(* IEC 61131-3 sources: tf-plc/examples/models/structured_text (part 7) *)

    weights_2 : ARRAY[0..287] OF REAL := [-0.187368, -0.051744, -0.039838, -0.182706, 0.020143, 0.109520, 0.194103, 0.170830, 0.202326, -0.167691, -0.195653, -0.237644, 0.106375, -0.036592, -0.006802, 0.135748, 0.022817, -0.062333, -0.017378, 0.128592, 0.187297, 0.185332, -0.152342, -0.201742, -0.104000, 0.041331, 0.068691, -0.044867, -0.198049, 0.149257, 0.125627, -0.021191, 0.074122, -0.145982, 0.118018, -0.081354, -0.131859, -0.051540, 0.168976, 0.046712, -0.040107, -0.054049, 0.084196, -0.269932, -0.139673, -0.139174, 0.131241, -0.010010, 0.138380, -0.188378, -0.036906, 0.057354, 0.008294, -0.113937, -0.038322, -0.006458, -0.001382, 0.096871, -0.011427, -0.108642, -0.113846, 0.096256, -0.134778, -0.045314, 0.048023, -0.015410, -0.087083, 0.081638, 0.095536, 0.014215, 0.110213, 0.167564, 0.020146, -0.133820, -0.078020, 0.007872, -0.044209, 0.044677, 0.131990, -0.089845, 0.145099, -0.119614, -0.106027, -0.091758, 0.077236, 0.042917, 0.118902, 0.120238, -0.244683, 0.045377, 0.197385, -0.131725, 0.193356, 0.124749, -0.181955, 0.108950, 0.119074, -0.070678, -0.009053, -0.087902, -0.065026, 0.183027, -0.196468, 0.195945, -0.166252, -0.165656, -0.164554, -0.076295, 0.139092, 0.190423, -0.007008, 0.013343, 0.018061, -0.073660, -0.022792, 0.075813, 0.097410, 0.177929, -0.145417, 0.025251, 0.175258, -0.197919, -0.079814, -0.340062, -0.006446, 0.052857, 0.114206, 0.051889, 0.145295, -0.146757, 0.093871, -0.111949, -0.084611, -0.067383, -0.099881, -0.057531, -0.233824, -0.186072, 0.174656, 0.076755, 0.009728, 0.104689, 0.106295, -0.179713, -0.113384, 0.079812, 0.132616, 0.004269, -0.171604, -0.030952, -0.045874, -0.015698, 0.004115, 0.010316, -0.183566, 0.082135, 0.082901, 0.090530, 0.143641, -0.040666, -0.152231, 0.207951, 0.124544, 0.016117, 0.046549, 0.030973, 0.043746, 0.036781, -0.086853, -0.171788, -0.013353, 0.078074, -0.141704, -0.113534, -0.045675, 0.082511, 0.031405, 0.099222, 0.061383, -0.090559, 0.025971, 0.117368, -0.137792, -0.203968, -0.087473, 0.150403, 0.221516, -0.053973, 0.100427, -0.012862, 0.224251, 0.226762, -0.101491, 0.057445, 0.086675, 0.134510, -0.058083, -0.216293, -0.036254, -0.225297, -0.080859, 0.008825, 0.033891, 0.143634, 0.059084, 0.023081, 0.094791, -0.194769, -0.001480, 0.073488, 0.115785, -0.061513, -0.130487, 0.057053, 0.185202, -0.062696, -0.098506, -0.052882, -0.012272, -0.177827, 0.048385, 0.121327, 0.044788, -0.111825, -0.129649, 0.139996, 0.051313, -0.047422, -0.002531, -0.233266, -0.124867, -0.128167, -0.082153, -0.073802, 0.102312, -0.003983, 0.033367, -0.024256, -0.227793, -0.130058, -0.093124, -0.002918, 0.156583, -0.133267, -0.070283, -0.019832, 0.240679, 0.192125, 0.226900, -0.215979, -0.037737, -0.027495, 0.257100, 0.067004, 0.162718, -0.035639, -0.025185, 0.145988, -0.062046, 0.179573, 0.208897, -0.050213, 0.200720, 0.185337, 0.195171, 0.145625, 0.199399, 0.174908, -0.021887, 0.128953, -0.153483, -0.080969, -0.116301, 0.002837, 0.088707, 0.122016, -0.069452, -0.073120, -0.099167, -0.086314, 0.211113, 0.213622, 0.087920, -0.150208, -0.143647, -0.111789, 0.093171, 0.048712];
    bias_2 : ARRAY[0..2] OF REAL := [0.178373, 1.153172, -1.176576];

END_VAR

VAR
    (* Buffer allocation variables *)
    buffer_0 : ARRAY[0..95] OF REAL;
    buffer_1 : ARRAY[0..127] OF REAL;

    (* Temporary computation variables *)
    i : DINT;
    j : DINT;
    sum : REAL;
    max_val : REAL;
    exp_sum : REAL;

END_VAR

(* Layer 0: Fused Linear + RELU *)
FOR j := 0 TO 127 DO
    sum := 0.0;
    FOR i := 0 TO 4 DO
        sum := sum + input_data[i] * weights_0[i * 128 + j];
    END_FOR;
    buffer_1[j] := MAX(sum + bias_0[j], 0.0);
END_FOR;

(* Layer 1: Fused Linear + RELU *)
FOR j := 0 TO 95 DO
    sum := 0.0;
    FOR i := 0 TO 127 DO
        sum := sum + buffer_1[i] * weights_1[i * 96 + j];
    END_FOR;
    buffer_0[j] := MAX(sum + bias_1[j], 0.0);
END_FOR;

(* Layer 2: Fused Linear + SOFTMAX *)
FOR j := 0 TO 2 DO
    sum := 0.0;
    FOR i := 0 TO 95 DO
        sum := sum + buffer_0[i] * weights_2[i * 3 + j];
    END_FOR;
    output_data[j] := sum + bias_2[j];
END_FOR;

max_val := output_data[0];
FOR i := 1 TO 2 DO
    IF output_data[i] > max_val THEN
        max_val := output_data[i];
    END_IF;
END_FOR;

exp_sum := 0.0;
FOR i := 0 TO 2 DO
    output_data[i] := EXP(output_data[i] - max_val);
    exp_sum := exp_sum + output_data[i];
END_FOR;

FOR i := 0 TO 2 DO
    output_data[i] := output_data[i] / exp_sum;
END_FOR;

END_FUNCTION_BLOCK

(* ---- test6_52k.st ---- *)
FUNCTION_BLOCK NeuralNetworkFB

VAR_INPUT
    input_data : ARRAY[0..4] OF REAL;
END_VAR

VAR_OUTPUT
    output_data : ARRAY[0..2] OF REAL;
END_VAR

VAR CONSTANT
    weights_0 : ARRAY[0..1279] OF REAL := [-0.070155, -0.038928, -0.060831, 0.071798, 0.002485, -0.001928, 0.071168, 0.040746, -0.011541, 0.011445, 0.033770, -0.092213, 0.017192, -0.118437, -0.098900, -0.051498, 0.004445, -0.006958, -0.025937, -0.127331, -0.033657, -0.020618, -0.089709, 0.067849, 0.032140, 0.027497, 0.034283, 0.044327, -0.041753, -0.071082, -0.023682, -0.090062, 0.088008, 0.007363, -0.073022, -0.031094, 0.042343, -0.067819, -0.017369, 0.056200, -0.086665, 0.056540, 0.024530, -0.093938, 0.012128, -0.109124, 0.043440, -0.042579, -0.016699, 0.004629, -0.082224, 0.015294, 0.014115, 0.027542, 0.014956, -0.021326, -0.135801, -0.044497, 0.006702, -0.013372, 0.013572, -0.004992, -0.067393, 0.015628, -0.044148, -0.024818, -0.001204, -0.007329, -0.112170, -0.094539, 0.009056, -0.031292, 0.066635, -0.026743, 0.002959, -0.164818, 0.041633, -0.146296, -0.119213, -0.024292, -0.025669, -0.181450, -0.006220, -0.075742, -0.011598, -0.002342, -0.026022, -0.097560, -0.021554, -0.012841, -0.050252, -0.103415, -0.029755, 0.012920, -0.010506, 0.006163, -0.086429, -0.082030, 0.041432, -0.020474, 0.059144, -0.007111, 0.003627, -0.155405, 0.002022, -0.031367, 0.028444, 0.041676, 0.054722, -0.002389, -0.071904, -0.012697, -0.021735, 0.006464, 0.051797, -0.067293, -0.057014, 0.035573, -0.061071, -0.045083, 0.003018, 0.041802, -0.097514, 0.002537, -0.057788, -0.071212, -0.054268, -0.012065, -0.017229, -0.022461, 0.063413, 0.005719, 0.022329, -0.099895, -0.169818, -0.108498, -0.092381, -0.012462, -0.023149, -0.024445, 0.001542, -0.032483, -0.113439, -0.054737, -0.004174, -0.010661, -0.019861, 0.037820, -0.132428, 0.022416, 0.011167, -0.055828, -0.034627, -0.058847, 0.018462, 0.025207, 0.008687, -0.013364, 0.049810, -0.020141, -0.018092, 0.025560, -0.021438, -0.034213, -0.023112, -0.027428, -0.112417, -0.060424, -0.006416, -0.000760, -0.237476, -0.086897, -0.081624, -0.070778, -0.009070, 0.027652, -0.129067, -0.014944, 0.070686, -0.006345, 0.018438, -0.048882, -0.056557, 0.062420, -0.013772, 0.014728, -0.015230, -0.076275, 0.001375, -0.011276, 0.055686, -0.049352, -0.030465, -0.023252, 0.003113, -0.023272, -0.035683, -0.076872, -0.011587, 0.004628, -0.030451, -0.045972, -0.004618, -0.025772, -0.087139, 0.004941, -0.025864, 0.024506, -0.078173, -0.092430, 0.019720, -0.007388, -0.031572, -0.029024, -0.016634, 0.007754, -0.131151, 0.000328, -0.051390, -0.012149, 0.023158, -0.010932, 0.001055, 0.019128, -0.102080, -0.010931, -0.004006, 0.002197, -0.046069, -0.077169, 0.041212, -0.009728, 0.006004, -0.136275, 0.041067, 0.023654, 0.053500, 0.007832, -0.052076, -0.010449, -0.061968, 0.004481, -0.017595, -0.114258, -0.086593, -0.011651, 0.022509, -0.070902, -0.014800, -0.082160, -0.123492, -0.043907, 0.016663, -0.004434, -0.054333, 0.003070, 0.089158, 0.025455, 0.057796, -0.060061, -0.053971, -0.149259, -0.048506, -0.131124, -0.069589, -0.080767, -0.101356, 0.024470, 0.060420, 0.024438, -0.048683, 0.003822, 0.001343, -0.000167, 0.044828, 0.070380, -0.072733, -0.003184, 0.066587, -0.008192, -0.074305, -0.068878, -0.004405, -0.115034, 0.052002, 0.015329, -0.068499, 0.086396, 0.005960, -0.052240, 0.085370, -0.002848, -0.093293, 0.056188, -0.044788, -0.007773, 0.056717, 0.055797, 0.034819, 0.070412, 0.016734, 0.026962, -0.057618, 0.037052, -0.052987, -0.121634, 0.024814, -0.146882, -0.013487, -0.083349, -0.024382, 0.026361, 0.101833, -0.002916, -0.006728, 0.015952, -0.015001, -0.004409, 0.042099, -0.126239, -0.019967, -0.013365, -0.089322, -0.006933, 0.059515, 0.037254, 0.045940, -0.074429, 0.040376, -0.027424, -0.080917, 0.035436, -0.094184, 0.086872, 0.085092, -0.091239, -0.026700, 0.043759, -0.012511, 0.063707, -0.027418, -0.008543, -0.119174, 0.009577, -0.061811, -0.094772, -0.022777, 0.022945, -0.005291, -0.032016, -0.059554, 0.046357, 0.075232, 0.040890, -0.148068, -0.049176, -0.063437, -0.004632, -0.026976, 0.105835, -0.039771, -0.031932, 0.011247, -0.132174, -0.032898, -0.073880, 0.088190, -0.053595, -0.043657, -0.188433, 0.014483, -0.032608, 0.091753, -0.101293, 0.051511, 0.070593, 0.004308, -0.037419, 0.076578, -0.054873, 0.099081, 0.003978, -0.081189, -0.127868, 0.054014, 0.114358, -0.023209, -0.011056, -0.110387, 0.098939, 0.080905, 0.080982, 0.096756, -0.078019, 0.020367, -0.011403, -0.049023, 0.027064, 0.045508, -0.029634, -0.027102, -0.001639, -0.051489, 0.038324, -0.060108, -0.090780, -0.070994, 0.013411, 0.029360, 0.048912, 0.032128, -0.033461, -0.088759, -0.006212, -0.115797, -0.025116, -0.056739, -0.064863, -0.018670, -0.114987, -0.056438, -0.030989, 0.092064, 0.189426, -0.025521, 0.023734, 0.049321, 0.059772, 0.003554, 0.131488, 0.021443, -0.112435, 0.054834, 0.073230, -0.001986, -0.073395, -0.088302, -0.088925, -0.006384, -0.017310, -0.022798, -0.173727, -0.023516, 0.107446, -0.011929, -0.035021, 0.039987, -0.033331, 0.028726, 0.007168, -0.073183, -0.021234, 0.039145, 0.072611, -0.171738, 0.066412, 0.031766, -0.144949, -0.042576, 0.096573, 0.008219, -0.068725, 0.015551, 0.032414, 0.043340, 0.033251, -0.078822, -0.124831, -0.110806, -0.004724, 0.045751, -0.038142, 0.191380, -0.055027, 0.060193, -0.041085, -0.025719, 0.040618, -0.056256, -0.008186, 0.069378, -0.035653, -0.084666, -0.038777, -0.058272, 0.019557, -0.136677, 0.065821, -0.102945, 0.050225, 0.018768, -0.064491, -0.091170, -0.006610, -0.032372, -0.123312, -0.026740, 0.070938, 0.001682, 0.065152, 0.035602, -0.010920, -0.117728, -0.045748, -0.028254, 0.012258, 0.147745, -0.019861, 0.060016, -0.048321, 0.020267, -0.102670, 0.020371, 0.036374, 0.049515, -0.085354, -0.004292, 0.032160, -0.047433, 0.015542, 0.003641, -0.001895, 0.039274, -0.046615, -0.016797, 0.007867, 0.096931, -0.006988, -0.073010, 0.025101, -0.081308, 0.030847, 0.031478, 0.015346, -0.066517, -0.199175, 0.092511, -0.083915, -0.144285, 0.058104, -0.086546, -0.018784, 0.035585, -0.058032, 0.018627, 0.052126, 0.017639, -0.000476, 0.115320, -0.064683, -0.022925, 0.007203, -0.020902, -0.037572, -0.042251, -0.046520, -0.123537, 0.049099, -0.212938, 0.041265, 0.029031, 0.034293, 0.038876, 0.019368, -0.166769, -0.036728, 0.011981, -0.056179, 0.014853, -0.017817, -0.052471, -0.052235, -0.109694, -0.017080, 0.027348, 0.072501, -0.023639, 0.039061, -0.021487, 0.004655, -0.077402, -0.030520, 0.049986, 0.015832, -0.107897, 0.019971, 0.077300, -0.067741, -0.016473, -0.016751, -0.142127, 0.027512, -0.076044, -0.049235, -0.036304, 0.005174, 0.034315, -0.048157, -0.019821, 0.034346, 0.021618, -0.014229, -0.108075, 0.031648, 0.023075, -0.146272, 0.066495, -0.103423, -0.090994, -0.007711, 0.138765, 0.023170, -0.011847, -0.025818, 0.004740, -0.090616, -0.039913, -0.036852, 0.018737, 0.024087, -0.099178, 0.090088, -0.022893, -0.002647, -0.036183, 0.054486, -0.109386, 0.009673, -0.054158, -0.036976, 0.037600, 0.022299, -0.092783, -0.059639, 0.001632, -0.018608, -0.112979, 0.022739, 0.040180, -0.030441, -0.105134, 0.033549, -0.106905, -0.046508, -0.094102, 0.000469, 0.057010, 0.023167, -0.086274, 0.045263, -0.049488, -0.052119, -0.037550, -0.022030, -0.010889, 0.003728, -0.008856, -0.083921, 0.133954, -0.080053, -0.017677, 0.094552, 0.068978, 0.020386, -0.025452, -0.168631, -0.090440, -0.195507, -0.003636, -0.084083, -0.068182, 0.058592, 0.029474, 0.040437, 0.061063, 0.025880, -0.001188, 0.000644, 0.010631, -0.110092, -0.000888, -0.141433, 0.108213, -0.022925, 0.000002, -0.130711, -0.062924, 0.008210, 0.019788, -0.175506, -0.039343, 0.045400, 0.123293, 0.092991, 0.016389, 0.004282, -0.004402, 0.075178, 0.003878, -0.106472, -0.002041, -0.004386, -0.036288, -0.002075, -0.062324, -0.014999, 0.041272, -0.017299, -0.065019, 0.063675, -0.028323, 0.020868, 0.058101, -0.043334, -0.045801, -0.052023, -0.069590, 0.053231, -0.069505, -0.033325, -0.063689, 0.014256, -0.067391, 0.005150, 0.014229, -0.018608, -0.039890, -0.104577, -0.153014, 0.020215, -0.030304, 0.036193, -0.106386, 0.008862, 0.040607, 0.011998, -0.043155, -0.008992, -0.005723, -0.012143, 0.037371, -0.016482, 0.095962, 0.051428, 0.012461, 0.050556, -0.075283, 0.013162, -0.012846, 0.062124, 0.080743, -0.025501, 0.139815, -0.065035, -0.005680, 0.005855, 0.048577, -0.014476, 0.120541, 0.069732, 0.030624, 0.049617, -0.192638, -0.032519, -0.154690, -0.022641, -0.025504, 0.012953, -0.027163, -0.031450, 0.065519, -0.104127, 0.037112, -0.119223, -0.095449, 0.035030, 0.034269, 0.024936, -0.046396, -0.025763, 0.005578, -0.043447, 0.019468, 0.028594, 0.004105, -0.158852, 0.010332, -0.055373, -0.080652, -0.053025, 0.093439, -0.167693, -0.056412, 0.084124, 0.138518, 0.010848, 0.047750, 0.065364, -0.054384, -0.045877, -0.157582, -0.058733, 0.018936, 0.010344, -0.077384, 0.028530, -0.036928, -0.080216, -0.012947, -0.183244, -0.072780, 0.075381, 0.062871, -0.028872, -0.298677, -0.122305, 0.024540, -0.183726, -0.086483, 0.028399, -0.020734, -0.022262, -0.050299, 0.060296, -0.118434, 0.011326, -0.046636, -0.025086, 0.066485, 0.015072, -0.007407, -0.044429, 0.119766, -0.047552, 0.063841, 0.005677, -0.020033, -0.024924, -0.233876, -0.022696, -0.111984, -0.043489, -0.051726, 0.036200, 0.070647, -0.001496, 0.052031, 0.090468, -0.004369, -0.060146, 0.019014, -0.042590, 0.009331, 0.075433, 0.015205, 0.045605, -0.016796, -0.001694, -0.110277, -0.107970, -0.011359, 0.017214, -0.087149, -0.066041, -0.040559, 0.002534, 0.000869, -0.049051, -0.134641, -0.071958, -0.090083, -0.033740, -0.027785, -0.014719, -0.067009, 0.054519, -0.112509, -0.141188, -0.101297, 0.027771, -0.021707, -0.026334, -0.046971, 0.081692, -0.052515, 0.042934, 0.002791, -0.025111, -0.005613, -0.003938, -0.041332, -0.026735, -0.021925, -0.056798, 0.066753, -0.013360, 0.035447, 0.029946, -0.050330, -0.020345, 0.102162, -0.016480, -0.009511, 0.017979, -0.000835, -0.016305, -0.005105, -0.034165, -0.094269, -0.030100, -0.018412, -0.009383, 0.003034, 0.058877, -0.094282, -0.001475, -0.008207, -0.135370, -0.018500, -0.028991, 0.023336, -0.155066, 0.068173, 0.106962, 0.025825, -0.009390, 0.192936, -0.002078, -0.033218, -0.064921, -0.042340, 0.023166, 0.001465, 0.003338, -0.087242, 0.088695, -0.064151, 0.023704, -0.042815, 0.040228, -0.088100, 0.029738, 0.052976, -0.017066, -0.013374, -0.115260, -0.151356, -0.057710, -0.126411, 0.031555, -0.056856, 0.036591, 0.034966, 0.008604, -0.002094, -0.092756, -0.202693, 0.028386, 0.024546, 0.076751, 0.017080, -0.018400, -0.037468, 0.032381, -0.089056, -0.187506, 0.129519, -0.021868, -0.080211, 0.100733, 0.030251, -0.004738, -0.024252, -0.009992, -0.027219, -0.172047, 0.029982, -0.126244, 0.126345, -0.019377, 0.012645, -0.025258, -0.065075, 0.028387, -0.041856, -0.017149, 0.030092, 0.000136, -0.004336, -0.093402, -0.012175, 0.005064, 0.021007, 0.024673, 0.024129, -0.034974, 0.004802, -0.013058, -0.053403, -0.190563, -0.019771, -0.090807, 0.061242, -0.032385, 0.046829, 0.005640, -0.098551, 0.083228, -0.062776, -0.092552, -0.069659, -0.059411, -0.109861, -0.007731, -0.057467, -0.123494, 0.004573, -0.083022, -0.016332, 0.051041, 0.110085, 0.073775, 0.004332, 0.020398, -0.023250, -0.240979, 0.044898, -0.046601, -0.058876, 0.054855, 0.074309, -0.081339, -0.042678, -0.073336, -0.128968, -0.047388, 0.046222, -0.051490, -0.121539, -0.014110, 0.015559, -0.096600, -0.026040, 0.032576, -0.048588, -0.136002, -0.095979, 0.036955, 0.120072, 0.117148, -0.211939, 0.082600, -0.083967, 0.111170, -0.045167, -0.052241, -0.135401, -0.065841, -0.088071, -0.020966, -0.022402, -0.022904, 0.015520, 0.135462, -0.039160, 0.030723, 0.095178, -0.072782, -0.122238, 0.017292, 0.137500, -0.023816, -0.043778, 0.078469, -0.029312, -0.022650, 0.019829, -0.054630, 0.004616, -0.052215, -0.042087, -0.029251, -0.010856, 0.017121, 0.000070, -0.000649, -0.167285, -0.133736, -0.115300, -0.070077, -0.072475, -0.028821, 0.017386, -0.026148, -0.075110, -0.140864, -0.265319, 0.034329, -0.032104, -0.108525, 0.078500, -0.021793, -0.019431, -0.080346, 0.010413, -0.075056, -0.007622, 0.000705, 0.074607, -0.090247, -0.168186, -0.039990, 0.031701, -0.071391, -0.018511, 0.014074, -0.022277, -0.023848, -0.025741, 0.026712, -0.067890, -0.028615, -0.066786, -0.023857, 0.044643, -0.013439, 0.111842, -0.073162, 0.005626, 0.026295, 0.080199, -0.108263, 0.001735, -0.108968, -0.149550, -0.043386, -0.001566, 0.012777, -0.011432, -0.195532, -0.000366, -0.033416, -0.085170, -0.005145, -0.030513, -0.069574, -0.100038, -0.027521, -0.074923, -0.100165, -0.104816, -0.065458, -0.013671, -0.442613, 0.025321, -0.030204, 0.013435, -0.012925, 0.006500, -0.379789, -0.014098, -0.052213, -0.030067, -0.087624, 0.038926, -0.044570, 0.059827, -0.018701, -0.029826, -0.133173, -0.116575, -0.012915, -0.023978, -0.024605, -0.153727, 0.037398, -0.021229, -0.068256, 0.080290, 0.051136, -0.059677, -0.024896, -0.248148, -0.052647, -0.045824, -0.042903, -0.291025, -0.024924, -0.014856, -0.032847, -0.013471, -0.064484, -0.000900, -0.064762, 0.063787, -0.061784, 0.022854, 0.069113, -0.139692, -0.025717, 0.024155, 0.025020, 0.013773, -0.025551, -0.028811, 0.002795, -0.056229, -0.253997, -0.059094, -0.055135, -0.027552, -0.055112, -0.061042, -0.090559, -0.302910, -0.153096, -0.108954, 0.002854, -0.065210, -0.058173, 0.042017, -0.152229, -0.018775, -0.276441, 0.115907, -0.061645, -0.046450, 0.088557, -0.030303, 0.108731, -0.035072, -0.089776, -0.036277, 0.031124, -0.120535, -0.084175, -0.034725, -0.048802, -0.314331, 0.044946, -0.064024, 0.040152, -0.048355, -0.067662, -0.021274, -0.042630, -0.228118, -0.142731, -0.022468, -0.072343, -0.034337, -0.025426, -0.029231, -0.028560, -0.059697, -0.185525, -0.011706, -0.098026, 0.066904, -0.028047, 0.102726, 0.096580, -0.092999, -0.048373, -0.263141, 0.136710, -0.097510, -0.041869, 0.014649, -0.041501, -0.043015, -0.089343, -0.077332, -0.101542, -0.098549, -0.095657, -0.183604, -0.095671, -0.010110, -0.157311];
    bias_0 : ARRAY[0..255] OF REAL := [1.761415, 0.448067, -0.616874, -0.484059, 0.264607, -0.939340, 1.879217, 0.387234, -0.224406, -0.592480, 0.573221, -0.500961, -1.606627, 0.053632, -0.815345, -0.331633, -0.254809, 0.114883, 0.034678, -0.491211, -0.556383, 0.517875, -0.619894, -0.175753, -1.234692, -0.794876, 0.608074, -1.463195, -0.042061, -0.962730, -0.235608, 0.198914, -0.023740, 0.011105, 0.650481, 0.174745, 0.899415, -0.358974, -0.603442, -1.367541, -0.065719, -0.929502, -0.847885, -0.365598, -0.106994, -0.493744, -0.071272, -0.507953, -0.072654, 0.642076, -0.468674, -0.864381, -1.117401, -0.245438, -0.073791, -0.435633, 0.299667, -0.095896, -0.052645, 0.095357, -0.586712, -0.615622, -0.026960, -0.250394, -0.784761, -0.225061, -0.657271, -0.407327, -0.230763, -0.098783, -0.037782, 0.199574, 0.593063, -0.725165, -0.492830, 0.248655, -1.223977, 0.003933, -0.103927, -0.255865, -0.239717, 0.080054, -0.552899, -0.238874, -1.349266, 0.138204, -1.088216, -0.206781, -0.391251, -0.378652, -0.585402, -0.228141, -0.377184, -0.224824, -0.723177, -0.617806, 0.083839, -0.155374, 1.478903, -0.308232, -0.179639, -0.159381, -0.263020, -0.181034, -0.507353, -0.264171, -1.168516, -0.972790, 0.189400, 0.139605, 0.125825, -0.717963, -0.294487, -0.057633, 0.015071, 0.269775, -0.534699, -0.084028, -0.079780, -0.401683, 0.027464, 0.074169, -0.013114, 0.126892, -0.778323, 0.311368, -0.224082, -1.059481, -1.343553, -0.005818, -0.149338, 0.081988, -0.058032, -0.328252, -0.384153, 0.146061, -0.012248, -0.017525, -0.254924, -0.230246, -0.753802, -0.348697, -0.681305, -0.580557, -0.063855, 1.148852, 0.216549, 1.353733, -0.041907, -0.766222, -0.039394, -0.722909, -0.515027, -0.293167, -1.141858, -0.532181, -0.700502, -0.093383, 0.853853, -0.491534, -0.364100, 1.343948, 0.206487, -0.739496, -0.120556, -0.194485, 0.531750, -0.071946, -0.429285, -1.223201, -0.799083, -0.240277, -0.253012, -1.097437, 1.321796, -0.732158, -0.643209, 0.023920, -1.042058, -0.577268, -0.130637, -0.380038, -0.697286, 0.272227, -0.397080, -0.299311, -0.152759, -0.012990, -0.102990, -0.175804, 0.514636, 0.076499, -0.173979, -0.501178, -0.362724, -0.373031, -0.193449, 0.413115, -0.477030, 0.085947, -0.924347, -0.343727, 0.956858, -1.252704, 0.042583, -0.986913, 0.150553, 0.331016, 0.022171, 0.308270, -0.172095, -0.276784, -0.621540, -0.314609, 0.217584, 0.068779, -0.080378, -0.521706, -0.216527, -0.760283, -0.076289, 1.077613, 0.342408, 1.537670, -0.199558, 0.696804, -0.477082, -0.216091, -0.627426, -0.344922, -0.476790, 0.048585, -0.653165, 0.220433, -1.102417, 0.015778, -1.255825, -1.064247, 0.158786, 1.424948, -0.014341, -1.144714, 0.264992, -0.409402, -0.673654, 0.344695, -0.371929, -0.803940, 0.197236, 0.139407, -0.046033, -0.167134, -0.541114, -0.539192, -0.470981, -0.991606];

    weights_1 : ARRAY[0..50175] OF REAL := [0.019087, 0.112252, 0.211727, 0.072814, 0.087899, -0.175614, -0.015506, 0.164059, 0.236532, -0.229048, -0.055866, 0.004746, 0.085537, -0.126006, -0.170778, 0.039044, -0.227048, -0.200908, 0.085609, -0.210631, 0.017052, 0.078471, -0.091614, -0.312604, -0.219523, -0.039882, 0.227878, 0.098304, 0.053254, 0.175391, 0.027453, 0.004954, 0.256044, 0.220982, -0.118379, -0.043911, 0.113699, -0.067441, 0.121477, -0.081606, 0.017963, -0.108318, -0.122663, 0.122943, -0.098493, -0.129229, -0.104070, -0.040965, -0.030263, 0.103501, 0.114757, -0.033213, -0.097106, -0.003870, -0.064622, -0.031450, 0.136162, 0.043457, 0.119389, 0.086272, 0.086328, -0.054092, 0.022835, 0.076201, 0.115069, -0.146640, -0.019403, 0.182401, -0.070480, 0.040452, 0.252047, 0.027936, 0.131226, -0.044332, -0.068760, -0.075233, 0.136624, 0.010865, 0.031996, 0.217943, 0.132278, 0.094806, -0.081434, -0.018107, -0.011303, -0.132485, -0.155610, 0.010216, 0.251893, 0.008599, 0.088021, -0.110349, -0.184611, -0.165733, -0.023405, 0.070966, 0.052070, -0.066027, 0.206689, -0.139396, 0.065651, 0.040476, 0.265397, 0.200300, -0.161854, -0.035440, -0.100544, 0.060114, 0.132822, 0.181317, 0.162731, -0.157100, 0.032291, -0.024872, 0.026177, -0.062704, -0.227261, -0.061749, 0.001810, 0.143090, 0.297814, -0.094348, -0.189725, 0.023125, 0.100221, -0.079787, 0.014617, 0.045027, 0.126831, 0.107187, -0.033158, 0.172206, 0.084450, 0.023537, -0.137875, -0.059479, -0.015502, 0.066624, -0.388477, 0.056747, 0.095752, -0.076781, -0.090368, -0.033154, 0.006288, 0.066518, -0.177086, 0.016229, 0.237689, -0.198316, -0.126118, -0.093328, 0.283691, -0.024487, -0.033743, -0.047251, 0.048239, 0.011724, 0.182427, -0.122201, -0.063529, 0.153458, -0.024413, 0.046109, -0.057552, -0.027173, 0.109429, 0.110716, 0.187617, 0.078747, 0.105684, 0.073501, -0.010930, 0.094036, 0.255130, -0.016355, 0.064772, 0.166211, 0.051418, -0.100114, 0.103828, -0.122074, -0.013134, -0.013142, 0.051070, -0.141888, -0.073589, 0.047752, 0.118184, -0.150595, -0.069933, -0.111839, 0.201886, 0.157238, -0.000566, -0.241842, -0.103816, -0.167649, 0.036014, -0.071474, -0.197229, -0.093806, -0.117186, -0.121392, 0.090752, 0.057172, -0.101006, -0.146829, -0.162285, -0.114287, 0.041882, -0.021359, 0.039685, -0.051023, -0.088828, -0.130283, 0.071467, -0.027591, 0.063893, -0.060089, -0.039073, -0.080926, -0.039526, -0.175741, -0.072726, -0.002156, -0.064652, -0.032380, -0.078773, -0.139573, -0.095449, 0.025900, 0.061990, 0.011282, -0.073379, -0.164573, -0.087662, -0.047434, -0.138482, 0.065975, 0.141275, 0.072849, 0.009651, 0.000184, 0.034366, -0.001639, 0.064527, -0.039849, 0.042872, -0.078356, -0.159165, -0.127313, 0.015479, -0.087568, 0.051244, -0.121865, 0.175445, 0.066785, -0.115017, -0.018106, -0.043598, -0.076265, 0.050338, 0.012569, -0.034868, 0.027134, -0.010178, -0.155097, -0.073559, -0.000278, -0.203096, -0.004941, -0.078585, -0.036923, -0.136309, 0.039640, 0.015160, -0.024950, -0.040108, 0.099179, -0.043566, -0.138085, 0.057145, -0.027623, 0.116453, 0.067655, -0.149188, -0.011659, -0.000152, -0.117239, -0.058557, -0.025922, -0.115761, -0.008718, 0.041052, 0.021877, -0.164530, -0.025719, 0.039448, -0.033210, -0.094054, -0.074904, -0.038552, -0.028109, 0.020906, 0.042368, -0.050518, -0.069741, -0.009646, -0.030400, 0.121980, -0.068921, -0.010179, 0.075115, -0.071092, -0.000068, 0.128066, -0.175240, -0.048073, -0.201908, 0.025278, -0.106169, -0.136777, -0.038482, -0.042894, -0.052749, 0.034706, -0.067714, 0.011700, -0.130630, 0.012471, 0.040072, 0.030638, 0.185444, 0.078900, -0.113858, 0.072917, -0.095026, -0.064184, -0.069011, -0.084066, -0.010202, -0.007493, -0.054461, 0.132179, -0.108565, -0.133447, -0.020019, 0.089484, 0.010921, -0.015147, -0.073809, -0.164842, 0.019242, -0.128817, -0.021889, -0.098907, -0.155679, -0.077994, -0.055610, -0.079722, -0.093138, 0.089238, -0.071704, -0.084965, 0.003876, 0.010080, -0.184207, -0.008479, 0.002302, -0.123802, 0.014025, 0.039673, 0.027165, 0.140232, 0.081911, -0.104612, -0.136547, -0.125663, -0.017690, -0.028861, -0.128213, 0.053530, -0.037016, -0.005354, -0.007881, -0.072455, 0.075998, -0.150186, 0.003538, 0.025154, -0.181750, -0.005627, 0.015931, -0.145865, 0.164566, -0.022345, -0.086018, 0.052187, -0.007339, 0.163025, 0.085218, 0.076081, 0.144517, -0.071499, -0.039545, -0.047413, 0.016911, 0.129909, 0.120274, 0.052777, 0.029113, 0.102280, 0.120183, 0.012646, 0.080433, -0.019135, -0.114755, 0.075379, -0.077169, 0.044199, -0.147909, -0.122363, -0.066505, -0.016582, -0.016903, -0.069173, -0.002722, -0.042748, -0.019419, -0.013751, 0.110063, -0.042846, 0.029374, 0.013619, -0.084677, -0.082738, 0.017447, -0.019679, 0.008661, 0.089650, 0.223866, -0.037423, 0.058718, 0.223306, 0.035864, 0.061035, -0.054710, 0.075441, 0.058958, 0.202108, -0.101563, -0.099383, -0.008222, -0.200740, 0.097243, 0.014732, 0.154570, 0.043766, -0.009304, -0.055844, -0.018659, 0.183471, -0.023827, 0.070002, 0.041760, 0.167490, -0.048266, 0.108233, -0.010787, 0.121722, -0.003856, 0.025528, 0.020465, -0.052595, -0.048578, -0.036409, 0.000491, -0.016168, 0.053307, -0.145291, 0.054400, 0.187202, -0.089671, -0.101879, 0.162248, -0.019973, -0.055917, 0.119184, -0.150383, 0.042248, 0.096906, 0.109155, 0.080165, -0.009909, 0.280200, 0.051996, 0.042644, 0.000768, 0.002605, 0.072514, 0.213357, 0.038522, 0.085074, 0.070995, 0.219419, -0.074172, 0.008887, 0.246615, -0.095728, -0.020076, 0.116962, 0.027811, -0.013989, 0.056890, 0.101884, 0.060451, -0.099294, 0.022870, 0.156072, -0.047571, -0.026024, 0.058590, 0.019635, 0.026216, -0.001581, -0.081485, 0.033548, 0.034559, -0.034313, 0.048365, 0.110622, 0.094056, -0.001664, -0.018744, 0.050562, 0.021697, 0.056702, -0.092299, -0.073527, 0.006214, -0.079798, -0.052168, -0.086453, -0.006532, -0.010577, -0.029513, 0.105852, -0.275099, -0.128755, 0.041453, -0.093995, -0.003681, -0.124704, -0.124020, -0.049122, 0.117641, 0.059697, -0.044566, -0.101940, 0.188092, 0.142056, 0.134078, 0.041127, 0.035474, 0.107212, 0.060624, 0.034643, -0.181532, 0.039691, 0.012068, -0.031569, 0.090305, 0.069827, 0.143646, -0.038929, 0.079717, 0.128726, -0.068412, -0.046522, 0.105732, -0.025602, 0.079163, -0.096699, 0.045994, 0.034854, -0.067040, 0.086313, 0.064069, 0.036678, -0.156208, -0.150338, -0.102526, 0.039301, 0.086361, -0.024633, -0.132891, 0.080287, -0.100965, -0.057234, -0.111725, -0.022540, -0.090631, 0.031524, -0.120615, -0.017978, -0.022298, -0.006987, 0.061163, -0.102908, -0.148379, -0.098665, 0.018615, 0.056827, 0.089001, -0.013134, -0.003036, 0.143445, -0.010353, -0.062452, -0.013643, 0.092925, -0.034422, 0.085092, -0.043912, 0.076237, -0.048921, 0.056351, 0.061761, -0.141086, 0.003610, -0.085852, -0.045372, -0.121835, 0.088956, 0.082596, 0.034770, -0.057173, 0.029236, -0.166666, -0.009784, -0.116007, 0.000360, -0.056035, -0.068974, -0.045856, -0.091816, 0.026982, -0.136249, 0.016789, -0.079818, -0.083522, -0.032031, -0.117626, -0.064185, -0.216489, -0.129358, -0.072896, -0.075290, 0.053919, 0.022993, -0.031171, 0.036235, -0.062525, -0.079568, 0.104918, -0.111249, 0.090243, -0.156623, 0.106249, 0.110953, -0.002011, 0.011957, 0.076677, -0.117035, 0.045182, 0.084106, 0.054265, 0.049279, -0.170700, 0.088931, 0.077295, -0.106536, -0.223289, -0.180796, -0.054039, 0.063236, -0.039010, -0.003974, -0.097592, -0.099271, -0.088824, 0.036501, -0.121148, 0.071922, 0.064697, -0.030513, -0.146272, 0.033028, 0.146114, -0.181025, 0.025671, -0.066351, 0.005915, -0.036995, -0.065130, 0.010359, 0.143837, -0.194034, -0.035653, 0.072018, -0.101430, -0.324173, -0.106044, -0.043522, -0.049253, -0.088946, 0.142913, 0.064938, -0.135467, -0.037628, -0.108382, -0.075162, 0.025261, -0.026427, -0.002965, -0.103873, 0.026990, 0.118669, -0.077579, -0.118062, 0.075373, -0.055841, 0.047908, -0.016173, -0.000047, 0.001842, -0.132699, -0.101972, -0.085123, -0.123046, 0.083153, -0.157092, -0.147615, -0.186562, -0.079440, -0.104795, -0.187915, 0.067444, -0.061773, -0.064322, -0.030680, -0.058348, -0.057221, -0.095582, -0.133214, -0.052529, 0.121469, -0.059717, 0.041280, -0.148639, 0.101247, 0.064651, 0.078919, -0.041949, -0.182256, -0.070102, -0.029421, -0.115502, -0.129157, -0.025260, -0.034863, -0.042848, 0.080907, 0.051103, -0.032286, -0.061058, 0.069918, -0.038627, -0.005238, -0.002159, 0.084238, -0.109072, -0.080085, 0.127401, 0.106197, -0.017038, -0.080919, 0.011097, 0.049521, 0.059727, 0.024202, 0.088085, -0.092945, -0.052078, -0.042216, 0.048724, 0.046643, -0.045592, -0.176796, -0.037914, -0.008196, -0.042904, -0.077948, 0.020485, 0.026218, 0.061671, 0.059945, -0.016648, -0.121312, -0.098689, -0.181613, 0.078740, 0.023735, -0.098268, -0.071533, 0.035284, -0.056109, -0.001989, -0.139051, -0.020433, -0.004766, -0.007580, -0.174961, -0.092434, 0.066625, -0.117502, -0.037798, 0.057671, 0.053905, -0.065360, -0.019672, -0.186390, 0.002110, 0.100599, -0.014125, -0.004204, 0.122479, -0.104440, 0.035850, -0.152272, -0.026409, 0.114577, -0.067488, -0.091784, 0.008339, 0.052320, 0.048703, -0.062640, 0.025489, 0.095889, -0.023739, -0.097751, -0.099172, 0.053132, 0.114207, -0.177148, 0.105202, -0.111281, 0.038844, -0.015349, 0.056444, 0.054711, 0.136033, -0.082014, 0.010470, -0.030293, -0.099113, -0.047619, -0.181317, 0.103047, 0.127858, 0.078801, -0.086867, -0.117279, -0.033613, 0.019201, -0.180484, -0.154765, 0.061346, -0.064952, -0.056183, 0.084271, 0.102972, 0.065615, -0.111835, 0.056108, 0.176568, 0.016379, 0.017522, -0.142013, -0.007219, -0.104620, -0.144636, -0.063979, -0.060847, -0.032692, 0.122917, -0.147106, -0.062755, 0.012541, -0.148126, -0.043110, 0.021487, -0.009996, 0.061543, -0.206080, -0.195564, -0.020537, -0.133944, 0.025850, 0.096806, -0.112063, 0.029370, -0.049795, -0.056473, 0.055213, -0.151802, -0.160091, -0.151661, -0.038781, 0.036104, 0.053520, -0.132503, -0.032326, -0.077364, -0.217113, 0.053834, -0.219743, 0.105419, -0.095950, -0.151808, -0.066669, -0.081858, 0.098166, -0.021824, -0.067333, -0.019496, 0.015563, -0.059110, -0.076128, 0.178659, 0.091090, -0.074106, 0.070255, -0.077358, -0.112879, 0.077412, 0.025083, 0.026152, 0.012809, -0.142545, -0.087881, -0.015273, 0.178429, 0.170337, -0.106502, 0.054853, 0.021515, -0.089748, -0.100349, -0.164853, 0.000667, -0.090071, -0.008077, 0.185323, -0.085372, -0.112397, 0.014247, -0.083588, -0.036136, 0.127643, 0.064369, 0.073729, -0.050948, -0.014044, -0.182222, 0.056814, -0.056092, -0.040727, -0.213120, -0.098599, 0.045975, -0.181463, -0.071185, 0.100344, 0.052472, -0.215122, -0.065159, 0.015217, 0.032520, 0.094486, -0.197438, -0.026454, -0.044753, -0.152395, -0.051332, -0.019524, -0.172293, 0.082108, 0.142434, 0.074673, 0.074597, 0.078569, -0.072255, -0.136009, -0.056322, -0.054084, -0.104861, 0.044404, 0.076383, 0.033862, 0.080257, -0.058024, -0.078371, -0.097096, -0.063691, -0.029839, 0.044378, 0.078426, 0.033354, -0.070337, 0.138203, -0.142656, -0.056512, 0.021528, -0.066354, -0.083081, -0.236461, 0.064244, -0.153117, -0.029091, 0.042190, -0.117686, 0.145115, -0.048079, 0.099946, -0.071859, 0.059696, -0.095557, -0.054787, -0.122110, -0.088782, 0.083703, 0.048141, -0.064529, 0.005618, -0.097177, -0.110536, -0.142819, -0.065839, -0.094944, 0.018961, -0.099151, -0.198094, -0.013984, -0.011091, -0.008252, 0.022140, -0.039377, -0.010458, -0.208391, -0.091304, -0.078158, -0.049752, 0.125188, -0.100087, 0.097491, -0.116807, 0.004508, -0.070719, -0.002883, -0.030286, -0.030703, 0.005226, -0.262217, 0.022196, 0.015927, -0.040104, 0.068360, -0.026407, 0.046189, -0.049886, 0.173153, 0.108369, -0.022076, 0.064689, 0.085553, 0.000238, 0.044140, 0.093514, -0.045166, -0.012393, 0.079811, -0.082676, -0.056477, -0.087986, -0.100695, -0.041185, -0.146482, 0.023451, -0.058040, 0.058801, -0.107925, -0.152068, -0.172320, 0.044384, 0.052113, -0.172874, -0.170240, 0.014697, 0.150143, 0.081321, -0.030740, -0.113979, 0.022836, -0.167214, -0.050602, -0.099422, -0.131082, 0.038192, -0.082917, -0.108151, -0.052472, -0.134135, -0.045075, -0.064432, 0.250552, -0.143789, 0.015460, 0.180920, 0.029685, -0.050402, 0.035008, -0.073346, 0.071804, -0.157414, 0.052726, -0.118639, 0.065929, 0.069186, -0.253910, -0.017151, 0.089519, 0.183066, 0.137547, 0.122671, -0.145832, -0.008087, -0.051812, -0.036468, -0.046325, 0.043646, -0.134134, -0.129915, 0.044372, -0.091126, -0.050619, 0.050467, -0.013290, -0.031310, -0.114490, 0.042256, 0.070883, 0.047820, 0.008023, 0.104225, 0.125312, 0.034384, -0.039841, 0.094834, 0.042942, -0.005580, -0.257027, -0.154987, 0.009421, 0.045741, 0.080904, 0.035393, 0.111025, 0.082148, -0.089763, 0.035221, 0.094880, 0.108935, 0.001577, -0.023088, -0.037592, 0.033744, 0.075051, -0.100634, -0.053072, 0.026299, -0.003795, 0.127786, 0.094785, 0.232596, -0.056839, 0.033139, -0.090313, -0.149171, 0.117668, 0.174688, 0.097817, -0.145184, 0.068671, 0.180850, -0.030937, 0.215770, 0.156902, -0.119691, 0.059523, -0.055236, -0.226490, -0.237438, -0.127971, -0.000791, 0.089595, -0.034488, 0.138498, -0.114008, -0.028960, -0.095210, 0.029992, 0.065373, -0.151819, 0.062377, -0.041755, -0.059274, -0.054100, -0.021659, 0.089076, 0.127801, -0.023952, 0.062740, -0.032144, 0.187913, -0.136559, -0.009302, -0.007558, -0.169485, -0.084244, -0.059545, 0.105821, -0.120696, 0.141241, 0.203729, 0.148026, 0.088018, -0.080925, 0.096096, 0.027410, -0.156046, -0.158756, 0.032207, 0.007221, 0.344494, -0.036998, -0.047743, 0.016457, 0.005089, -0.000682, 0.026303, -0.014775, 0.272801, -0.041455, 0.040938, 0.034764, 0.050673, -0.038220, 0.033246, 0.098095, 0.027850, -0.073006, 0.074952, 0.005706, 0.013382, -0.220796, 0.209334, 0.253340, 0.031337, 0.113429, 0.034453, 0.138160, 0.212788, 0.110564, 0.160061, 0.014191, 0.106261, -0.065506, 0.137208, 0.003077, 0.046537, -0.163562, -0.144258, 0.061503, 0.115026, 0.044925, -0.009267, 0.176470, 0.109477, -0.039916, 0.146964, 0.099196, 0.162142, 0.030322, -0.117109, 0.178354, 0.090466, -0.161766, 0.029943, -0.106840, -0.093958, 0.130050, -0.092636, -0.082686, 0.043057, -0.182247, -0.096600, -0.133091, 0.119896, -0.046350, -0.116248, 0.022831, 0.122150, -0.086858, 0.044733, -0.128481, 0.018598, -0.042498, -0.018465, 0.121027, -0.045440, -0.043158, 0.112994, 0.066515, -0.055506, 0.001144, 0.001762, 0.128164, -0.065124, -0.054133, 0.214650, 0.041804, 0.315379, -0.032408, 0.087979, 0.072041, -0.196844, 0.080406, 0.153377, -0.137726, -0.022882, 0.227910, 0.062962, -0.147406, 0.159909, -0.097056, -0.016344, -0.160364, 0.119470, -0.030065, 0.065594, -0.051290, 0.007540, -0.129645, -0.129634, -0.144952, 0.107958, 0.022748, -0.052174, -0.087933, 0.025262, 0.066282, 0.039028, -0.114060, -0.033210, -0.030558, 0.055064, -0.064431, -0.213004, -0.010090, -0.107847, -0.006497, -0.144362, 0.336409, -0.050992, -0.051211, 0.062435, -0.039551, -0.094448, -0.045941, -0.073822, 0.133791, 0.063238, -0.032661, -0.072728, -0.010004, 0.012471, 0.067459, -0.130388, 0.066889, -0.184211, -0.082500, -0.053863, -0.072569, -0.052074, 0.048992, 0.081268, -0.091059, -0.053469, -0.175719, -0.087657, -0.209073, 0.016879, 0.031966, -0.084577, -0.177720, -0.081343, 0.101700, -0.153151, -0.138370, -0.075105, -0.008808, -0.074839, -0.050318, -0.163576, -0.170850, -0.221416, -0.110951, 0.081662, -0.028462, 0.047567, -0.184248, 0.040988, -0.091325, -0.143539, -0.030374, -0.002269, 0.152714, -0.017201, -0.094564, -0.052210, 0.041706, -0.090776, -0.131064, 0.015830, -0.150425, -0.154221, -0.068794, 0.060521, -0.191235, -0.001042, 0.282362, 0.042888, 0.055028, 0.098971, 0.038474, 0.014420, -0.022587, 0.035149, 0.047814, -0.025055, -0.021019, -0.111718, -0.287602, 0.000253, 0.050583, 0.012616, -0.040234, 0.154187, -0.077570, -0.045584, 0.044512, -0.047277, 0.007406, -0.014795, -0.181500, -0.125628, -0.021537, -0.046749, -0.140914, -0.053525, -0.243101, -0.137482, -0.104698, -0.096924, 0.033680, -0.056733, -0.030535, -0.075371, -0.102772, -0.183080, 0.049507, -0.100398, 0.036516, -0.210650, -0.021577, -0.077714, -0.159015, 0.183548, 0.037474, -0.016995, -0.046999, -0.227799, -0.079963, -0.026326, -0.037037, -0.091802, -0.113556, -0.060374, -0.009194, 0.096339, -0.025744, -0.082264, 0.103064, -0.117133, -0.039137, 0.033967, -0.087033, 0.174108, -0.132678, -0.167555, -0.008391, 0.004518, 0.023418, 0.029971, 0.004577, -0.076275, -0.121223, 0.051243, -0.016593, -0.073084, 0.117548, 0.027623, 0.088855, -0.164806, -0.057957, -0.058351, 0.076715, 0.019879, -0.008117, -0.117966, 0.187369, -0.072366, 0.178441, 0.093355, -0.116011, -0.138751, -0.062116, 0.012776, -0.008796, -0.163777, 0.067828, -0.116379, -0.085175, 0.024777, -0.116945, 0.017072, -0.128596, -0.113390, -0.038784, -0.124178, -0.126629, 0.006454, 0.099044, -0.091827, -0.007732, -0.160089, -0.078124, -0.009004, -0.004980, -0.013874, -0.102244, 0.081286, -0.020725, -0.018777, 0.020967, -0.080072, -0.066568, -0.053473, -0.020241, -0.088039, -0.095797, -0.141911, -0.164115, -0.077702, 0.016036, -0.011268, -0.045965, 0.014893, 0.012777, -0.102961, -0.189625, -0.095094, -0.049763, -0.075690, -0.120070, 0.028730, -0.067642, -0.001965, -0.007239, 0.064283, -0.151160, 0.044597, 0.014399, -0.062381, 0.002024, -0.083654, -0.064107, -0.119602, 0.022915, -0.080297, 0.013349, 0.062126, -0.072363, -0.207237, 0.003734, -0.043662, -0.158454, -0.114404, -0.101448, 0.020741, -0.206459, 0.059534, 0.090559, -0.143550, 0.001672, -0.031304, -0.038508, 0.053129, 0.175834, -0.014710, 0.036988, 0.019318, -0.027118, -0.038198, -0.136480, -0.175305, 0.018628, -0.031914, -0.024771, -0.010782, 0.033243, -0.155769, 0.067826, 0.003758, -0.039986, 0.073341, -0.109548, -0.063142, 0.076973, 0.012936, 0.115559, 0.059937, -0.018252, 0.059264, 0.008156, 0.055209, -0.020416, -0.028660, -0.093089, 0.070549, 0.079156, -0.054899, 0.045430, -0.146777, 0.199928, 0.191229, -0.108392, -0.009619, -0.022477, 0.075113, 0.048136, 0.132529, -0.016129, 0.125690, 0.024077, -0.002285, 0.022616, -0.134391, 0.047702, -0.029570, -0.115425, 0.069332, 0.001313, 0.079069, -0.113597, -0.112819, -0.019466, -0.113795, -0.040433, 0.056663, 0.122918, 0.026737, -0.034013, -0.107641, 0.026462, 0.036141, -0.031089, -0.054573, 0.007394, 0.060948, 0.030305, 0.077312, -0.007448, 0.030940, -0.002564, -0.136700, 0.062775, -0.130955, -0.051405, -0.134777, 0.029866, -0.063722, -0.118298, 0.014863, -0.041507, -0.046326, -0.099231, 0.012791, -0.089044, -0.134637, 0.191558, -0.076247, 0.074888, 0.015094, -0.011294, 0.011376, -0.162267, -0.135580, -0.059208, -0.103904, -0.056071, -0.085404, 0.114298, 0.032905, 0.115623, -0.051892, -0.038895, 0.015444, -0.039494, 0.035762, 0.070795, -0.157048, 0.038876, -0.196186, -0.045179, -0.077474, -0.007454, 0.005102, 0.066898, 0.027204, 0.009113, 0.052094, -0.065906, -0.171679, 0.046485, -0.098911, -0.007187, 0.000240, -0.033393, 0.070073, -0.030711, 0.073362, 0.035598, -0.002507, -0.201307, 0.028633, 0.080203, -0.196043, -0.065957, -0.125021, 0.001547, -0.192467, -0.151143, 0.004591, 0.119832, -0.070920, 0.086491, 0.142954, 0.045717, 0.061341, -0.202144, -0.060203, -0.063361, 0.034158, -0.014267, -0.133672, -0.084147, -0.068462, 0.055255, 0.091635, -0.001075, -0.013580, -0.000664, -0.099291, -0.061880, 0.056597, 0.013572, -0.112947, -0.073521, 0.069699, 0.026268, -0.121181, -0.118742, -0.064180, -0.091876, 0.082797, -0.212855, -0.067485, -0.011989, -0.055563, -0.113979, -0.085965, -0.023988, -0.079515, 0.054800, -0.062980, -0.053606, -0.013759, 0.014781, -0.032490, -0.023336, 0.179701, -0.113594, -0.011894, 0.057133, 0.070240, 0.151126, -0.113374, 0.022945, -0.020242, -0.011959, 0.048784, -0.018162, -0.004894, -0.050443, -0.106047, 0.066109, -0.044677, 0.050467, -0.095524, -0.159400, 0.101974, 0.159742, 0.080277, -0.092075, 0.087559, -0.052313, 0.031599, 0.030421, -0.118346, 0.000175, 0.071803, -0.040223, -0.179201, -0.055939, 0.103731, -0.078320, -0.012671, 0.056494, 0.030093, -0.079507, 0.109278, -0.065657, -0.102386, -0.085533, 0.050784, -0.205683, -0.046242, -0.066881, 0.060181, -0.120047, -0.076139, -0.201692, -0.100922, -0.021243, 0.015871, -0.078541, -0.002240, -0.030480, -0.095572, -0.072460, -0.228379, 0.122723, 0.072628, -0.252539, -0.277393, 0.006553, 0.009668, -0.154670, 0.002855, -0.092451, -0.008875, -0.039893, -0.040272, -0.034766, -0.116732, -0.077112, -0.141940, 0.029427, 0.068693, 0.222056, 0.187592, 0.030192, 0.038319, 0.112310, -0.194210, -0.066446, -0.000920, 0.130781, 0.072736, 0.077486, -0.187105, -0.120419, -0.128611, -0.143621, 0.010328, -0.081794, 0.054265, -0.019573, 0.010238, 0.057413, -0.159222, -0.036712, -0.093249, -0.087319, 0.081351, -0.001184, -0.181214, 0.126413, -0.190884, -0.080189, -0.055854, -0.028841, -0.027709, 0.120972, 0.116504, -0.121195, -0.107296, 0.041077, 0.020492, 0.087747, 0.043422, 0.126991, -0.044143, -0.118220, -0.020730, -0.083720, -0.018610, 0.035537, 0.026469, -0.096193, 0.194933, -0.012480, -0.093044, -0.098956, 0.072297, -0.115272, -0.063073, 0.115923, 0.046369, -0.007494, 0.045403, 0.037994, 0.098409, 0.132605, 0.017922, 0.045034, 0.023139, 0.050274, -0.078886, 0.041988, -0.023474, 0.085313, -0.110226, -0.169473, -0.236922, -0.182666, -0.162326, -0.053805, 0.135236, -0.330935, -0.060417, 0.164037, 0.061803, -0.082402, -0.126387, -0.118802, 0.005750, -0.043583, -0.071514, -0.060441, -0.153771, -0.083721, -0.095956, 0.145971, -0.019170, 0.037685, -0.158148, -0.066579, -0.104269, -0.044769, -0.027317, -0.155952, -0.079424, 0.097705, 0.078596, -0.092878, 0.029170, -0.035781, 0.109035, -0.122391, 0.035075, -0.023706, 0.052735, -0.052661, -0.145526, 0.028236, -0.027213, -0.054233, -0.030098, -0.018636, -0.055844, -0.209197, -0.106560, 0.081238, 0.109522, -0.205381, 0.099706, -0.091235, 0.001473, -0.117953, 0.019389, -0.177502, 0.102457, -0.072657, -0.221911, -0.067212, -0.031332, 0.137509, -0.034266, 0.006808, -0.139460, -0.045928, -0.022443, 0.016579, 0.164751, -0.028440, -0.093767, -0.025979, 0.015073, -0.140818, -0.025925, -0.172505, -0.121721, -0.001821, -0.029625, -0.090522, -0.014405, -0.034766, -0.164906, -0.133973, -0.083389, -0.077585, -0.028641, -0.208091, 0.212780, -0.124050, 0.070248, 0.010817, -0.142993, 0.081598, 0.053776, -0.111811, -0.008867, 0.003158, -0.162539, 0.009218, 0.122464, -0.009644, 0.000799, -0.143111, -0.101835, -0.024264, -0.154475, -0.106086, 0.114155, -0.058152, -0.058630, -0.090407, 0.131540, 0.054424, -0.042507, -0.127363, -0.027258, -0.010863, -0.203317, -0.054742, -0.051424, -0.034125, -0.112695, -0.138449, -0.075680, -0.028747, 0.117785, 0.004196, -0.044447, 0.107136, -0.189101, -0.064540, 0.026183, -0.057381, -0.104361, 0.008995, 0.016744, -0.023086, -0.165401, -0.165560, 0.095167, -0.044776, -0.145051, 0.063015, -0.077605, -0.153339, -0.088327, -0.231164, -0.181101, 0.048101, -0.097803, -0.026143, -0.064404, 0.079467, -0.023290, -0.103390, -0.009408, 0.053774, 0.093235, -0.029657, -0.182546, 0.026099, -0.033375, -0.009190, 0.032830, -0.107149, -0.032436, 0.052238, -0.263541, 0.037051, 0.029552, 0.056791, -0.252337, -0.093024, 0.062986, 0.060941, -0.007081, -0.043596, 0.032539, 0.074691, -0.070949, -0.077239, 0.015646, -0.169756, 0.095029, 0.013989, 0.075577, -0.011142, 0.016903, -0.012740, 0.011193, -0.046114, -0.002273, 0.027345, -0.045302, -0.054550, 0.153139, 0.020801, -0.097795, -0.061557, 0.066842, -0.104187, 0.005899, -0.025695, -0.038670, -0.142454, -0.013696, -0.069709, -0.142114, -0.066628, 0.062358, -0.021167, 0.169802, -0.135716, -0.066359, 0.053064, -0.040778, -0.086801, -0.075866, -0.156887, 0.075032, 0.123029, 0.022092, -0.121280, 0.035238, -0.127091, -0.095882, 0.038687, -0.057998, -0.007676, -0.132060, -0.038721, 0.037607, -0.035195, 0.080879, -0.051269, -0.031614, -0.081667, -0.093973, 0.016498, -0.019444, 0.098232, -0.054880, -0.087299, -0.120085, 0.002443, 0.018968, -0.155720, 0.112201, -0.059064, -0.035621, 0.036116, -0.027004, 0.086542, -0.120361, -0.027599, -0.151020, -0.053445, -0.135930, -0.118498, -0.037287, 0.006014, 0.099481, 0.090013, 0.043544, -0.112433, 0.104463, -0.034088, -0.155445, 0.041483, -0.054522, -0.149758, -0.018893, -0.072810, 0.184066, 0.043246, 0.086769, 0.072659, -0.105562, 0.061482, 0.109777, 0.016986, -0.044340, 0.031875, -0.144521, 0.013169, 0.043181, 0.093284, 0.074468, 0.184385, -0.051247, 0.073586, 0.077568, -0.054899, -0.067590, 0.159844, 0.048175, 0.095335, -0.060264, -0.118752, 0.144120, 0.082507, 0.012317, 0.089650, 0.002438, -0.062258, -0.037796, -0.121273, -0.082937, -0.071170, 0.072036, -0.107927, 0.018476, -0.006050, -0.001458, 0.012120, -0.041194, 0.056650, 0.017839, -0.024416, -0.161634, 0.027470, 0.023890, -0.015523, -0.047890, -0.122740, 0.009995, 0.004588, -0.022069, -0.037033, -0.036915, -0.039307, -0.347291, -0.068661, 0.166712, -0.133946, -0.030192, -0.047225, -0.022415, -0.120439, -0.073758, 0.148790, -0.054552, -0.074957, 0.157835, -0.096706, 0.074303, -0.088984, 0.072778, -0.201510, -0.123792, -0.028434, 0.170391, -0.035797, 0.108130, -0.103771, 0.034279, -0.096463, -0.005054, 0.124541, -0.125290, 0.089416, 0.042414, -0.035823, -0.055076, -0.104552, -0.023449, 0.033631, -0.069096, -0.025499, 0.114698, -0.016353, -0.159610, -0.125573, -0.142339, -0.082444, -0.183814, -0.021964, -0.079264, -0.304383, -0.002767, -0.132536, -0.096325, 0.067301, -0.104082, -0.214176, -0.095786, 0.040320, -0.110418, 0.149169, -0.073481, 0.061703, -0.193209, -0.067774, -0.088267, 0.000754, -0.153742, -0.265316, -0.030388, -0.140454, -0.092963, -0.021300, 0.137379, 0.032352, 0.032325, -0.112175, 0.003457, -0.206673, -0.130931, -0.098123, -0.078656, -0.056412, -0.243341, 0.029190, 0.143076, -0.211348, 0.007599, -0.059515, -0.112692, -0.092114, -0.102004, 0.133464, -0.242659, 0.068407, -0.154321, -0.036645, -0.130005, 0.072732, -0.129623, -0.024830, -0.126686, -0.157732, -0.054263, 0.114031, 0.104240, -0.028981, -0.026594, -0.061592, -0.083907, -0.070554, -0.087867, -0.066700, -0.030122, -0.269097, 0.100608, -0.046372, -0.028717, -0.133911, -0.069868, 0.099228, -0.170559, 0.062093, 0.002236, -0.296094, -0.192442, 0.064883, -0.094957, -0.181423, -0.041546, -0.100217, -0.044501, -0.140602, -0.243408, -0.025761, -0.086285, -0.063519, -0.056726, -0.167487, 0.047246, -0.125957, -0.132760, 0.126514, -0.187582, -0.135405, 0.140214, 0.032933, 0.038661, 0.092960, -0.121865, -0.021323, -0.043739, 0.093263, -0.046070, -0.119628, 0.137099, -0.001587, 0.071807, -0.028075, -0.198663, -0.057680, 0.025364, -0.058248, -0.134835, -0.121286, 0.027014, -0.057707, -0.187913, 0.032960, -0.163665, 0.041245, -0.199973, -0.143757, -0.052779, -0.168909, -0.146372, -0.002339, -0.214776, 0.039984, -0.019443, -0.108600, 0.024349, -0.105047, -0.182450, 0.001472, -0.013896, -0.057009, -0.164951, -0.101318, -0.138836, -0.161650, -0.210835, -0.003415, -0.009011, -0.068053, -0.064274, 0.005296, -0.133336, -0.007012, 0.012130, -0.097760, -0.435152, -0.044470, 0.035301, -0.154601, -0.068135, -0.146037, 0.065529, -0.109874, -0.049675, 0.140885, -0.029697, -0.192225, 0.003500, -0.144885, -0.189061, -0.085242, -0.090926, -0.003198, -0.228940, 0.021831, -0.197883, -0.045680, 0.131188, -0.116335, 0.018045, -0.020853, -0.178866, -0.168448, -0.035180, -0.174030, -0.058121, 0.017344, -0.016081, -0.246462, -0.053458, -0.154282, -0.178749, 0.052529, -0.147745, 0.077385, -0.062275, -0.115843, -0.005264, 0.003910, 0.049700, -0.020530, -0.192279, -0.079080, 0.087107, -0.325585, -0.061374, 0.092730, 0.080280, -0.124476, 0.013983, -0.153576, -0.022479, 0.023825, 0.020818, -0.028854, -0.121934, -0.107864, -0.056019, -0.052255, 0.078968, 0.011126, 0.012962, -0.059262, -0.029813, -0.138145, -0.034773, 0.054480, 0.069958, -0.055701, -0.003352, 0.009370, -0.017522, -0.009066, -0.126615, -0.002882, -0.192078, -0.136099, -0.150764, 0.050751, 0.073025, -0.081593, -0.068313, -0.190202, -0.101080, 0.066659, -0.124887, -0.038662, 0.073330, -0.054553, -0.305221, -0.003392, 0.058004, -0.047934, 0.040097, 0.102967, -0.026782, 0.025573, -0.086253, -0.095216, 0.095567, -0.115651, -0.113359, -0.074895, -0.067474, -0.193817, 0.024670, 0.005042, -0.043217, -0.181589, -0.139558, 0.120287, -0.046967, 0.105773, -0.079070, -0.235334, -0.029267, 0.056830, 0.026388, -0.151306, 0.046752, -0.224455, 0.095211, -0.012172, -0.019097, 0.060606, -0.058891, -0.221758, 0.126744, -0.013248, -0.203035, 0.035841, -0.156769, 0.095524, -0.021415, 0.075800, -0.062436, -0.083513, 0.219822, -0.020604, 0.006724, -0.165978, -0.372533, -0.119710, 0.044033, 0.008928, -0.433636, -0.234675, -0.146079, 0.003303, -0.046552, -0.112135, -0.077509, -0.158093, -0.234958, -0.078717, 0.213535, 0.059069, 0.191849, 0.065640, 0.143610, -0.239684, -0.076163, -0.070503, 0.011417, -0.024035, 0.207786, -0.105763, -0.200766, 0.002038, -0.072414, 0.054924, 0.077387, 0.026869, -0.156442, -0.009138, -0.058285, -0.199708, -0.019956, -0.100663, -0.109681, -0.037448, 0.256107, -0.099835, -0.080525, -0.019100, -0.033991, -0.147076, -0.093837, -0.029817, -0.052364, -0.136723, 0.027086, 0.084430, 0.022162, -0.190539, 0.035415, 0.000806, -0.035769, -0.385158, -0.357358, -0.221977, -0.067018, 0.075678, -0.110639, 0.015855, 0.030232, 0.022461, 0.023747, 0.015568, -0.100060, -0.364533, -0.040461, -0.004988, -0.228169, -0.074997, -0.016723, -0.082738, -0.211165, -0.329567, -0.028588, -0.059708, -0.051029, 0.101628, 0.128107, 0.025882, -0.004721, 0.070833, -0.144995, -0.047396, -0.059485, -0.174326, -0.196945, -0.177992, -0.103623, -0.016748, -0.079357, -0.114142, -0.040439, 0.075442, 0.071951, -0.121837, -0.131791, 0.173629, -0.141120, 0.027474, -0.093048, -0.033247, -0.052539, -0.100527, 0.084374, 0.046823, 0.037147, -0.179601, -0.096900, -0.131676, -0.142185, 0.059563, -0.045363, -0.044397, -0.123087, -0.023015, -0.076475, -0.055046, -0.026545, -0.019593, -0.091789, -0.015027, 0.077177, -0.023897, 0.083421, -0.021897, 0.113625, -0.116027, -0.054452, 0.017473, -0.024014, -0.148910, -0.110849, -0.011972, -0.166899, 0.063058, 0.024954, -0.017574, -0.028549, -0.132254, -0.090857, -0.109773, -0.141056, -0.022536, 0.024924, -0.048091, -0.016754, -0.098519, 0.080100, -0.098552, -0.069122, -0.113134, 0.025553, -0.111853, 0.060200, -0.140128, -0.094525, 0.053798, -0.059619, -0.116877, -0.033758, 0.057168, 0.099797, 0.002290, -0.020689, -0.011083, -0.110233, -0.096956, 0.067461, -0.006061, -0.133520, -0.062682, -0.123421, -0.067516, 0.067293, -0.084571, -0.078932, 0.012629, 0.038806, -0.055639, 0.007363, -0.024023, -0.063624, 0.115203, 0.119328, -0.000051, -0.025234, -0.123329, 0.091965, -0.017763, -0.153317, -0.013709, -0.050928, -0.235270, -0.161229, -0.056051, -0.075273, -0.124565, -0.147145, -0.001261, -0.152334, -0.187168, -0.047326, -0.052173, -0.238113, 0.065726, 0.104003, -0.066369, 0.022359, -0.142507, 0.091698, -0.061968, -0.062454, 0.025669, -0.002330, 0.125744, -0.090312, -0.175322, -0.076810, -0.103594, -0.009597, -0.162850, -0.095368, 0.081653, -0.040522, 0.011559, 0.058787, 0.034153, 0.018117, 0.060779, 0.049629, 0.008666, -0.023060, 0.007225, -0.029763, 0.049383, -0.145896, -0.102978, 0.019372, 0.065187, -0.185356, 0.010111, -0.056371, -0.084967, -0.030131, -0.151355, -0.068010, 0.002111, -0.039701, -0.201487, -0.260601, -0.002647, -0.073961, 0.006952, -0.078208, -0.081915, -0.065358, 0.162113, 0.074604, -0.035159, -0.000763, -0.143871, -0.010183, -0.008682, -0.081857, 0.045224, -0.135508, 0.000319, -0.198289, -0.147073, -0.046908, 0.036359, -0.133954, 0.002975, 0.108507, -0.138581, -0.045861, 0.015162, -0.075112, -0.013375, 0.047677, -0.093441, 0.037267, -0.075997, 0.061607, -0.068909, 0.049660, -0.140163, 0.069048, 0.011648, -0.152991, 0.041181, 0.046013, 0.003656, 0.012783, 0.203628, -0.058242, 0.167972, -0.026348, -0.122479, -0.069336, 0.052834, -0.039294, 0.008059, 0.056264, 0.130947, -0.093885, -0.144072, 0.015358, 0.037974, 0.138899, -0.119804, 0.049484, -0.018998, -0.138845, -0.028653, -0.130479, -0.095948, -0.061333, -0.051929, 0.152148, -0.062989, 0.036603, 0.134599, 0.140234, 0.037752, 0.039781, 0.059013, 0.108256, 0.019346, 0.000797, 0.003160, -0.014864, 0.028225, 0.017749, -0.020234, 0.065106, -0.034647, 0.062206, -0.018270, -0.078950, 0.014991, 0.041244, -0.032646, -0.040795, 0.034070, -0.067503, -0.135368, -0.091426, 0.086328, -0.042814, 0.033086, -0.026986, 0.041271, -0.114991, 0.010664, -0.003690, 0.146406, -0.114275, -0.086341, 0.094540, 0.001637, -0.030737, 0.071344, 0.085621, -0.182983, 0.051418, -0.019718, 0.072537, -0.093087, 0.111494, -0.101459, -0.023699, 0.071369, 0.018671, 0.001229, 0.059204, -0.013593, 0.074542, -0.110264, -0.055075, -0.027838, -0.054335, 0.097348, 0.020577, 0.068916, 0.107039, 0.011772, -0.072780, -0.084506, 0.106147, -0.138462, -0.057223, 0.019620, -0.050388, 0.029875, 0.138136, 0.053163, 0.055840, -0.176175, 0.114934, 0.016680, -0.068455, -0.087203, 0.064099, -0.056567, -0.168697, 0.077517, -0.214364, -0.001430, -0.020959, -0.086716, -0.056709, 0.144707, 0.053366, 0.102451, 0.090011, 0.039274, 0.017870, -0.103485, 0.116097, -0.040037, -0.054777, 0.126079, -0.074423, 0.011791, -0.100010, 0.062148, 0.033072, 0.005502, -0.038822, 0.008529, -0.117446, 0.023762, -0.112772, -0.009901, 0.009360, -0.057126, 0.190816, 0.073941, 0.018355, -0.130529, 0.012463, 0.100470, -0.030437, 0.181699, -0.044676, -0.019230, -0.093345, -0.093089, 0.029931, 0.110651, 0.046043, 0.171809, 0.082464, 0.001066, -0.074358, 0.126926, -0.028155, -0.046436, 0.050406, -0.168920, -0.072015, -0.033478, -0.050125, -0.043479, 0.031158, -0.044136, 0.095465, 0.023192, -0.072044, -0.062716, -0.036005, 0.113594, 0.099973, -0.018794, -0.004461, -0.190591, 0.031607, -0.116120, 0.004099, -0.085797, 0.089681, 0.022658, 0.148813, -0.124902, 0.090635, 0.014614, -0.097756, -0.242078, 0.073628, 0.019843, -0.054724, -0.059661, 0.006279, 0.024353, -0.168932, 0.053927, 0.006301, -0.074176, -0.023818, 0.028727, -0.057886, -0.052302, 0.020428, -0.068597, -0.047236, -0.079005, -0.091185, -0.073569, -0.088530, 0.060150, -0.131975, -0.036506, -0.018834, -0.038552, -0.122502, 0.054835, 0.075879, -0.021335, 0.146962, -0.058336, -0.087290, 0.089687, -0.021143, -0.010161, 0.122782, -0.095042, -0.146120, 0.208879, -0.054203, 0.010463, -0.050359, -0.081405, 0.038086, -0.041686, -0.205757, -0.168329, -0.025926, 0.015814, 0.072949, -0.063454, -0.005879, -0.086528, -0.086613, -0.081872, -0.111511, -0.044107, 0.001502, 0.097951, -0.070983, 0.013071, -0.218000, 0.045928, 0.036345, 0.015297, -0.063999, -0.134623, -0.143680, 0.010347, -0.166799, -0.077430, -0.094337, -0.041325, 0.007421, 0.085554, -0.220417, -0.074392, -0.045473, -0.004537, -0.107514, 0.104693, -0.067416, -0.117774, -0.100649, -0.131449, 0.003238, -0.029459, 0.098295, -0.031098, 0.083079, 0.046918, 0.049274, 0.008466, -0.062693, 0.098637, -0.108772, 0.062500, -0.074120, 0.046568, -0.017530, -0.063932, -0.038669, 0.033951, 0.199346, -0.050113, -0.138489, 0.040220, -0.058408, 0.099074, -0.152265, 0.113193, 0.104128, 0.096634, -0.045871, -0.136480, 0.006801, 0.015815, -0.126718, 0.075590, 0.016429, 0.064568, -0.058904, 0.069883, 0.187780, 0.053879, -0.072304, -0.081966, -0.094970, -0.126066, -0.142198, 0.006573, 0.001783, -0.006990, 0.016942, -0.021147, 0.132214, -0.008446, 0.016273, -0.083971, -0.117231, -0.041870, 0.019675, -0.128394, 0.012964, 0.019175, -0.044400, -0.051952, -0.204019, 0.132498, 0.149170, 0.056909, -0.020648, -0.037201, 0.059877, -0.044375, 0.038615, 0.000627, 0.142140, -0.040076, 0.015490, -0.016664, 0.088257, -0.198647, -0.069621, 0.011015, 0.127128, -0.104116, 0.098732, -0.127153, 0.098776, -0.108447, -0.000428, -0.082623, -0.026132, -0.016761, -0.038015, 0.121798, 0.034316, 0.090678, -0.067154, 0.089492, 0.019632, -0.038679, 0.099009, 0.057944, 0.029281, 0.000409, -0.027494, 0.062662, -0.124168, 0.040687, 0.022160, -0.055331, -0.048190, -0.080587, -0.028514, 0.043123, -0.245596, -0.182641, 0.044531, -0.024949, 0.007206, 0.010216, -0.148411, -0.044334, -0.019283, 0.126113, 0.082067, -0.190736, 0.017685, 0.023508, 0.042169, -0.079757, 0.122315, -0.036046, -0.069359, -0.051944, -0.062178, 0.115055, 0.040306, -0.183491, 0.019392, -0.019991, 0.018811, -0.112608, -0.137771, 0.030295, -0.027283, -0.134316, 0.090266, -0.107783, -0.010321, -0.135497, 0.072288, -0.084060, -0.129109, 0.079897, -0.016866, 0.043828, -0.174852, 0.062438, 0.079805, -0.003929, -0.118412, -0.032092, -0.023406, 0.037815, 0.070854, 0.008882, -0.013117, -0.036381, -0.145240, -0.095026, -0.032649, -0.106797, -0.112104, 0.031933, 0.068449, -0.029149, -0.098384, -0.082480, 0.000643, -0.103027, 0.033714, 0.086354, -0.008428, 0.110576, -0.007864, -0.097262, -0.180885, 0.034460, 0.006498, -0.038993, -0.081411, -0.225106, -0.041844, -0.129164, -0.064087, -0.106992, -0.042072, -0.155786, -0.037159, 0.058244, 0.007018, -0.292664, 0.072258, -0.249745, -0.121693, -0.182519, -0.153451, -0.076374, -0.001731, -0.047619, -0.053593, 0.116778, -0.107736, -0.094979, -0.098637, -0.034375, -0.055126, 0.087810, -0.042993, -0.130296, -0.005233, -0.073222, -0.078988, -0.005794, -0.115612, 0.032973, 0.050318, -0.010285, -0.077051, -0.216627, -0.031803, 0.124005, -0.102523, -0.069515, -0.080839, 0.001438, -0.023432, 0.015457, -0.050717, -0.029156, -0.075381, -0.037715, 0.123255, -0.056802, -0.042032, 0.100244, -0.162414, -0.035163, 0.005517, -0.131325, -0.092598, -0.049279, -0.020315, 0.030483, 0.051690, -0.096460, -0.147453, -0.085629, -0.064820, 0.046792, -0.009387, -0.030789, -0.013869, 0.015571, -0.162979, -0.119113, -0.136663, 0.000783, -0.052611, -0.074448, -0.026619, -0.072115, -0.072530, -0.091429, -0.035569, -0.061765, 0.119485, -0.068363, -0.287902, -0.018046, -0.022451, 0.000028, 0.076027, 0.034049, -0.123502, 0.020447, 0.075165, -0.023378, 0.055744, -0.058038, -0.062636, 0.121339, -0.013051, 0.037661, -0.029063, 0.054065, -0.140765, 0.002105, 0.012374, -0.134888, 0.044262, -0.027604, -0.175688, -0.058845, 0.171828, 0.009248, -0.029104, -0.016661, 0.223975, 0.130438, -0.038260, -0.017648, -0.069363, -0.022101, 0.111524, -0.109093, 0.102940, -0.151455, 0.208134, -0.072306, -0.031215, -0.069374, -0.101493, -0.254544, 0.067483, -0.018431, 0.013245, 0.013553, 0.076736, -0.055793, -0.024447, 0.060326, 0.083566, 0.039073, -0.095280, 0.014408, 0.044301, -0.070744, -0.190903, -0.008299, 0.018804, 0.022930, -0.108671, 0.014493, 0.064324, -0.141594, -0.129037, -0.030659, 0.062191, -0.149435, -0.159981, 0.044609, 0.119048, 0.142492, 0.094042, 0.029357, 0.051722, -0.056652, -0.023510, 0.127183, -0.016280, -0.038552, -0.198949, -0.147464, 0.087198, 0.031614, 0.036145, -0.017352, -0.038559, -0.086792, -0.031823, 0.103093, 0.008135, 0.067778, -0.134567, -0.088446, -0.050763, -0.030137, -0.050223, -0.119532, 0.040044, -0.005919, 0.061318, -0.054375, -0.082281, -0.097600, -0.068808, -0.084127, -0.105033, 0.002077, -0.082140, 0.062786, -0.066852, -0.006593, 0.005070, -0.016905, 0.092082, -0.176027, 0.204910, 0.093863, -0.119235, -0.115423, -0.274976, -0.225057, 0.046238, -0.149975, -0.079404, -0.332325, 0.124737, -0.058707, 0.061638, 0.110805, 0.127129, -0.165928, -0.185743, -0.035228, -0.176918, -0.008101, 0.068449, -0.063268, -0.166279, -0.030102, -0.118573, -0.227808, -0.024509, -0.137099, -0.012383, -0.066046, -0.042926, 0.005177, -0.094976, -0.013117, 0.018711, -0.051383, -0.016900, -0.007156, -0.020425, 0.073003, -0.078669, 0.014017, 0.039352, 0.020145, -0.043552, -0.005199, 0.091879, 0.060729, -0.090801, 0.054089, -0.061018, 0.119698, -0.115594, -0.099541, -0.053763, -0.038999, -0.095404, -0.003955, 0.018399, 0.182729, -0.179721, -0.079970, -0.261002, -0.196496, -0.216771, -0.031651, -0.032150, -0.003531, 0.026535, 0.167153, -0.131749, -0.055433, 0.090566, -0.060284, -0.005399, -0.048728, -0.007436, -0.000272, -0.012569, 0.021800, 0.029359, -0.030026, -0.096823, -0.070797, -0.105219, -0.061489, -0.011105, 0.111241, -0.035469, 0.019216, -0.019821, 0.057768, -0.095234, -0.070371, 0.057568, 0.068834, 0.165882, 0.038837, -0.179494, -0.112829, 0.088466, 0.045454, 0.039259, 0.070924, -0.102202, -0.058179, 0.031527, 0.046909, -0.062567, -0.174287, -0.093190, 0.119169, -0.023643, 0.105330, 0.022387, 0.067000, -0.010873, 0.057861, 0.040474, 0.026070, -0.116047, -0.000810, 0.011510, 0.007864, -0.139058, -0.034463, 0.073313, 0.067841, -0.081335, 0.060430, -0.071300, -0.081929, -0.035771, 0.020305, -0.025826, 0.048588, -0.008804, -0.126809, -0.193321, -0.066686, 0.101628, -0.029525, 0.118877, -0.017622, -0.030064, 0.022763, -0.118488, -0.106003, 0.007339, -0.032362, 0.175508, 0.106023, 0.078912, 0.061872, -0.139555, -0.016383, -0.006526, -0.042544, 0.011826, -0.012201, 0.076302, -0.003576, -0.163289, 0.078688, 0.002217, -0.008301, -0.093748, 0.007359, -0.112806, 0.076594, 0.042535, 0.221136, -0.206835, -0.229130, 0.035516, 0.104121, -0.014032, 0.095444, -0.130961, -0.030264, -0.040374, -0.012330, -0.025552, -0.020989, 0.059928, 0.046894, 0.110158, -0.213501, -0.005954, -0.069962, 0.036661, -0.048987, 0.069931, -0.037897, -0.050485, 0.069588, -0.033645, 0.082831, 0.059432, 0.078829, -0.173516, -0.011831, 0.007269, 0.093592, -0.224196, 0.195422, 0.129130, -0.017316, -0.065978, 0.071086, -0.095350, 0.071101, 0.103121, 0.004518, 0.038557, 0.023136, -0.060841, 0.058827, -0.009534, -0.222815, -0.051922, -0.039274, -0.134631, -0.037860, 0.086253, -0.174725, -0.145306, 0.060124, -0.127489, -0.073043, 0.049601, 0.192907, -0.123709, -0.129380, 0.016020, 0.015858, -0.136824, -0.069150, 0.086734, 0.021087, -0.031258, -0.053344, -0.027790, -0.007340, 0.033700, -0.076475, 0.061390, 0.027040, 0.004191, -0.007257, 0.102520, -0.194497, -0.064849, 0.030611, 0.048210, 0.070614, -0.072884, 0.040259, 0.019559, -0.082818, 0.064373, 0.082822, 0.066337, -0.026658, 0.048960, 0.029637, -0.033332, 0.015372, 0.031995, -0.113763, -0.062519, 0.070400, 0.127192, 0.122241, 0.012558, 0.070762, -0.071880, 0.013834, -0.031658, 0.070073, 0.102732, -0.106265, 0.048822, -0.169062, 0.123907, 0.111989, 0.128458, -0.093820, -0.076286, 0.033886, -0.011811, 0.047638, 0.051459, -0.079107, -0.046385, -0.020387, 0.021618, 0.044388, 0.040465, -0.140248, -0.164357, 0.015417, -0.072033, -0.055933, 0.049196, 0.030368, 0.064201, 0.019329, -0.095539, 0.004250, -0.031017, -0.050449, -0.022888, -0.021269, 0.019517, 0.121720, 0.035497, 0.072216, -0.108030, 0.074772, -0.029942, 0.102610, -0.070233, 0.076666, -0.063612, 0.047368, -0.055417, -0.006878, -0.101862, -0.024956, -0.073378, -0.097012, 0.025693, -0.021930, -0.070376, -0.087773, -0.131919, -0.035085, -0.048346, -0.068094, 0.029060, -0.050153, 0.026375, -0.106136, 0.071767, 0.035678, 0.052745, 0.009462, 0.105244, -0.127938, 0.037765, -0.149585, -0.132042, -0.082670, -0.132427, -0.001540, -0.172115, 0.071959, -0.140200, -0.031160, 0.014245, 0.081011, -0.168253, -0.022828, -0.044315, 0.012108, 0.122460, 0.034895, -0.061572, -0.014355, -0.199724, -0.013875, -0.051021, -0.114935, -0.090823, 0.036393, -0.211950, 0.059983, -0.040143, 0.001740, 0.029647, 0.079594, -0.032817, -0.167964, 0.074551, 0.090106, -0.012153, 0.058021, -0.020662, -0.010300, -0.164301, 0.106935, 0.260431, -0.029741, -0.007944, -0.001828, -0.166766, 0.061915, -0.084093, -0.009174, 0.009618, 0.066373, 0.043103, -0.092679, 0.064870, 0.043049, 0.073493, -0.088806, -0.000102, -0.053090, -0.024611, -0.105786, -0.354259, 0.038793, -0.056625, 0.016190, -0.131007, -0.028511, -0.051598, 0.054320, 0.157242, 0.070199, 0.067184, 0.084486, -0.068777, -0.002112, 0.013564, 0.213083, -0.066406, 0.016064, -0.083865, -0.002959, -0.089523, -0.007364, 0.019501, 0.020058, 0.067514, -0.012181, 0.021012, 0.015207, -0.070544, 0.071557, -0.083219, -0.025638, -0.279106, -0.067233, -0.066479, -0.090283, -0.097288, -0.041080, 0.026277, 0.011736, -0.121760, -0.172139, 0.051294, -0.159049, -0.002481, -0.021770, -0.036156, -0.059248, -0.006296, 0.074399, 0.059307, -0.043883, -0.107494, -0.034386, 0.061804, -0.090981, -0.016392, 0.022166, 0.055119, -0.025145, -0.121037, -0.135580, -0.058106, 0.022025, 0.050271, 0.030859, 0.116210, -0.089142, 0.112157, -0.005407, -0.110430, -0.014726, -0.162739, -0.100278, 0.118483, -0.120908, -0.079123, -0.055674, -0.130761, 0.023478, -0.151181, 0.133052, -0.055106, -0.127126, -0.013812, -0.140643, -0.161795, 0.167317, -0.123816, -0.121085, -0.220647, -0.165418, -0.009087, -0.050460, -0.068853, -0.055026, 0.071934, -0.054732, 0.058304, -0.023844, 0.017639, -0.120493, -0.118126, 0.058040, 0.041169, -0.055727, -0.021230, 0.075947, 0.083886, 0.070128, -0.104871, -0.047722, -0.045510, -0.122013, -0.158473, 0.155251, -0.070215, -0.094254, 0.079598, -0.018151, 0.106714, -0.040596, 0.016450, -0.065476, 0.139143, -0.096886, -0.004576, 0.069536, -0.234696, 0.057974, -0.023785, 0.065491, 0.024792, 0.055723, -0.115271, -0.185299, 0.088142, -0.150510, -0.132312, 0.085020, 0.003106, -0.146295, 0.056258, -0.051820, 0.030736, -0.038717, -0.068603, 0.023153, 0.054021, -0.089970, 0.048851, 0.026736, -0.097624, -0.027582, -0.097729, -0.204503, -0.091907, 0.067270, -0.023791, -0.035106, 0.062176, 0.026610, -0.172351, -0.124447, -0.113672, -0.192875, 0.036261, -0.096645, -0.089714, -0.029796, -0.005171, -0.031457, -0.084642, 0.039710, -0.111771, -0.135783, -0.048955, -0.128304, -0.281269, -0.205512, -0.120098, -0.047603, -0.122811, -0.284401, 0.124258, -0.167586, 0.119977, -0.037083, 0.039982, -0.108833, -0.177149, -0.138470, 0.164335, -0.012523, -0.094132, 0.088551, 0.070285, -0.037885, 0.015147, -0.182813, 0.037156, 0.015818, 0.017367, -0.026103, -0.059657, -0.074451, -0.072117, -0.032202, 0.057886, 0.001654, 0.058711, 0.100391, 0.015541, 0.004152, 0.021422, -0.112271, 0.060068, -0.153015, -0.010529, 0.161568, 0.050634, 0.053643, -0.114443, 0.063591, -0.136020, -0.126297, -0.025016, -0.010572, -0.169593, 0.022024, -0.170734, -0.005525, 0.040260, 0.197998, -0.083081, 0.079327, -0.039900, -0.100057, -0.137291, -0.088154, -0.099276, 0.022371, -0.192036, -0.154942, -0.073324, -0.158078, -0.112393, -0.027118, -0.002877, -0.040991, -0.012942, -0.019356, -0.009375, -0.051952, -0.006641, 0.022929, 0.015091, 0.108199, 0.040318, -0.088270, -0.190541, -0.016933, -0.116838, -0.056290, -0.051902, 0.159244, 0.020761, -0.052232, -0.123964, 0.098832, -0.036826, 0.077738, -0.107882, 0.037663, -0.005430, 0.090681, 0.078899, 0.061013, -0.152627, 0.122984, -0.036893, -0.123482, -0.020064, 0.128325, -0.022540, -0.087252, -0.084057, 0.024780, 0.031234, -0.110676, -0.064162, -0.100468, 0.078091, 0.094900, -0.020669, -0.010057, -0.170540, -0.118959, 0.027017, 0.007574, -0.012434, -0.029411, 0.024195, 0.013798, -0.006570, 0.045159, -0.029393, 0.087169, -0.108666, -0.007843, -0.212875, -0.066675, -0.079006, -0.007737, -0.066800, -0.119319, -0.071637, 0.087302, -0.010658, 0.049033, -0.074197, -0.021607, -0.049924, -0.097063, 0.012777, 0.074501, -0.008716, -0.054696, 0.005727, -0.024067, 0.025372, -0.055069, 0.092109, 0.129738, -0.115144, -0.123790, -0.050720, 0.067710, -0.057972, -0.070279, -0.053308, -0.016014, -0.213560, -0.138886, -0.014101, 0.016838, -0.203820, 0.016753, 0.068865, -0.060205, 0.001634, 0.088078, 0.144537, -0.145244, -0.066068, -0.025455, -0.067123, 0.041828, -0.019499, -0.003338, -0.012798, -0.001443, -0.065340, -0.023787, -0.088199, -0.106870, 0.086379, -0.058711, -0.049113, -0.065910, -0.094060, -0.006762, 0.001172, -0.041658, 0.187839, -0.002685, -0.049181, -0.039465, -0.018347, -0.100779, 0.001526, -0.056302, 0.025021, 0.038479, 0.040542, -0.100450, -0.024246, -0.153138, -0.042795, -0.167190, 0.050730, 0.058303, 0.141334, 0.044526, 0.058873, 0.143144, -0.003947, -0.137729, -0.107334, -0.031527, -0.013312, 0.008832, -0.081272, -0.009417, 0.050453, 0.030817, -0.017685, -0.022402, -0.105225, -0.044858, 0.031899, 0.209029, -0.122391, -0.052477, 0.071320, -0.128502, 0.111084, 0.021287, 0.052869, -0.063602, 0.010122, -0.011385, 0.096793, 0.079424, -0.120927, 0.067186, -0.048985, -0.064627, -0.007341, 0.023025, -0.063792, -0.205782, -0.231632, 0.176161, 0.015777, -0.137782, -0.180000, 0.071903, 0.074973, 0.003187, -0.037289, -0.041300, 0.093357, 0.003070, 0.004946, -0.039536, 0.052924, -0.077118, -0.043539, -0.089842, 0.012481, -0.097825, 0.032228, 0.032803, -0.006559, -0.041052, 0.055771, 0.049250, -0.072071, 0.000555, -0.158054, -0.047668, 0.064026, -0.090133, -0.056910, -0.069543, 0.007716, -0.027090, -0.214130, 0.014789, 0.116021, 0.049864, -0.136626, -0.058964, -0.042253, -0.042876, -0.005233, 0.055879, -0.183548, 0.089182, -0.125520, -0.353067, -0.039579, -0.048661, 0.051359, 0.140446, -0.071182, 0.084293, 0.069767, -0.257759, -0.044037, 0.044264, 0.038131, 0.008525, -0.154235, -0.059081, -0.066722, -0.147072, -0.012935, -0.101006, -0.111193, -0.114904, -0.169241, -0.024248, -0.036257, -0.034095, -0.018850, -0.140328, 0.103927, 0.091620, -0.007594, 0.206907, -0.179893, -0.144197, -0.162345, -0.235265, -0.078595, 0.061855, 0.093645, -0.208349, 0.202928, -0.030785, -0.105420, -0.033730, 0.018039, -0.138314, -0.190440, -0.141635, -0.206586, -0.090117, -0.049468, 0.001742, -0.059584, 0.208721, -0.134961, -0.014449, -0.252731, -0.046835, -0.001556, 0.138565, -0.062602, -0.063364, -0.160925, 0.084114, -0.027819, 0.155323, 0.149241, -0.104495, 0.065426, -0.142228, 0.052523, 0.005036, 0.019921, 0.002065, -0.127720, -0.193936, 0.116309, 0.034046, 0.020931, -0.116367, -0.065739, 0.010041, 0.074589, -0.353351, 0.095083, -0.057956, -0.034941, -0.240649, -0.012093, 0.001841, 0.096869, 0.010607, -0.167603, 0.054229, -0.063451, 0.040409, -0.176723, -0.193609, -0.103997, 0.050583, 0.040682, -0.082689, -0.073978, -0.007730, -0.043997, -0.011804, -0.219556, 0.017417, -0.259160, -0.087331, 0.030993, -0.072511, -0.160959, 0.062435, -0.015777, 0.042320, -0.109450, -0.017929, -0.013224, -0.007667, -0.045710, 0.081555, -0.081590, 0.024863, 0.103802, 0.068328, 0.004972, -0.142102, 0.171601, -0.079264, 0.074034, -0.076115, -0.056089, -0.001458, 0.002992, -0.035799, -0.112966, 0.068335, -0.046580, 0.097477, -0.161258, 0.078815, -0.069136, -0.202961, 0.034632, 0.177494, 0.003361, 0.022094, -0.104555, 0.124067, -0.009735, -0.181372, -0.011347, -0.043229, -0.132056, -0.087328, 0.066275, 0.177827, -0.026487, 0.050161, -0.027391, -0.234901, -0.027400, 0.073541, 0.034326, -0.100667, -0.038750, -0.058635, 0.077274, -0.060283, -0.076280, 0.022281, -0.040350, 0.074530, 0.043840, 0.060370, -0.078876, -0.056489, -0.035180, -0.030065, -0.237865, -0.318128, -0.301313, -0.255828, -0.106176, -0.053712, -0.227579, -0.317563, 0.096685, -0.075482, -0.198823, -0.080253, -0.153323, -0.246145, 0.006940, -0.056832, -0.031839, 0.071877, -0.031331, 0.165473, -0.100327, -0.083314, -0.100532, 0.042583, -0.014250, -0.177487, -0.028345, -0.278858, -0.012439, 0.086701, -0.087000, -0.073942, -0.017157, -0.042504, -0.042694, 0.093031, -0.053962, 0.127976, -0.132878, -0.014213, -0.091103, 0.093184, 0.050163, -0.230994, -0.150712, -0.109024, -0.063372, -0.336799, -0.312854, -0.042271, -0.226193, 0.055687, -0.131053, -0.071251, -0.072520, 0.114967, 0.045656, 0.051232, -0.119355, -0.171894, -0.221023, 0.018411, 0.032920, 0.134339, -0.135054, -0.049884, -0.029561, -0.039570, -0.142715, -0.041482, 0.046223, -0.173790, -0.045243, -0.086247, -0.045548, 0.042026, -0.024140, 0.077375, -0.302607, -0.086558, -0.061781, -0.119913, -0.119284, -0.008287, -0.175886, -0.171918, -0.024500, -0.125627, -0.092559, 0.014638, -0.075982, 0.054568, -0.006950, -0.110091, 0.037974, -0.219119, -0.027641, 0.022667, -0.153284, -0.000749, -0.220263, 0.103250, 0.034734, 0.024665, 0.076157, -0.028593, 0.072082, -0.052632, 0.095849, 0.103157, -0.165127, 0.080316, -0.048514, -0.022748, -0.206790, -0.146238, 0.069649, -0.190162, -0.042363, -0.340200, 0.007838, -0.160703, 0.006019, -0.103791, -0.051032, -0.033010, -0.099389, 0.021179, -0.192430, -0.061862, 0.032382, -0.110685, -0.062021, -0.035522, 0.109707, -0.120194, -0.099254, -0.138626, -0.077244, -0.345918, -0.124968, -0.060890, 0.046749, -0.182168, -0.106649, 0.014851, -0.212767, -0.143423, -0.144982, -0.065700, 0.007375, -0.099657, -0.073219, -0.065716, -0.290818, 0.090189, 0.005988, -0.147241, -0.321131, 0.210350, 0.046649, -0.222738, 0.018152, -0.019001, 0.001682, -0.309273, 0.098494, 0.075877, 0.032993, -0.011009, 0.109583, -0.174735, 0.083916, -0.254488, -0.057528, 0.024951, -0.205341, -0.090027, -0.256734, -0.064818, -0.006019, 0.014347, 0.169761, -0.011176, -0.183641, 0.012745, 0.043913, -0.030311, 0.081231, -0.137382, 0.062949, -0.179174, -0.052289, -0.075042, -0.127989, 0.158258, -0.213642, -0.059370, -0.083067, -0.109815, -0.135388, -0.162379, -0.149021, -0.148926, 0.018193, 0.116225, 0.131065, -0.182030, -0.030722, -0.112650, -0.132146, -0.226270, -0.013420, 0.065049, -0.085130, 0.087276, -0.028201, 0.066678, -0.060049, 0.066215, -0.062750, -0.067686, -0.018457, -0.249217, -0.174732, -0.063654, -0.006502, -0.039753, -0.040925, -0.026650, -0.058890, -0.137708, -0.165330, -0.166913, 0.048548, 0.067538, -0.044563, -0.054172, -0.078971, -0.182682, -0.048775, 0.047979, 0.012105, -0.105830, -0.121161, 0.112348, -0.206445, -0.047934, -0.172699, -0.120474, -0.033503, -0.225469, 0.040884, -0.087056, -0.080658, 0.004721, -0.148746, -0.058141, 0.143784, 0.050056, -0.105954, 0.085693, -0.120785, -0.037798, -0.072123, -0.058360, 0.005898, -0.078844, -0.063817, -0.159657, -0.065893, -0.042136, 0.067940, -0.075101, -0.068093, 0.020318, 0.038773, -0.121779, -0.021761, 0.031203, 0.103322, -0.201332, 0.011897, -0.125572, -0.039899, 0.019069, -0.166649, -0.128293, -0.094189, -0.191566, -0.122018, -0.026998, -0.000909, -0.048215, -0.179536, 0.012462, -0.195282, -0.063502, 0.040172, 0.038928, -0.001782, 0.050483, -0.003399, 0.082924, -0.047069, 0.064684, -0.092930, -0.013999, -0.155452, -0.106217, -0.139255, -0.090622, -0.128016, -0.105196, -0.049479, -0.194068, -0.025392, 0.004534, 0.024651, -0.082864, -0.154700, -0.065623, -0.177129, 0.023307, -0.085556, -0.065003, -0.129646, -0.111127, -0.201984, -0.050015, -0.117825, -0.190668, -0.105333, -0.231333, 0.044077, -0.237960, -0.081157, -0.046089, -0.110983, -0.025395, -0.094720, 0.066964, 0.038372, 0.003291, -0.057970, -0.117265, -0.093706, -0.039399, 0.042631, -0.058309, 0.051876, 0.013534, 0.002871, -0.091221, -0.003213, -0.132414, 0.070791, -0.113376, 0.029239, -0.016615, -0.006595, -0.102526, -0.070712, -0.056679, -0.005617, -0.033267, 0.010031, -0.113016, 0.137521, -0.154730, 0.003475, -0.005504, -0.040435, 0.035114, -0.134986, -0.142605, -0.043632, 0.062881, 0.138186, 0.148977, -0.018421, 0.033164, -0.120793, -0.033611, -0.083884, -0.202340, -0.096178, -0.120465, -0.016010, -0.201323, -0.221043, 0.090821, -0.062656, -0.012505, 0.140315, 0.040534, -0.170789, 0.055697, -0.005037, 0.152574, -0.009388, -0.030754, -0.024707, -0.098266, 0.124520, 0.007352, -0.183326, 0.002242, -0.037593, -0.248234, -0.234266, 0.041432, 0.045260, -0.027262, -0.146485, -0.067432, -0.158447, -0.002866, 0.138439, 0.123212, 0.139566, -0.046841, -0.026258, -0.062751, -0.153209, -0.012915, -0.138870, -0.170053, 0.062011, 0.201011, 0.013705, -0.046314, -0.252945, -0.067020, -0.200699, 0.103472, 0.141969, -0.144532, -0.009951, -0.077417, 0.071902, 0.087401, 0.003713, -0.063515, -0.099458, 0.107891, -0.011111, -0.033340, -0.224779, -0.090469, -0.116634, -0.031903, 0.026906, -0.159280, -0.188582, -0.109893, -0.020799, 0.026646, -0.102106, -0.033525, -0.014341, -0.149950, -0.046837, 0.051059, -0.054983, 0.116017, -0.098745, 0.099157, -0.149697, -0.000369, -0.019704, -0.104088, -0.060612, 0.058308, 0.154298, -0.057151, 0.035382, -0.107946, -0.176635, -0.063819, 0.119062, 0.056988, 0.069292, 0.004755, -0.132571, 0.048062, -0.157931, 0.085473, -0.065378, -0.072987, 0.018363, -0.176662, -0.025007, -0.094934, -0.191868, 0.028081, -0.072941, -0.069393, -0.140983, -0.179762, -0.151091, -0.282862, 0.114129, -0.192220, -0.135408, -0.022252, 0.124224, -0.078155, 0.054697, 0.050932, -0.233139, 0.092454, -0.041110, 0.071595, -0.020727, 0.011350, 0.066303, -0.214162, 0.158539, -0.083198, 0.023187, -0.023669, -0.038224, 0.136018, -0.009429, -0.032847, -0.135606, -0.018868, -0.051015, 0.011957, -0.060587, 0.038051, -0.011923, -0.113846, -0.033875, 0.244218, -0.036167, -0.275983, -0.102944, 0.011877, -0.047084, -0.043470, -0.106849, -0.012651, -0.184507, -0.122470, 0.024159, -0.166503, -0.131644, -0.085184, 0.004409, -0.000878, -0.121915, -0.112303, 0.024609, 0.060290, -0.082798, 0.049786, -0.246568, 0.004352, -0.148725, 0.021286, -0.232052, -0.018071, -0.163646, 0.070554, -0.007011, -0.161741, -0.000683, -0.231500, 0.138742, -0.026339, -0.154162, 0.107181, 0.003394, -0.067754, 0.149846, -0.092296, 0.003603, -0.134236, 0.098595, -0.142246, -0.045995, 0.096693, -0.101018, 0.029978, -0.045512, -0.101356, -0.117173, -0.003216, -0.065060, -0.131147, -0.110735, -0.047827, -0.200189, -0.027589, 0.063349, 0.132574, 0.136775, 0.075750, -0.181700, -0.089665, -0.164006, -0.184219, -0.009370, 0.088857, -0.052762, 0.043799, -0.075966, -0.129669, 0.084338, -0.007650, -0.124359, -0.074182, -0.128766, -0.150456, -0.064212, -0.107116, -0.008709, -0.126514, -0.069019, -0.112430, -0.114633, -0.126730, -0.113512, 0.025661, -0.169623, -0.017119, -0.057899, -0.005661, -0.048900, -0.114584, 0.037027, -0.076457, -0.079287, -0.099734, -0.126212, 0.036002, -0.108459, 0.054582, -0.177255, 0.095167, -0.038280, 0.026968, -0.052959, -0.038532, -0.115334, -0.210202, -0.134265, 0.126788, -0.071944, -0.029726, -0.169808, -0.115966, -0.155919, -0.171447, -0.080516, -0.155142, -0.039512, -0.177812, 0.036762, 0.010263, 0.091706, 0.040420, 0.104264, 0.026940, -0.245864, -0.115407, -0.044642, -0.106949, -0.015493, 0.040031, -0.093103, -0.134806, -0.061764, -0.027225, -0.091250, 0.007098, -0.057456, 0.021300, -0.179846, -0.019114, 0.009270, -0.110567, 0.048575, -0.099010, -0.003344, 0.083025, -0.006456, -0.011886, -0.016583, 0.011467, 0.002636, -0.113170, 0.112991, 0.073400, -0.130569, -0.014177, 0.004643, 0.020862, 0.099399, 0.040879, -0.157895, 0.062050, 0.019117, -0.000425, -0.131230, -0.174731, -0.023369, -0.173640, 0.090590, -0.135031, -0.038181, -0.048123, -0.074457, -0.008519, 0.032649, -0.062126, -0.002087, -0.133384, -0.140551, 0.081924, 0.083734, -0.185832, -0.147438, -0.162754, -0.035581, 0.008188, -0.073188, 0.022239, -0.108829, -0.118786, -0.036144, -0.187280, -0.070367, 0.072721, -0.055795, -0.043381, 0.115585, -0.010152, 0.074035, -0.072858, -0.184007, -0.014374, -0.006369, -0.072652, -0.067585, -0.122697, -0.068328, 0.004126, -0.005717, 0.138271, 0.062095, -0.034098, 0.029267, -0.195223, -0.019633, -0.096798, 0.103674, -0.185196, 0.061397, -0.213207, -0.116905, -0.106247, -0.061949, 0.075754, -0.075825, -0.134546, 0.064293, -0.154000, -0.116425, -0.179501, -0.129644, -0.121097, 0.045113, -0.010748, -0.076206, -0.029711, -0.070059, -0.074360, -0.107677, -0.212284, -0.009636, 0.153082, -0.073643, -0.126213, -0.088668, -0.052478, -0.106809, -0.047123, -0.100750, -0.015008, -0.074365, -0.004169, 0.031174, 0.060896, -0.111481, -0.027885, 0.047293, -0.073483, 0.018885, -0.058645, -0.098454, 0.063430, 0.019321, 0.078739, -0.078548, -0.024898, -0.113623, -0.065624, 0.017729, -0.001427, 0.018534, -0.239710, -0.058684, -0.022833, -0.036651, 0.103555, 0.059009, -0.003478, 0.111956, 0.071430, -0.042661, 0.088415, -0.106775, 0.042357, 0.038417, -0.038890, 0.064800, 0.077590, -0.102851, -0.123961, -0.128363, -0.052264, 0.078162, 0.143426, 0.012485, 0.020982, 0.059972, -0.013609, 0.087362, 0.055179, -0.021269, -0.068835, -0.009070, -0.027865, 0.073036, 0.014250, -0.062541, 0.179711, -0.119455, -0.111965, -0.135092, 0.090705, 0.084936, -0.068984, 0.044766, -0.071048, -0.020513, 0.105601, -0.047047, -0.127774, -0.068160, -0.002632, -0.074276, 0.028333, 0.025773, 0.038226, 0.126947, 0.019851, 0.026171, -0.058855, 0.067985, -0.091429, -0.040910, -0.040918, -0.002734, 0.237528, -0.122513, 0.119352, 0.016308, -0.009054, 0.004646, 0.028383, -0.009004, -0.004986, -0.209295, -0.030813, 0.045471, 0.084432, -0.033264, 0.157485, -0.244621, -0.047432, -0.040875, -0.087464, 0.072070, -0.084548, 0.088671, -0.013828, -0.039330, -0.078418, 0.087568, -0.157741, 0.032354, 0.153782, -0.040007, 0.007079, 0.021593, -0.011677, -0.009944, 0.000616, -0.020386, 0.036395, -0.052643, 0.002615, -0.068611, 0.110874, -0.052375, 0.047151, 0.009505, -0.098234, 0.004062, -0.031044, -0.130578, -0.080585, 0.108634, 0.211836, -0.160036, 0.050490, -0.049799, -0.068982, 0.152096, -0.129201, 0.089162, -0.080535, -0.020980, 0.012785, 0.100578, -0.008088, -0.109889, -0.090028, -0.060347, -0.151361, -0.057072, -0.082086, 0.130174, 0.190820, 0.040677, -0.069706, -0.099310, -0.136301, -0.112940, 0.005231, -0.030931, 0.008851, 0.120883, -0.019179, -0.034036, 0.055993, -0.003319, 0.052478, 0.036688, 0.050758, -0.030257, -0.067326, -0.064982, 0.048491, -0.102794, -0.087367, -0.034301, -0.040039, 0.038896, -0.024724, -0.092245, -0.065347, -0.147426, 0.118013, -0.060222, 0.052951, -0.226288, -0.237047, -0.061178, -0.230657, -0.032082, -0.078217, -0.107607, -0.001522, 0.052151, -0.003073, -0.037628, 0.009810, -0.209219, -0.216506, 0.041800, -0.098418, -0.065091, 0.018265, -0.051001, 0.149972, -0.011067, 0.016410, -0.224507, -0.052983, 0.005925, -0.278784, -0.024275, -0.114292, 0.076839, -0.030100, 0.071480, -0.015511, 0.041225, -0.032440, 0.025451, 0.020257, -0.068521, 0.020632, -0.116585, -0.147196, 0.021319, -0.132461, 0.135136, -0.279936, -0.099179, -0.051155, 0.033701, -0.306621, -0.141106, 0.099972, -0.234686, -0.024711, -0.132101, -0.053029, -0.082780, 0.090621, -0.065364, -0.046228, -0.182134, -0.085472, -0.224502, 0.009544, -0.138506, 0.113056, -0.116512, -0.111174, -0.102671, -0.000312, -0.159848, 0.002543, 0.080654, -0.145143, 0.111835, 0.052046, -0.260529, -0.024181, 0.156036, 0.017216, -0.212793, -0.079634, 0.000314, -0.192572, 0.032106, 0.014458, -0.011897, 0.096570, -0.071616, -0.018941, -0.004634, -0.008209, -0.142824, -0.079830, -0.130547, -0.080873, -0.139269, -0.222421, 0.013443, -0.084103, -0.226175, 0.040040, -0.249905, -0.039435, 0.042496, -0.024337, 0.076529, -0.109987, -0.033235, 0.089273, 0.005339, -0.031642, -0.285567, -0.112764, -0.116521, 0.052380, -0.039599, 0.036167, -0.136547, -0.067657, 0.021359, -0.189110, 0.012975, -0.170424, 0.089639, -0.250668, -0.204663, 0.008947, -0.170911, -0.148201, -0.242466, -0.194375, -0.028420, -0.296033, -0.220690, 0.104261, 0.006708, -0.103990, 0.004449, -0.299824, 0.065232, -0.212815, -0.177501, 0.079562, -0.043524, -0.115562, -0.303115, -0.004339, -0.045696, -0.034874, -0.163167, -0.048578, -0.082554, -0.079933, -0.012845, 0.023816, -0.090273, 0.035741, 0.045743, -0.164459, -0.263946, -0.176890, -0.099645, -0.279956, 0.063192, -0.052036, 0.125513, 0.099416, -0.007535, 0.030265, 0.023289, -0.247125, -0.124591, -0.299876, -0.098520, -0.265750, -0.050896, -0.083600, -0.102819, -0.092958, -0.175001, -0.065079, 0.029904, -0.041108, 0.082096, -0.044955, -0.159301, 0.057211, 0.056031, 0.052836, 0.070892, -0.153919, 0.013841, 0.001777, 0.000606, -0.093088, 0.060846, 0.089582, 0.005010, -0.054190, -0.074912, -0.029806, 0.069457, -0.061827, 0.041562, 0.053823, 0.048874, 0.085202, -0.008177, -0.029291, -0.172957, 0.040184, 0.087182, -0.114856, 0.106522, 0.138453, 0.024833, 0.050895, -0.025308, -0.046946, -0.112008, 0.049229, -0.022544, -0.017056, -0.054639, 0.147016, -0.139312, -0.022634, 0.015071, 0.060604, -0.301776, 0.091533, 0.057683, 0.023693, -0.056226, 0.187903, 0.048753, -0.083164, -0.092987, -0.078251, 0.064422, -0.190629, 0.062076, -0.052302, -0.069556, 0.033059, -0.060851, 0.228138, -0.044445, 0.019021, -0.068587, 0.172532, 0.034094, 0.104441, 0.206123, 0.077166, 0.315495, 0.144576, 0.079441, -0.113239, -0.005448, 0.112641, -0.001555, 0.054804, -0.053929, 0.087100, 0.049489, -0.021477, -0.058918, 0.000143, -0.053988, -0.063802, -0.018350, 0.094156, -0.037203, 0.067540, 0.263895, -0.225524, 0.095939, 0.034292, -0.154265, 0.137819, -0.119476, -0.003095, -0.071214, 0.123800, -0.061237, -0.025781, 0.090561, -0.077738, -0.098151, 0.070266, 0.148180, -0.136632, 0.122344, 0.085899, 0.043281, 0.057419, -0.001230, 0.031488, 0.013429, 0.054926, 0.077757, 0.058796, -0.012630, -0.156000, 0.051647, 0.012689, 0.097659, -0.039534, -0.039320, -0.057098, -0.047859, -0.050465, 0.027420, -0.142272, -0.019090, 0.190193, -0.267886, -0.040023, 0.089000, 0.063264, -0.227978, 0.003133, -0.063791, -0.104393, -0.063922, -0.004581, -0.049739, 0.096768, -0.042555, -0.177506, 0.042341, -0.060417, 0.072109, 0.044944, -0.048122, 0.043807, -0.070190, 0.019914, -0.121995, 0.103866, 0.002795, 0.012369, -0.165886, -0.110502, 0.019797, 0.029332, 0.075793, -0.046033, -0.214286, 0.076646, -0.023658, -0.031422, -0.007743, -0.115799, -0.049526, 0.002732, -0.009482, -0.179054, -0.239059, -0.041616, 0.057661, 0.122279, 0.038445, -0.015027, -0.036295, 0.036404, -0.163587, 0.044521, -0.023259, 0.116695, -0.080991, -0.056708, 0.019669, 0.114631, 0.070372, -0.145250, 0.131769, -0.124991, -0.147875, -0.104377, -0.026882, -0.012139, 0.131385, -0.055657, -0.027237, -0.054583, 0.181610, -0.028852, 0.027004, 0.092996, 0.018451, 0.020626, -0.004800, -0.178736, -0.030948, 0.016116, 0.036279, 0.017265, 0.083754, -0.013935, -0.413245, 0.002049, -0.021967, 0.004100, -0.054738, -0.008824, 0.150547, -0.069833, 0.060684, -0.059523, -0.043138, -0.005046, 0.025590, -0.206904, -0.038874, -0.118424, 0.052409, -0.036360, 0.067520, 0.036175, -0.075486, -0.105673, -0.043315, 0.079365, -0.072885, -0.044304, -0.049019, -0.117884, 0.202290, -0.017531, -0.142211, -0.119516, -0.034071, -0.115559, -0.205617, -0.164347, 0.039050, 0.219275, -0.056106, 0.019855, 0.070524, -0.098473, 0.214637, -0.125352, -0.064590, -0.124605, -0.072919, -0.109593, 0.015672, 0.012934, 0.154695, 0.010199, -0.100290, 0.012294, 0.034686, 0.000914, -0.018744, -0.010204, 0.056258, -0.064827, -0.071388, 0.137941, -0.138939, -0.153039, -0.101525, -0.093202, 0.037150, -0.039741, -0.068534, 0.228263, -0.139131, 0.148880, -0.041225, 0.011089, -0.073455, 0.032564, -0.013035, 0.020794, -0.012186, -0.073676, -0.045944, 0.026938, 0.019576, -0.017539, -0.099100, -0.251001, 0.106873, 0.063030, 0.010082, -0.068810, -0.005070, 0.006611, 0.043471, 0.088478, -0.010074, -0.309880, 0.060114, -0.325942, -0.284395, -0.244246, -0.226015, -0.147776, 0.129598, -0.080098, -0.068881, -0.165190, 0.113538, -0.095689, 0.080384, -0.011301, -0.147173, -0.021866, -0.097806, 0.006477, -0.032457, -0.114424, -0.070816, -0.007928, 0.070626, -0.150725, -0.069766, -0.083430, -0.100562, -0.006620, 0.092270, -0.089088, -0.019240, -0.041119, -0.035952, 0.005314, -0.107924, -0.155270, -0.035930, -0.095558, 0.000519, 0.063002, 0.094141, -0.031756, -0.066855, 0.079373, 0.002617, -0.121688, -0.041882, -0.001301, 0.069679, 0.051575, -0.091434, 0.063585, -0.060677, 0.033963, 0.092952, 0.040896, 0.025723, 0.062367, -0.066843, -0.029888, 0.048257, -0.176524, -0.180826, -0.259579, -0.241548, 0.138721, -0.266718, -0.100950, -0.057154, -0.188945, -0.190449, 0.083462, 0.060090, -0.065373, 0.120924, -0.017394, -0.140515, -0.076177, -0.013031, -0.138269, -0.159254, -0.122982, -0.033596, -0.089379, -0.310128, -0.069055, -0.133560, 0.095270, 0.003196, 0.072595, -0.126204, -0.059154, 0.021256, -0.058287, -0.022640, -0.011537, -0.082270, -0.054105, -0.007676, 0.095299, -0.041807, 0.118270, -0.253711, 0.087193, -0.059264, -0.108399, -0.123590, -0.005547, -0.047855, -0.108316, -0.221977, -0.119323, 0.131010, -0.051542, 0.032114, -0.055739, -0.068716, -0.138649, 0.002839, -0.031513, -0.224230, -0.110836, -0.144376, 0.046193, -0.203395, 0.103428, 0.011748, -0.011735, -0.063248, -0.043122, 0.018604, -0.010570, 0.038960, 0.025297, -0.257196, -0.137335, -0.104559, -0.093162, -0.024476, 0.068027, 0.084284, -0.059774, 0.138552, -0.055876, 0.052538, 0.027068, 0.030896, -0.163971, 0.097678, -0.070661, 0.069303, -0.219138, 0.008191, -0.011582, -0.041124, -0.023351, -0.082302, -0.043655, 0.005960, -0.075897, -0.052605, 0.001408, -0.199729, 0.072058, -0.017318, 0.016427, -0.151145, -0.001472, 0.142264, -0.048777, 0.101990, -0.041138, 0.082658, -0.097336, 0.052946, -0.135756, -0.072700, 0.039878, -0.117289, -0.225615, -0.130753, -0.080712, 0.037287, -0.070572, -0.074469, -0.023543, -0.065783, -0.018177, -0.227092, -0.095051, -0.015707, -0.193063, -0.108783, 0.012936, -0.122908, 0.057342, 0.012714, 0.103698, -0.275800, 0.001813, 0.052442, -0.070676, 0.144010, -0.059181, -0.094266, -0.125235, 0.087360, -0.110083, 0.025357, -0.120082, -0.107047, -0.082422, -0.199879, -0.075280, -0.095451, 0.016574, -0.430656, -0.023910, 0.029310, 0.037135, 0.080677, 0.139308, -0.105955, -0.038941, 0.077471, -0.086711, -0.049622, -0.075540, -0.067497, 0.042646, -0.157886, 0.065480, 0.018957, -0.012346, -0.096677, -0.148701, -0.119283, -0.110039, -0.091678, -0.036272, 0.267150, 0.161700, -0.068283, -0.129597, -0.037997, -0.040621, -0.163531, -0.202857, 0.038415, 0.004041, -0.127266, -0.130256, 0.044529, -0.135039, -0.252686, -0.086361, 0.088269, 0.006058, -0.351844, -0.023699, -0.033725, 0.108113, 0.055382, 0.102414, -0.121660, -0.066178, -0.063924, -0.043102, -0.076272, -0.204561, -0.059988, 0.008608, -0.155681, 0.054499, -0.212230, 0.008318, 0.031357, 0.094706, 0.037514, -0.089915, -0.105109, 0.048553, -0.095235, -0.012629, 0.043971, 0.146252, -0.026723, -0.218903, -0.188803, -0.003134, 0.165470, -0.102761, 0.019301, -0.074284, -0.052182, -0.143883, 0.039945, 0.066022, -0.027883, -0.109704, 0.056820, -0.088451, 0.094519, 0.026121, -0.022222, -0.095235, -0.067143, 0.005722, 0.002492, 0.001559, 0.127276, -0.091291, -0.026150, 0.058415, 0.060466, -0.080306, -0.094774, 0.057244, -0.093002, 0.054175, -0.063672, -0.006247, -0.111771, 0.073924, -0.149225, 0.007993, 0.230540, -0.096407, -0.081608, -0.089691, 0.022328, -0.077599, -0.029877, -0.001232, 0.016035, -0.118801, 0.042010, -0.015797, 0.058093, -0.141764, -0.007488, -0.032952, -0.125286, -0.236151, -0.060023, -0.000622, -0.061421, 0.010168, 0.058249, -0.087213, -0.111364, 0.106728, -0.018600, -0.035531, -0.116702, 0.140167, -0.061769, 0.111921, -0.008269, 0.009932, 0.036478, -0.102906, 0.050895, -0.122497, -0.107010, -0.026406, -0.116585, -0.053251, 0.041053, 0.094679, -0.021909, -0.074826, 0.011758, -0.121206, -0.069241, -0.147942, -0.112058, 0.007187, -0.004502, 0.053438, 0.002035, -0.013085, -0.038182, 0.003369, 0.022272, -0.017221, -0.094104, -0.055067, -0.034853, -0.022019, -0.087427, -0.019453, 0.080296, 0.018579, -0.109028, -0.036942, 0.062725, 0.040806, 0.034439, -0.227817, -0.013252, -0.060824, 0.056471, 0.080571, -0.006350, 0.010245, -0.097759, 0.024435, -0.047851, 0.067234, -0.046803, 0.163759, -0.391462, -0.038932, 0.009626, -0.136950, 0.084936, 0.050089, 0.031731, -0.108119, -0.033166, 0.094296, -0.086680, 0.081069, -0.037968, 0.037624, -0.038006, 0.353144, -0.130406, -0.102309, -0.046086, -0.180522, 0.068060, -0.134004, 0.079770, -0.059921, -0.002682, 0.016200, -0.230064, -0.006365, 0.035671, -0.116726, -0.093313, -0.045209, -0.210396, 0.080679, -0.041469, 0.000953, 0.017819, 0.090033, 0.012055, -0.043019, -0.012821, 0.019102, 0.109330, -0.016058, 0.049063, -0.020861, 0.004419, -0.121496, 0.041127, 0.116340, 0.017037, 0.054861, -0.095722, -0.024278, -0.040030, 0.087291, -0.068626, 0.064245, -0.021232, 0.055709, -0.129635, 0.092954, 0.017129, -0.075201, -0.148911, -0.042940, -0.094641, 0.108574, -0.066127, -0.028810, -0.102399, -0.090231, -0.017655, 0.079484, 0.011201, 0.015540, 0.022494, -0.004773, 0.091144, 0.062537, -0.428748, 0.044852, -0.015092, -0.087267, 0.114469, 0.169045, 0.057102, -0.066398, -0.009621, 0.024939, -0.001454, 0.036395, 0.019006, -0.234321, 0.142400, -0.331585, -0.150466, 0.241073, 0.108930, -0.021447, 0.058396, -0.482788, -0.091035, -0.107536, -0.101664, -0.152037, -0.108371, 0.009085, 0.281593, -0.002084, 0.038859, 0.105054, -0.131732, 0.096901, 0.000391, 0.198297, -0.049248, 0.050973, 0.066640, -0.003508, -0.001302, 0.124295, 0.197946, 0.087457, -0.164022, -0.047376, -0.103433, -0.267538, -0.083386, -0.051565, 0.233261, -0.100204, -0.030512, 0.066832, 0.049244, 0.019032, 0.193260, -0.090655, -0.140362, -0.096783, 0.243392, -0.026520, 0.119233, -0.005179, 0.028697, 0.024563, 0.080306, 0.014968, 0.067599, 0.173052, -0.052262, 0.083409, -0.124701, 0.044567, 0.291395, -0.017722, -0.056514, 0.086671, -0.093821, -0.031019, 0.114987, 0.005162, 0.081580, -0.027616, -0.198549, -0.203164, 0.097296, -0.147139, 0.115885, -0.035681, 0.000469, -0.032310, -0.095778, 0.182911, 0.068391, -0.317023, 0.246631, -0.057790, -0.167751, -0.003747, -0.080907, -0.207857, -0.056642, -0.132882, -0.078114, -0.210339, 0.138950, -0.023764, 0.009760, 0.051332, -0.135663, 0.040227, 0.232177, 0.039467, 0.216335, 0.134154, 0.096650, 0.039413, -0.050756, -0.276895, -0.005592, 0.147525, 0.000143, 0.034048, 0.131670, -0.215526, -0.175415, -0.088560, -0.101385, 0.074786, -0.026813, 0.063419, -0.023831, 0.019993, -0.191051, -0.160473, -0.153954, -0.058446, 0.010033, 0.250177, 0.017043, 0.127271, -0.165826, -0.155869, 0.096138, -0.019851, 0.066812, 0.005574, -0.039117, -0.221569, 0.150096, 0.142523, -0.055788, 0.222872, -0.350393, -0.084237, 0.215530, -0.241407, -0.319469, -0.097555, -0.229763, 0.129265, -0.143222, -0.052377, 0.122224, 0.055148, 0.093053, -0.011391, 0.120728, -0.400474, 0.183664, -0.025779, -0.067148, 0.012948, -0.193259, -0.038374, 0.015175, -0.125006, -0.000041, 0.007739, -0.007303, 0.024060, -0.096750, 0.091304, -0.074519, 0.236791, -0.037402, 0.091167, 0.043035, 0.145834, 0.089429, -0.008756, 0.148863, -0.116460, 0.094209, -0.007873, -0.197845, 0.081624, 0.055729, -0.084881, -0.060415, 0.039872, 0.055261, -0.129359, -0.011897, -0.073712, -0.067248, 0.107567, -0.207694, -0.154339, 0.090828, -0.011646, -0.096151, -0.096878, -0.124147, 0.069117, -0.107470, -0.171480, -0.010510, -0.012728, -0.043061, -0.054314, 0.016108, 0.032545, -0.313261, 0.123909, -0.093523, -0.003303, -0.123799, 0.106550, -0.014859, -0.163313, -0.018512, 0.077892, -0.061060, 0.037134, -0.217362, 0.034427, 0.060850, 0.058817, -0.008752, -0.141350, -0.000556, 0.095569, -0.167081, 0.096559, 0.145674, -0.035669, 0.103803, -0.031012, -0.061175, 0.064222, 0.000865, -0.031753, 0.079531, -0.116977, 0.000496, -0.150999, -0.119892, 0.056187, -0.098254, -0.065829, 0.047606, -0.114490, 0.111535, -0.081114, 0.090718, 0.067603, -0.035286, 0.028478, 0.192873, -0.085653, -0.021023, -0.147715, -0.098158, 0.053874, 0.008672, -0.041263, -0.084760, -0.095584, -0.105270, -0.012682, 0.002068, -0.041103, 0.122153, -0.099839, 0.082916, -0.049016, 0.040548, -0.245296, 0.075127, -0.297715, 0.170777, 0.027686, -0.016806, -0.101644, -0.203755, -0.147320, 0.088120, 0.039443, -0.006866, 0.049442, 0.042585, 0.071830, 0.023308, 0.021130, -0.125034, 0.106879, -0.099024, -0.042310, 0.001047, -0.101916, 0.054259, 0.003841, -0.087030, -0.122064, -0.069948, 0.158193, -0.059470, 0.022294, 0.022473, -0.060818, -0.059952, 0.086759, 0.085727, 0.068051, 0.132968, -0.029760, 0.051655, 0.016397, -0.062367, -0.200357, 0.001294, -0.045131, 0.046592, -0.201232, -0.046121, 0.130199, -0.103015, 0.021650, -0.359971, 0.071979, -0.015335, 0.035486, 0.076642, -0.116027, -0.027801, 0.202821, 0.056537, -0.102226, -0.037000, 0.012584, 0.016879, -0.075182, -0.208140, 0.008511, -0.157799, 0.024613, -0.006218, 0.096047, -0.147258, 0.169007, 0.098633, -0.069358, -0.044213, -0.104673, 0.136840, 0.046401, -0.024259, -0.034505, -0.047192, 0.112113, -0.081351, -0.114710, 0.047780, -0.027445, 0.070165, -0.052432, -0.153688, -0.157400, -0.004623, 0.107485, -0.179106, -0.071405, 0.173559, -0.054587, 0.061498, 0.023673, -0.080052, -0.175788, -0.065897, 0.021448, -0.035865, -0.048381, -0.042757, -0.064784, -0.128405, -0.041365, -0.124137, -0.057286, -0.144628, -0.089853, -0.140542, -0.041059, -0.259039, -0.161653, -0.019118, -0.041375, -0.079743, -0.066026, 0.076689, 0.002165, -0.027631, -0.131822, 0.114350, -0.063772, 0.025738, 0.093149, -0.125397, 0.077307, 0.029262, 0.090769, 0.042265, 0.071741, -0.173886, -0.024086, -0.151982, 0.051664, 0.016177, -0.179608, -0.059366, 0.039677, 0.072239, -0.085272, 0.204670, -0.016208, -0.038905, -0.080776, -0.197591, -0.062611, 0.074910, -0.139481, 0.032362, -0.002150, 0.053697, 0.136421, 0.072979, -0.086532, -0.054828, -0.112088, -0.149604, -0.018966, -0.120115, -0.011177, 0.152373, -0.019728, -0.134224, -0.026858, -0.015776, -0.132020, 0.075652, -0.041383, 0.052949, 0.036571, -0.029895, -0.037042, 0.257425, -0.069155, -0.172190, -0.017338, -0.125099, -0.071720, 0.082069, 0.005878, -0.078337, -0.034573, 0.012823, -0.059406, 0.024743, 0.078684, 0.020644, -0.079392, 0.125603, 0.066693, 0.073477, -0.120026, 0.114695, -0.167785, -0.180297, -0.077668, -0.044978, 0.109999, -0.009595, -0.088992, 0.098004, 0.053936, 0.038034, 0.049447, -0.011029, -0.019755, -0.104290, 0.054483, 0.044779, 0.136844, 0.004614, -0.094669, -0.050751, -0.128855, -0.027082, -0.110179, -0.004412, -0.040491, 0.026778, -0.127453, 0.017492, 0.106550, 0.087260, 0.043570, -0.040508, -0.123998, -0.149300, 0.082800, -0.009258, -0.074452, 0.039313, -0.039820, -0.143552, -0.194717, -0.020422, -0.059472, -0.001922, -0.125253, -0.063311, -0.045461, -0.236528, -0.172445, 0.052553, -0.116265, 0.115972, -0.213337, 0.092230, -0.027490, -0.000182, 0.082562, -0.041257, -0.008972, -0.122839, 0.274415, 0.109278, 0.048399, -0.132140, -0.033941, -0.185868, -0.122004, -0.200874, 0.158324, -0.042495, 0.133882, -0.103728, -0.013877, -0.012684, 0.048308, 0.146684, -0.074297, -0.064098, -0.033528, -0.223986, -0.117125, -0.031415, 0.051833, -0.121259, 0.108601, 0.049620, 0.034460, 0.053613, -0.134198, -0.084861, 0.037319, 0.022362, -0.175359, -0.099740, -0.025546, 0.046172, 0.032650, -0.003429, 0.004825, 0.078618, -0.044242, -0.081354, 0.048675, 0.154771, 0.139684, 0.077857, 0.044689, 0.139226, -0.083394, 0.140889, -0.006850, -0.115875, -0.001764, -0.042841, -0.059069, 0.050093, 0.033704, 0.063383, -0.075940, -0.045793, -0.095938, -0.096622, -0.004037, 0.039769, -0.019860, -0.170245, -0.038382, 0.067936, 0.056963, -0.021990, -0.126511, -0.181764, -0.030561, -0.081386, 0.040101, 0.071358, 0.016876, 0.015981, -0.036226, 0.064199, -0.047012, 0.077724, -0.112252, 0.063974, 0.095152, -0.056482, -0.051551, -0.126540, 0.060914, -0.030415, 0.014991, -0.034487, -0.006545, -0.022412, 0.123924, 0.110464, 0.029478, -0.129586, 0.144443, -0.048478, 0.054766, -0.046752, 0.037760, 0.113994, -0.054598, 0.118662, -0.048556, -0.064770, 0.119864, 0.034002, 0.040106, -0.076394, 0.064934, -0.166691, -0.113654, -0.106979, 0.179735, 0.082032, -0.062233, 0.043271, 0.064004, -0.012171, -0.081993, -0.071759, 0.028651, 0.049354, 0.042135, 0.024370, -0.101661, 0.090055, -0.123460, -0.176882, -0.060202, 0.193661, 0.082213, 0.050434, 0.075429, 0.031679, 0.007674, 0.006209, 0.040638, 0.013304, -0.044054, 0.092766, 0.039404, 0.017965, -0.066457, 0.009775, 0.096898, 0.014578, 0.043078, -0.061313, 0.026144, 0.014209, 0.038553, 0.060709, -0.115241, -0.078499, -0.189108, 0.006277, 0.039076, -0.038230, 0.111487, -0.045661, -0.253270, -0.159281, -0.054387, -0.111773, -0.092274, -0.078992, -0.046930, -0.009864, 0.029940, -0.068203, -0.080995, -0.063545, -0.000177, -0.030146, -0.071874, -0.024588, 0.008756, -0.089195, 0.020603, -0.043050, 0.003308, 0.117677, -0.017131, -0.167368, 0.057341, -0.206633, -0.018500, -0.125875, 0.072440, 0.055050, -0.021160, -0.171466, 0.060741, 0.047147, 0.146068, 0.044785, -0.133120, -0.070677, 0.071426, -0.037817, -0.074171, 0.100956, 0.038334, -0.156232, -0.128066, -0.048403, 0.059180, -0.088396, 0.035431, 0.059809, 0.143804, 0.045680, -0.032423, -0.105142, 0.089472, -0.054756, -0.004429, -0.130174, 0.030888, -0.016487, -0.082202, 0.043408, -0.000698, -0.074150, 0.079063, -0.094060, -0.095340, 0.055669, -0.034617, 0.083389, -0.010516, -0.019169, -0.023193, -0.067218, 0.044397, 0.100727, 0.048729, -0.158545, 0.124266, -0.033724, -0.145200, -0.080494, -0.044302, 0.104630, -0.130038, -0.154880, 0.107940, 0.003191, 0.131200, -0.130978, 0.047669, 0.065334, 0.077375, -0.106480, 0.088012, 0.037535, 0.042488, 0.090607, 0.137824, -0.008669, -0.101677, -0.184534, -0.138476, -0.054582, 0.079867, 0.035970, 0.001917, -0.068120, -0.135967, 0.102798, 0.024775, 0.042193, -0.132265, -0.035761, -0.151369, 0.029782, -0.045628, 0.042019, 0.110204, -0.033531, -0.004614, 0.131817, -0.046070, 0.000385, 0.038949, -0.044634, -0.046085, -0.069308, -0.077016, -0.157528, -0.100282, -0.124366, 0.010469, -0.057137, 0.013507, -0.139499, -0.008197, -0.177102, -0.021311, -0.081361, 0.050594, -0.102543, 0.050923, -0.108387, -0.013324, 0.001300, 0.001279, 0.021783, -0.041397, -0.036915, -0.068590, 0.002459, -0.037978, 0.030943, -0.068744, 0.012101, -0.047375, -0.028442, 0.075993, -0.187879, -0.089378, 0.101595, -0.106171, 0.072103, -0.130742, 0.008578, -0.038851, -0.052058, 0.102527, 0.002941, -0.053597, 0.018529, 0.056583, -0.067537, 0.132166, -0.025882, 0.080517, 0.064038, 0.050145, 0.076148, 0.041465, 0.054728, 0.120442, -0.015132, -0.063461, 0.000197, -0.041931, 0.051238, -0.227326, -0.038384, -0.111589, -0.020015, 0.087732, -0.053595, -0.155597, -0.030490, -0.142064, -0.116703, 0.131133, -0.011561, 0.005489, 0.092907, -0.113460, -0.022442, 0.089790, -0.041265, -0.119890, 0.093668, 0.033458, -0.014817, -0.103150, -0.037031, -0.095662, -0.059424, 0.051945, 0.096441, -0.075278, -0.109345, 0.003531, -0.053480, 0.199159, -0.125129, 0.034727, -0.052539, 0.126900, -0.108887, 0.062140, 0.055142, -0.069992, -0.083367, -0.027290, 0.033349, -0.047463, 0.066577, -0.065565, -0.129255, -0.070388, 0.029641, 0.165064, -0.147484, -0.109609, -0.176327, -0.047287, 0.233845, 0.107735, 0.061204, -0.061482, 0.044542, -0.080909, -0.007254, 0.006470, -0.033812, -0.150050, 0.065363, 0.059720, -0.016550, 0.018407, -0.094693, 0.088850, -0.075472, 0.092270, -0.214399, -0.349119, -0.177875, -0.237755, 0.021986, -0.051285, -0.195538, -0.223448, 0.126320, -0.184303, 0.024546, 0.115601, -0.204682, -0.173590, 0.017084, -0.134358, -0.091495, 0.064555, -0.055793, 0.090095, -0.097523, -0.190886, -0.078572, -0.194769, -0.009541, -0.250876, -0.020967, -0.370949, -0.160997, 0.056440, 0.089165, -0.153007, 0.051737, -0.108668, 0.018730, -0.005430, -0.264685, -0.247486, 0.020381, -0.005046, -0.072410, -0.202923, 0.149560, -0.117934, -0.050618, -0.033601, 0.041118, -0.162456, -0.259964, -0.137796, -0.124810, -0.038378, -0.028650, 0.100601, -0.000323, 0.018635, 0.032044, 0.005985, -0.155438, -0.202218, -0.081175, -0.002397, 0.065370, -0.050640, -0.102691, -0.091998, 0.006711, -0.062667, -0.205063, -0.051216, 0.012970, -0.101359, 0.168295, -0.028440, -0.023571, -0.174264, -0.194553, -0.035303, -0.206787, 0.106729, -0.017883, 0.018088, -0.062559, -0.020252, -0.076702, -0.223246, 0.025267, 0.009155, -0.044875, -0.022596, -0.113842, -0.024619, 0.011273, 0.029876, 0.046657, -0.236425, 0.105234, -0.079894, -0.111110, 0.153420, -0.146143, -0.091187, 0.022492, -0.067567, 0.009346, 0.083891, -0.115654, -0.008510, -0.064810, 0.065514, -0.326266, -0.030651, -0.003527, -0.134215, 0.016874, -0.097387, 0.011332, -0.129982, -0.027326, -0.242507, 0.038544, -0.065785, 0.118840, -0.010276, -0.200083, -0.105642, -0.186978, -0.069463, -0.072862, -0.072958, -0.077455, -0.194077, -0.010206, 0.021857, -0.085078, 0.031880, -0.147325, -0.086478, 0.109013, -0.191527, 0.025970, -0.078010, -0.085603, -0.167570, -0.077861, -0.119435, -0.109889, -0.146821, -0.182258, 0.056908, -0.120645, -0.010153, -0.050628, -0.145768, -0.097812, 0.084200, -0.271823, -0.106954, -0.199802, -0.002869, 0.040377, -0.252813, -0.114376, -0.094717, 0.081723, -0.010119, -0.084258, 0.006563, -0.012868, -0.121665, 0.085701, 0.020440, 0.024905, -0.124158, -0.048420, -0.012248, -0.100398, 0.008222, -0.244239, -0.092114, 0.071340, -0.049353, -0.141145, -0.152273, -0.188029, -0.217547, -0.060223, 0.021635, 0.125767, -0.005546, -0.170207, -0.213838, -0.004280, -0.023733, -0.118602, 0.123620, -0.173784, 0.014813, -0.142633, 0.051898, -0.059044, -0.098280, 0.013531, -0.174650, -0.055657, 0.092495, -0.042626, -0.078719, 0.044875, -0.007605, -0.043100, -0.086732, 0.049609, -0.014925, 0.040290, -0.023229, -0.005411, -0.043770, -0.006721, 0.016083, -0.087251, 0.022676, 0.057785, 0.056474, -0.142925, -0.254302, 0.008490, 0.010880, 0.016469, -0.158888, 0.052813, -0.025294, -0.020891, 0.168973, -0.130871, -0.068044, -0.138257, -0.126572, -0.087591, -0.132399, -0.035596, 0.001123, 0.093956, -0.001976, 0.007599, 0.097369, 0.187154, 0.217177, -0.107044, 0.023385, 0.015443, -0.049306, 0.134378, 0.098033, -0.077941, 0.033518, 0.179742, -0.049879, -0.144649, -0.156646, -0.085051, -0.144673, -0.116438, -0.018280, 0.142060, -0.031180, -0.121672, -0.061326, 0.053946, 0.017202, 0.000225, -0.093835, 0.056120, -0.001719, -0.071326, -0.158532, -0.128717, -0.142458, 0.060298, -0.116890, -0.221100, -0.094133, -0.078987, -0.056930, -0.032493, -0.126196, 0.005333, -0.030141, -0.065553, -0.213953, -0.028467, 0.062379, -0.059273, -0.119248, -0.170932, 0.052533, -0.097945, -0.160574, 0.078791, -0.131505, 0.220568, -0.111222, 0.084937, 0.162765, -0.091586, -0.002178, 0.014124, -0.083940, -0.247372, -0.328510, -0.178806, -0.007460, 0.139914, 0.026030, -0.127236, -0.088720, -0.008045, -0.136318, 0.295165, -0.051141, -0.043954, -0.016702, 0.025800, -0.247979, -0.035388, 0.069338, 0.043921, -0.227293, 0.139283, -0.212946, -0.116182, -0.019968, -0.099572, -0.097621, 0.073169, -0.091537, -0.202207, -0.037710, -0.117191, -0.040970, -0.209013, -0.135316, -0.100025, 0.007262, 0.100535, 0.032030, -0.223818, -0.101891, -0.010894, -0.012561, 0.018039, -0.010113, 0.056236, -0.129501, 0.128219, -0.000976, -0.032505, 0.011035, -0.148862, -0.101120, 0.027355, -0.118809, -0.212871, -0.193850, -0.118938, 0.113809, -0.022841, -0.027402, -0.128962, 0.060370, 0.087865, -0.117466, -0.025503, -0.036726, 0.107224, 0.062965, 0.033539, -0.024567, 0.060654, -0.140398, -0.083720, -0.143479, 0.073556, -0.083323, 0.099104, -0.022402, -0.134861, -0.077045, -0.014021, -0.081538, -0.130357, 0.163631, -0.025978, -0.112235, 0.041836, -0.222431, 0.033324, -0.034433, -0.005476, -0.068053, 0.008753, 0.022241, -0.199432, -0.154473, 0.001395, -0.090821, 0.025841, -0.030150, 0.023481, -0.041840, 0.020952, -0.052650, -0.071931, -0.096689, 0.086854, 0.098036, -0.103514, -0.058979, 0.042190, -0.189950, 0.078408, 0.011228, 0.104774, -0.039605, 0.027176, 0.023668, 0.063830, 0.008654, -0.069560, -0.142516, 0.096959, -0.062095, -0.093737, 0.003341, -0.123725, -0.145982, -0.071856, -0.018916, 0.074633, 0.056809, -0.080350, -0.055707, -0.252271, -0.030153, 0.062091, 0.104247, -0.139357, -0.043126, -0.004199, 0.031975, 0.171925, -0.025330, 0.031431, 0.028461, 0.160238, -0.114811, 0.096076, 0.015363, -0.049762, 0.006046, 0.049991, -0.049690, -0.025874, -0.084546, -0.039526, -0.031447, 0.026012, -0.150950, 0.045561, -0.179861, -0.141825, -0.190913, 0.168930, 0.021148, -0.210207, -0.081464, -0.051435, 0.015618, 0.010068, -0.078482, 0.079999, -0.005103, -0.001583, -0.106754, -0.053040, 0.134666, -0.103973, -0.133197, -0.172819, -0.089912, -0.102125, -0.004049, -0.144938, -0.044799, 0.017609, 0.028087, -0.186880, 0.022129, -0.047641, 0.096061, 0.074608, 0.093799, -0.009796, 0.138890, 0.158604, -0.230045, 0.109919, 0.058715, -0.106906, 0.097979, -0.041540, -0.087849, 0.037612, -0.136964, -0.160305, 0.117065, -0.009550, -0.101019, -0.039538, 0.029232, -0.004359, -0.019188, -0.086537, -0.036029, -0.111042, -0.074288, 0.001880, -0.051332, -0.045676, 0.029895, -0.201280, 0.052392, -0.044205, -0.098054, -0.044305, -0.003635, -0.085970, -0.066238, -0.110275, -0.083808, 0.024810, -0.088122, -0.106489, -0.064459, -0.116226, -0.067340, -0.080634, -0.014090, -0.012480, 0.007719, -0.021866, -0.132769, 0.075265, -0.051277, -0.015249, -0.148978, 0.014954, -0.004848, -0.093557, -0.128523, 0.035598, -0.154549, 0.059168, 0.032158, -0.004963, -0.148362, -0.021251, -0.088713, -0.131030, 0.147592, 0.045032, 0.013228, -0.025086, -0.131792, -0.009908, -0.010853, 0.040607, -0.083759, -0.132125, -0.168778, 0.009768, -0.050261, -0.114085, 0.023028, -0.136889, -0.058954, 0.087401, -0.037836, -0.096303, -0.234171, -0.204516, -0.094771, 0.052591, -0.148327, -0.058006, -0.199830, -0.046292, -0.210680, -0.051253, 0.063777, -0.144981, -0.118098, -0.008743, -0.054151, -0.097203, 0.015885, -0.021338, -0.153848, -0.075778, -0.039126, 0.013967, -0.231632, 0.005151, -0.020251, 0.026812, -0.122740, -0.168010, 0.145150, 0.089490, -0.024984, 0.032448, -0.005715, -0.144827, 0.021090, -0.217637, -0.020910, -0.085483, -0.168754, -0.070271, -0.139269, 0.225343, -0.095481, -0.065741, 0.025330, -0.082543, -0.149963, -0.043008, -0.018774, -0.301091, -0.033695, -0.101770, -0.133392, -0.045676, -0.007970, 0.098803, -0.005709, -0.048782, -0.103976, -0.014214, -0.063620, -0.136189, -0.034490, -0.175192, -0.233079, -0.177615, -0.007253, -0.062822, -0.029856, 0.115531, -0.196426, 0.039692, -0.065515, -0.009751, 0.034923, 0.136139, -0.066956, -0.144927, -0.082048, -0.044002, -0.036737, -0.093503, -0.106894, -0.111050, 0.007599, -0.217490, 0.064781, -0.047759, -0.127391, -0.040671, -0.074441, -0.054767, -0.208065, -0.079214, -0.166916, -0.041664, -0.122026, 0.046899, -0.037273, 0.004644, -0.003699, 0.052568, -0.002906, -0.005951, -0.032636, -0.005986, 0.086892, 0.079617, 0.120825, -0.165474, -0.126605, -0.184790, 0.047207, 0.086339, 0.007256, -0.027942, -0.030436, 0.063300, 0.027635, -0.075450, 0.031114, -0.019140, -0.021321, -0.103346, -0.087294, -0.216489, -0.049224, -0.046734, -0.048599, -0.102252, -0.158751, -0.009598, -0.014824, -0.139822, -0.110484, -0.012594, -0.097070, 0.061686, -0.097509, -0.080113, -0.041393, -0.001189, -0.175889, -0.122972, -0.148223, -0.006309, -0.136843, 0.016994, -0.023399, 0.006604, -0.080547, 0.018724, -0.030717, -0.004633, 0.082414, -0.034810, -0.114533, -0.200852, 0.077348, -0.124813, -0.160216, 0.085978, -0.091679, -0.113977, -0.098598, -0.019291, 0.010486, -0.020708, 0.023483, -0.078105, -0.198628, -0.063552, -0.182152, -0.001497, -0.116789, -0.069976, 0.054799, -0.185914, -0.103471, -0.053294, 0.013392, -0.000283, -0.173953, -0.160021, 0.066364, -0.132256, 0.026621, 0.049999, 0.006015, -0.067647, -0.111593, 0.006528, -0.120489, 0.086464, -0.028477, -0.126583, 0.023727, -0.036052, -0.068816, 0.029023, 0.091770, -0.086417, -0.202998, 0.102035, 0.021192, -0.138966, -0.066661, -0.042755, 0.069576, 0.082676, 0.030048, 0.023544, 0.049181, 0.071094, -0.090772, 0.159520, -0.013024, -0.060194, -0.024197, 0.021748, -0.056526, -0.122751, -0.022633, 0.040948, -0.007057, 0.000660, 0.015864, -0.119033, -0.055183, -0.041637, 0.082067, 0.202985, -0.126217, 0.058517, -0.186618, -0.164244, -0.117197, 0.117264, -0.037941, 0.144326, 0.117817, -0.143155, -0.120373, 0.059379, -0.015998, 0.129441, 0.102603, -0.168307, 0.022757, 0.055692, 0.035244, -0.033921, 0.039584, 0.145143, 0.086604, 0.138755, 0.037306, 0.184470, 0.042106, -0.029435, 0.171252, -0.066781, 0.049509, -0.055383, -0.030688, 0.092210, 0.105111, 0.035383, 0.038922, -0.153657, -0.067618, -0.004333, 0.024085, -0.012770, -0.116875, -0.147133, -0.072813, -0.038606, -0.044393, 0.068440, -0.065242, 0.012901, 0.144540, 0.058488, -0.101759, -0.019200, -0.164944, 0.083646, 0.041071, -0.117177, -0.041042, 0.117127, 0.103637, 0.034374, 0.147890, 0.148181, 0.090025, -0.039972, 0.026569, 0.021120, 0.036281, -0.016481, 0.163098, -0.167052, 0.169746, -0.049437, -0.100761, 0.139744, 0.199236, -0.045132, 0.073574, 0.138724, 0.152708, 0.015515, -0.235317, -0.083777, 0.101449, 0.155208, -0.057176, -0.071294, -0.012780, 0.046534, 0.142596, 0.036461, -0.044901, -0.074952, -0.016466, -0.164205, -0.044506, 0.008057, -0.093140, -0.015293, -0.067676, 0.026181, -0.142597, -0.044704, -0.056948, -0.157955, 0.115896, -0.064407, 0.034523, -0.110229, -0.098640, 0.125366, -0.029666, -0.090292, -0.045377, 0.051192, 0.099469, 0.076341, -0.021487, 0.022678, 0.046532, -0.114265, 0.017596, 0.020906, 0.049867, -0.078729, 0.012482, -0.030830, 0.122245, -0.129228, -0.029695, 0.169707, 0.026927, -0.084974, -0.040726, 0.059866, -0.011297, 0.094366, -0.130847, -0.069302, 0.035898, -0.155049, 0.066666, 0.088505, -0.060840, 0.100026, 0.099498, -0.110579, 0.086674, -0.127839, 0.016847, -0.054148, -0.117150, -0.198573, -0.070323, -0.026335, -0.098061, 0.017791, -0.014273, 0.079347, -0.018737, 0.179263, -0.002305, -0.050560, 0.015780, 0.041119, 0.086307, 0.001544, -0.013693, -0.119414, 0.066853, 0.119617, -0.217106, -0.023742, -0.006741, -0.010344, -0.024386, -0.131517, -0.028753, 0.084555, 0.021678, 0.023710, -0.010395, 0.047469, -0.052382, 0.098786, -0.008376, -0.069907, 0.085366, -0.165001, -0.028077, 0.015751, 0.085235, -0.010250, 0.002429, 0.203278, -0.093468, -0.053033, 0.072789, 0.043867, 0.062264, 0.099703, 0.154054, 0.079033, -0.056707, -0.070698, 0.121270, -0.117285, -0.148616, 0.086448, -0.090539, 0.030692, 0.034122, -0.093544, -0.089995, 0.059018, -0.038828, 0.037126, -0.136537, 0.070475, -0.046117, 0.053130, 0.170559, 0.053956, 0.018535, -0.030878, 0.022160, -0.077642, -0.189230, 0.059160, -0.062924, -0.180665, -0.099824, -0.098950, 0.002466, -0.019390, -0.004555, 0.020420, -0.024363, 0.058931, 0.073766, 0.068702, -0.087764, -0.032242, 0.073636, 0.071197, 0.097383, -0.173730, 0.029280, -0.054453, -0.015248, -0.148534, -0.084479, 0.005111, 0.130577, -0.105668, 0.079299, 0.003235, -0.081081, -0.130359, 0.070253, -0.110694, 0.037081, -0.041315, 0.074619, 0.071535, 0.024587, -0.174044, -0.094007, 0.118237, -0.024835, -0.046728, 0.182307, 0.088483, -0.023628, -0.036965, 0.019472, -0.045045, 0.039440, 0.017264, 0.097226, -0.022984, -0.003118, -0.304042, -0.047657, -0.051791, 0.158829, -0.066265, 0.097961, -0.058862, 0.019016, -0.090564, 0.005688, -0.070917, 0.116594, -0.056278, -0.076547, 0.003080, 0.142880, 0.018680, -0.096846, 0.048738, 0.142879, 0.031667, -0.128994, -0.090995, -0.063082, 0.073211, -0.043917, -0.113743, -0.063416, -0.071807, -0.035187, 0.110351, 0.053724, -0.117475, 0.020538, -0.026410, 0.062344, 0.052451, -0.013615, -0.147677, 0.056842, -0.057224, 0.039454, 0.100180, -0.039484, 0.014294, 0.168338, -0.076061, 0.046241, 0.080953, -0.117992, 0.000434, -0.012340, 0.115420, 0.014703, -0.036446, 0.018519, -0.147867, 0.019952, -0.044170, -0.043352, 0.049652, 0.043997, -0.070146, -0.024542, -0.142537, -0.028954, -0.029349, 0.022060, 0.008983, -0.053424, -0.016003, 0.006247, 0.061104, 0.050734, 0.032107, -0.044257, 0.092995, 0.057502, 0.017627, 0.091503, 0.118991, 0.013152, -0.169037, 0.125871, -0.176133, -0.019289, 0.111911, 0.009510, 0.008829, -0.157112, -0.016608, 0.042768, -0.072247, 0.058393, -0.117136, 0.017748, -0.057995, -0.129622, -0.014803, -0.066282, 0.015524, 0.127418, -0.074217, 0.024822, -0.197154, 0.042987, -0.081507, 0.067740, 0.060346, 0.118172, -0.094873, 0.048237, -0.033816, 0.092007, -0.014019, -0.087272, 0.028185, -0.184813, 0.087166, 0.025336, 0.005554, 0.051941, 0.011025, 0.030366, 0.013038, 0.194331, 0.074825, -0.224661, 0.159764, 0.014123, 0.109104, 0.109942, -0.080625, -0.101255, 0.148388, 0.070335, -0.003718, 0.003288, -0.027729, 0.127294, -0.099893, -0.019717, -0.001185, -0.006413, -0.071276, 0.006979, -0.116613, 0.053450, -0.046211, -0.016818, 0.105791, 0.120337, 0.078001, -0.106814, 0.023293, 0.062645, -0.037335, 0.018961, -0.034720, 0.100587, 0.006601, 0.018247, 0.080920, -0.133658, -0.100272, 0.144770, 0.005372, -0.105028, 0.043350, -0.073430, 0.116246, -0.105507, 0.083417, 0.076652, -0.001708, 0.255886, -0.103664, -0.121963, 0.029488, -0.106733, 0.096946, 0.109316, 0.095282, -0.063873, 0.038397, 0.273502, -0.014831, -0.045789, 0.148320, -0.116517, -0.119054, -0.087235, 0.062254, -0.145052, 0.084778, -0.075057, -0.301261, 0.043413, 0.068367, 0.125284, -0.063389, -0.023944, 0.053126, 0.147260, 0.119572, -0.053608, 0.033723, -0.004656, -0.119163, 0.096190, -0.146080, 0.046461, -0.170626, -0.088610, -0.036965, -0.036090, -0.102746, -0.126298, -0.018096, -0.029234, 0.056686, -0.083532, 0.019483, 0.049426, -0.101021, -0.073348, 0.053829, -0.080902, -0.021208, -0.073556, 0.105784, 0.213869, -0.025465, -0.064158, -0.381028, 0.063233, -0.094779, 0.187027, -0.006644, -0.069662, 0.002580, -0.053224, 0.045534, -0.028284, 0.136176, -0.016081, 0.028095, 0.034772, -0.022276, -0.178128, -0.041598, 0.005843, -0.086407, -0.007446, 0.028685, -0.022599, 0.089290, 0.319908, 0.075521, -0.003703, 0.010279, -0.097664, -0.072643, -0.024213, 0.100523, -0.033696, -0.002511, -0.133648, 0.002638, 0.134987, -0.057933, -0.092656, -0.105945, -0.126956, 0.084314, -0.001516, -0.186977, 0.020002, -0.193135, 0.020655, 0.036038, -0.031342, -0.175460, -0.180554, 0.009570, -0.154066, -0.099684, -0.025210, -0.020764, 0.087913, -0.076385, 0.107840, -0.146812, 0.032364, 0.094126, 0.058828, -0.144958, -0.004610, -0.118794, -0.065217, -0.039490, -0.013315, 0.054885, 0.075500, -0.051281, -0.042950, -0.132541, -0.124352, -0.211332, -0.037289, -0.216332, 0.021722, -0.020196, -0.171414, -0.035075, 0.056188, -0.000126, -0.012344, 0.116943, -0.227331, -0.066375, -0.087067, 0.009563, -0.040385, 0.097734, -0.101710, -0.046529, -0.051028, -0.104818, -0.144603, -0.105879, -0.014701, -0.129602, -0.016104, -0.183929, -0.059448, -0.055404, 0.094317, -0.126847, 0.019051, -0.033867, -0.039139, -0.050566, -0.094930, -0.194191, 0.085933, -0.367069, 0.046000, -0.104139, -0.097389, -0.027324, 0.069076, -0.061382, -0.091633, 0.015271, 0.014288, 0.020243, -0.125450, -0.226755, -0.031114, -0.100411, 0.111216, -0.009450, -0.078539, -0.116103, -0.140027, -0.087181, -0.191718, -0.070862, -0.069203, 0.042169, -0.072331, -0.100808, -0.013237, 0.009791, -0.089520, -0.180334, 0.005710, 0.107547, -0.057965, -0.242825, -0.077640, -0.229659, -0.107370, -0.130146, -0.026662, -0.141512, 0.058331, 0.079186, 0.004357, -0.219632, -0.058070, -0.238432, -0.047663, 0.072005, 0.019580, -0.175580, 0.133436, 0.014942, -0.112805, -0.041108, -0.004388, 0.078067, 0.055282, -0.013928, -0.021361, -0.102965, -0.022910, 0.190479, 0.038260, -0.011673, -0.129639, 0.134730, -0.086246, -0.041449, 0.040545, -0.195004, -0.019456, 0.086908, -0.119246, -0.014457, -0.066465, -0.091412, 0.048372, 0.043623, 0.056843, -0.022895, -0.120414, 0.022003, 0.046297, -0.080718, 0.076534, 0.178156, -0.178485, -0.136854, -0.017726, -0.008594, -0.013896, -0.056431, -0.326249, -0.082323, 0.065994, -0.087436, 0.027198, 0.038487, -0.080040, 0.000551, -0.060412, -0.001544, 0.008370, 0.047446, -0.059820, -0.116183, -0.087526, -0.084095, -0.087297, 0.081780, -0.084317, 0.090931, -0.003402, -0.050849, 0.112515, -0.157019, -0.276175, -0.075481, -0.059869, 0.036397, -0.000340, -0.009834, -0.151082, -0.055476, 0.016659, -0.102365, 0.191112, -0.102762, -0.031264, 0.028062, -0.154118, 0.022473, -0.028108, -0.136331, -0.073106, 0.083459, 0.092774, 0.010394, 0.010209, -0.015374, -0.041251, 0.018496, -0.015994, -0.094139, 0.075551, -0.032961, 0.068024, 0.028211, 0.062287, -0.048844, -0.022653, 0.006049, -0.049675, -0.141361, -0.102663, 0.032909, -0.064709, -0.114736, 0.028978, -0.065624, -0.056909, -0.031948, -0.017085, -0.140236, -0.180262, 0.041230, 0.057634, -0.042320, 0.086991, -0.024393, 0.108087, -0.103073, 0.090662, -0.018796, -0.098772, -0.051831, -0.099601, -0.063665, -0.091446, 0.099636, -0.020757, 0.031888, -0.031037, -0.005659, 0.112928, -0.047007, -0.028184, -0.017555, -0.056931, -0.168266, -0.096296, -0.069911, -0.047682, -0.173247, 0.030497, 0.089311, 0.082698, 0.055852, -0.132705, -0.091753, -0.000630, 0.052152, -0.079904, -0.017650, 0.063140, 0.045963, 0.010155, -0.112527, 0.021262, 0.073684, 0.059862, 0.009121, -0.081018, 0.084145, 0.043122, 0.018955, 0.001018, 0.002494, -0.052652, 0.006007, -0.075843, -0.025851, -0.062350, -0.073561, -0.155721, 0.040309, 0.068766, -0.035629, 0.056447, 0.117070, -0.052542, -0.119053, -0.107729, -0.102704, 0.056566, -0.054978, -0.082882, -0.117422, 0.042796, -0.000199, 0.016556, -0.256099, -0.070111, -0.023579, -0.006253, 0.062201, 0.147156, 0.050702, -0.007044, 0.073158, 0.085700, -0.024150, 0.078223, 0.086409, -0.072242, 0.046618, 0.108160, -0.174050, -0.107874, 0.127690, -0.139733, -0.006462, 0.036263, 0.078073, -0.050308, 0.016359, -0.052203, -0.085708, 0.019010, -0.011554, -0.116066, -0.061254, -0.022967, -0.227917, -0.018254, -0.048215, 0.007526, -0.036657, 0.047089, 0.013774, -0.034044, -0.112435, -0.094616, 0.033609, -0.188234, 0.152140, 0.084898, -0.107788, -0.049830, -0.055038, -0.028252, -0.054747, -0.024485, -0.017384, -0.073533, 0.031411, 0.031480, 0.044878, 0.087346, 0.013158, -0.120802, -0.044465, 0.042307, -0.043693, 0.034963, 0.051188, -0.114605, 0.022636, 0.094169, 0.041304, 0.129952, -0.086016, -0.036860, 0.098597, -0.028515, -0.233841, -0.012574, -0.038106, 0.142052, -0.122946, 0.022597, -0.108827, -0.161925, 0.136554, -0.073705, -0.075164, 0.050270, -0.113360, -0.027091, -0.037795, 0.135926, 0.023007, -0.179968, 0.039523, 0.114981, -0.081676, 0.044021, 0.008575, -0.035012, -0.130764, 0.057064, -0.045369, -0.034859, -0.100056, -0.106044, -0.162867, -0.106885, -0.111643, -0.141240, 0.083862, -0.133622, -0.013784, 0.142567, -0.025397, -0.075783, 0.165546, -0.045950, 0.016735, -0.041263, -0.133181, -0.110367, -0.218113, -0.088805, -0.103892, 0.061520, -0.048347, 0.062326, -0.017489, -0.030911, -0.062898, -0.021963, 0.242810, 0.025943, 0.106521, -0.070253, 0.050554, 0.067029, -0.003385, 0.012045, -0.000830, -0.090342, -0.161640, 0.043597, -0.082577, 0.010252, 0.023988, -0.018043, -0.190813, -0.118497, -0.121469, 0.037608, 0.129419, 0.035159, -0.126327, -0.037070, -0.028592, 0.047085, -0.023773, -0.012030, 0.055689, 0.074148, 0.029489, 0.044009, 0.052038, -0.059163, -0.025433, -0.172589, 0.053325, 0.046766, 0.012789, -0.120103, 0.119155, -0.075167, -0.075945, -0.126783, -0.043503, -0.164872, -0.023662, 0.004837, 0.054638, -0.229084, -0.192464, -0.121554, 0.057940, 0.033658, -0.086682, -0.058215, 0.073858, -0.139716, 0.024769, 0.097304, -0.095555, -0.066120, -0.305383, -0.075664, 0.017603, 0.172361, 0.011219, -0.055651, -0.146251, -0.005335, -0.004105, -0.120963, 0.070451, -0.016917, -0.124862, 0.089318, 0.044002, -0.001771, -0.091858, 0.109983, -0.033500, 0.012604, -0.081997, -0.079272, 0.041373, 0.005885, -0.228869, 0.068199, -0.037632, 0.071898, 0.251602, -0.107793, -0.050886, -0.091756, -0.203825, -0.165251, 0.109858, 0.095500, -0.051785, 0.060635, -0.053082, -0.086777, 0.079521, -0.154866, 0.000997, -0.042849, -0.056831, 0.006285, -0.019673, -0.003617, -0.131736, 0.008258, -0.246536, 0.087187, -0.045319, 0.053514, -0.127200, 0.013877, -0.183917, -0.043583, 0.015669, -0.105153, -0.035255, -0.071183, -0.059093, -0.070308, -0.127914, 0.057378, 0.073274, -0.013615, -0.050868, -0.098035, -0.173268, -0.146615, 0.088664, 0.012823, 0.044644, -0.034901, -0.056601, -0.067925, -0.049439, -0.188231, 0.079631, -0.083042, -0.093555, 0.023727, -0.186291, 0.020614, -0.068362, 0.053272, -0.002033, 0.058610, -0.173109, 0.112715, 0.054360, -0.034868, -0.009817, 0.005929, -0.104932, -0.246230, -0.224867, -0.075170, -0.048756, 0.122310, 0.006069, -0.229542, 0.053796, -0.133409, 0.061239, 0.032309, 0.147751, -0.005645, 0.072127, -0.015657, 0.133921, -0.024546, -0.059587, 0.027752, -0.079260, -0.170856, -0.117589, -0.033127, -0.014851, -0.163960, -0.019863, -0.017465, 0.106070, 0.031654, -0.094260, -0.157940, 0.026296, -0.145314, -0.208231, -0.099917, -0.009463, -0.099642, -0.050368, 0.124722, -0.056147, 0.021536, -0.010428, -0.064955, 0.089510, -0.114330, -0.047571, -0.042184, -0.053861, -0.051968, -0.142291, -0.069270, -0.041878, -0.180094, 0.068377, 0.015211, -0.159702, 0.048156, 0.153419, 0.040829, 0.076509, -0.013538, -0.029691, 0.006143, -0.123903, -0.353122, 0.031193, -0.147568, 0.145407, -0.140318, 0.042785, -0.175349, -0.021035, -0.018479, -0.032797, 0.003186, -0.049331, 0.062884, -0.009876, -0.017983, 0.161882, 0.048737, -0.175836, -0.109206, -0.175934, -0.023401, 0.036002, 0.078386, -0.078901, -0.126181, 0.150031, 0.066221, -0.087101, -0.089790, -0.059253, -0.033897, -0.036377, 0.066118, 0.118529, -0.151079, 0.186617, -0.077682, -0.047121, 0.067008, -0.280852, -0.036436, -0.071966, -0.140291, -0.075102, 0.045806, -0.161650, -0.052586, 0.112875, -0.150060, -0.096994, -0.070530, -0.057995, -0.140867, -0.103700, -0.009514, -0.068845, -0.078290, -0.143776, -0.169109, -0.058759, -0.135924, 0.160528, -0.057830, -0.044408, 0.006477, -0.021510, -0.113184, -0.079740, -0.111221, -0.013740, 0.030159, -0.019819, 0.043001, -0.023639, -0.006348, -0.025693, 0.123897, -0.167645, 0.213983, 0.008189, -0.024895, -0.076585, -0.038526, -0.009165, 0.142749, -0.253920, 0.098266, -0.023862, -0.059127, -0.200217, -0.012129, -0.008253, 0.050106, 0.128204, 0.064484, 0.019574, 0.108876, 0.091993, -0.228872, 0.035731, -0.003206, 0.016731, -0.174505, -0.032594, 0.001252, 0.128174, 0.026790, 0.018068, -0.026198, 0.013321, -0.120149, -0.026221, 0.093478, -0.054973, 0.074660, 0.043212, -0.026289, -0.168483, -0.087013, 0.098342, -0.152687, -0.170789, 0.155834, -0.194697, -0.008745, 0.031344, -0.055731, -0.049699, 0.053822, 0.031670, -0.093430, 0.035759, 0.049842, -0.034841, -0.022870, -0.117492, -0.236812, 0.031399, -0.061935, -0.140886, -0.080660, 0.032678, -0.024031, -0.018796, 0.027493, -0.055735, -0.070906, 0.005528, 0.040037, -0.022803, -0.019349, 0.074163, -0.165675, -0.098578, -0.118681, -0.006050, 0.070484, -0.014614, 0.031527, -0.056811, 0.024859, 0.030932, 0.165601, -0.115130, -0.049246, -0.076288, -0.045846, 0.034802, -0.006072, 0.132238, 0.033077, 0.080409, 0.085701, -0.048732, -0.021165, -0.071395, -0.213272, 0.001368, 0.026006, 0.056703, 0.030494, 0.065061, -0.067255, 0.037546, 0.030709, 0.097234, -0.051068, 0.115002, 0.088447, 0.017987, -0.036787, -0.077183, -0.090074, -0.040965, 0.121228, 0.029440, -0.064205, -0.060446, 0.140337, -0.080121, 0.076058, -0.035049, -0.100415, -0.067477, 0.098861, 0.059098, 0.110137, 0.079657, -0.084156, -0.133281, 0.014878, 0.091782, 0.005532, -0.187822, 0.101822, 0.011838, 0.017463, 0.112538, -0.017211, -0.065418, 0.235493, 0.054089, 0.147176, -0.087423, -0.059838, 0.037099, 0.023708, 0.045870, -0.006962, -0.032980, -0.067077, 0.067784, -0.029464, -0.036382, 0.008963, -0.204239, -0.156968, 0.057770, 0.019753, -0.037834, 0.025573, -0.073082, 0.080685, -0.051962, 0.051800, -0.017096, -0.062929, 0.015842, -0.037474, -0.077980, -0.016682, -0.025164, -0.029561, -0.128855, -0.060379, -0.114090, 0.032669, -0.101440, 0.009349, -0.186647, -0.134202, 0.007123, -0.080913, -0.161299, 0.066349, -0.114912, 0.087805, -0.105849, -0.063411, 0.072154, -0.049064, -0.016927, 0.033458, 0.001917, -0.002014, 0.204346, 0.142631, 0.048653, 0.070003, -0.028448, -0.077633, -0.057995, -0.000431, 0.034120, -0.072120, 0.004294, -0.065416, -0.138701, 0.052053, 0.054738, 0.004186, 0.075987, 0.025781, 0.100008, 0.006173, -0.002671, 0.132038, -0.067688, 0.009316, 0.071962, -0.092067, 0.039820, 0.054608, -0.066626, 0.062243, -0.032009, -0.111331, -0.063792, 0.010918, 0.007507, -0.164606, -0.065931, -0.081069, -0.040328, -0.016404, -0.058618, 0.003151, -0.043152, 0.176332, 0.025580, -0.028547, -0.176311, -0.057942, 0.003372, 0.119560, 0.013266, -0.009865, -0.026428, 0.041093, -0.086451, 0.248209, -0.062104, -0.166841, 0.033292, 0.076545, -0.084711, -0.048468, 0.135539, -0.038221, -0.114337, -0.059129, 0.028118, 0.012321, -0.174759, 0.057674, 0.019802, 0.012922, -0.014849, -0.016069, 0.112891, -0.079790, -0.003197, 0.037654, 0.035599, -0.116782, -0.252279, -0.063665, -0.043144, 0.053982, -0.112467, 0.014827, 0.084605, 0.095304, 0.007492, 0.072378, 0.080161, -0.038290, -0.044538, 0.040011, -0.010893, 0.172533, 0.018024, 0.058256, -0.136609, -0.065971, 0.045392, 0.000254, 0.093012, 0.095824, 0.101547, 0.011248, 0.075520, -0.156232, -0.002681, 0.025294, 0.095404, -0.022035, -0.037930, -0.058540, -0.145160, -0.149642, -0.153581, 0.016153, -0.071728, 0.049940, -0.145765, 0.087358, 0.013887, -0.084610, -0.033622, 0.057979, -0.051256, -0.013590, 0.004323, 0.002204, 0.096511, 0.069835, -0.120925, 0.031582, -0.114119, 0.250629, 0.094299, 0.117886, 0.095517, -0.014982, -0.067955, 0.128354, -0.091506, -0.027878, 0.058715, 0.067631, -0.078936, 0.029895, -0.150339, -0.062390, 0.044752, -0.010997, 0.019415, 0.014300, 0.005096, -0.061742, -0.076706, -0.021229, -0.007999, 0.073269, -0.191618, 0.040091, 0.060849, -0.014392, -0.002520, 0.004526, 0.042337, 0.013382, -0.124605, 0.075761, 0.049341, 0.054852, 0.086052, 0.077612, -0.021126, 0.061452, -0.215456, 0.021030, 0.068245, -0.166381, -0.016099, 0.092261, -0.031255, -0.077567, -0.116549, 0.003587, -0.005023, 0.000405, -0.030602, 0.082284, 0.000382, 0.054953, 0.073340, -0.093532, 0.022639, -0.029975, -0.053221, 0.109408, -0.058406, -0.025490, -0.005300, -0.083054, 0.043711, 0.117144, 0.104686, 0.049200, -0.035299, 0.032636, -0.141892, 0.119466, -0.101731, 0.012251, 0.064773, 0.017995, 0.008142, 0.087301, -0.006923, 0.023042, -0.049533, 0.007703, -0.050253, -0.127481, 0.062545, 0.002228, -0.052134, -0.068017, -0.015901, 0.006291, 0.004868, 0.018001, -0.057128, 0.021766, 0.048399, 0.011980, 0.119909, -0.029855, -0.098146, 0.130535, 0.117855, 0.109109, 0.063490, -0.005151, -0.088425, 0.021349, -0.021715, 0.018073, -0.127977, -0.059910, -0.050422, 0.114490, -0.003207, -0.136542, 0.059025, 0.067964, -0.138546, 0.001892, 0.039257, 0.118726, 0.050033, -0.051535, 0.014530, -0.038214, -0.144600, -0.009352, -0.023279, -0.121206, -0.035867, -0.127557, -0.180835, 0.164152, 0.032351, 0.057177, 0.055231, 0.019786, -0.069579, -0.213699, 0.035767, -0.043928, -0.121789, 0.016473, -0.062504, 0.010528, -0.108932, -0.022767, 0.140302, -0.079811, -0.071962, -0.209977, -0.108367, 0.095807, -0.111089, -0.005972, -0.098901, 0.001168, -0.030703, -0.099747, 0.043024, 0.013817, 0.004147, -0.058279, -0.191894, -0.069057, -0.099445, -0.135400, 0.015166, 0.061659, 0.024829, 0.023265, 0.027158, -0.034233, -0.019249, 0.054152, -0.139799, -0.139263, -0.008389, 0.116566, -0.153132, -0.079141, -0.118352, 0.079200, -0.056278, -0.026452, -0.053211, -0.134522, -0.052625, 0.097024, -0.178102, 0.068767, -0.013983, -0.024566, -0.185938, -0.115049, 0.101773, 0.173322, 0.052996, 0.276921, -0.005077, 0.131549, 0.165202, 0.124667, 0.049748, 0.049771, -0.107103, 0.015139, 0.096201, -0.063182, -0.148635, -0.104358, -0.042369, 0.020327, 0.057761, -0.054728, -0.075224, -0.019680, 0.072565, 0.077025, -0.135953, 0.059662, 0.044110, -0.106754, -0.171349, 0.198336, -0.129622, -0.069572, -0.017677, 0.021989, -0.024541, -0.053189, 0.044967, -0.102041, 0.070593, -0.095802, -0.048216, 0.059130, -0.077050, -0.029985, -0.117988, -0.025894, 0.162537, 0.001679, -0.125865, -0.067199, -0.022875, 0.000398, -0.078279, -0.081510, -0.113201, -0.105033, -0.026187, 0.088747, -0.009140, -0.056726, -0.078485, -0.143280, 0.060964, -0.032844, 0.070814, -0.130627, -0.111308, -0.158879, 0.096151, -0.060557, 0.051451, -0.131444, -0.164386, -0.162636, -0.025842, 0.014788, -0.063375, -0.128550, 0.177143, -0.015911, -0.078745, 0.111220, -0.062524, -0.092734, 0.078611, -0.098103, 0.060231, 0.005971, -0.030148, -0.087836, -0.037196, -0.087765, 0.089605, -0.074122, -0.098283, 0.086429, 0.006048, -0.107308, -0.127141, 0.107449, 0.022448, 0.072796, -0.060733, -0.100252, -0.083407, -0.099515, 0.009762, -0.068191, -0.059841, 0.013648, -0.202719, -0.144398, 0.033505, 0.061672, -0.001443, -0.182640, 0.049812, -0.083249, 0.064124, 0.053720, -0.033791, 0.056776, -0.089521, -0.076365, -0.007643, 0.003800, -0.059844, 0.054176, 0.086809, 0.075863, -0.059941, -0.136158, -0.023925, -0.090318, 0.000217, -0.007239, -0.018444, -0.074410, -0.055030, 0.088063, -0.182837, -0.138123, -0.085601, -0.091443, -0.006739, 0.022858, -0.055435, 0.024634, 0.133234, -0.013144, 0.113602, -0.105965, 0.048865, -0.197711, -0.136751, 0.065697, -0.021738, -0.020856, -0.098692, 0.027762, -0.176309, -0.105591, 0.034446, -0.073073, -0.042501, 0.069289, 0.046891, -0.097975, -0.146949, -0.146675, 0.018055, -0.045944, 0.053389, 0.143237, 0.140190, 0.041611, -0.076793, -0.099553, -0.128396, -0.072306, -0.124234, -0.130288, -0.106267, -0.074224, -0.086666, -0.091989, 0.103535, -0.016252, -0.134184, -0.027887, -0.140756, -0.100259, -0.015901, -0.028394, -0.149708, -0.122279, 0.012344, 0.082801, -0.148535, 0.104546, 0.009124, 0.002504, 0.019203, -0.067298, -0.024391, 0.108015, -0.025879, 0.006084, 0.160548, -0.137075, 0.003340, 0.213151, -0.092671, 0.018159, -0.014164, 0.028064, -0.078276, -0.180295, 0.007342, -0.090920, 0.034161, 0.166572, 0.063671, -0.179594, -0.052427, -0.049676, 0.010783, -0.015752, -0.073376, 0.022851, -0.267236, 0.141386, -0.162151, -0.003006, -0.030870, -0.037759, -0.167205, 0.029051, 0.070623, 0.035191, 0.009115, 0.021677, -0.089117, 0.077844, -0.179437, 0.061892, -0.031638, -0.099240, -0.005649, -0.104061, 0.013049, -0.025086, -0.065634, -0.010691, 0.060415, -0.066028, -0.044047, -0.171913, -0.151293, 0.077762, -0.105070, 0.028585, 0.053779, -0.053717, 0.027245, 0.049920, -0.046015, 0.059541, -0.112515, -0.091451, -0.190892, -0.028940, -0.214434, 0.019865, -0.014777, -0.021537, -0.108209, -0.135514, 0.066939, -0.121798, 0.006864, 0.002213, 0.025791, 0.029141, -0.039185, -0.113929, -0.049977, -0.118579, 0.014141, 0.001444, -0.126466, -0.031304, 0.070617, -0.106682, -0.074144, -0.010001, 0.120183, -0.088579, 0.091692, -0.059496, -0.123072, 0.136135, -0.075894, 0.038026, -0.079725, 0.019509, 0.039074, -0.014544, -0.162935, 0.006108, 0.069590, -0.165580, -0.162726, -0.102671, 0.124794, 0.177552, -0.061786, 0.092424, -0.087871, 0.003020, -0.114115, 0.006950, 0.075406, 0.053756, -0.172153, 0.089267, 0.028655, 0.152431, 0.106032, 0.019915, -0.063168, 0.032387, 0.020009, -0.129434, 0.047699, 0.164224, -0.096366, -0.059017, -0.034837, 0.111875, -0.077690, -0.184036, -0.029098, -0.098524, -0.102672, 0.011326, 0.047258, 0.095350, 0.000405, 0.009580, 0.064386, -0.020766, -0.004319, -0.076974, -0.036920, 0.034011, -0.065528, -0.017410, -0.016508, -0.002091, 0.029483, -0.138785, -0.020239, -0.051472, 0.005860, 0.093470, -0.111514, 0.037871, 0.044907, 0.031009, 0.039143, -0.069019, -0.016582, 0.008915, -0.167552, -0.027772, 0.026449, 0.011598, 0.070179, 0.040630, 0.003834, 0.004875, -0.013500, -0.097471, -0.084086, -0.083261, -0.010578, -0.108506, 0.027612, -0.108314, 0.011878, 0.151437, -0.073757, 0.063326, 0.063680, 0.050593, 0.006069, 0.133256, 0.144176, -0.011904, 0.100271, 0.065117, -0.051765, -0.123202, -0.011145, -0.065397, -0.233520, -0.116338, -0.072892, -0.010288, -0.117758, -0.263255, -0.129320, -0.080238, 0.156201, 0.088115, 0.059220, 0.093655, -0.164460, -0.049598, -0.095991, -0.086657, -0.038450, -0.115876, -0.063028, -0.089367, -0.034471, 0.041378, 0.103871, 0.043801, 0.088701, -0.117042, -0.099865, 0.003084, -0.127849, -0.039886, 0.130072, -0.042420, 0.099195, 0.045954, -0.004092, -0.054251, -0.044969, -0.062797, -0.061660, -0.090294, 0.078700, 0.017290, -0.026370, -0.041976, -0.018638, 0.092204, 0.095606, -0.056530, -0.063051, -0.076196, 0.106822, -0.089183, -0.082122, 0.080038, 0.035343, 0.071318, -0.020126, -0.030967, -0.074179, 0.079528, 0.004116, -0.036716, 0.002349, 0.046550, 0.013934, -0.168303, 0.058565, -0.039214, -0.102998, 0.119397, 0.156250, -0.008968, 0.033022, 0.072586, 0.039182, 0.178555, 0.030400, 0.028062, 0.012452, 0.063616, 0.011140, -0.067570, 0.064047, 0.023183, -0.079947, 0.020568, 0.145432, -0.042589, -0.088513, 0.036398, 0.030347, -0.119827, -0.090826, 0.107782, -0.073441, -0.101210, 0.017490, -0.187816, -0.133791, 0.133743, 0.124610, 0.089537, -0.001632, -0.061080, -0.040848, 0.069088, 0.144801, -0.187087, 0.132161, 0.052537, 0.050073, -0.095321, 0.105963, -0.113581, -0.099277, -0.017741, 0.067251, 0.009021, -0.110608, 0.074434, 0.017481, -0.072057, 0.069138, -0.139169, -0.029193, -0.040788, -0.080506, -0.035487, 0.026556, -0.070083, 0.043547, -0.058873, -0.100772, -0.003194, 0.055339, -0.008688, -0.035706, 0.002001, 0.058450, 0.144096, -0.014168, -0.071943, 0.043440, 0.124256, 0.055023, -0.002750, -0.074196, 0.110832, 0.078298, -0.026749, -0.135911, -0.124625, -0.082140, -0.077322, -0.130755, -0.178140, -0.034902, -0.091923, 0.080372, 0.056911, -0.016695, -0.113012, 0.066029, -0.086475, -0.091969, 0.175351, 0.108957, 0.052052, -0.114937, -0.056842, -0.069490, 0.077391, -0.041332, -0.083332, 0.156843, -0.088905, -0.055907, -0.081896, 0.021310, 0.013324, -0.021883, -0.102334, 0.098233, 0.078277, 0.116115, -0.161238, -0.065386, -0.114773, -0.010476, 0.037619, 0.011903, 0.120994, -0.102421, -0.058744, -0.114603, 0.029886, 0.002742, 0.010915, -0.010118, 0.096707, -0.084630, 0.033244, 0.025245, 0.037932, -0.135450, 0.055104, -0.048576, 0.022220, 0.004110, 0.019060, -0.072560, -0.086262, -0.018641, 0.047792, -0.029146, -0.104912, -0.010956, 0.003854, -0.054019, 0.101513, -0.062776, 0.095478, 0.017286, -0.032747, 0.040655, -0.107236, 0.099701, -0.031741, 0.042656, -0.019910, -0.139714, -0.083407, -0.205610, -0.064838, -0.088966, -0.002475, 0.036755, 0.115221, -0.080641, -0.032659, 0.097438, -0.150376, -0.111857, -0.036984, 0.200731, -0.049128, 0.037679, -0.244369, 0.249312, -0.088724, 0.019072, -0.033821, -0.033679, -0.120427, -0.168260, -0.152952, -0.082231, -0.013921, 0.064537, -0.100772, -0.070762, 0.132940, 0.025851, -0.034372, 0.073477, 0.131358, 0.037405, -0.019334, 0.019583, -0.032638, -0.141897, 0.032864, -0.034396, 0.046419, -0.179922, -0.031577, 0.032264, -0.052588, 0.074201, -0.104608, 0.129805, 0.048165, -0.145889, 0.010923, 0.038807, -0.167107, 0.088594, 0.071233, 0.022715, -0.009977, 0.032354, -0.153355, 0.215031, 0.072684, -0.100893, -0.041009, -0.075564, -0.054332, 0.032531, -0.094763, 0.137496, 0.086833, 0.001649, -0.255322, -0.110593, 0.088414, -0.035349, 0.055580, -0.116333, 0.007994, 0.093696, 0.018478, -0.038420, -0.067808, -0.075585, 0.026028, -0.051669, 0.109467, -0.178950, 0.095638, -0.125675, 0.118970, 0.117680, 0.057013, 0.044610, 0.052066, -0.039249, -0.017673, -0.110420, -0.153433, -0.118427, -0.067390, -0.058137, 0.113123, -0.017957, 0.025160, -0.052458, 0.110550, 0.069565, -0.100847, -0.045675, 0.039920, -0.016841, -0.146486, 0.045277, -0.070795, -0.124312, -0.105563, -0.000388, -0.070452, -0.149859, 0.072526, 0.063527, -0.039524, 0.205809, -0.142528, 0.020870, 0.039052, -0.081472, 0.133929, 0.009704, -0.192122, -0.088153, -0.171554, -0.145384, 0.091197, 0.010014, -0.252314, 0.123595, 0.049866, -0.004045, -0.022608, -0.047581, 0.006379, -0.111861, 0.061456, -0.022511, 0.141158, 0.090272, -0.078931, -0.115785, 0.023610, -0.226771, -0.011266, 0.017915, -0.257406, 0.066873, -0.233122, 0.162009, -0.106780, 0.095696, 0.020969, -0.115322, -0.077852, -0.113105, 0.062498, 0.022420, 0.081641, -0.033092, -0.097032, 0.078533, -0.272336, 0.042639, 0.026189, -0.075359, -0.082953, 0.223244, -0.141986, -0.043632, -0.105225, 0.044779, -0.047352, 0.027948, 0.057636, -0.156457, 0.019646, -0.072059, 0.024275, -0.166494, -0.106689, -0.055403, 0.131450, -0.067107, 0.027383, 0.044595, -0.097701, -0.064108, -0.017052, 0.102321, -0.062845, -0.069732, -0.126782, 0.167127, -0.035825, -0.031903, -0.062586, -0.105736, -0.005309, 0.057495, -0.058550, -0.182121, 0.081607, -0.088159, 0.063443, -0.123381, 0.032293, -0.190995, 0.043385, 0.016147, 0.089450, 0.082112, -0.167787, -0.061621, 0.052680, 0.067742, 0.021218, -0.018484, -0.128717, -0.025581, 0.019114, -0.005618, -0.005687, 0.119374, 0.045428, 0.109199, 0.004786, -0.023340, 0.189729, 0.002662, -0.067457, -0.057660, -0.123217, -0.135085, -0.130367, 0.150391, -0.090935, 0.011361, -0.061593, 0.057744, 0.009307, 0.110663, 0.102082, -0.147567, 0.008066, 0.038584, -0.223765, 0.021189, 0.024957, 0.121172, -0.074707, -0.125421, -0.049682, 0.119886, -0.104690, 0.110235, -0.036904, -0.008463, -0.120817, -0.029453, -0.022796, -0.046087, -0.049844, -0.068031, -0.099763, -0.082477, -0.083889, 0.096684, 0.032236, 0.000173, -0.107304, -0.052242, 0.005163, 0.044463, 0.058579, -0.113025, -0.014318, -0.046181, -0.111803, 0.065300, -0.173579, 0.031159, -0.058183, 0.004448, -0.061769, -0.056523, 0.032539, -0.000833, -0.091855, 0.005328, 0.168343, 0.081518, -0.092745, -0.068590, 0.095623, -0.013579, -0.070150, 0.041259, -0.137630, 0.142439, -0.071447, 0.041106, -0.187764, -0.106597, -0.151517, -0.104379, -0.119442, -0.063553, 0.050259, 0.076666, 0.023008, -0.129864, 0.070793, 0.030543, -0.142995, 0.136369, -0.022709, -0.023904, -0.075720, -0.057190, -0.030240, 0.110762, -0.173628, -0.020137, -0.122421, -0.011872, -0.105578, 0.036741, -0.015677, 0.079807, 0.004213, -0.103816, -0.003347, 0.015432, -0.140343, 0.000313, 0.041789, -0.019587, 0.053668, 0.036036, 0.055283, 0.162987, 0.126810, 0.020708, 0.104890, -0.029222, -0.027070, -0.155727, 0.098905, -0.178437, -0.016479, -0.179767, 0.026909, -0.006697, -0.039101, -0.195305, 0.031821, -0.031385, 0.007960, -0.038008, -0.116526, -0.064848, -0.033827, 0.010934, 0.112762, -0.041082, -0.099393, 0.020702, 0.070839, -0.130618, -0.077543, -0.092264, 0.024305, 0.078055, -0.026116, -0.319611, -0.043447, 0.057132, -0.018438, 0.013670, -0.108971, 0.045521, -0.106579, 0.003851, 0.023077, 0.045209, -0.144587, 0.028511, -0.024399, 0.069510, -0.095599, -0.089656, -0.016466, 0.045517, -0.212998, 0.070608, 0.056141, -0.090286, -0.054132, -0.127218, -0.080899, 0.156112, 0.126947, -0.111526, 0.042017, 0.048016, -0.123050, -0.119971, 0.139588, -0.044479, -0.089293, -0.083710, 0.072706, -0.014947, 0.067960, -0.074196, -0.169187, 0.024284, -0.038276, -0.111662, 0.054071, -0.007674, -0.100655, 0.080137, 0.155313, 0.062300, -0.146968, -0.107370, -0.060392, -0.078736, -0.089332, 0.018335, -0.017227, -0.031229, 0.050022, 0.009749, -0.134290, -0.028178, -0.122374, -0.132132, -0.093704, -0.066764, -0.123792, -0.088862, -0.045613, -0.005067, -0.135762, -0.032379, -0.015399, -0.013180, 0.071819, -0.091811, 0.149170, 0.121337, 0.072309, -0.016779, 0.081041, 0.001551, 0.065818, 0.141771, 0.014132, -0.070345, -0.144173, 0.059088, 0.081668, 0.000222, -0.174888, -0.020680, -0.064189, 0.012913, -0.019586, -0.055034, 0.048848, -0.025120, -0.084461, -0.024080, -0.042400, 0.015810, -0.070292, -0.023865, -0.047495, -0.021893, -0.079151, -0.163985, 0.056327, -0.180487, -0.119865, -0.009391, 0.053912, -0.202381, -0.068965, -0.013284, -0.057958, -0.062920, -0.055044, -0.136395, 0.016048, 0.024469, -0.041205, -0.097683, -0.051884, -0.112903, 0.042250, -0.178784, 0.046920, -0.077854, 0.014314, -0.061381, -0.009955, -0.079560, 0.011765, -0.061536, 0.069027, -0.003603, -0.117969, 0.082827, -0.084717, -0.128681, 0.006991, -0.014820, -0.052593, -0.039872, -0.011079, -0.107412, 0.032533, -0.029613, -0.069842, -0.009202, -0.068834, -0.119997, 0.010852, 0.151022, -0.150633, 0.081234, -0.004150, -0.124901, -0.177795, -0.137991, 0.121514, -0.039556, -0.133238, -0.265938, 0.011924, -0.121484, -0.068070, -0.105859, 0.117016, -0.176013, -0.063238, 0.008318, 0.054851, -0.319088, -0.150540, 0.055535, -0.056724, -0.113417, 0.042275, -0.039503, 0.035291, 0.009051, -0.126682, -0.116374, -0.091274, -0.137280, 0.053867, -0.037876, 0.010112, -0.008681, -0.019385, -0.078334, 0.012022, 0.034034, -0.016876, 0.028024, -0.188394, 0.055451, -0.138682, 0.123592, -0.051746, -0.028986, -0.090465, -0.123360, 0.053939, -0.213269, -0.008455, -0.101097, 0.010272, 0.082468, 0.062646, -0.132475, -0.015266, -0.126872, -0.027742, 0.047301, -0.108053, -0.037131, -0.039888, 0.094057, -0.192836, -0.034694, -0.132764, 0.092752, -0.030817, 0.061407, -0.029966, -0.132207, 0.058899, -0.023508, 0.050375, -0.025942, -0.059796, -0.142306, 0.007094, -0.072795, -0.116458, 0.061279, -0.092803, 0.030340, 0.051941, -0.127177, -0.084702, -0.120618, -0.145221, 0.123566, -0.101117, 0.108863, 0.094850, -0.052774, -0.164404, -0.117233, -0.171548, -0.133281, 0.122970, 0.037372, -0.073976, 0.004655, -0.006506, 0.065590, -0.051171, -0.030132, 0.019964, 0.040968, 0.040799, 0.025088, -0.008009, 0.058267, 0.197864, -0.217122, 0.027370, 0.018346, 0.011890, 0.101624, 0.019860, -0.122945, -0.054878, 0.199421, 0.049386, -0.061107, -0.028567, 0.048603, -0.103112, -0.100327, -0.024560, -0.023639, -0.246423, 0.045630, -0.035495, -0.039201, 0.017587, 0.118315, 0.030165, 0.046554, -0.219168, -0.109447, -0.241147, -0.008819, -0.019019, -0.156078, -0.044191, 0.090972, -0.031428, 0.063539, 0.064059, -0.058227, 0.265565, 0.040689, -0.036580, -0.111835, -0.090304, 0.047114, 0.001143, 0.001769, 0.022658, 0.031365, -0.039906, -0.029568, -0.037080, 0.088753, -0.132843, 0.009510, 0.085387, 0.055867, -0.190581, -0.019242, -0.090193, 0.118820, 0.148269, -0.055975, -0.043012, -0.032311, -0.158217, 0.049658, 0.017344, -0.150169, 0.091127, 0.022166, -0.088728, -0.145596, -0.054122, 0.051215, -0.074363, -0.083826, -0.163946, -0.007142, -0.099919, -0.116580, -0.163169, 0.105273, -0.204947, 0.130460, -0.039979, 0.050460, -0.063712, 0.009308, -0.063543, -0.160996, 0.008848, -0.024465, -0.113122, 0.055610, -0.158658, 0.070925, 0.289531, -0.087784, -0.016100, -0.108610, -0.006233, 0.042598, 0.009191, 0.108710, -0.008725, 0.005459, 0.049419, 0.061070, -0.208630, 0.022826, -0.287140, -0.129666, 0.035811, 0.048743, -0.006997, 0.014588, 0.042310, 0.095712, -0.005673, 0.040387, -0.249745, 0.093631, -0.059398, -0.081665, 0.001288, -0.000780, 0.006156, -0.088044, 0.061199, 0.109891, -0.103270, -0.028618, -0.005685, 0.153504, -0.118974, -0.096677, -0.023130, -0.097554, 0.022345, -0.088674, 0.176985, 0.125978, -0.265733, 0.041104, -0.045222, 0.206667, -0.032983, -0.076561, -0.108777, 0.141796, -0.095317, -0.110539, -0.074529, -0.023034, -0.032948, 0.107128, 0.025753, -0.207666, 0.004432, 0.130989, -0.063144, 0.016618, 0.110759, 0.045596, 0.039150, -0.014618, -0.077881, 0.070665, 0.004207, 0.051469, 0.002884, -0.100441, -0.000088, -0.139682, -0.052668, -0.057368, -0.014944, -0.089759, 0.026773, -0.056171, -0.008287, 0.064725, 0.036485, -0.006702, -0.036267, 0.023898, -0.144961, -0.042268, -0.057178, 0.099478, -0.074139, 0.056709, 0.147983, 0.026204, -0.007750, -0.100426, 0.049950, -0.067916, -0.037823, -0.004289, -0.042476, -0.023900, -0.179094, -0.072012, -0.110743, -0.000756, 0.046749, 0.001618, -0.080831, -0.068553, 0.092001, 0.084706, -0.037441, 0.041781, -0.085560, 0.076832, -0.081460, -0.067917, -0.137638, -0.001120, -0.066712, 0.010076, -0.146626, 0.047666, -0.017881, 0.093422, -0.110473, -0.082845, 0.037945, -0.111446, 0.064162, -0.046592, -0.004358, -0.030300, 0.065886, -0.063683, 0.030202, 0.028271, 0.049200, -0.020017, 0.069631, -0.050258, 0.006300, -0.110245, -0.013887, -0.118653, -0.093656, -0.068289, -0.125733, 0.052534, 0.075075, 0.048373, 0.003397, -0.077926, 0.127948, 0.025344, -0.056226, 0.079405, -0.081135, 0.050076, 0.102633, -0.024290, -0.070104, 0.026106, 0.148397, -0.140319, -0.012523, -0.196315, 0.130236, -0.066226, -0.119930, 0.014568, 0.005455, 0.072263, -0.133198, -0.034132, -0.001908, 0.023534, 0.095981, -0.004799, 0.003506, 0.061427, 0.116113, 0.212175, 0.091466, -0.036203, 0.063250, -0.049133, -0.086836, 0.013985, -0.069891, 0.047338, -0.044120, -0.015496, -0.069202, 0.075003, -0.019173, -0.239135, -0.026026, -0.075501, -0.105459, -0.117095, 0.034156, -0.155261, 0.069690, -0.079490, 0.149018, -0.088810, -0.115692, -0.103067, 0.011903, 0.027513, -0.028234, -0.082526, -0.122664, -0.074731, 0.086495, -0.212197, -0.082558, -0.111297, -0.092932, 0.068878, -0.096141, 0.137638, -0.050192, -0.053021, 0.003830, 0.088637, -0.066690, -0.045786, 0.023034, -0.074406, -0.047010, 0.084054, -0.049755, -0.009146, -0.079542, -0.038100, -0.024057, -0.144806, -0.123414, 0.072089, 0.021832, 0.130648, 0.049912, -0.097114, -0.023306, -0.112885, -0.073522, -0.000337, -0.002180, -0.121885, -0.075804, 0.138907, -0.037699, 0.100722, 0.121603, 0.119196, 0.140969, -0.047207, -0.022625, 0.039147, -0.068928, 0.035597, -0.037826, 0.009639, -0.081580, -0.065033, 0.102838, 0.002353, 0.125513, -0.068058, 0.008167, 0.059143, -0.185954, -0.140429, -0.039520, -0.058812, 0.073344, 0.031944, -0.023056, -0.043570, -0.006348, 0.060347, 0.013847, -0.079951, -0.078248, 0.026536, -0.131832, 0.031295, 0.043907, 0.186870, -0.070787, -0.079799, -0.173385, 0.026502, -0.050949, 0.074125, -0.049186, 0.204260, -0.051565, -0.143952, -0.052918, 0.078572, 0.067268, -0.195333, -0.060673, 0.043771, 0.138226, -0.112341, -0.002389, 0.084836, -0.006384, 0.086212, 0.021731, 0.034017, 0.025197, -0.137225, -0.020678, -0.050217, 0.072907, -0.077849, -0.070681, -0.103132, 0.024816, 0.029600, -0.090109, -0.073017, -0.046757, -0.040423, 0.131861, -0.018746, -0.029654, -0.151850, 0.041985, -0.044289, 0.014706, 0.098207, -0.036492, 0.058522, -0.119023, -0.012702, -0.080019, -0.081847, -0.030915, 0.184260, -0.006190, -0.037579, 0.008337, 0.038173, -0.081274, -0.057346, -0.048092, 0.046972, -0.126911, -0.140979, 0.023641, -0.056539, -0.019317, 0.060584, 0.057391, 0.046372, 0.119824, 0.004635, -0.099276, 0.065243, 0.088890, -0.134364, -0.031032, -0.085402, 0.065100, -0.015915, 0.017244, 0.097986, 0.031873, 0.067153, -0.069140, 0.095763, 0.117611, 0.033261, -0.014280, 0.201685, 0.129493, -0.008498, -0.100629, 0.013834, 0.022671, -0.159155, -0.096295, -0.013456, 0.074912, -0.080146, -0.017790, 0.023552, 0.121003, -0.131714, 0.024075, -0.070230, 0.101975, -0.028594, 0.022039, -0.025031, 0.175170, -0.101650, 0.050307, -0.022270, 0.048799, -0.141531, 0.134389, -0.059346, -0.123160, -0.117868, -0.015703, 0.164039, -0.093275, 0.104867, 0.082938, -0.005743, -0.113308, 0.088400, -0.014370, 0.118553, -0.032119, 0.123753, -0.099368, 0.053641, 0.048019, 0.053823, -0.110684, -0.089871, 0.013991, -0.077578, 0.016918, -0.160641, 0.071110, 0.183884, 0.013650, 0.181181, -0.068486, -0.003686, 0.117471, 0.091117, -0.063793, -0.016996, -0.006267, 0.049699, -0.108153, -0.020417, -0.119411, 0.001593, 0.032612, -0.067360, 0.041969, -0.073078, -0.096689, -0.099396, -0.007337, 0.054754, 0.059520, -0.039050, -0.158701, -0.028301, 0.096485, 0.011547, 0.070117, 0.089033, -0.029638, 0.142382, 0.010569, 0.070191, 0.155189, -0.135327, -0.018185, -0.079641, 0.064296, 0.013108, -0.106697, -0.126362, -0.052873, -0.074320, 0.134129, 0.064948, -0.050449, 0.062760, -0.133347, -0.049682, 0.080780, 0.022304, 0.005054, -0.123499, 0.210905, -0.110427, -0.068541, -0.169460, -0.045076, -0.178270, -0.097912, 0.028378, -0.029404, 0.000813, -0.192335, -0.034953, -0.026014, 0.077939, -0.100451, 0.174856, -0.147401, -0.071003, -0.075948, -0.042117, 0.048287, -0.011969, -0.011023, 0.135941, 0.095647, 0.075413, -0.147577, 0.037868, 0.041693, -0.020464, 0.020361, -0.080870, -0.077560, -0.171915, 0.046623, 0.129781, -0.131711, -0.037536, -0.058485, 0.124164, 0.012518, -0.141082, 0.060374, -0.008513, -0.008720, -0.000675, 0.104861, 0.049048, 0.061642, -0.025407, -0.006148, -0.056567, -0.103724, -0.179839, -0.073242, -0.088265, 0.083841, -0.053084, 0.032628, -0.024596, -0.081899, 0.037132, 0.059074, -0.143452, -0.131956, -0.254585, -0.024783, -0.157500, -0.079619, 0.068568, -0.037012, -0.200841, -0.094134, 0.090209, -0.286411, -0.273429, -0.077239, 0.087489, -0.043448, -0.098900, -0.039552, -0.051895, -0.131918, 0.088290, -0.047997, -0.023557, -0.163662, -0.116258, 0.064838, 0.093891, 0.014904, -0.018867, -0.172079, -0.002953, 0.010954, -0.002794, -0.092602, -0.069013, -0.019282, -0.066516, 0.071706, -0.016927, 0.148502, -0.007161, 0.082247, 0.071821, 0.014291, 0.186900, 0.167817, -0.107659, -0.010856, -0.002988, 0.106383, -0.124647, 0.071860, -0.149682, -0.002490, -0.069928, -0.057323, 0.128782, -0.043889, -0.039711, 0.131359, -0.005369, -0.170873, -0.145924, -0.047822, -0.028993, -0.038302, 0.074167, 0.011167, 0.131153, -0.040917, -0.009803, -0.121045, 0.088992, 0.042072, -0.019775, -0.110818, -0.060206, -0.061538, -0.128559, 0.019565, -0.000150, 0.029852, 0.036151, -0.158231, -0.147201, -0.141388, -0.174529, -0.023372, 0.037747, -0.178336, 0.090450, 0.016820, 0.029661, 0.099155, 0.024946, 0.182540, -0.111873, -0.002652, 0.056514, 0.024216, 0.064501, 0.046612, -0.066156, 0.082944, -0.057203, -0.071593, 0.106939, 0.049906, -0.086589, 0.051523, -0.116651, 0.033245, -0.130907, 0.014014, 0.042548, 0.010418, -0.044963, 0.168636, -0.057893, -0.309024, -0.124572, -0.034757, -0.119483, -0.058967, 0.078096, -0.097026, -0.230863, -0.043768, -0.032686, 0.131498, -0.072125, -0.164778, -0.124109, -0.088285, -0.010503, -0.001398, 0.063682, -0.143395, -0.155429, 0.082853, -0.205063, -0.053938, -0.105975, 0.041091, -0.116360, 0.034777, 0.038050, 0.047948, -0.086172, -0.099639, -0.149289, -0.085304, -0.154557, -0.074231, -0.039891, -0.048104, 0.134820, -0.058958, -0.121195, -0.094806, -0.024033, 0.102207, -0.068049, -0.071385, -0.141066, -0.006113, 0.049865, 0.080745, 0.079258, -0.091284, 0.027119, -0.052096, 0.021640, -0.016085, -0.083321, -0.067459, -0.001165, -0.103750, -0.141927, -0.019292, 0.115588, 0.101403, 0.089368, -0.118942, -0.177770, 0.055272, -0.053997, -0.090448, 0.168764, 0.024968, 0.012351, 0.145804, 0.049664, -0.173331, -0.061380, -0.067240, -0.204206, 0.022689, 0.096952, -0.155183, -0.131862, -0.058738, 0.100340, 0.007350, -0.029143, -0.089373, -0.108398, -0.010219, 0.114033, 0.004062, 0.022615, -0.247742, 0.169187, -0.183502, -0.308132, -0.158414, -0.164285, -0.266544, -0.056286, -0.135477, -0.188695, 0.189810, -0.085147, -0.080511, -0.009016, -0.131912, 0.083162, 0.003723, -0.032230, -0.172643, 0.051144, -0.100920, -0.045979, 0.174359, -0.114859, -0.232716, -0.184882, 0.201520, 0.006254, 0.075164, 0.072967, -0.091255, -0.021814, 0.035959, -0.099314, -0.081107, -0.087921, 0.210618, 0.171652, -0.034510, -0.052451, -0.226987, -0.179563, 0.058824, -0.000284, -0.124525, 0.104071, -0.041868, -0.109456, -0.085792, -0.159886, -0.011803, -0.040487, 0.080665, -0.114301, 0.014244, -0.031036, -0.133985, -0.159286, -0.036111, -0.104772, -0.061291, 0.091626, -0.136008, -0.310572, -0.135250, -0.131231, -0.064772, -0.146589, -0.098854, -0.054291, -0.009274, -0.152290, 0.019807, -0.077080, -0.016605, -0.074567, -0.123505, -0.107446, -0.055716, -0.064364, -0.025709, -0.173395, -0.017298, 0.046922, 0.016869, 0.090106, -0.021745, 0.044139, 0.064979, 0.004368, 0.063977, 0.024753, -0.179060, 0.006250, -0.003597, 0.097358, -0.103543, -0.115145, 0.048455, 0.017660, -0.150214, -0.199876, 0.105956, -0.143896, 0.164959, -0.081769, -0.130550, -0.033411, -0.075401, -0.083636, 0.023904, -0.064415, -0.061457, 0.031747, -0.042950, -0.035863, -0.124639, 0.070450, 0.105752, -0.115221, -0.080083, 0.094326, 0.019244, -0.060915, -0.052440, -0.020201, -0.169664, -0.065440, 0.067407, -0.020561, -0.078617, 0.189411, -0.071829, 0.011068, -0.135542, -0.075788, -0.034750, 0.088439, 0.071458, -0.114173, 0.044123, -0.152317, -0.106766, -0.082335, -0.046169, 0.035586, -0.018735, 0.018497, 0.052016, 0.036186, 0.038248, 0.038954, -0.099696, 0.034589, 0.022162, -0.081159, 0.042907, 0.059233, 0.218299, -0.078373, -0.127584, 0.053013, -0.038744, -0.023968, -0.139958, -0.014361, -0.013901, 0.020718, -0.087895, 0.032014, 0.057295, -0.109014, 0.043334, -0.044511, -0.164600, 0.066105, 0.035714, 0.181224, -0.013391, 0.042073, -0.022554, -0.216032, -0.010137, 0.082759, 0.073752, -0.030774, -0.159402, -0.094531, -0.202544, 0.075383, -0.043392, 0.116174, -0.049710, -0.133177, 0.101723, -0.046693, -0.084987, 0.004854, -0.001749, 0.032836, 0.078622, 0.070970, 0.061395, -0.053867, 0.049998, -0.026357, -0.071005, 0.035014, 0.062845, -0.177548, -0.110835, 0.151710, 0.156921, -0.059244, -0.061717, -0.021035, -0.009422, 0.056087, -0.109959, -0.107224, 0.087484, -0.084872, 0.060892, -0.053537, 0.066478, -0.160982, -0.040918, 0.109693, -0.024174, -0.045169, -0.018981, -0.018261, -0.099940, -0.017234, -0.072194, 0.089905, 0.079699, -0.179323, -0.082941, 0.052770, -0.067798, -0.087390, -0.046137, -0.087998, 0.006718, 0.017122, 0.004019, -0.031008, 0.177938, -0.005663, -0.065119, -0.046674, -0.090693, -0.007379, -0.046700, -0.062839, -0.098728, -0.141635, 0.091530, -0.079104, 0.158699, -0.023878, 0.038523, 0.120187, 0.034197, -0.048666, -0.065291, -0.066037, 0.011198, -0.075972, 0.041551, -0.140488, -0.117688, 0.091185, -0.080890, -0.002220, 0.025841, 0.016287, -0.147594, -0.064506, -0.008641, 0.023581, -0.096798, 0.062919, -0.179257, -0.037550, -0.199473, -0.075922, -0.043124, -0.036486, 0.016031, -0.044078, 0.063245, 0.005192, -0.076360, -0.001038, -0.063924, -0.041309, 0.031655, 0.138983, 0.167282, -0.077055, -0.072577, 0.028729, 0.006019, -0.081206, -0.053918, 0.050163, 0.044136, 0.042295, -0.068000, -0.159764, 0.117371, -0.096574, 0.010563, -0.100315, 0.041871, -0.147818, 0.053674, -0.024026, 0.061230, -0.106162, -0.123938, 0.000400, 0.063486, -0.111592, 0.084607, 0.070192, -0.096462, -0.045426, -0.155077, 0.081567, -0.109509, -0.058975, 0.068798, -0.078239, -0.125721, -0.145479, -0.119095, -0.028073, 0.098282, -0.155986, -0.051509, -0.001554, 0.014250, -0.017716, -0.045553, -0.037882, -0.082993, -0.067491, -0.227437, 0.007573, 0.125899, 0.015535, -0.117273, -0.005296, -0.130783, -0.102131, 0.002598, -0.117912, -0.179784, -0.034990, 0.037375, -0.003457, -0.037261, 0.001791, 0.063201, -0.055223, -0.207887, -0.096360, -0.140250, 0.020367, 0.029245, -0.029970, -0.007991, -0.086212, -0.130629, -0.053171, -0.081327, -0.037310, -0.081707, -0.014015, 0.011476, 0.053945, 0.015119, 0.006924, -0.026748, -0.026001, 0.088071, -0.108830, -0.062385, -0.038127, 0.030167, 0.009795, 0.035196, -0.091004, 0.070469, -0.045263, -0.033707, 0.109188, -0.139747, 0.041768, -0.050309, -0.004094, -0.072738, -0.107733, -0.079963, 0.073909, 0.014545, 0.057171, -0.095321, -0.025378, 0.172856, -0.357176, -0.175981, 0.019981, -0.123289, -0.048143, -0.111007, -0.103803, -0.187832, 0.144336, 0.046719, -0.111635, -0.094448, -0.112618, -0.136532, 0.081794, 0.067138, -0.038896, 0.030332, -0.244143, 0.034912, -0.272812, -0.119743, -0.026279, 0.016985, 0.074681, 0.043394, -0.248657, -0.127179, -0.028224, -0.133274, -0.035398, 0.107135, -0.045204, -0.072436, -0.073072, 0.144140, -0.154109, -0.011226, -0.181613, -0.036841, 0.114447, -0.023506, 0.178908, -0.111000, -0.083440, -0.000344, 0.110140, -0.042072, 0.006894, -0.015615, 0.023543, -0.061773, -0.057837, -0.056921, 0.142575, -0.012320, -0.091801, -0.125325, 0.118552, -0.182365, -0.230805, 0.081077, -0.058391, -0.044054, 0.106606, -0.020311, 0.194673, 0.029758, 0.005443, -0.025449, -0.018370, 0.127148, 0.024376, -0.138707, -0.092678, 0.088502, 0.022457, -0.028558, -0.066970, -0.125999, 0.053323, -0.006283, 0.095246, 0.038603, -0.069583, 0.129398, -0.024059, -0.093443, 0.087249, -0.087165, -0.036556, -0.154683, 0.075927, 0.010197, 0.077885, 0.006816, 0.048219, -0.038183, -0.168387, 0.041427, -0.103426, -0.008712, -0.007329, -0.005463, 0.107093, -0.007103, -0.091703, -0.074642, -0.063147, -0.080201, -0.091817, 0.119461, -0.103350, 0.090934, -0.031393, 0.020690, -0.002636, 0.066288, -0.080477, 0.015577, -0.131176, 0.027206, -0.139583, 0.075939, 0.155993, -0.098572, -0.058825, 0.080711, 0.101954, 0.026476, -0.035724, 0.028400, 0.025196, -0.100343, -0.024790, -0.028119, -0.025263, 0.218690, 0.037524, -0.014539, -0.016316, -0.138716, 0.068898, 0.046415, 0.120024, 0.030067, -0.115819, 0.035953, 0.017114, -0.260552, -0.013727, -0.041275, 0.110036, 0.036220, 0.047773, -0.024850, 0.203019, -0.090583, 0.058193, -0.003884, 0.009515, 0.024219, 0.087722, -0.043945, -0.048927, -0.062343, 0.067466, 0.045941, -0.047886, -0.099357, 0.140116, 0.008315, 0.092327, 0.005796, 0.042696, 0.006813, -0.157580, 0.082506, 0.079066, 0.026358, 0.170491, 0.034774, 0.309763, -0.089545, 0.078149, -0.059208, -0.089624, -0.079200, -0.062669, -0.068732, 0.113953, -0.153646, -0.049365, -0.086183, 0.014803, -0.031617, -0.276162, 0.004709, 0.063716, 0.087172, -0.085288, -0.116403, 0.032284, 0.102077, -0.045606, 0.110988, 0.191683, -0.069036, -0.126728, -0.097068, 0.013032, -0.122050, 0.031847, 0.016111, -0.077666, 0.142026, -0.042203, 0.041702, 0.102575, -0.075914, 0.043869, 0.127272, 0.180861, 0.089377, -0.082308, -0.088805, -0.098911, 0.014522, -0.039510, -0.021699, 0.009183, -0.044061, 0.164444, -0.144224, 0.051224, -0.126179, 0.007907, 0.020060, 0.010195, 0.017738, -0.123518, -0.161929, 0.024462, -0.136711, 0.040650, -0.090715, -0.057321, 0.023655, -0.064388, 0.002333, 0.189350, 0.096084, -0.117327, -0.040680, -0.000380, 0.051453, -0.122050, 0.066692, 0.102878, -0.000282, -0.035689, -0.038609, 0.032819, -0.055119, -0.077957, -0.041580, 0.008804, 0.082709, 0.115855, -0.007322, 0.124409, -0.036626, 0.091791, 0.077641, -0.020331, -0.059326, 0.323560, -0.127440, 0.121264, 0.092116, -0.019106, -0.027575, 0.013279, -0.027665, 0.101155, -0.066060, -0.026076, -0.034940, -0.117651, -0.107220, -0.062832, 0.014014, -0.016903, 0.024933, 0.105646, 0.016177, -0.078408, 0.085231, 0.020674, -0.063290, -0.232416, -0.032389, -0.002516, -0.119637, -0.188774, -0.100241, 0.094044, 0.046349, -0.095352, 0.191381, 0.044782, -0.067372, 0.196835, 0.071395, -0.091749, 0.020104, -0.072873, -0.121414, 0.129531, 0.038624, -0.111784, 0.149050, 0.079947, -0.160348, -0.039183, 0.088891, 0.018703, 0.093371, 0.122789, -0.022360, -0.145400, 0.044720, 0.028135, -0.137110, 0.011212, 0.011919, 0.114673, -0.010383, -0.004032, -0.085528, 0.058187, -0.006600, -0.055640, 0.058126, -0.048009, 0.115441, 0.123526, -0.082301, -0.017909, 0.022394, -0.075382, -0.114615, -0.022811, -0.106910, -0.056158, 0.176262, -0.008423, -0.082961, -0.158921, 0.013675, -0.181225, 0.070484, -0.187474, -0.042635, 0.079374, 0.014120, 0.144204, -0.088668, 0.071560, -0.123290, 0.018902, 0.076623, 0.062018, 0.222840, 0.100903, -0.080990, -0.176777, 0.008644, -0.051300, 0.060589, 0.117769, 0.190801, -0.018287, 0.003568, -0.001525, 0.050220, 0.154228, -0.015234, -0.112422, 0.089921, -0.028921, -0.045779, -0.064905, 0.062984, -0.060759, -0.012231, -0.066016, 0.054217, -0.087021, 0.125804, -0.018614, -0.045735, -0.005982, -0.035009, -0.000716, 0.102242, -0.009767, 0.092864, -0.170815, 0.080770, -0.052609, -0.235050, -0.196485, 0.075399, 0.029695, -0.160762, 0.001117, -0.112996, 0.002315, 0.045865, 0.012134, 0.022349, 0.059729, 0.075417, 0.104514, -0.051013, 0.137940, -0.060266, -0.078633, 0.093913, -0.068935, -0.137966, 0.124349, 0.082477, -0.126461, 0.090575, 0.018632, -0.163887, 0.123277, 0.211229, 0.024822, 0.016630, 0.000918, -0.109438, 0.101868, 0.082858, 0.003562, -0.066384, -0.012807, -0.004292, -0.056848, -0.000222, -0.056179, -0.001758, 0.053283, -0.047175, 0.164752, 0.000997, -0.086290, -0.103196, 0.201135, -0.087160, -0.125284, -0.089701, 0.016414, 0.111908, 0.061438, 0.020211, -0.020750, -0.086879, 0.089234, 0.022832, -0.138379, -0.045833, 0.040893, -0.144509, -0.080925, -0.011411, -0.124583, -0.039173, -0.184302, -0.022296, 0.064990, -0.125734, -0.115565, -0.050936, 0.110658, -0.106247, -0.028823, -0.107931, 0.123934, 0.160904, 0.001104, -0.111379, -0.101642, -0.060340, 0.000560, -0.123326, -0.103958, -0.048370, 0.113178, -0.009385, -0.032542, 0.061356, -0.226527, 0.183049, -0.051576, 0.007074, 0.020996, -0.029956, 0.087978, -0.033889, 0.069824, -0.074142, -0.033008, 0.030035, 0.041298, 0.110235, -0.013265, -0.075770, 0.121023, 0.043532, 0.121320, 0.111573, 0.099570, 0.027683, -0.170866, -0.103084, 0.009494, -0.184655, 0.116323, -0.112740, 0.034669, -0.005142, -0.013207, -0.110010, -0.106708, 0.067000, 0.131227, 0.122356, -0.057793, 0.045124, 0.009096, 0.171616, -0.218069, 0.015552, 0.036884, 0.030539, -0.148281, 0.028426, -0.139040, 0.011773, 0.065358, -0.046925, 0.061677, -0.162704, 0.113025, 0.209498, -0.205784, 0.051843, -0.151169, -0.099341, 0.016522, -0.012910, 0.161770, 0.089924, -0.055962, -0.187244, 0.017719, 0.077225, 0.113443, -0.019793, -0.039471, 0.067440, 0.049999, 0.065232, -0.010693, 0.123569, -0.064139, 0.067362, 0.210042, -0.001623, 0.009151, -0.039895, 0.037838, 0.006616, 0.111341, -0.090087, 0.018426, 0.041388, -0.006807, -0.004753, -0.082602, -0.123184, 0.068558, -0.090778, 0.032170, -0.031681, 0.006096, 0.089758, -0.063980, -0.042450, -0.095492, 0.001666, 0.058184, 0.010080, -0.042796, -0.303294, -0.118538, 0.028633, -0.072922, -0.011903, 0.061174, -0.166933, -0.089984, -0.068056, 0.117004, 0.020598, -0.070455, 0.035025, 0.090618, -0.054127, 0.068089, 0.055644, -0.030162, -0.051667, -0.012264, -0.131969, 0.023615, 0.096261, 0.013959, -0.030424, -0.034181, 0.087614, 0.137821, -0.108047, -0.106818, 0.019304, -0.111396, 0.107478, 0.054541, -0.153921, 0.063225, -0.062444, -0.046817, 0.045400, 0.104512, 0.110243, -0.085787, -0.152936, 0.086180, 0.029016, 0.145205, 0.058811, 0.000691, -0.061966, -0.114173, 0.121291, 0.200687, 0.006909, -0.065793, 0.214574, -0.040366, -0.053571, 0.126848, -0.074250, -0.091723, -0.151027, -0.198496, -0.026685, -0.012008, -0.042739, -0.094497, 0.151782, 0.132502, -0.114303, -0.088279, 0.009073, 0.077949, -0.164075, -0.054721, 0.103719, 0.026009, -0.065078, -0.035922, -0.065365, 0.014611, 0.014216, -0.131645, 0.084891, -0.204964, 0.027011, -0.167069, -0.043863, -0.083072, -0.029014, 0.076728, 0.069180, 0.048855, 0.144067, -0.140662, -0.219493, -0.315313, -0.095045, -0.129247, 0.149055, 0.026327, -0.007564, -0.057315, 0.006108, 0.089624, -0.014232, -0.005397, -0.081347, 0.050245, -0.032150, -0.111387, -0.141349, 0.006915, 0.076999, -0.060059, 0.145200, -0.082196, -0.226437, 0.041883, 0.045317, -0.090782, -0.016556, 0.051287, 0.037361, 0.057331, -0.085139, 0.014322, 0.176369, 0.065758, 0.079379, 0.044255, 0.133420, 0.140504, -0.080284, -0.234938, -0.082424, 0.059711, -0.100801, -0.041125, 0.027355, 0.064588, -0.050632, 0.001280, 0.011044, 0.124484, -0.107595, 0.021952, 0.095942, 0.136534, 0.084252, -0.048643, -0.010310, -0.129241, 0.158870, 0.111010, 0.039259, -0.024912, 0.020902, 0.250763, 0.025447, 0.075809, 0.097576, -0.240308, -0.147681, 0.060312, 0.007368, -0.029402, 0.081576, -0.013667, -0.100552, 0.118213, 0.101974, 0.080528, -0.125057, -0.080648, 0.078270, 0.135748, -0.182905, 0.133466, 0.006646, -0.013119, 0.079543, 0.057211, 0.044228, 0.026523, -0.111011, 0.129118, -0.042804, 0.077692, 0.101381, -0.038876, -0.096832, -0.081224, -0.150828, 0.031621, 0.062783, -0.035207, -0.177913, -0.030542, 0.037812, -0.087570, 0.084436, 0.147625, -0.023855, -0.165518, -0.018027, -0.035425, -0.094745, -0.002921, -0.053945, 0.113779, -0.139220, 0.084383, -0.208019, 0.032335, 0.002005, -0.079142, -0.063103, -0.161241, -0.003593, -0.018557, -0.130288, -0.034748, -0.035129, -0.095381, -0.126881, -0.131888, 0.182379, -0.119569, 0.096713, -0.045289, 0.016826, 0.016836, -0.068506, -0.161875, -0.012195, -0.048651, -0.111086, 0.073611, -0.182571, -0.089407, 0.007126, -0.043112, -0.030441, -0.029143, -0.029153, 0.015871, 0.164175, 0.020930, -0.009362, 0.007836, 0.005621, 0.081839, 0.048213, -0.104880, -0.050029, -0.043068, -0.025476, -0.003050, 0.065640, -0.159300, -0.062435, 0.044716, -0.134378, -0.028276, 0.039114, -0.203654, -0.023298, 0.029064, 0.016876, -0.018051, -0.182941, 0.041382, -0.069137, 0.015442, 0.103035, 0.071962, -0.188009, 0.053828, 0.029102, -0.084726, 0.034979, -0.059858, 0.060045, -0.128648, 0.095838, -0.082166, -0.048656, 0.017629, -0.023032, -0.076154, -0.024883, 0.006203, 0.005178, -0.195829, 0.026233, 0.005153, -0.023113, 0.211180, -0.066783, -0.125651, -0.164240, -0.017767, -0.042364, 0.045382, -0.141899, -0.038479, -0.052341, -0.152083, 0.042215, -0.056505, -0.257887, 0.090060, -0.192554, 0.037245, -0.041820, 0.035012, 0.012130, 0.005073, 0.019344, -0.279248, -0.030301, -0.064028, -0.086505, -0.019835, -0.044353, -0.197645, -0.014713, -0.023174, -0.096084, 0.073707, 0.041478, 0.085772, -0.127784, -0.044026, 0.037630, -0.078844, -0.169069, -0.117906, 0.023153, 0.005944, -0.046030, -0.089251, -0.058312, -0.075363, -0.099344, -0.057399, -0.051115, -0.108404, -0.046521, 0.093463, -0.120489, -0.143000, -0.000267, -0.163673, -0.240637, -0.077972, 0.019007, -0.260116, 0.079041, 0.088254, -0.054506, -0.103494, -0.135238, -0.077800, -0.005250, -0.126676, -0.068769, -0.028756, 0.039602, -0.308959, -0.151636, -0.169359, -0.001637, -0.487497, 0.030400, 0.062971, -0.046121, 0.133442, -0.064024, 0.024673, 0.024815, 0.130226, -0.072183, -0.101276, 0.027488, 0.021635, 0.079487, -0.217187, 0.074702, 0.019141, -0.011343, -0.134009, -0.053123, 0.069660, 0.075233, -0.027180, -0.065754, -0.101036, -0.107677, -0.045596, -0.064476, -0.336248, 0.024901, 0.039350, -0.094050, -0.036781, -0.082126, 0.017655, -0.078614, 0.128242, 0.127736, -0.092031, -0.150956, -0.049799, -0.082485, -0.141244, -0.088754, -0.081184, -0.142922, -0.099401, -0.163044, -0.062089, -0.027656, 0.078150, -0.089297, -0.050178, -0.074635, -0.003084, 0.076410, -0.243720, 0.007771, -0.023352, 0.050574, 0.002885, -0.052320, -0.050091, -0.012712, -0.055721, -0.042558, -0.039952, -0.100553, 0.074929, 0.097035, 0.010956, 0.079516, -0.093751, 0.081081, -0.039998, -0.026042, 0.079244, -0.055945, -0.100060, 0.023160, -0.092379, -0.005294, 0.039101, -0.106008, -0.086293, -0.242168, -0.018669, 0.038574, 0.032505, -0.126690, -0.094387, 0.034300, 0.004193, -0.017159, -0.120254, -0.113458, -0.102097, 0.081951, 0.136937, -0.064308, 0.002330, 0.016353, -0.014900, 0.029018, 0.090221, -0.076198, -0.128383, 0.000982, 0.091236, -0.000148, -0.031967, -0.032721, -0.183407, -0.056565, 0.052303, -0.031605, -0.125046, -0.011006, -0.025648, -0.044112, -0.029899, 0.002989, -0.063107, 0.013810, -0.007273, 0.061670, -0.016886, 0.035317, -0.174748, -0.079989, 0.058199, -0.038522, -0.215839, 0.109675, -0.135975, -0.023130, -0.120692, 0.019169, 0.010695, 0.069548, -0.158105, -0.166730, 0.117633, -0.007436, 0.017465, -0.046398, -0.102279, -0.026032, -0.082995, -0.075174, -0.080788, -0.070499, -0.056753, 0.077399, -0.108739, -0.046231, -0.071926, -0.121704, 0.072146, -0.145813, 0.048030, 0.088703, 0.018115, -0.147766, -0.161801, -0.164951, -0.104652, 0.064708, -0.168957, -0.007862, 0.020270, -0.094294, -0.031751, 0.031626, -0.054499, 0.009148, 0.093348, -0.043682, -0.195768, -0.000648, -0.009219, -0.169233, -0.041102, -0.080846, -0.140144, -0.014707, -0.088930, -0.071610, 0.147743, 0.025774, -0.091062, 0.002799, 0.005369, -0.171770, -0.123444, -0.176960, 0.088401, -0.047115, -0.094210, -0.150602, -0.063748, -0.051055, -0.014534, 0.045157, 0.144435, -0.128236, 0.082982, -0.126417, -0.013623, -0.043854, -0.050465, 0.019470, -0.068566, 0.023245, -0.118397, -0.220180, -0.111128, -0.112833, -0.115314, -0.038779, 0.082352, 0.034994, -0.234940, 0.073097, -0.154521, 0.057690, -0.155433, -0.048403, -0.073139, 0.000171, -0.100069, 0.034560, -0.090277, 0.007480, -0.139258, -0.002163, -0.094367, -0.079620, 0.133494, -0.109177, -0.004047, 0.119496, -0.110113, -0.034933, -0.057675, -0.137793, -0.102979, -0.059684, -0.040742, -0.187174, -0.029054, 0.051475, 0.010664, -0.007966, 0.090412, -0.158862, -0.154982, -0.172921, 0.016640, -0.040697, 0.039850, -0.158309, 0.152518, 0.112021, -0.168384, -0.050420, -0.067774, -0.150069, 0.062537, -0.013488, 0.054311, 0.036449, -0.072385, -0.093626, -0.087783, -0.038044, -0.039856, 0.027907, -0.130311, 0.033926, 0.144025, -0.305648, -0.278876, 0.122221, 0.057812, -0.071425, -0.261186, -0.054685, -0.100456, -0.172137, -0.191036, -0.070172, -0.016576, -0.076825, -0.098216, -0.094922, 0.142153, -0.084559, 0.069768, -0.117660, -0.159791, -0.021623, -0.034006, -0.085896, -0.007119, 0.135768, 0.057278, -0.000914, -0.111993, -0.222658, -0.076019, 0.072155, 0.047460, -0.169691, -0.071772, 0.004112, 0.059826, 0.061738, 0.109072, -0.080407, 0.004209, -0.038069, -0.146115, -0.147275, 0.031881, -0.091320, 0.159537, -0.015666, -0.011673, -0.016089, -0.171758, -0.134062, 0.033748, -0.023272, 0.049681, 0.000108, -0.043827, -0.099283, -0.069869, 0.065807, -0.116147, -0.114700, 0.048021, -0.030477, -0.104627, -0.257900, -0.150163, 0.058206, 0.255237, 0.155329, 0.051146, -0.088804, -0.058971, -0.142647, -0.091106, -0.120802, 0.072117, -0.114869, 0.007108, -0.083243, 0.114050, 0.135860, -0.110131, 0.036561, -0.079140, 0.025921, 0.137167, -0.041169, 0.000771, -0.060994, -0.191125, 0.119128, -0.083160, 0.108090, -0.057821, -0.245877, 0.002509, -0.115137, 0.041161, -0.033730, 0.100739, 0.122225, 0.029930, -0.026227, -0.079364, -0.094628, 0.033069, -0.025509, -0.158890, -0.156364, -0.062096, 0.026385, -0.036410, -0.161739, -0.082481, -0.169919, 0.091816, -0.057677, 0.029939, 0.081368, 0.002616, 0.068092, -0.052572, -0.064738, -0.112983, -0.009426, -0.050856, 0.139589, 0.051782, 0.063048, 0.085820, -0.029943, 0.101476, -0.032045, 0.053984, 0.197348, 0.239349, -0.055386, 0.002940, -0.124035, -0.027564, -0.101614, -0.074520, -0.016393, -0.155695, -0.121885, -0.068266, 0.015463, 0.045026, 0.106196, -0.141566, -0.001388, -0.018729, -0.055595, -0.070923, -0.047641, -0.239714, 0.239208, 0.062660, -0.066641, -0.207199, -0.076718, -0.265493, -0.038027, 0.010601, -0.108380, 0.136665, 0.021135, -0.178722, 0.224150, -0.068012, -0.027623, -0.008935, -0.070803, -0.048991, -0.074546, -0.156380, -0.066519, -0.082300, 0.044561, 0.087007, 0.157449, -0.048698, -0.217021, -0.016243, 0.044466, -0.061711, -0.023584, -0.026482, 0.009349, -0.009980, -0.012853, 0.150369, -0.138211, -0.112839, 0.163934, 0.003320, -0.024404, -0.139909, -0.037415, -0.116248, 0.010126, 0.031576, 0.117399, -0.056380, 0.158353, -0.106196, 0.151490, -0.025320, -0.074568, -0.062269, 0.041034, 0.058914, 0.053256, -0.016671, -0.062167, 0.008511, 0.075931, -0.082685, -0.069736, 0.051131, -0.180733, -0.007652, -0.046045, -0.103759, -0.025397, 0.010131, -0.102340, 0.008972, 0.012948, 0.077738, -0.126575, -0.000996, -0.090176, -0.063450, 0.017244, -0.000997, 0.019657, 0.010015, -0.094581, 0.018820, -0.054627, -0.055552, -0.082878, -0.026258, -0.045633, 0.006511, -0.029255, -0.019331, -0.104048, 0.046328, -0.172793, 0.029631, 0.012027, -0.009913, 0.038542, 0.054126, -0.108417, 0.048737, -0.090855, 0.016476, 0.033121, 0.028162, -0.084012, -0.056915, -0.180447, 0.126347, -0.095744, 0.006007, -0.006856, -0.002880, 0.047899, -0.009251, 0.023142, 0.047274, -0.078170, -0.005424, 0.024086, -0.034878, 0.037492, -0.018241, -0.089003, -0.019465, 0.100686, -0.056628, -0.159634, 0.109580, -0.061640, -0.010156, 0.046175, -0.011571, 0.092869, 0.045422, 0.028524, 0.125218, 0.079603, -0.011606, 0.035303, -0.044672, -0.033770, 0.009879, 0.021275, -0.156359, -0.015981, 0.090250, -0.011820, 0.081658, -0.073627, -0.128115, -0.085366, 0.045775, 0.035075, -0.134144, -0.081137, -0.109089, 0.006441, -0.119817, 0.050244, -0.141799, 0.096967, -0.020395, -0.048100, 0.181003, -0.134623, 0.027337, 0.028929, 0.088732, -0.137056, -0.040084, -0.115209, -0.022431, -0.058035, -0.154763, 0.044022, 0.083362, 0.071474, 0.115832, 0.045587, -0.020550, 0.139317, -0.115715, -0.063439, -0.042596, -0.136558, 0.112930, -0.017084, -0.092073, -0.006800, 0.098358, -0.017931, 0.091014, 0.004409, 0.159458, -0.116385, 0.139750, -0.011399, 0.007657, 0.027491, 0.052502, -0.061179, -0.059304, -0.022624, -0.001960, -0.066615, 0.007496, 0.103956, 0.092674, -0.081031, 0.007707, 0.054774, 0.074479, 0.035191, -0.045323, 0.010824, 0.045403, -0.010966, 0.048137, 0.035432, 0.057088, -0.055390, 0.028289, 0.076932, -0.166971, 0.001552, -0.036624, 0.031977, -0.011835, -0.031084, 0.045131, -0.008995, 0.063358, 0.109222, -0.162888, -0.030121, -0.049310, -0.119691, 0.071709, 0.129508, 0.045527, -0.064341, 0.011660, 0.117412, 0.011102, 0.035715, -0.135933, -0.086265, -0.065980, -0.063551, -0.117420, -0.179986, 0.110206, -0.126410, -0.068528, 0.020789, 0.029749, -0.013837, 0.055492, 0.090846, -0.004521, -0.074961, -0.018985, 0.003356, 0.024347, -0.021865, -0.130275, 0.015662, -0.035687, -0.140468, -0.070399, -0.031895, 0.002007, -0.064431, 0.026745, 0.000377, 0.095061, 0.172417, -0.008487, -0.037975, 0.077662, -0.058646, 0.034540, -0.130048, -0.099697, -0.000451, -0.059104, -0.089409, 0.067595, -0.135208, -0.032450, 0.016034, 0.136228, 0.034588, -0.059121, -0.047132, -0.025282, -0.088552, 0.063232, 0.044240, 0.026976, 0.034748, -0.119132, -0.096194, -0.150992, -0.017542, -0.125540, 0.053755, -0.076088, 0.060464, -0.100372, -0.119278, -0.054451, -0.221072, 0.042404, 0.033865, 0.112092, 0.019241, 0.018585, -0.076705, 0.097773, 0.163267, 0.111988, -0.048274, -0.077819, 0.112439, 0.024774, 0.063494, -0.028155, -0.010944, 0.042872, 0.090565, 0.082363, 0.030676, 0.157270, -0.005872, 0.012095, -0.081497, 0.050578, -0.017874, 0.088733, -0.032323, 0.083409, -0.042252, 0.060798, 0.009940, -0.251880, 0.063182, -0.164492, 0.004256, 0.011699, -0.037491, 0.036372, 0.093843, -0.087296, -0.105318, 0.095442, 0.055748, 0.037783, -0.055858, -0.043060, 0.172289, -0.110312, -0.055369, -0.142614, -0.019995, 0.020991, 0.046109, 0.056649, -0.200987, -0.083776, -0.070854, -0.083067, 0.060203, -0.027742, -0.045846, 0.111465, 0.188390, 0.026930, -0.069393, 0.145816, 0.040620, -0.109045, -0.028680, -0.027303, -0.015006, 0.031287, 0.019745, 0.036146, 0.023915, 0.084229, 0.067373, 0.053604, 0.118510, -0.014261, -0.124910, -0.105372, -0.011164, 0.032891, -0.001700, 0.094137, -0.017909, -0.072197, 0.179959, -0.137023, -0.011381, 0.066719, 0.158299, -0.095013, -0.046147, 0.056521, 0.042264, 0.053665, -0.090748, 0.066021, 0.042920, -0.133441, -0.053457, 0.118874, 0.092501, 0.056136, 0.069697, 0.005763, 0.097342, 0.093161, 0.096128, -0.130737, -0.083529, -0.096484, -0.103742, -0.136896, 0.099534, 0.071537, -0.068584, -0.153971, -0.012881, -0.008713, -0.012220, 0.016575, -0.003102, -0.005143, -0.035460, 0.040832, -0.160089, 0.307463, 0.020397, -0.023416, -0.108971, -0.277689, 0.035924, -0.168752, -0.282633, 0.020468, -0.133384, 0.198190, 0.100644, -0.083823, 0.038001, -0.152785, 0.113105, 0.052075, 0.111278, -0.017641, 0.233588, 0.007135, 0.033648, -0.169085, -0.039322, -0.060834, 0.132972, -0.082724, -0.090602, 0.008478, -0.014768, -0.182214, -0.072840, 0.030284, 0.170262, 0.002479, 0.094199, -0.129648, -0.196034, -0.089743, 0.195658, -0.050180, -0.230216, 0.110695, -0.060859, 0.139957, -0.121455, -0.116562, -0.146889, -0.010570, 0.050300, -0.050577, -0.059620, 0.098131, -0.137836, -0.164386, -0.041408, 0.092876, -0.043351, 0.153389, -0.097176, -0.123896, 0.114372, 0.081428, -0.049703, 0.175488, 0.028359, -0.147893, -0.112860, -0.074831, -0.078798, -0.055760, -0.025268, -0.018889, -0.026304, 0.069107, 0.035208, -0.036046, -0.207759, 0.193942, -0.004204, -0.053837, 0.025900, -0.371767, -0.097312, 0.031078, 0.028670, 0.010728, 0.039374, -0.034194, -0.035870, 0.179436, -0.015043, -0.212089, -0.129427, -0.308552, 0.006712, -0.038968, 0.060219, 0.112703, 0.007373, 0.011357, -0.055519, -0.151708, -0.119542, 0.012559, -0.048777, 0.008291, 0.041474, -0.027022, -0.101673, -0.037004, 0.063628, 0.027479, -0.066297, -0.022611, 0.046507, 0.030160, 0.180064, -0.322292, -0.091838, -0.112675, -0.019362, 0.001195, 0.004539, -0.112638, -0.077903, -0.023614, -0.010806, 0.065590, 0.072952, -0.057277, -0.102507, 0.116151, -0.154472, -0.021552, 0.019796, 0.024687, 0.118586, -0.128829, 0.023802, -0.528765, -0.056560, -0.195169, 0.042301, -0.249384, 0.068405, -0.059520, 0.044273, -0.271580, 0.068062, 0.009979, -0.067876, -0.052320, -0.044412, -0.073393, 0.191855, 0.005509, -0.034342, -0.075552, -0.156541, 0.010502, -0.077892, -0.005620, -0.079229, -0.319871, 0.066958, -0.203147, 0.171216, -0.200940, -0.006504, -0.130760, -0.368090, -0.010430, -0.118878, -0.133881, 0.029188, 0.114151, -0.368001, 0.020258, 0.078614, -0.070301, -0.087747, -0.161443, -0.197219, -0.066592, -0.068844, -0.170809, 0.119841, -0.075351, -0.097806, -0.108387, -0.076627, -0.035600, 0.151364, -0.082774, -0.066000, -0.120995, -0.164203, -0.053792, 0.060274, -0.079060, -0.060286, -0.061511, -0.100237, -0.105739, -0.015906, 0.040535, -0.010384, 0.006486, -0.067986, -0.116884, -0.023942, 0.058058, -0.245378, -0.000253, 0.007754, 0.004051, -0.200858, -0.310581, 0.061930, -0.178233, -0.090671, -0.038474, -0.006355, 0.030476, 0.178537, -0.060244, -0.128843, -0.075104, -0.165197, -0.095786, 0.067853, -0.043876, -0.008125, 0.051160, -0.046712, -0.088557, -0.058489, -0.068221, -0.071611, -0.044476, -0.170194, 0.025402, 0.001642, -0.042850, -0.013632, -0.017275, -0.036231, -0.216151, -0.000422, -0.113024, -0.067446, -0.033640, 0.080441, -0.057246, -0.165256, 0.022464, 0.097545, -0.058914, -0.100476, -0.081696, 0.011489, -0.038522, -0.078397, -0.114505, -0.181027, 0.041087, -0.000496, -0.268919, -0.065545, -0.274440, -0.107762, -0.051025, 0.002191, 0.075199, 0.110132, -0.074540, 0.088741, -0.086127, -0.033153, 0.028605, -0.008037, 0.033031, 0.049192, -0.101470, -0.136583, -0.206854, -0.181798, 0.006568, -0.258157, -0.030957, 0.006671, 0.034127, 0.039343, -0.081687, 0.116287, -0.195556, 0.043986, -0.217705, -0.078405, -0.152222, -0.237463, -0.175828, 0.041795, -0.048437, -0.171395, -0.039346, -0.085348, 0.009353, -0.212410, -0.109350, -0.057938, -0.113495, -0.042734, -0.131125, 0.040959, -0.143058, -0.171990, -0.038400, 0.042455, -0.021875, 0.006071, 0.024088, -0.120658, -0.170335, -0.119022, -0.199620, -0.089280, 0.001702, 0.072163, 0.084214, -0.274301, -0.031417, -0.101694, -0.147700, -0.146983, 0.059620, -0.098990, 0.046360, -0.051268, 0.011907, -0.326126, -0.086965, -0.048541, -0.078468, -0.035505, 0.006236, -0.041448, -0.293279, -0.029129, 0.014596, 0.060871, -0.060039, 0.124411, -0.006676, -0.025302, -0.097741, 0.057392, -0.088959, -0.082568, -0.018777, -0.134726, -0.054937, -0.141388, -0.212196, -0.001030, -0.027800, 0.082991, -0.031669, -0.004372, 0.170266, -0.022411, 0.036907, -0.041662, -0.102473, 0.003605, -0.076284, 0.063524, -0.086817, 0.032802, 0.047621, -0.210525, -0.049201, -0.063718, -0.128533, -0.138321, 0.048572, 0.201510, 0.094769, -0.291992, 0.128337, -0.113310, 0.147517, 0.160398, -0.051065, -0.052084, -0.031363, -0.126257, 0.060359, 0.102055, 0.076961, 0.059705, 0.101775, 0.025887, -0.057929, 0.048544, -0.059357, 0.037749, -0.072379, -0.078706, 0.054695, 0.071995, -0.043339, -0.106895, -0.008926, 0.137627, 0.036395, 0.165492, -0.194587, 0.096473, -0.048646, -0.199876, -0.034250, 0.023906, 0.020264, 0.159783, 0.081500, -0.073903, -0.182742, -0.126642, -0.060582, -0.236132, -0.013397, -0.073764, -0.002617, 0.027301, -0.033506, -0.143472, 0.061572, 0.054707, -0.095656, -0.069344, -0.030714, 0.035716, 0.040579, 0.001267, -0.109901, -0.072523, 0.208149, -0.017536, 0.014136, -0.219299, -0.158779, 0.095729, 0.063366, 0.025587, 0.108768, 0.000757, -0.076636, 0.223175, -0.063240, 0.030207, -0.078421, -0.136474, 0.041888, 0.192825, 0.144390, 0.103944, -0.042203, -0.222443, 0.262696, 0.124754, -0.015907, 0.365553, -0.231536, 0.260485, 0.101092, -0.079657, 0.140515, 0.035824, 0.038867, -0.071086, 0.180249, -0.035909, -0.047954, -0.034799, -0.137327, 0.067856, 0.181976, 0.043365, 0.040262, -0.003775, -0.020471, -0.029652, -0.082841, -0.113689, -0.097262, -0.106070, 0.082860, 0.030253, 0.031376, -0.098148, 0.089366, -0.142643, -0.128563, -0.109276, 0.090629, 0.018449, -0.007374, -0.368284, -0.211911, -0.005975, -0.090456, 0.061098, 0.039377, 0.135873, -0.082363, -0.058697, -0.145966, -0.064763, 0.037727, 0.155858, -0.027704, -0.155850, 0.026980, -0.078058, -0.038918, -0.058350, -0.009093, 0.110381, -0.045063, 0.069269, -0.165425, 0.154204, -0.055350, 0.130687, 0.049426, -0.022432, -0.066480, -0.011072, 0.118946, -0.064072, -0.168473, 0.050074, -0.066652, -0.018681, 0.092186, -0.111227, 0.046570, 0.151367, -0.053032, -0.234081, -0.070440, -0.139607, -0.000417, -0.070927, -0.107108, -0.135102, -0.000505, 0.088675, -0.006865, -0.028102, -0.000199, 0.030573, -0.078332, 0.091662, 0.124858, -0.069430, 0.133203, -0.053896, 0.086447, -0.034824, 0.166367, 0.015704, 0.075996, -0.018268, -0.085917, -0.064583, -0.196273, -0.125712, 0.058592, -0.193440, -0.063253, 0.088275, -0.018739, 0.026075, 0.035964, -0.189806, 0.162809, 0.076796, 0.003422, 0.006565, 0.058542, -0.087384, -0.025940, -0.062405, 0.065928, -0.013199, 0.007280, -0.068904, -0.071317, -0.075671, -0.009538, -0.005839, -0.116345, -0.018000, 0.055596, -0.125714, -0.178347, -0.116251, -0.166843, -0.113068, -0.022950, -0.007958, 0.092812, -0.014910, -0.062165, -0.067439, -0.189931, -0.088393, -0.174443, 0.101382, 0.219828, 0.159775, 0.022230, 0.167976, -0.184782, 0.080681, 0.075894, 0.051332, 0.044857, -0.016451, 0.102872, -0.129677, 0.117374, 0.046232, -0.013733, 0.027209, 0.028393, -0.049094, 0.116998, 0.123416, -0.142752, -0.032790, 0.072149, -0.049734, 0.194955, -0.066874, -0.089755, 0.000431, 0.043680, -0.022933, -0.137649, -0.133008, 0.035702, -0.112459, -0.215144, -0.060830, -0.071465, 0.077486, -0.083728, 0.049104, 0.114668, 0.113037, -0.022607, 0.128139, -0.022262, 0.178903, -0.015749, 0.025887, -0.148035, 0.051418, 0.032117, -0.040875, 0.045884, 0.024038, 0.054504, -0.020718, 0.054978, -0.086993, -0.061364, 0.037002, 0.121759, -0.165966, 0.106900, -0.095924, 0.100117, -0.023694, -0.336584, -0.079893, 0.007482, 0.000948, -0.086585, 0.067844, -0.091541, 0.075152, 0.030825, 0.032736, 0.040487, 0.089523, 0.185976, 0.128702, -0.129056, -0.117647, 0.124900, 0.114344, -0.183619, 0.014275, -0.056272, -0.161142, -0.028327, 0.076695, -0.015015, 0.015684, -0.073595, -0.120191, -0.139483, 0.067938, -0.143839, -0.067700, -0.058627, 0.035017, -0.120056, -0.056611, -0.143474, -0.139919, -0.129282, 0.070750, 0.064641, 0.044440, -0.055120, -0.109692, 0.046853, 0.034897, 0.064838, 0.164852, -0.130617, -0.166449, -0.076645, -0.006160, 0.116861, 0.094355, 0.171337, -0.057472, -0.107632, -0.039988, 0.144537, 0.120877, -0.096528, -0.033428, -0.042885, -0.126656, -0.039495, -0.115820, 0.082919, -0.042180, -0.057450, -0.027469, 0.080236, -0.014780, -0.176412, -0.107095, 0.060287, 0.024326, 0.081527, -0.133074, 0.040501, 0.149740, 0.003260, 0.064305, -0.066201, 0.135863, -0.110508, 0.064224, -0.018478, -0.097851, -0.064903, -0.058445, 0.089384, -0.028956, -0.061775, 0.014616, -0.048824, -0.059620, -0.086199, 0.113536, -0.150780, -0.071185, -0.000607, 0.019294, -0.071356, -0.047454, -0.119500, -0.073540, 0.054943, -0.132369, -0.017115, 0.011438, -0.152603, -0.042400, -0.079245, 0.064180, -0.143842, 0.095470, -0.086749, -0.037729, -0.075675, -0.032210, -0.009267, -0.104218, 0.320924, -0.088893, -0.051534, 0.107530, -0.073505, 0.016447, -0.082996, 0.007302, -0.008158, 0.067813, 0.092828, -0.025175, 0.022487, 0.164771, 0.058614, -0.083011, -0.012903, -0.066108, -0.209505, -0.098660, 0.051666, -0.083428, -0.051739, -0.117397, -0.000056, -0.063386, -0.012033, -0.066626, -0.160435, 0.034906, -0.145679, 0.047362, 0.066292, 0.069332, 0.115532, -0.036764, 0.006236, -0.046650, 0.126974, 0.076756, 0.046814, 0.008800, -0.109934, -0.102685, -0.113948, -0.032470, -0.023226, 0.085949, 0.092421, -0.015744, -0.156410, 0.014473, -0.071952, 0.042415, -0.003722, 0.084175, 0.097660, -0.087803, -0.008410, 0.042073, 0.036199, 0.186011, -0.089011, -0.080704, -0.088910, -0.082585, 0.028971, 0.126664, -0.123477, -0.027863, 0.040612, 0.007409, 0.104474, 0.041520, -0.129605, 0.223421, -0.049891, -0.055381, 0.016186, 0.161468, -0.036252, -0.037176, -0.069897, -0.076128, -0.044350, -0.000245, -0.126827, 0.086317, -0.124838, -0.022698, -0.070213, 0.077768, 0.012275, 0.031332, -0.100231, -0.222669, -0.005904, -0.075661, 0.154336, -0.074540, -0.126616, -0.091444, 0.135117, -0.034197, -0.144844, 0.008807, 0.125667, -0.064608, -0.000964, -0.124643, 0.038319, -0.164437, -0.002721, -0.024967, 0.023320, -0.013231, -0.067340, 0.059161, 0.116125, 0.279915, 0.052820, 0.083363, 0.047709, -0.024974, -0.122166, 0.008307, 0.018329, 0.065969, -0.012040, -0.067998, -0.105463, 0.115613, -0.092663, 0.087921, -0.000891, 0.065248, -0.025333, 0.034332, -0.039855, 0.055734, -0.049337, -0.003783, -0.054005, -0.106749, -0.097568, -0.100315, 0.116387, -0.048267, -0.041810, -0.073130, 0.128502, 0.115899, 0.199680, 0.065991, 0.142224, 0.090686, 0.018895, 0.172825, -0.061233, -0.096433, 0.038688, -0.218101, 0.013180, 0.055648, 0.003417, 0.064400, -0.113315, -0.018900, -0.004269, 0.043582, -0.019807, 0.196399, 0.119204, 0.064619, 0.159048, 0.064958, -0.170559, 0.042283, -0.054435, 0.032379, 0.250167, -0.013789, -0.163083, -0.026576, -0.064139, 0.189430, 0.210244, -0.100577, 0.027830, -0.008100, -0.029073, -0.036478, 0.056039, -0.105392, 0.042745, -0.201113, -0.106627, 0.013472, -0.033761, -0.016741, -0.112588, -0.114113, -0.231826, 0.032898, 0.079047, 0.045482, -0.045386, -0.071009, -0.138409, -0.241049, 0.075442, -0.093576, -0.065396, -0.049194, -0.212993, -0.126846, 0.002913, 0.066706, -0.017569, -0.082167, -0.089653, 0.137427, 0.067217, 0.181396, -0.121815, -0.119787, -0.045991, -0.155547, -0.245716, -0.071119, 0.078826, 0.008661, -0.032027, 0.066143, -0.161863, -0.016999, -0.106182, 0.085898, -0.124126, -0.045065, 0.040804, -0.115499, -0.126095, -0.035421, -0.035062, -0.045318, 0.026523, -0.043984, 0.103963, 0.031667, 0.110852, 0.093245, 0.212724, 0.042155, 0.025032, 0.048845, 0.011084, -0.050865, -0.034240, -0.125505, -0.078821, 0.104235, -0.073305, 0.186337, -0.137245, 0.016577, -0.177905, -0.051540, -0.296186, 0.076247, 0.100367, 0.106215, 0.080465, -0.125691, 0.022984, -0.064328, 0.105904, -0.092480, -0.019046, -0.129299, 0.024605, 0.027402, 0.122172, 0.113609, 0.100319, -0.102733, -0.134529, -0.144077, -0.079293, 0.019035, -0.117612, 0.072842, -0.025710, 0.040649, 0.065982, -0.028206, -0.108644, -0.071989, 0.047922, 0.116442, 0.083601, -0.128099, -0.022526, 0.049384, 0.028470, -0.011948, -0.207043, -0.099292, 0.015090, 0.007786, 0.171823, 0.051995, 0.068854, -0.079143, -0.020266, 0.046016, -0.052680, 0.087447, 0.083039, 0.000027, 0.070786, -0.315182, 0.048407, -0.011329, -0.057845, 0.060909, 0.225151, -0.044462, 0.018324, -0.023694, -0.095112, -0.068342, -0.063069, -0.112960, -0.154926, 0.093112, 0.003885, -0.069050, 0.051977, -0.013295, -0.174460, -0.059060, 0.028969, 0.048624, 0.122202, 0.053740, -0.063442, -0.030741, -0.361136, 0.178486, -0.036004, -0.339672, -0.169732, -0.102179, 0.270307, -0.080804, -0.087639, 0.011147, -0.065261, -0.051427, 0.054001, -0.094697, -0.092222, -0.280283, 0.083252, -0.220621, 0.036896, 0.071002, -0.045281, -0.178552, -0.203823, 0.090639, 0.004757, 0.028989, -0.038759, -0.011798, 0.161178, -0.097314, -0.002167, -0.094795, -0.071009, -0.047110, -0.057002, -0.032261, 0.066076, 0.087537, -0.081959, 0.053049, 0.059220, 0.044483, -0.035741, 0.144774, 0.061637, -0.206811, -0.054893, -0.092820, -0.071536, -0.066922, -0.069521, -0.046925, 0.156458, -0.020098, -0.121932, -0.192638, 0.102676, -0.014818, 0.088685, -0.140784, -0.074543, -0.116281, -0.098058, -0.202357, 0.040523, -0.034219, 0.121212, -0.131530, -0.120047, 0.030389, -0.112277, 0.022772, -0.048996, -0.256811, -0.002802, 0.086857, 0.066414, -0.180253, -0.017675, -0.284616, 0.041162, -0.010707, 0.111667, -0.116346, 0.014701, -0.327735, 0.068724, -0.126564, -0.227005, -0.045223, -0.049902, 0.111259, 0.033342, 0.047022, 0.052884, -0.340481, 0.368088, -0.165115, -0.197323, -0.124023, -0.068378, -0.238443, 0.002227, -0.133849, -0.135646, -0.143093, 0.100112, 0.059449, -0.077897, -0.001072, -0.094999, -0.167501, -0.040998, -0.017341, 0.281206, 0.057099, 0.217038, 0.015425, 0.024542, -0.050718, -0.094203, 0.103381, 0.038484, -0.242024, 0.251324, -0.030859, -0.062215, 0.085182, -0.102509, -0.085683, 0.089534, -0.209980, -0.178250, -0.037584, 0.033385, -0.193466, -0.282743, -0.046690, -0.028280, -0.027464, 0.057314, 0.031520, -0.170652, 0.099192, 0.011038, -0.032152, 0.158005, -0.050825, -0.115137, -0.114336, -0.068624, -0.093966, 0.031900, -0.024054, 0.098169, -0.059631, 0.065816, -0.351718, -0.384688, -0.159168, -0.288895, 0.233973, -0.148545, -0.028034, 0.001684, -0.043015, -0.050082, 0.054740, 0.079895, -0.140123, 0.038322, -0.097631, -0.204046, -0.084985, -0.045660, -0.012765, -0.040171, -0.131433, -0.007506, -0.011067, -0.153732, 0.093226, -0.163989, -0.043763, -0.107820, 0.012576, -0.122260, 0.120028, -0.098802, 0.175834, -0.109518, 0.161750, -0.119233, 0.096761, -0.035737, 0.029333, -0.005993, -0.056085, 0.106855, -0.069718, -0.006663, 0.049973, 0.126339, 0.074147, 0.058531, 0.018339, -0.048632, -0.112337, -0.001410, 0.046342, 0.138121, -0.011390, -0.143779, -0.042757, -0.062626, -0.062553, 0.026099, 0.132057, -0.040008, -0.014840, 0.007015, 0.000093, 0.070233, -0.063470, 0.003634, -0.189420, -0.128313, -0.130246, -0.000441, 0.021424, 0.065122, -0.030535, 0.065647, -0.061027, 0.087881, -0.136154, -0.054728, -0.144556, 0.018630, 0.030484, -0.052261, 0.113272, -0.116564, -0.174536, 0.072725, 0.030650, 0.021080, -0.137506, -0.050612, -0.020428, 0.038438, 0.042995, -0.001327, 0.145723, 0.104995, -0.056887, -0.099358, -0.047546, 0.146644, -0.067370, 0.034138, -0.079475, 0.005502, 0.025765, -0.063036, -0.018628, 0.100001, 0.047332, -0.138308, -0.043247, 0.007983, 0.021408, 0.068238, 0.066436, 0.100959, -0.044965, 0.012126, 0.071389, -0.010680, 0.042006, 0.031463, -0.017144, -0.040904, -0.071610, 0.058630, -0.032955, -0.062732, 0.069315, 0.012460, -0.063941, 0.051844, 0.005627, 0.076232, 0.012775, -0.027814, 0.021609, -0.013577, 0.044895, 0.009881, 0.120327, -0.030484, -0.148966, -0.092186, -0.110996, 0.066970, -0.011837, -0.057818, 0.016802, -0.058288, 0.078379, -0.079894, -0.037784, -0.130764, -0.065733, 0.040432, 0.132959, -0.004977, -0.012492, 0.020928, 0.003784, -0.088909, 0.068814, 0.029971, 0.031611, 0.038344, -0.013008, -0.117760, 0.006041, 0.029923, -0.071571, -0.108762, 0.002438, -0.033683, 0.081630, -0.097764, -0.090767, -0.037246, -0.009887, 0.076186, 0.078398, -0.042506, -0.012910, -0.025561, 0.059783, -0.123285, 0.031707, 0.087698, 0.056091, -0.012902, -0.074122, -0.043413, -0.085910, -0.129046, -0.040367, 0.089386, -0.063205, -0.060609, 0.024605, 0.128820, -0.012152, 0.082219, 0.013183, 0.047644, 0.023604, 0.002073, -0.043316, -0.080378, 0.017161, 0.054294, 0.086921, 0.023395, -0.080999, 0.046552, 0.146831, -0.042326, 0.053970, -0.034743, -0.053440, 0.004967, 0.051390, -0.070346, -0.110926, -0.138882, -0.021597, -0.094029, 0.079391, -0.060203, 0.080002, 0.113989, -0.116836, 0.079855, 0.024356, 0.101703, -0.027800, -0.149133, -0.092881, -0.040804, 0.128732, -0.015060, -0.177092, 0.101395, -0.286897, 0.028872, -0.074029, -0.205722, -0.089968, 0.061380, -0.024066, -0.006812, -0.052673, 0.003066, 0.035160, 0.020565, 0.105719, -0.127204, -0.025101, 0.084794, 0.047702, -0.003641, -0.130909, 0.120980, 0.070639, -0.122633, -0.079569, 0.000352, -0.024636, -0.038007, -0.131251, -0.058447, -0.055328, -0.148788, -0.123086, 0.042158, 0.029993, -0.121521, -0.029143, -0.114386, -0.126273, -0.086333, 0.013196, -0.008037, 0.006405, 0.137056, 0.121034, 0.116405, -0.026293, -0.090119, -0.065223, 0.025044, -0.228797, -0.066962, -0.019798, -0.075618, -0.056786, -0.086517, 0.022684, -0.173819, -0.066175, -0.010761, 0.099537, 0.025852, -0.111482, 0.113874, 0.038300, 0.060297, 0.036274, 0.045349, -0.122489, -0.131460, 0.183640, -0.023977, 0.050190, -0.039938, 0.006953, 0.045183, -0.065856, 0.015684, 0.050115, -0.116690, -0.011207, 0.035594, 0.094016, -0.139569, 0.033834, 0.128953, 0.099280, 0.098581, 0.046639, 0.054146, -0.058905, 0.092906, 0.046509, -0.224702, 0.093248, 0.050235, -0.010220, 0.074364, 0.132874, 0.050564, -0.115791, -0.065832, 0.066869, -0.103556, -0.052147, -0.067143, -0.001604, -0.027839, -0.014756, 0.069925, -0.088333, -0.112830, 0.050093, 0.071044, -0.139848, 0.099580, -0.108372, 0.003698, 0.190302, 0.162524, -0.137041, -0.124691, 0.065886, 0.061069, 0.002685, -0.217956, -0.036640, -0.046029, -0.327825, -0.023569, -0.113346, -0.003659, 0.030995, -0.202784, -0.174494, -0.082433, 0.082772, 0.034516, -0.012607, 0.199323, 0.158663, -0.069788, 0.113870, -0.005797, -0.137303, -0.067433, -0.006648, -0.189994, 0.175670, 0.193236, 0.041285, -0.075724, 0.082742, 0.086096, -0.011698, -0.011979, 0.013573, 0.098424, 0.051249, 0.049755, -0.032411, -0.078271, -0.037287, 0.105532, 0.002624, 0.191292, -0.134677, 0.099643, 0.060532, -0.070464, 0.215996, 0.066156, -0.046027, -0.007805, -0.027779, -0.055128, -0.028633, 0.035950, 0.004933, 0.065899, 0.020462, -0.320631, -0.281836, -0.273960, -0.323316, -0.417855, 0.092839, -0.030649, -0.380760, -0.062099, -0.136621, -0.010011, -0.036197, -0.142359, -0.167171, 0.003355, -0.096666, 0.106582, 0.040090, -0.101636, 0.017084, -0.157042, -0.157552, -0.030074, 0.055561, -0.047112, -0.088888, -0.086941, -0.175848, 0.037857, -0.184962, 0.056730, -0.055691, -0.013950, -0.045562, -0.100605, 0.158319, 0.195275, -0.033661, -0.051825, -0.115900, 0.002260, -0.070431, 0.251626, -0.238041, 0.140575, -0.071205, -0.047368, -0.120220, -0.205366, -0.079129, -0.354571, 0.001661, 0.071426, -0.135514, 0.047972, -0.087575, -0.044821, -0.096199, -0.200207, -0.190467, -0.252624, 0.049106, 0.073404, -0.035235, -0.164789, -0.103069, 0.025979, -0.096175, -0.105324, -0.083405, -0.134133, -0.321873, 0.046789, -0.058813, -0.072129, -0.064387, -0.035135, -0.026167, -0.321781, -0.121761, -0.147044, -0.376803, -0.212131, 0.080955, -0.061756, -0.154342, -0.164446, -0.043938, -0.145949, -0.028498, -0.249823, 0.010698, -0.091574, 0.007385, 0.044565, -0.277106, 0.079391, -0.062550, -0.247786, 0.079277, -0.198747, -0.049940, -0.032398, 0.009787, 0.036465, -0.013508, 0.043144, -0.068525, -0.022465, 0.016634, -0.329112, -0.013769, -0.060301, 0.029990, -0.207255, -0.104420, -0.110378, -0.065189, 0.042188, -0.115952, -0.048335, -0.089090, 0.125813, -0.009546, -0.219733, -0.019574, -0.322814, -0.165793, -0.164985, -0.155910, -0.062158, -0.310582, -0.135369, 0.003705, -0.158794, -0.049494, -0.052545, -0.125965, -0.061428, -0.414918, -0.149543, -0.078155, -0.153025, 0.046215, -0.220992, -0.016386, -0.008890, -0.097929, -0.034545, -0.138515, -0.011945, -0.188789, 0.069118, -0.028001, -0.293557, 0.091387, -0.093256, -0.005673, -0.223653, -0.117339, -0.167852, -0.245122, -0.091290, -0.104819, -0.019394, 0.045247, -0.033260, 0.201083, -0.064026, -0.154743, -0.082042, -0.295479, -0.095284, -0.444657, -0.087330, -0.097887, -0.198394, 0.017064, -0.223860, -0.064489, 0.022250, -0.097288, 0.125187, -0.022067, -0.232618, 0.094854, -0.097888, -0.075581, 0.073562, -0.112346, -0.136780, 0.033985, -0.125276, -0.321069, 0.032384, 0.099893, 0.024167, 0.054283, 0.034128, -0.092456, -0.019133, 0.088654, -0.083230, -0.118362, -0.015762, 0.037959, -0.079354, 0.039312, -0.150997, -0.094924, 0.015776, -0.126137, -0.081712, 0.055804, -0.078698, 0.007256, -0.091899, -0.135883, -0.031552, -0.008581, -0.038109, -0.080549, 0.033400, -0.010590, 0.061655, -0.042998, 0.093812, 0.070115, -0.092453, -0.046645, -0.046337, 0.053829, -0.035560, -0.095752, -0.041504, -0.140637, -0.108931, -0.044518, -0.163751, -0.015510, 0.018417, -0.133559, 0.060327, 0.055841, -0.084184, -0.040802, -0.005292, 0.003381, 0.018329, 0.116703, -0.059311, -0.049561, -0.053835, -0.035965, 0.058987, 0.049497, 0.044153, -0.037292, -0.141432, -0.161087, -0.121527, 0.117311, -0.030272, -0.001184, -0.055795, -0.002486, -0.068789, 0.034904, -0.010284, 0.036350, 0.078311, -0.059228, -0.015435, -0.077254, -0.064175, -0.123681, 0.041613, 0.089121, -0.002873, -0.114284, 0.029440, -0.017309, -0.044754, -0.026124, 0.039786, -0.081021, -0.095334, 0.118441, -0.081264, -0.115500, 0.046917, -0.077877, 0.029928, -0.102471, 0.014797, -0.090446, 0.017926, 0.048931, 0.067393, -0.095960, -0.174307, -0.039299, -0.041900, 0.127161, -0.041253, 0.118785, -0.061346, -0.123313, -0.037561, -0.004211, -0.117890, 0.015136, 0.105246, -0.121119, -0.123018, -0.028441, -0.014214, 0.055299, 0.051977, 0.000731, 0.096077, -0.052905, -0.094523, 0.138934, 0.111123, 0.026282, -0.009975, 0.094072, 0.014219, -0.006404, -0.025369, -0.121986, 0.047188, -0.002728, 0.040961, 0.057789, -0.106470, -0.122462, 0.052882, 0.155134, 0.055254, -0.117730, -0.008940, -0.208140, -0.031824, -0.093844, -0.027801, -0.079768, 0.032856, 0.043761, 0.000708, -0.063234, -0.032128, 0.015770, -0.115096, -0.082891, 0.048678, -0.056779, -0.073184, -0.039189, 0.027632, -0.074326, 0.108843, -0.063087, -0.015077, -0.040940, 0.005305, 0.035519, 0.065066, 0.087835, -0.064585, 0.034441, -0.066236, -0.111902, 0.088476, -0.005130, -0.015603, 0.066666, 0.085037, 0.007765, 0.117824, -0.084906, -0.142216, -0.093463, 0.004740, 0.075673, -0.077250, 0.120591, -0.332697, -0.041148, -0.033691, -0.129794, -0.101185, 0.010905, -0.006170, -0.185505, -0.064564, 0.037324, -0.101491, 0.000366, -0.152152, 0.056040, 0.017028, -0.026707, -0.328550, -0.087478, -0.071055, -0.028419, 0.065051, -0.094925, -0.150722, -0.007161, -0.091055, -0.060933, -0.103757, 0.000752, 0.017284, 0.036489, -0.020032, 0.054709, 0.005742, -0.001819, -0.073051, 0.071649, -0.099291, -0.013985, -0.035283, -0.103378, 0.077881, -0.182806, 0.012076, 0.061502, 0.019338, -0.017459, 0.003289, -0.249176, 0.048872, 0.071768, -0.058683, -0.044261, -0.098442, -0.067731, -0.135689, 0.110124, 0.015198, -0.132140, 0.014221, -0.052108, 0.003471, -0.090089, -0.080421, -0.028540, 0.046194, -0.017742, 0.060060, -0.030137, -0.179193, -0.080912, -0.105910, -0.066747, -0.056803, -0.031311, -0.198117, -0.186682, 0.062273, -0.091352, -0.168795, 0.036792, -0.128357, -0.030541, 0.003755, -0.005971, -0.008363, -0.143691, -0.003922, 0.027619, 0.066269, -0.120075, 0.015092, 0.091244, -0.244811, -0.052686, 0.052174, -0.108148, 0.018901, -0.042860, 0.003212, 0.025170, 0.070424, 0.008142, 0.256699, -0.027637, -0.042487, -0.027892, -0.126491, -0.067974, 0.171102, -0.105774, -0.128959, -0.079572, -0.098444, -0.023540, -0.040118, -0.113935, -0.084683, -0.114781, -0.085792, 0.034368, -0.200892, -0.169142, 0.011520, -0.015275, -0.100881, 0.008438, -0.058977, 0.026906, -0.267861, 0.078009, 0.026461, -0.107124, -0.178896, -0.157631, 0.047328, -0.025748, -0.040126, 0.012371, 0.050066, 0.097968, -0.013780, -0.033341, -0.095901, -0.053693, 0.198500, -0.071247, 0.022768, -0.042791, -0.032637, 0.006505, -0.087021, -0.000076, -0.032508, 0.035979, -0.033953, 0.031686, -0.198845, 0.058936, -0.061763, -0.101328, -0.131337, 0.044351, 0.146480, 0.009326, -0.067068, -0.102900, 0.095212, -0.072848, -0.090250, -0.036714, 0.029892, -0.116298, -0.027662, -0.062231, 0.038844, -0.038784, -0.146376, -0.166188, 0.313560, -0.014587, -0.028223, -0.060164, -0.031235, -0.019822, -0.111088, -0.068100, -0.170124, -0.033628, -0.165687, -0.055185, 0.073528, -0.085137, -0.069467, -0.049083, -0.100256, 0.002354, 0.108595, -0.051864, 0.104063, 0.050921, -0.061192, -0.096299, 0.109858, 0.055076, 0.028130, -0.045724, -0.080546, -0.038850, 0.125929, -0.037071, -0.013955, -0.031692, -0.107318, 0.085611, -0.057431, -0.119878, -0.070149, 0.037998, -0.098855, -0.054922, 0.049407, 0.069929, -0.067527, 0.013999, 0.060339, -0.057807, -0.167466, -0.020730, -0.100983, -0.151332, -0.053338, 0.057532, -0.032879, -0.078396, -0.058914, -0.097518, 0.037446, -0.036823, -0.091370, 0.159987, -0.041251, -0.117258, -0.175549, 0.100423, -0.027831, 0.157677, -0.115334, 0.032967, -0.016487, 0.063812, 0.132784, 0.006840, -0.060574, 0.126458, -0.035177, -0.051341, -0.027286, -0.149214, -0.054435, 0.017076, 0.044087, 0.112145, -0.204964, 0.133145, 0.047321, 0.095190, -0.027215, -0.013910, 0.049583, 0.119319, -0.138798, 0.010634, 0.104724, 0.070723, -0.040704, -0.052029, -0.075257, 0.024035, -0.141484, 0.067893, 0.073598, -0.249688, 0.162998, 0.114631, 0.121823, -0.230230, -0.098277, -0.003301, 0.075494, 0.065268, 0.096625, -0.101807, 0.001191, 0.114923, 0.081898, 0.123994, 0.092250, 0.001312, -0.024086, 0.149521, 0.122739, 0.036923, 0.008668, -0.037993, 0.119124, -0.022211, 0.147741, 0.022628, -0.077001, 0.058671, -0.039667, 0.040180, -0.059933, 0.113862, -0.109439, -0.020264, -0.019407, 0.085476, -0.016839, -0.166066, -0.134895, -0.065935, 0.055401, 0.161524, 0.090011, 0.047616, -0.057956, 0.268957, 0.003896, 0.076125, -0.014026, 0.178900, -0.024760, -0.142704, -0.030860, -0.154514, -0.020011, -0.005124, -0.171485, -0.110742, 0.007665, -0.024232, 0.033851, 0.095018, -0.043649, 0.005022, 0.049750, 0.061858, -0.052117, 0.146874, 0.051195, 0.049508, 0.034214, -0.037279, 0.120692, -0.156351, -0.077434, 0.007859, 0.082764, 0.001432, -0.109189, -0.039274, -0.093652, -0.144355, -0.077210, 0.110319, -0.110534, 0.026715, 0.004551, 0.067639, 0.097769, 0.209425, 0.057577, 0.121009, 0.001004, 0.008010, -0.069654, 0.012200, -0.163975, -0.018584, 0.051852, 0.058262, -0.195871, -0.008093, -0.069087, -0.113725, -0.035638, 0.005737, -0.024957, -0.046218, -0.026900, -0.044425, -0.135961, 0.061226, 0.134940, 0.004697, -0.010512, 0.062074, 0.003400, -0.057330, 0.201516, -0.073157, -0.007947, -0.198857, -0.051318, -0.258609, 0.077456, -0.050570, -0.177912, 0.074926, 0.084481, 0.069762, -0.028691, 0.006759, -0.083524, -0.049425, -0.047759, 0.005801, -0.071233, 0.160923, -0.034509, -0.005583, -0.067399, 0.073877, -0.162912, -0.068442, 0.186825, 0.048431, -0.260859, 0.005083, 0.080071, 0.090315, -0.073162, 0.134181, 0.001289, -0.076654, 0.029558, 0.008495, 0.071675, -0.065701, -0.082156, -0.044954, 0.034952, -0.057017, 0.024779, -0.099009, 0.003829, -0.025087, 0.012239, -0.116820, 0.074734, -0.024627, -0.140065, 0.034288, 0.084276, 0.099425, 0.160483, 0.079851, 0.117225, 0.030030, -0.175479, -0.090567, -0.047473, -0.049218, -0.133766, -0.113354, -0.173324, 0.013594, 0.006190, 0.011925, 0.070885, 0.042836, -0.063331, 0.063460, 0.157142, -0.110262, -0.139218, -0.000370, -0.096600, 0.053864, -0.079215, -0.059331, 0.055188, 0.065775, -0.035835, -0.079258, 0.028979, -0.206867, 0.030253, 0.132931, -0.043722, 0.222228, -0.118610, -0.001973, 0.000565, 0.105224, 0.095284, -0.026608, -0.247171, -0.026762, 0.077891, 0.017440, 0.018515, 0.028772, 0.060826, 0.031960, 0.060915, -0.115517, -0.055242, -0.003539, -0.011686, -0.009660, -0.119105, 0.097084, -0.047040, -0.037964, -0.182104, -0.056219, -0.045938, -0.144456, -0.212142, -0.169760, 0.011684, 0.100647, -0.036757, 0.099388, 0.006961, 0.047116, -0.038425, -0.136439, 0.164479, -0.050046, 0.090201, 0.078795, 0.022470, 0.089379, -0.069072, 0.052122, -0.057131, -0.233778, -0.037374, 0.014706, 0.087299, -0.095431, 0.115591, -0.131035, 0.097803, -0.024574, -0.314615, 0.044222, 0.188964, 0.027303, 0.059504, 0.009073, 0.121399, 0.016886, -0.054758, -0.169657, -0.139456, 0.028155, 0.018538, 0.052148, 0.146474, -0.255966, 0.077720, -0.060795, 0.022088, 0.049411, 0.080412, 0.192936, -0.078614, 0.003615, -0.126701, -0.053882, -0.058713, 0.064483, -0.011054, -0.000738, 0.030828, -0.086642, 0.077441, 0.027402, -0.051702, -0.190825, 0.078878, -0.055278, 0.011310, 0.005660, 0.071821, 0.067429, 0.029839, -0.123993, -0.114707, -0.049661, -0.167617, 0.056342, -0.116663, 0.046143, 0.029724, -0.081427, 0.041639, 0.051811, -0.020210, 0.129666, -0.050771, 0.188207, 0.032444, -0.137360, -0.057769, -0.020588, 0.030857, -0.057394, 0.000165, -0.000621, 0.007913, 0.095192, 0.022772, -0.149600, -0.085870, 0.033742, 0.015381, -0.007207, -0.072266, -0.013185, -0.263171, -0.197043, 0.082751, 0.067706, -0.235078, 0.061937, 0.034586, -0.033142, -0.031018, 0.054441, 0.014488, 0.043356, 0.165276, 0.020465, 0.026978, -0.007448, -0.130390, -0.040962, 0.093885, -0.029519, 0.151588, 0.058191, -0.035450, -0.045470, -0.052258, -0.008227, -0.096110, 0.128421, 0.041831, -0.004093, 0.000744, 0.000220, -0.174368, 0.002190, -0.045175, -0.058838, -0.002403, -0.167034, -0.013614, -0.118622, -0.020385, -0.097728, 0.014369, -0.001716, -0.071835, -0.005660, 0.079677, -0.017964, -0.129655, -0.139002, -0.109957, 0.101661, -0.058004, -0.009959, -0.023073, 0.067251, -0.120252, -0.134495, 0.101426, -0.129498, 0.018512, 0.017842, 0.036049, -0.053081, 0.060214, -0.044770, 0.063738, 0.009737, 0.059572, -0.062405, -0.174845, -0.048404, -0.015829, -0.046462, 0.156257, -0.081339, 0.017098, -0.004372, 0.014883, -0.118947, -0.098997, 0.074073, -0.039814, -0.004702, 0.039182, -0.037912, 0.081815, 0.031044, -0.099265, 0.077115, -0.083712, -0.042703, -0.250900, -0.166667, 0.071617, 0.075986, -0.159852, -0.142337, -0.131475, 0.160736, -0.149554, -0.064750, 0.087684, 0.024418, -0.040513, 0.090897, -0.127098, -0.010633, -0.066225, -0.043778, 0.040936, 0.057844, -0.267469, 0.000931, 0.054244, -0.077933, 0.124728, 0.069738, -0.045607, -0.020835, -0.356803, 0.007945, -0.148171, -0.033532, 0.065665, -0.064175, 0.179317, -0.085005, 0.027863, -0.261506, 0.076569, 0.042682, 0.100302, -0.069790, -0.100066, 0.048303, -0.106157, -0.091787, 0.116303, 0.004552, -0.041670, 0.063340, 0.082825, -0.068005, -0.105224, -0.022005, 0.022982, 0.010475, 0.019081, -0.004345, -0.215589, 0.126259, -0.038649, 0.099271, 0.101168, 0.009555, -0.175877, -0.038100, 0.162414, -0.059705, -0.122116, 0.078227, -0.010089, -0.024037, 0.030286, 0.223085, 0.052676, -0.067553, 0.028301, -0.084342, -0.026597, 0.015056, -0.036686, -0.001457, 0.037651, -0.015583, 0.052154, -0.063114, -0.053204, -0.155237, -0.093895, -0.046258, -0.073418, 0.003406, 0.064511, 0.019325, -0.184678, -0.017165, -0.031616, -0.123489, -0.069799, 0.361381, 0.092272, -0.004060, 0.008062, 0.043219, -0.141910, -0.050251, 0.002551, 0.060260, -0.046441, -0.132724, -0.013720, -0.067291, -0.014790, -0.165338, 0.040678, -0.068499, -0.034852, -0.188337, 0.046784, 0.045634, 0.022247, 0.015906, 0.016942, 0.024885, 0.015514, 0.020077, 0.026067, -0.092715, -0.119386, -0.031013, -0.004238, 0.049967, -0.097354, -0.008325, -0.072182, -0.045106, -0.194680, -0.015742, 0.017410, 0.000134, -0.038757, -0.050300, -0.104252, -0.045844, -0.077165, 0.007889, -0.011204, -0.040528, 0.097182, -0.003449, -0.049089, -0.072533, -0.078685, -0.115992, -0.007082, -0.050899, -0.096230, 0.043973, -0.074465, -0.022626, -0.032246, -0.013314, -0.052089, -0.125287, -0.138799, 0.036846, -0.121875, 0.103521, 0.024576, -0.057750, -0.026243, -0.082276, 0.046250, 0.013340, 0.001795, -0.009054, 0.106019, -0.103261, 0.103401, -0.160286, -0.060691, -0.094014, 0.112333, 0.128201, -0.096710, -0.038025, 0.035923, 0.045668, -0.016678, -0.031534, -0.034349, -0.123206, -0.056150, -0.019148, -0.093186, -0.016536, -0.349115, -0.069248, -0.133397, -0.107857, -0.069917, 0.003013, -0.074416, -0.069234, 0.122266, 0.082947, -0.042563, -0.103198, 0.011277, -0.137110, 0.074876, 0.009112, 0.089675, 0.058513, -0.051016, -0.029926, 0.125699, -0.132190, -0.066214, -0.040979, 0.148902, -0.006171, 0.048697, -0.067727, -0.072220, 0.014549, -0.071796, -0.066780, 0.054162, -0.129418, -0.013728, -0.003547, 0.099971, 0.022282, -0.127128, -0.108193, -0.041520, 0.085874, 0.192319, -0.067525, 0.127843, -0.148406, -0.237751, -0.065256, -0.111757, 0.042962, -0.053458, 0.027547, -0.050078, -0.128561, 0.256082, 0.040443, 0.026108, 0.084282, 0.007726, 0.011843, 0.019832, -0.046665, -0.086357, -0.048966, -0.089083, 0.014328, -0.087195, 0.013074, -0.013402, -0.020059, 0.050874, -0.223518, 0.079337, -0.101486, 0.104044, -0.077222, 0.076144, -0.071063, -0.174972, -0.103591, -0.063536, 0.056479, -0.008231, -0.089534, -0.058432, -0.071028, -0.104539, 0.025890, -0.090563, -0.074682, -0.031716, -0.069125, -0.006225, -0.025241, -0.091135, -0.140160, 0.118179, -0.000858, -0.008358, 0.084175, 0.043443, -0.031612, -0.030553, -0.051145, -0.037136, -0.019582, 0.025805, -0.063706, -0.059474, 0.045085, 0.031876, -0.118870, 0.008425, -0.085046, 0.022466, 0.002574, 0.026983, -0.113695, -0.102028, -0.079537, 0.015512, 0.031698, -0.003478, 0.063516, 0.067535, 0.039897, -0.100763, -0.012151, 0.077709, -0.105966, -0.029072, 0.145351, 0.033875, -0.152267, 0.042528, -0.056599, -0.093187, -0.122141, -0.066502, 0.017661, 0.006524, 0.005956, -0.268206, -0.100266, -0.045581, -0.089011, 0.091104, 0.020957, -0.018513, -0.105020, 0.098319, -0.190358, -0.033712, 0.087400, -0.077930, -0.082555, -0.135251, -0.024772, 0.006085, -0.133967, 0.043046, -0.051226, -0.068687, -0.192576, -0.037178, 0.036400, 0.035664, -0.148301, 0.019482, -0.077409, -0.044221, 0.039328, 0.079281, -0.066808, 0.012500, 0.097220, 0.062767, -0.133576, 0.101343, 0.133730, -0.071188, 0.126486, -0.019371, 0.039823, -0.086438, 0.056880, 0.127526, 0.013699, -0.055537, 0.044520, -0.160393, -0.121234, -0.052648, -0.018657, -0.013512, -0.018087, -0.103853, -0.015687, 0.110502, -0.018452, -0.024131, -0.000849, -0.099036, 0.042808, -0.120268, -0.046553, 0.009323, 0.045664, -0.003770, 0.005568, 0.095911, -0.019236, -0.131976, 0.063919, 0.076454, -0.030544, -0.043730, 0.009750, -0.134336, -0.145342, 0.029552, -0.142949, 0.132252, -0.010223, -0.049474, 0.052000, -0.113810, -0.011091, -0.042991, 0.041066, 0.178327, -0.136655, -0.051790, 0.028465, -0.021827, 0.022607, 0.120952, -0.073410, -0.106257, 0.023091, 0.045165, -0.103191, -0.110413, -0.004590, 0.021639, 0.132746, -0.080934, -0.132735, -0.031588, -0.018021, 0.018236, -0.052814, -0.008881, 0.001844, -0.082097, -0.197083, -0.144542, -0.060567, 0.000027, -0.117389, 0.022598, 0.016634, 0.039845, -0.015449, 0.083081, 0.014805, -0.140595, -0.093013, -0.032607, 0.045805, 0.006147, -0.081341, 0.147312, 0.010461, -0.003364, 0.205523, 0.001380, 0.053981, 0.048998, 0.182210, 0.002855, 0.222965, 0.009416, 0.055693, -0.096885, -0.006528, 0.116391, -0.059499, 0.000731, 0.034951, 0.091454, 0.113145, 0.001312, 0.009179, -0.013135, -0.078863, -0.037471, 0.039266, 0.053128, -0.023409, 0.073082, -0.011298, -0.010303, 0.116783, 0.018333, 0.028235, -0.056586, 0.091289, 0.043691, -0.110287, 0.090128, 0.005065, -0.135777, 0.108977, -0.175943, 0.043058, -0.113012, -0.033682, 0.022186, 0.045497, -0.052043, 0.158929, -0.048146, 0.024324, 0.112652, -0.007714, 0.096802, -0.064846, -0.082411, 0.043617, 0.011072, 0.037090, 0.116538, 0.003904, -0.121821, -0.123068, 0.029614, 0.038660, -0.064324, -0.071319, 0.006559, -0.143664, -0.050745, -0.029431, 0.014222, -0.087014, -0.023900, -0.062313, -0.112864, -0.053301, -0.026519, 0.072306, 0.088529, 0.094502, -0.074899, 0.014262, 0.022109, -0.057802, 0.000986, 0.026476, -0.052176, 0.245442, -0.018599, -0.023649, 0.090455, -0.021206, -0.012673, 0.118805, 0.061044, -0.103424, 0.183295, 0.033015, 0.092308, 0.010473, -0.069715, -0.110400, -0.023787, 0.184404, -0.044797, -0.035279, 0.034516, 0.058686, -0.228944, 0.026470, -0.069006, -0.081788, 0.008825, 0.049616, -0.145408, -0.039585, 0.107517, -0.046487, -0.184303, -0.028285, 0.025653, 0.033715, -0.119180, 0.042948, -0.005413, -0.085142, -0.040762, 0.050793, -0.004620, -0.083096, -0.004455, 0.035890, 0.093139, -0.039772, -0.024004, -0.059905, -0.124434, 0.044264, -0.110011, 0.053954, -0.057285, -0.025424, -0.152110, 0.029913, -0.243578, 0.051619, -0.072731, -0.116399, 0.122813, 0.069034, -0.091741, -0.042464, 0.154047, 0.032020, -0.012484, -0.103777, 0.082985, -0.028860, 0.193411, -0.121123, 0.027701, -0.085851, 0.202340, 0.067212, 0.127585, 0.097247, 0.077295, -0.086294, 0.012446, 0.062375, 0.012216, 0.119178, 0.083426, -0.015650, 0.025358, -0.103183, -0.007421, -0.059186, 0.032900, -0.073868, -0.149613, -0.053727, 0.108761, 0.056122, 0.003883, -0.125453, -0.079749, 0.099152, -0.053455, 0.014637, -0.039494, 0.000624, -0.044362, 0.005138, -0.067778, -0.036581, 0.079579, 0.129269, -0.033852, -0.031565, 0.160241, 0.004322, 0.081963, 0.032643, -0.061689, -0.153820, -0.061908, -0.090497, -0.036019, 0.134852, -0.176514, 0.162225, -0.018816, -0.095384, -0.005092, 0.001424, -0.051903, -0.016156, -0.177487, -0.078060, 0.041936, 0.021614, -0.002590, 0.096917, -0.106782, -0.109999, -0.234354, -0.079869, -0.134581, -0.045270, 0.083431, 0.096194, 0.066743, -0.017029, -0.068801, -0.031504, 0.088634, 0.119594, 0.059190, 0.003905, -0.077304, -0.036049, -0.084894, -0.025289, 0.039399, -0.067833, -0.016349, 0.021204, -0.074432, -0.064057, -0.021417, -0.148868, -0.019564, -0.046357, -0.172159, -0.105964, 0.069016, 0.019016, -0.105377, -0.156977, -0.111383, -0.172632, -0.118267, 0.043398, -0.003057, -0.161844, 0.061666, -0.056882, 0.104652, -0.140848, -0.111078, -0.006408, -0.105392, -0.116953, -0.112689, -0.006827, -0.091737, -0.093677, -0.166312, 0.021857, 0.096566, -0.128301, -0.110515, -0.139148, -0.145926, 0.099003, 0.035822, 0.090099, -0.177180, 0.070362, 0.129359, -0.178066, -0.033664, -0.180195, 0.063695, 0.032021, 0.151520, -0.179545, -0.038055, -0.041768, 0.105589, 0.097973, -0.038455, 0.074867, -0.023603, -0.035200, -0.068567, 0.020279, 0.093825, 0.089490, -0.160882, -0.074406, -0.115453, -0.137508, -0.203475, 0.016149, 0.009139, -0.025246, -0.024714, 0.021686, -0.059688, -0.033462, 0.055163, -0.062716, -0.126818, -0.028723, -0.030713, 0.148461, -0.063771, 0.104058, -0.081252, -0.052137, -0.112891, -0.023285, -0.099838, -0.027697, -0.115176, -0.068086, 0.011545, -0.090183, -0.019343, -0.153564, 0.028174, -0.083825, -0.020830, -0.103536, 0.120941, 0.018580, -0.145927, -0.030059, -0.098676, -0.017183, -0.179325, -0.040508, -0.101261, 0.120692, -0.075808, 0.005273, 0.014894, -0.086595, 0.065784, -0.001310, -0.102470, 0.052515, 0.077026, -0.016011, 0.084164, -0.202829, 0.125463, 0.124170, 0.105745, 0.096440, 0.035498, -0.157750, 0.078635, -0.215763, -0.044526, 0.026306, 0.043407, 0.049312, -0.131571, -0.045107, -0.102439, -0.006040, -0.034509, -0.043000, -0.227521, -0.239639, 0.066396, 0.023354, -0.069438, -0.110540, 0.055686, -0.152500, -0.115230, -0.080619, -0.036856, 0.090352, -0.131586, -0.065360, 0.033632, -0.055282, 0.025173, 0.000668, -0.157578, -0.065807, 0.076208, 0.047115, 0.072033, 0.119407, -0.176681, 0.018342, -0.095679, 0.192156, -0.018851, 0.110758, -0.024417, -0.026683, -0.218883, -0.108533, -0.097645, -0.003771, 0.011019, -0.180128, -0.067236, 0.026408, -0.024615, -0.117826, 0.005620, -0.116531, -0.119432, -0.013273, -0.126301, -0.040444, -0.087059, -0.011145, -0.174117, -0.029351, -0.097828, -0.108856, -0.121137, 0.034295, 0.041435, -0.081717, 0.070838, -0.135300, -0.010639, 0.069808, -0.017487, -0.128075, -0.023783, -0.008510, 0.056460, -0.130221, -0.090242, -0.125950, -0.064664, -0.140622, 0.100186, -0.208313, -0.020277, 0.046844, 0.023232, 0.120955, -0.001586, -0.118086, -0.104630, -0.113681, -0.152955, 0.027628, 0.049398, -0.041698, 0.113022, 0.010360, 0.020474, 0.040425, -0.022507, 0.128981, -0.094330, 0.038420, 0.007086, -0.133780, -0.073008, -0.043567, 0.099047, 0.045731, 0.017187, 0.037833, -0.035721, 0.019118, -0.030944, 0.045542, -0.034774, -0.050563, -0.047691, 0.067483, -0.143034, 0.097623, 0.121048, -0.185795, -0.002013, 0.047360, -0.028966, -0.081188, -0.060190, 0.006325, -0.148362, -0.013581, 0.007075, -0.029891, -0.143528, -0.107555, 0.051183, -0.011143, -0.258358, -0.124693, -0.069272, 0.101741, -0.080275, -0.090718, 0.006934, -0.042868, -0.003683, 0.013024, -0.111438, -0.029729, -0.008870, 0.075446, -0.046268, -0.097197, -0.012055, -0.071298, -0.084195, 0.007739, -0.080497, 0.075102, -0.041336, 0.052914, -0.035121, -0.065297, 0.022014, -0.023264, 0.017999, -0.148685, 0.017802, -0.049363, -0.059266, -0.256328, 0.033824, -0.090818, 0.039097, -0.011398, -0.061299, -0.007172, -0.029656, 0.050844, -0.120477, -0.051888, -0.062270, 0.098442, -0.036799, 0.050259, 0.089948, 0.022105, 0.063771, -0.026646, -0.024322, -0.106438, 0.120206, -0.047229, -0.006481, 0.060422, -0.074195, 0.069524, 0.054103, -0.015833, -0.085855, -0.059047, -0.037411, -0.037001, -0.121906, -0.103570, 0.064216, -0.222148, 0.120428, -0.155428, 0.046715, -0.044497, 0.023344, 0.054647, 0.093718, 0.149977, 0.048801, -0.150152, 0.003762, -0.159514, -0.098340, -0.038466, -0.136304, 0.064521, -0.115409, 0.017635, 0.017229, -0.007549, -0.106771, -0.016809, 0.029184, -0.074620, -0.017310, 0.051820, -0.095096, -0.027344, -0.097528, 0.087770, 0.004469, -0.026907, 0.076469, -0.095311, -0.088042, -0.110354, 0.047907, -0.042647, 0.078806, 0.082021, -0.062800, 0.067441, 0.042872, 0.004343, 0.055974, -0.012150, 0.037404, -0.150888, 0.019205, 0.001002, -0.042887, -0.048250, -0.151012, -0.002217, 0.083732, 0.052448, 0.123923, 0.095055, 0.118004, -0.054684, 0.023418, -0.074032, -0.049329, -0.068497, 0.012734, -0.084997, -0.112512, 0.046355, -0.038437, -0.039792, -0.014205, -0.124706, -0.050537, 0.075028, 0.027949, 0.029828, 0.054760, 0.019999, -0.083672, 0.054133, 0.130445, 0.044781, -0.041997, -0.065640, -0.070110, -0.015569, -0.100665, -0.119353, -0.034243, -0.039275, 0.071676, 0.022802, -0.019842, 0.046946, -0.021638, 0.063672, -0.159851, -0.176629, -0.021952, -0.087787, -0.008713, -0.031314, -0.039261, -0.051019, -0.091746, -0.080384, -0.029767, -0.005817, -0.006865, 0.024355, -0.087046, -0.085548, 0.160933, 0.040744, 0.095023, -0.067384, 0.056538, -0.097240, -0.009747, 0.035877, -0.183278, 0.003558, -0.094417, 0.120551, -0.040771, -0.084486, -0.133422, -0.108058, -0.136832, -0.010684, -0.129556, 0.049127, -0.060807, -0.060748, 0.060601, 0.132665, -0.056501, -0.093551, 0.131115, -0.005077, -0.040747, -0.025117, -0.039720, 0.032783, 0.049928, -0.059523, 0.008886, -0.105931, 0.167071, 0.002904, -0.070399, 0.001465, -0.071139, -0.064650, -0.104246, -0.097688, 0.034713, -0.063805, -0.064703, 0.095277, 0.005821, 0.086651, -0.040724, -0.012219, 0.017726, 0.006249, 0.046109, 0.232799, -0.015246, -0.038317, 0.029109, -0.149251, -0.082884, 0.062418, -0.109010, -0.015857, 0.234284, 0.003439, 0.152199, 0.034985, 0.151291, 0.059777, 0.022238, 0.009207, -0.113829, -0.141098, 0.034012, 0.061176, -0.012344, -0.103229, 0.022397, 0.078166, -0.042556, -0.099900, -0.185971, -0.078881, 0.002173, 0.158164, 0.056774, 0.013128, -0.141202, -0.033938, -0.306758, -0.052001, -0.082769, -0.060719, -0.113739, -0.032412, -0.026982, 0.018407, 0.043064, 0.075985, -0.215440, 0.038142, 0.034016, -0.059795, -0.000967, -0.124293, 0.074331, 0.004855, -0.179589, -0.003390, -0.091879, -0.035251, -0.220402, 0.054665, 0.059966, -0.011457, 0.081477, -0.036543, 0.125970, -0.039857, 0.048030, 0.028895, 0.008078, -0.001318, -0.039434, -0.001772, 0.016297, 0.071112, 0.085613, -0.002230, 0.113405, -0.127501, 0.173410, -0.069056, -0.144316, -0.045555, 0.060776, 0.046894, -0.043793, -0.126044, -0.044240, -0.093292, 0.002095, -0.121745, 0.101204, -0.111560, 0.023329, -0.019146, 0.027152, -0.151145, 0.042947, -0.043683, -0.057689, -0.178385, 0.026022, -0.090362, 0.028564, 0.054839, 0.041659, 0.056826, -0.128037, -0.038347, -0.148552, -0.078019, -0.071879, -0.011991, -0.054461, -0.305345, -0.056264, -0.129305, -0.029803, -0.098046, 0.111804, 0.028582, -0.146926, -0.314070, -0.056917, -0.041474, -0.203157, -0.087862, -0.072286, -0.055818, 0.058579, 0.098033, -0.079928, -0.184344, 0.060200, -0.091852, -0.127924, 0.019528, -0.028031, -0.207984, -0.165802, -0.133924, -0.092455, -0.228983, -0.011613, -0.085463, 0.096606, 0.177018, 0.131097, -0.067144, -0.012775, -0.137721, 0.101093, -0.137118, 0.223832, 0.083500, -0.142113, -0.077398, -0.044722, -0.035025, -0.003650, -0.146234, 0.030623, -0.019492, -0.127822, -0.025942, -0.031058, 0.072137, -0.034526, 0.101645, -0.095632, -0.087112, -0.256793, -0.146718, 0.045574, -0.124525, -0.090882, 0.119340, 0.110846, 0.021960, -0.069937, 0.006952, 0.300033, 0.002010, -0.088118, -0.132755, 0.045757, 0.014464, -0.036014, -0.130133, 0.062954, -0.075390, 0.024221, 0.094153, 0.100825, -0.049882, -0.062725, -0.218766, -0.290256, 0.062805, -0.154582, -0.138965, -0.027668, -0.136982, -0.205973, -0.093105, -0.113031, -0.052144, 0.079072, 0.035063, -0.169450, 0.004793, 0.017169, -0.033712, -0.070533, -0.097298, -0.076035, -0.019888, -0.278046, 0.127443, 0.014208, 0.115077, -0.051866, 0.054153, -0.059682, -0.074399, -0.133570, 0.079531, -0.123193, -0.005465, -0.072980, -0.008575, -0.139375, -0.138723, -0.067418, -0.033016, 0.054842, 0.022090, -0.066577, 0.027664, 0.075548, 0.023965, -0.081947, -0.046173, -0.049068, -0.061533, 0.077098, -0.035136, -0.003959, -0.206099, 0.052683, -0.053955, 0.019690, 0.103946, 0.108444, -0.120065, -0.070196, -0.025683, 0.065892, -0.103194, -0.059536, -0.121712, 0.054535, -0.001627, -0.151679, 0.066313, -0.110740, -0.111666, 0.104911, -0.005190, -0.012064, -0.013472, 0.017567, -0.208094, -0.066031, -0.003182, 0.128749, -0.003673, -0.022867, -0.064306, -0.105399, 0.002113, -0.035148, -0.060942, -0.069508, -0.051686, -0.043715, -0.053532, 0.104066, -0.055585, 0.089794, 0.054024, 0.030421, 0.070441, 0.032223, -0.145245, -0.122011, -0.027226, 0.001902, 0.066555, -0.082442, -0.010074, 0.040987, -0.117286, 0.003379, 0.039885, -0.013898, -0.029889, 0.048384, -0.118980, -0.091514, 0.141822, -0.011854, 0.000214, -0.016538, 0.037895, 0.063477, -0.118775, -0.137122, -0.086022, 0.067082, 0.063733, 0.030225, -0.003954, 0.024128, -0.082002, -0.048826, -0.031926, 0.045659, 0.105135, 0.179274, -0.108111, -0.096712, -0.016622, -0.141890, 0.049596, 0.054811, 0.055206, 0.072648, -0.022705, -0.108544, -0.093877, 0.126009, -0.031764, 0.064340, 0.091063, -0.194329, 0.004336, -0.021274, -0.069213, 0.032834, 0.031319, 0.078988, -0.084385, -0.107784, -0.133902, 0.080114, -0.077000, 0.066807, -0.088950, -0.073132, -0.049850, -0.139337, 0.011469, 0.017383, -0.011418, -0.099727, 0.102635, -0.041106, -0.037975, -0.034534, 0.002536, -0.020100, -0.075047, -0.106218, -0.076331, -0.183121, -0.038108, -0.179668, -0.000209, -0.030966, -0.009641, 0.004537, 0.010176, -0.055894, 0.019389, 0.029494, 0.042358, 0.058944, -0.132443, -0.137853, 0.017691, -0.013426, 0.017328, 0.060994, -0.030758, 0.098592, -0.126962, 0.037907, 0.013477, -0.053146, -0.071356, -0.154505, -0.073113, -0.038255, 0.069969, 0.057342, 0.004783, -0.211731, -0.093098, 0.056953, -0.061336, -0.070461, -0.067892, -0.156607, -0.075643, 0.092065, -0.070951, -0.191615, -0.110507, 0.014920, -0.026773, 0.097690, -0.054223, 0.047464, 0.005225, 0.020999, 0.120912, -0.004732, 0.005636, -0.004531, -0.119636, -0.120211, -0.053225, 0.095820, -0.162010, -0.175420, -0.003385, -0.189358, -0.146759, 0.036363, -0.234399, 0.155601, -0.123397, 0.065953, 0.196625, -0.005653, -0.015884, 0.161091, 0.115924, -0.164195, -0.105068, 0.074130, -0.163910, -0.112674, 0.003948, -0.114110, -0.028266, -0.035529, -0.018263, 0.119095, -0.080985, -0.048839, -0.138270, -0.093016, 0.054552, -0.127884, -0.028782, -0.228550, 0.047622, -0.049210, -0.106734, 0.142676, -0.086889, -0.129000, -0.251693, -0.010004, 0.086895, -0.057646, -0.163757, -0.026519, 0.003471, 0.027450, 0.034710, 0.079952, -0.095190, -0.192429, -0.335038, -0.107302, 0.167718, 0.053575, 0.033704, -0.021320, 0.020183, 0.000840, -0.053357, 0.173747, -0.091237, -0.115602, -0.056315, 0.064523, -0.124167, 0.136655, -0.014325, 0.026232, 0.095648, -0.251295, -0.178398, -0.075158, 0.067408, 0.205129, -0.017464, -0.017064, -0.081622, -0.152050, -0.054174, 0.046867, 0.091659, -0.123285, -0.104067, 0.168616, -0.120649, 0.022476, -0.064978, -0.085698, 0.213564, -0.136970, -0.031538, -0.121172, -0.113090, 0.171168, 0.010495, -0.007483, -0.262019, 0.091589, 0.016544, -0.105890, -0.167926, 0.005993, -0.062530, 0.041716, -0.010820, 0.078426, -0.091217, -0.052818, 0.121608, -0.020094, -0.197270, 0.117206, 0.163612, 0.196670, 0.107267, -0.145472, 0.003430, -0.118751, -0.160445, -0.045824, -0.176921, -0.187454, 0.118447, -0.191405, 0.146009, 0.002299, -0.075943, 0.002819, -0.234511, 0.062537, -0.161140, -0.018995, 0.014460, 0.097518, -0.048375, -0.010085, 0.065402, -0.033466, 0.037598, 0.131260, -0.054924, 0.071152, -0.136739, -0.049918, -0.120070, -0.101356, 0.000440, -0.100886, 0.087834, 0.017225, 0.145338, 0.091280, -0.106395, 0.107993, -0.008914, 0.010160, 0.025223, 0.010873, 0.040302, 0.059417, -0.187925, 0.238337, -0.016797, 0.154713, -0.054175, 0.063638, -0.126405, -0.194996, -0.072430, 0.025935, 0.086584, -0.207899, -0.009348, -0.135691, 0.049701, -0.121201, -0.132409, 0.062200, 0.093983, -0.146945, -0.271116, 0.114431, 0.002998, 0.143722, -0.008234, -0.025278, 0.135029, -0.047323, 0.023307, 0.085782, 0.096204, -0.026970, -0.190659, -0.037893, -0.018793, 0.082692, -0.026183, -0.082277, 0.091460, -0.020023, -0.066820, 0.198661, 0.057076, -0.063245, -0.056406, 0.068875, 0.139615, -0.062891, -0.014834, -0.010750, 0.033766, -0.059607, -0.012058, 0.033141, -0.002501, 0.017563, 0.087868, -0.177791, -0.097952, -0.024497, -0.091563, -0.123635, 0.002899, 0.078125, -0.069001, 0.044674, -0.064664, 0.097428, 0.015876, 0.021208, -0.126683, -0.082569, 0.187656, -0.017327, 0.015101, -0.079818, 0.017808, 0.145289, 0.046474, 0.055957, -0.009158, -0.119027, -0.089367, -0.139373, 0.169804, -0.163840, 0.002291, -0.036234, 0.067487, 0.051369, -0.008134, 0.075348, 0.033861, -0.154349, -0.067341, -0.073665, -0.018846, -0.103509, 0.009965, -0.036861, -0.003891, 0.051575, 0.099547, -0.109519, -0.029569, -0.019267, -0.076132, -0.136685, -0.023407, -0.054575, -0.029637, 0.097657, 0.172953, 0.071850, -0.024491, 0.018166, 0.064897, 0.010254, -0.114444, 0.059617, -0.044307, -0.070055, -0.200571, 0.008876, 0.029373, 0.050303, 0.044682, -0.145425, 0.058648, -0.013716, -0.130367, 0.164050, 0.141011, -0.025993, -0.212629, -0.117225, -0.047044, -0.168418, -0.114971, -0.163060, -0.028594, 0.017051, -0.128238, -0.015909, 0.054228, -0.146429, -0.160660, 0.051900, -0.164169, -0.141196, -0.128994, -0.060546, 0.019371, -0.112509, 0.015752, 0.138087, -0.006151, -0.022123, -0.126333, 0.117431, 0.009300, -0.052842, 0.086209, 0.016731, -0.048495, 0.016819, 0.088272, -0.048882, -0.085141, 0.136892, 0.035316, -0.112368, -0.005250, 0.052977, 0.084588, -0.144209, -0.055722, 0.060604, 0.039959, -0.033209, -0.055434, -0.129612, -0.092887, 0.073250, 0.083208, 0.028723, -0.142761, -0.148779, -0.154042, -0.038216, -0.067246, -0.070163, 0.101459, -0.050551, 0.114180, -0.079780, 0.005939, -0.226026, 0.014638, -0.001745, -0.052677, 0.131284, 0.037278, 0.031378, 0.045255, -0.098775, 0.017700, 0.085961, 0.058255, 0.022563, 0.002234, 0.006310, -0.094025, -0.132018, 0.141500, -0.129614, 0.046845, -0.035465, -0.067970, 0.082954, -0.074580, -0.083963, -0.121134, 0.065554, -0.075909, -0.159822, 0.026621, -0.162135, -0.089607, -0.131333, -0.187549, -0.164315, -0.142288, -0.070055, 0.013472, 0.138422, -0.146853, -0.075003, -0.003991, -0.001428, -0.078729, -0.132958, 0.037681, -0.169211, 0.134973, -0.129639, -0.010855, 0.121519, 0.041647, -0.201006, -0.008176, 0.047346, 0.031384, 0.111486, -0.158202, -0.100548, -0.100763, -0.121858, -0.180137, -0.142810, 0.036009, 0.037860, -0.098222, -0.044776, -0.027983, -0.125489, 0.067862, 0.072094, -0.055004, -0.156578, -0.000913, 0.047968, 0.062252, -0.182284, 0.032975, -0.047339, -0.057420, -0.051438, -0.084315, -0.035432, 0.016183, -0.170387, -0.066501, -0.102816, -0.115471, 0.039420, 0.015434, -0.053496, -0.002469, 0.036823, 0.016562, -0.099548, 0.066192, -0.062328, -0.094244, -0.064501, -0.078087, 0.037531, 0.035431, 0.038410, 0.137963, 0.015233, 0.042617, 0.014638, 0.059297, 0.065398, -0.120460, 0.038505, -0.005286, 0.038647, 0.102578, -0.013238, 0.031927, -0.026432, -0.041499, -0.016034, -0.002526, 0.141229, -0.018009, -0.061088, -0.013162, -0.013895, -0.065679, -0.004541, 0.150430, 0.106224, 0.100064, 0.035396, 0.127913, -0.057896, -0.126534, -0.075412, -0.073882, -0.025330, 0.022475, -0.107486, 0.008992, 0.025133, -0.133448, -0.086445, 0.158946, -0.191628, 0.053068, -0.075933, -0.057957, 0.053249, -0.007455, -0.007982, -0.161220, -0.074870, -0.146129, -0.070356, 0.024316, -0.075169, 0.055306, -0.150521, -0.065095, -0.025127, 0.011838, 0.076482, 0.006026, -0.091584, 0.061019, 0.070615, 0.038338, -0.077526, 0.049299, 0.038859, -0.120834, -0.074027, -0.114690, -0.117595, 0.098781, -0.089812, 0.023860, 0.041710, -0.188638, -0.118036, -0.127667, -0.132159, -0.162593, 0.040136, -0.233512, -0.104145, -0.110916, -0.016650, 0.181034, 0.153303, -0.009807, 0.030965, -0.019812, 0.025424, 0.050539, -0.063904, -0.059425, 0.019760, 0.035841, 0.137572, -0.024871, 0.110770, 0.009340, 0.011259, -0.100735, 0.045252, 0.016501, -0.042066, 0.074246, -0.053277, -0.041039, 0.100094, -0.021001, 0.022456, -0.137572, -0.228364, -0.100517, 0.020402, 0.057131, -0.043475, -0.117623, -0.060273, 0.014411, 0.060933, 0.025865, 0.057253, -0.033334, -0.107424, -0.032085, 0.081378, -0.068515, 0.011429, -0.029991, 0.025194, -0.035970, 0.026124, -0.148143, -0.068239, -0.106571, 0.110034, 0.052318, 0.120862, 0.026025, -0.066855, 0.100385, -0.026926, -0.065359, -0.032752, 0.052409, 0.020703, -0.107552, 0.043137, -0.075955, -0.096376, 0.014468, 0.085207, 0.052437, -0.091405, -0.081316, -0.040297, -0.034297, -0.036168, 0.063108, -0.122650, 0.044754, 0.002304, -0.075492, -0.042458, -0.029940, -0.031007, 0.018412, 0.035412, -0.048413, -0.077161, 0.171392, 0.069167, -0.130395, 0.059284, 0.066314, -0.170054, -0.106317, -0.059526, 0.003591, 0.251196, 0.021145, -0.074264, -0.065049, -0.053373, -0.083594, 0.056950, 0.049422, -0.039032, -0.038219, -0.104715, -0.148722, -0.017772, -0.132209, 0.038525, 0.093393, -0.024685, -0.095190, 0.034949, -0.082250, 0.007563, 0.065809, -0.067707, -0.151882, -0.156591, -0.021641, 0.054960, -0.187485, -0.064177, -0.100553, -0.062667, -0.047350, -0.041468, 0.128128, -0.202505, -0.148775, 0.072997, 0.009233, -0.120681, 0.066233, -0.155665, 0.021198, 0.001570, 0.131582, -0.067530, -0.253775, -0.016644, -0.023652, -0.091072, 0.006496, -0.035619, -0.088641, 0.125746, -0.060969, -0.076542, 0.021472, -0.163551, 0.012965, 0.057747, -0.107531, -0.034727, 0.035108, -0.125531, -0.077660, -0.028376, -0.064677, -0.138644, -0.061645, 0.057367, -0.015045, -0.118227, 0.006632, 0.066991, -0.070494, 0.026968, 0.077553, 0.076121, 0.075482, -0.112887, 0.128298, 0.025715, 0.011663, 0.117558, 0.073161, -0.043474, 0.051797, -0.078561, 0.040663, -0.014328, 0.057074, 0.015195, 0.068515, 0.041436, -0.033243, -0.125625, -0.080097, -0.032969, -0.031471, -0.023321, -0.171959, 0.027462, -0.042881, -0.115719, 0.048167, -0.005611, -0.092472, 0.010721, -0.009542, 0.129377, -0.314902, -0.166710, 0.036527, -0.053709, -0.066249, -0.053179, -0.038646, -0.058725, -0.056897, 0.060130, -0.098212, 0.027382, 0.041749, -0.005404, 0.139368, -0.070036, 0.021176, -0.081982, -0.030814, -0.067904, -0.007592, -0.039968, -0.022834, 0.018850, -0.021040, 0.034185, 0.072766, -0.123296, 0.099178, 0.192149, 0.065247, 0.014606, -0.146015, -0.072250, -0.063003, -0.085597, 0.048946, -0.068509, 0.170015, 0.029578, -0.052739, -0.044319, -0.052831, -0.072432, -0.097740, 0.002572, 0.239383, -0.177907, 0.069783, 0.115637, -0.004213, -0.014742, -0.108752, -0.076624, -0.024037, 0.045915, 0.049331, -0.118195, -0.044757, 0.024966, -0.226744, -0.057132, 0.019469, -0.014157, -0.136193, 0.022543, 0.023882, -0.104650, -0.025113, 0.081868, -0.087850, -0.067063, 0.193722, -0.050255, -0.220868, 0.111281, -0.028540, 0.015512, -0.153411, -0.164567, 0.039119, 0.028117, 0.155732, 0.106688, -0.105823, -0.102634, 0.066230, 0.057871, -0.039744, -0.041893, -0.037435, 0.132572, -0.132310, 0.001275, -0.064972, 0.011660, -0.006734, -0.197565, -0.176355, -0.123977, -0.115179, 0.003902, 0.176156, -0.080324, -0.107447, -0.004974, -0.038673, -0.157721, -0.058795, -0.067144, -0.152867, -0.050865, -0.053499, -0.116791, -0.032997, -0.134311, 0.047576, -0.076580, 0.094853, -0.103547, 0.044363, -0.045329, 0.017643, 0.071835, 0.137520, -0.014539, 0.229747, 0.060607, 0.067057, -0.064977, 0.197861, -0.139136, 0.013242, -0.172583, 0.005071, -0.034245, 0.067994, -0.011637, 0.042699, 0.017774, -0.026526, -0.125675, -0.059675, -0.199595, 0.067518, 0.080794, 0.163051, 0.033396, 0.003074, -0.007225, -0.024161, 0.070134, 0.083027, -0.170746, 0.001161, -0.052965, 0.017462, -0.015315, 0.013105, -0.114333, -0.059012, -0.101845, -0.001814, -0.134400, -0.084250, -0.003620, -0.025012, 0.001603, -0.046553, 0.205141, 0.032678, -0.019733, 0.080921, -0.138712, 0.109964, 0.095913, -0.005872, 0.056958, -0.176035, 0.032663, -0.087759, -0.197889, -0.143425, 0.095746, -0.121719, 0.240303, -0.023382, 0.064747, -0.031995, 0.039506, -0.137032, -0.108929, 0.068741, -0.097709, -0.096646, -0.088554, -0.009410, -0.026183, -0.043619, 0.239864, 0.054490, 0.041377, -0.120459, 0.011957, -0.113200, 0.079043, -0.059448, -0.047080, -0.085029, -0.098863, 0.006846, -0.027085, -0.015105, 0.090940, 0.048788, -0.078675, 0.110280, -0.001689, 0.008104, -0.050419, 0.043139, -0.097571, 0.083423, -0.250586, 0.024945, 0.152725, -0.022765, -0.078996, -0.090958, 0.081867, -0.053712, 0.080180, -0.152143, 0.110272, -0.107792, 0.052169, 0.018987, 0.118064, -0.106088, -0.128130, 0.236584, 0.148400, -0.034127, -0.034334, 0.035779, 0.029855, -0.018736, 0.078301, -0.133053, 0.059870, -0.171473, 0.191458, -0.023061, 0.008394, 0.110350, 0.153810, -0.056259, 0.000073, -0.118085, 0.002663, 0.117235, -0.031076, 0.196844, -0.021425, 0.074382, 0.145450, 0.159653, 0.007526, 0.058384, -0.104344, -0.034867, -0.001566, 0.048821, -0.010430, 0.051139, 0.008444, -0.028201, -0.198706, 0.026201, -0.162111, -0.151912, 0.063789, -0.007710, -0.127514, 0.013429, -0.073081, -0.074757, -0.022904, -0.144219, -0.052227, 0.006019, 0.173355, 0.201484, -0.152671, 0.114755, -0.165108, -0.086728, 0.185419, -0.082965, -0.073626, -0.221274, -0.073992, -0.019977, 0.039560, -0.024339, 0.013489, -0.134856, 0.062730, -0.064152, -0.148281, -0.111116, 0.018925, -0.014714, -0.219768, -0.155980, 0.052730, 0.194621, -0.128651, 0.010870, 0.137559, -0.027527, -0.038958, -0.147820, 0.093422, 0.038802, 0.074026, -0.057050, 0.072045, -0.037902, 0.133550, -0.079082, -0.062591, -0.089089, -0.032806, 0.153758, -0.041794, 0.048734, -0.036622, -0.082242, -0.094795, 0.042122, -0.137585, 0.048118, -0.112825, 0.122775, 0.079178, -0.206854, 0.020149, 0.101420, -0.006324, -0.043785, -0.075270, -0.009642, -0.037193, -0.032697, -0.108055, 0.082510, -0.002385, -0.191423, 0.061455, 0.082604, -0.092830, 0.088732, -0.228770, -0.027647, -0.040018, 0.066545, -0.132211, 0.027668, -0.061484, 0.039195, 0.065301, -0.037781, 0.078838, -0.033650, -0.102812, 0.085937, -0.116900, 0.008399, 0.024675, 0.058285, 0.150340, 0.022809, 0.131543, -0.016561, 0.067914, -0.144808, -0.093217, -0.248616, -0.031464, 0.041719, -0.075194, 0.004671, 0.065309, -0.072983, 0.067337, 0.153160, -0.075461, 0.128123, -0.118466, 0.006387, -0.157151, -0.016019, 0.015656, 0.053476, 0.047681, -0.006435, -0.091541, 0.084525, 0.000550, 0.075407, -0.097284, -0.027869, -0.023929, -0.015650, 0.066922, -0.057178, 0.010370, -0.086485, 0.048261, -0.065205, -0.127550, 0.017343, 0.042904, 0.075875, -0.017613, -0.073255, -0.021168, 0.004750, 0.024684, 0.041517, -0.099496, 0.156681, 0.079225, -0.006608, -0.132691, -0.007190, 0.042543, 0.132833, -0.034591, -0.153601, 0.027585, 0.126206, -0.041198, 0.017577, 0.013800, -0.243023, -0.036976, -0.147907, 0.022502, 0.017759, 0.058687, 0.045971, -0.071215, -0.165310, -0.042600, 0.060682, -0.007190, 0.109656, -0.088616, 0.066010, -0.142707, 0.061310, 0.072281, -0.090593, 0.084411, -0.038661, -0.029283, -0.074335, -0.109965, -0.021439, 0.120213, 0.019741, 0.013482, -0.053290, -0.113984, -0.103670, -0.095839, 0.071889, -0.195185, 0.024484, -0.177553, -0.069049, 0.038803, -0.129973, -0.054953, 0.002032, 0.080458, 0.027254, 0.089119, 0.007423, -0.108996, 0.080172, -0.011013, 0.131881, -0.122388, -0.110602, 0.023705, 0.090850, -0.208262, -0.019697, 0.042825, 0.141271, 0.022694, 0.006106, -0.058922, 0.001035, 0.069052, -0.073421, 0.026288, 0.129098, -0.035912, -0.086565, 0.002898, 0.095627, 0.028191, 0.089555, 0.112588, -0.076859, 0.126269, 0.064153, 0.159779, 0.182998, 0.037591, -0.161526, -0.003563, 0.016291, -0.024577, 0.028669, -0.041164, 0.160945, 0.052448, -0.165686, 0.037258, -0.194662, -0.127013, -0.050219, 0.020154, 0.056485, -0.095881, -0.069798, 0.052544, 0.024553, -0.172963, -0.022034, -0.076781, 0.071056, -0.083179, -0.127061, 0.028078, 0.067420, 0.009452, -0.122298, -0.159336, -0.074594, 0.050125, 0.146413, -0.009151, 0.012138, -0.210535, -0.039050, -0.055098, -0.069339, 0.043134, -0.055475, -0.091701, 0.044188, -0.115898, -0.167353, 0.005349, -0.084676, 0.058613, 0.051580, -0.049104, -0.195686, 0.046061, 0.138729, -0.085752, 0.060006, 0.044214, 0.056233, 0.051294, -0.074079, 0.098999, 0.028257, -0.163305, 0.060015, -0.071370, -0.078753, 0.023233, -0.100370, 0.159353, -0.120710, -0.024310, 0.168393, -0.078548, 0.152153, 0.025569, 0.076498, -0.038862, -0.124236, -0.083165, 0.001088, 0.036207, -0.071775, 0.129587, 0.076245, 0.047402, -0.067018, -0.044365, -0.084646, -0.000458, -0.068487, -0.045076, -0.091384, -0.026163, 0.010316, 0.125343, 0.090480, -0.141738, 0.093856, 0.117902, -0.195080, 0.013361, -0.169830, -0.005161, 0.086882, -0.115948, 0.132784, -0.002399, -0.147812, -0.083117, 0.157890, 0.045957, 0.091637, 0.066644, 0.065287, 0.034196, 0.018225, 0.101485, -0.114197, 0.058335, -0.103136, -0.068404, 0.009706, -0.044726, 0.098902, 0.096992, 0.119173, 0.045899, 0.015881, 0.077533, -0.273007, -0.035418, -0.112743, -0.041535, -0.007489, 0.142444, 0.036269, 0.058695, 0.068594, -0.065728, 0.096718, 0.143582, -0.106129, -0.115722, 0.047475, 0.163640, 0.044323, -0.082834, -0.088041, 0.023233, -0.162284, -0.118916, -0.035771, -0.118052, 0.052173, -0.073284, -0.168667, 0.117559, 0.061235, -0.120494, 0.186222, 0.048604, -0.050910, 0.017604, -0.134775, -0.168928, -0.003767, -0.147812, -0.079877, -0.016403, -0.068491, 0.000697, -0.038978, 0.048387, -0.097432, -0.062391, 0.039436, -0.080469, 0.019443, -0.113932, 0.085951, 0.059092, -0.081567, -0.165742, 0.044567, 0.131742, -0.133852, 0.045313, 0.148680, -0.032151, -0.056011, 0.207353, 0.133599, 0.071612, 0.064819, -0.018460, 0.106999, 0.131887, 0.074731, -0.097311, 0.035519, 0.045520, 0.092833, -0.099978, -0.130650, 0.023953, -0.056899, 0.009177, -0.129616, -0.092365, 0.047624, 0.067543, -0.092664, -0.015174, -0.134233, 0.002297, 0.066400, -0.029113, 0.143665, 0.104415, -0.060941, -0.151729, 0.009839, 0.056560, -0.025181, -0.117684, -0.022493, 0.080333, -0.159907, -0.005099, 0.094839, -0.087290, -0.140698, -0.000367, 0.149737, 0.144172, 0.133051, -0.082411, -0.063652, 0.099924, 0.124701, -0.001797, 0.093651, 0.123508, 0.125006, 0.110055, -0.027895, -0.035091, 0.078658, 0.099775, -0.086050, -0.111421, -0.023588, 0.031340, -0.064775, 0.053652, -0.119573, -0.013659, -0.014258, 0.039730, -0.058016, 0.051129, 0.082329, -0.070170, 0.033254, 0.044419, -0.037483, 0.069933, -0.035024, 0.027979, 0.029418, -0.024486, 0.031533, -0.059984, -0.029495, -0.005961, 0.033896, 0.064093, -0.075987, 0.171075, 0.097372, -0.111762, -0.151643, -0.027895, -0.040761, -0.000503, -0.062196, -0.056921, -0.330974, 0.014505, 0.055992, -0.036508, -0.008633, -0.185781, 0.016223, -0.161294, -0.157561, 0.089492, 0.042999, -0.058113, -0.003188, -0.283790, 0.112561, -0.102481, -0.112580, 0.006958, -0.116324, -0.031820, -0.136642, 0.029959, -0.026738, 0.070668, -0.059104, -0.073443, -0.101230, -0.088685, 0.003661, -0.080694, -0.132881, 0.095398, -0.146257, -0.115622, -0.013249, 0.026092, -0.069178, -0.127046, -0.043324, 0.028828, -0.211568, 0.005607, -0.188469, -0.289551, 0.000417, 0.014788, -0.035365, 0.035487, -0.087928, -0.045958, -0.032260, -0.113698, -0.098639, -0.039199, -0.044237, 0.012469, 0.086750, -0.053289, -0.090615, -0.186633, -0.056685, 0.022120, -0.077370, 0.051863, -0.240933, 0.082190, -0.126032, 0.064799, 0.002649, 0.129436, -0.052285, -0.010037, 0.124354, -0.061666, -0.267661, -0.150661, -0.041209, -0.025323, -0.026121, -0.097257, -0.032018, -0.034155, -0.025936, -0.093527, 0.047078, -0.129505, -0.047494, 0.130361, -0.139470, 0.080229, -0.060805, -0.056365, 0.146227, -0.190216, -0.057980, 0.031549, -0.117045, 0.160132, -0.118904, -0.088474, 0.008180, 0.075009, -0.058351, -0.060809, -0.133623, 0.110935, 0.125114, -0.140403, 0.011411, -0.138081, -0.142995, -0.032833, -0.039434, -0.026352, -0.136384, 0.032903, 0.012650, -0.308390, 0.185199, -0.085637, 0.026933, -0.067993, -0.131782, 0.102822, -0.153537, -0.115749, 0.040235, 0.133702, -0.169056, -0.059073, -0.277339, -0.102706, -0.156584, -0.240170, -0.029461, -0.075329, -0.251440, -0.069450, -0.033159, -0.081999, -0.163114, -0.102687, -0.124943, 0.092977, 0.022920, -0.069342, 0.002232, -0.040326, 0.153809, -0.130089, -0.026396, -0.093361, 0.039298, -0.105377, -0.315281, 0.164820, 0.004031, 0.012883, -0.040759, 0.008222, 0.027992, 0.020964, -0.209888, -0.155422, -0.200176, -0.131368, -0.018019, -0.124899, -0.058230, -0.112711, -0.059140, -0.237788, -0.088474, 0.034940, -0.012130, 0.078058, 0.004628, -0.089582, 0.116101, 0.000696, -0.030738, -0.042328, -0.132943, -0.059423, -0.046025, -0.078194, -0.043837, -0.082817, 0.057727, 0.055392, -0.195603, 0.028100, -0.139253, 0.014586, -0.135867, -0.064916, -0.097258, -0.095752, -0.054062, -0.033443, 0.022375, -0.017890, 0.015159, -0.035874, 0.012273, -0.155043, 0.037483, -0.203850, -0.111284, -0.164942, 0.095922, -0.011614, -0.157923, 0.021892, -0.220811, -0.007546, -0.024257, -0.100643, -0.047353, -0.138796, 0.011245, 0.087954, -0.037694, -0.059297, 0.085005, 0.045213, -0.025695, -0.021986, 0.002102, 0.024132, -0.047023, -0.037423, -0.070252, -0.091403, 0.145492, 0.036642, -0.045241, -0.096047, -0.026318, -0.154671, -0.022505, -0.081902, 0.077316, 0.029682, 0.035480, -0.118760, 0.042672, 0.039897, -0.199259, -0.113181, -0.205996, -0.160947, -0.142909, -0.060035, -0.005849, 0.026310, -0.178451, 0.015001, 0.018644, -0.110623, -0.003002, -0.102807, -0.037157, -0.055209, -0.024863, -0.097015, -0.149843, 0.017084, -0.163863, 0.117417, 0.055878, -0.134927, -0.015876, 0.109247, 0.027818, 0.067025, 0.079880, -0.126646, 0.016214, -0.053436, 0.083336, 0.085534, -0.000234, -0.054731, 0.077793, -0.092114, 0.057377, -0.042151, -0.005801, 0.012823, -0.093449, 0.001940, -0.052603, 0.143946, -0.066555, 0.060514, -0.167786, -0.028155, -0.156056, 0.029779, 0.008303, -0.006761, 0.033066, -0.093040, -0.119735, -0.113453, -0.022104, -0.025025, -0.037459, -0.171040, 0.080499, -0.126266, -0.045157, -0.168679, -0.111938, -0.016675, 0.063782, 0.005406, 0.099986, -0.022402, 0.008125, -0.101330, -0.206955, -0.121546, -0.125234, -0.144563, -0.033113, -0.071047, -0.030959, -0.056913, -0.012347, 0.063898, -0.034743, -0.137032, 0.024835, -0.036500, -0.203814, 0.032021, -0.083384, -0.073691, 0.050948, -0.093061, -0.011942, 0.000486, -0.074211, -0.058869, 0.051482, 0.031577, -0.097581, -0.087062, 0.009044, -0.007028, 0.011158, -0.124115, -0.040533, -0.094767, -0.222709, -0.204191, -0.107221, 0.128627, 0.224336, -0.088047, 0.044040, -0.105925, -0.013617, -0.104750, 0.053604, -0.037032, 0.083856, -0.103314, -0.003621, -0.131480, -0.081529, -0.123573, -0.097537, -0.118836, -0.088510, -0.035905, -0.128614, -0.045305, -0.003211, -0.086610, -0.139666, 0.091535, 0.082297, 0.062037, -0.068621, 0.090828, -0.064679, -0.105417, -0.053828, 0.025067, 0.086193, 0.054229, -0.211636, -0.049141, 0.046067, -0.101703, -0.099591, 0.008989, 0.208972, -0.058648, -0.109949, 0.010919, -0.235974, -0.077002, -0.071980, -0.033240, 0.011447, -0.128901, 0.096414, 0.183511, -0.087166, -0.085418, 0.069887, -0.145248, -0.098418, -0.100449, 0.098008, 0.066641, -0.122641, -0.109226, -0.104513, 0.019271, -0.027931, 0.039132, -0.069807, -0.125331, 0.007823, -0.040342, -0.125495, -0.041266, 0.055823, 0.092756, 0.005190, 0.069785, -0.046576, 0.058422, 0.104604, 0.061070, -0.107155, 0.034627, -0.108379, -0.190316, 0.135612, -0.010529, -0.078953, -0.113719, 0.013885, -0.128915, -0.038474, 0.009074, 0.052631, -0.018866, -0.099766, -0.009775, -0.042780, -0.145475, -0.034242, -0.080321, 0.024256, -0.108177, -0.078581, -0.019455, -0.171411, -0.091513, 0.209811, 0.007296, -0.223048, -0.054460, -0.072548, -0.025331, -0.035643, 0.045503, -0.120112, 0.022687, -0.041729, -0.051038, -0.039615, -0.193440, -0.034379, -0.165594, -0.117537, -0.197173, -0.151310, -0.028055, 0.032142, 0.055974, -0.106745, -0.176636, 0.027006, 0.038049, -0.047939, 0.067243, 0.030063, -0.037881, -0.080777, -0.059986, -0.027528, -0.180707, 0.058656, -0.008119, 0.186755, -0.082359, 0.124310, -0.106167, -0.183901, -0.105287, -0.050602, -0.291256, -0.083262, 0.047158, -0.090595, -0.009354, 0.159857, 0.022869, 0.000917, 0.004094, -0.125580, -0.196968, -0.095644, -0.078392, 0.036621, -0.090942, -0.089368, 0.010287, 0.040911, -0.050665, -0.099601, 0.077311, 0.027811, 0.064816, -0.136068, 0.139507, 0.039980, -0.052498, 0.029641, 0.011802, 0.077169, -0.019182, -0.048934, -0.047948, 0.055523, -0.240907, -0.138982, -0.139937, 0.092059, 0.005746, 0.121973, 0.069862, -0.044274, 0.009143, 0.013576, 0.006125, 0.097660, -0.283747, -0.209341, -0.043004, 0.045236, 0.069107, -0.088427, 0.018449, -0.241891, -0.090693, -0.138023, 0.013242, -0.068212, 0.073601, -0.144506, 0.073465, -0.139425, -0.116659, -0.070787, -0.008554, -0.001372, -0.097253, -0.058570, -0.167707, 0.107940, 0.050328, -0.122016, -0.145740, -0.062609, -0.015225, -0.042834, 0.170373, -0.125054, -0.160772, -0.019473, -0.011916, -0.033769, -0.067226, -0.007766, 0.090280, -0.038743, -0.070850, 0.111826, -0.023796, -0.073279, 0.003484, -0.123064, 0.018982, -0.108684, -0.037657, -0.109554, -0.045920, -0.115764, 0.051223, -0.046977, -0.052551, -0.085054, -0.026176, -0.153162, -0.163562, 0.029114, -0.053520, -0.131781, 0.112847, 0.013575, -0.120867, -0.092601, 0.058682, 0.041945, -0.225904, 0.095402, -0.035688, -0.050114, -0.025210, 0.030101, -0.030115, 0.071996, -0.130801, 0.104522, 0.074208, -0.022812, -0.168959, -0.062704, -0.123864, 0.020413, -0.205946, -0.081331, -0.128027, -0.148407, -0.029455, 0.013529, 0.038976, 0.103316, -0.117361, 0.110193, -0.003031, 0.017274, 0.022609, 0.090701, -0.061947, 0.081513, -0.031640, -0.095404, -0.120424, 0.116564, -0.055237, 0.034824, 0.041022, -0.142834, -0.123244, -0.101064, 0.031001, -0.003181, -0.009677, 0.031714, 0.081784, -0.115573, -0.059286, -0.076962, -0.092415, 0.083122, 0.035238, -0.119148, -0.045843, -0.111313, 0.003361, -0.036940, 0.041928, -0.033920, 0.005243, 0.161518, -0.133713, -0.107810, -0.013842, 0.042239, -0.050240, -0.009942, -0.140875, -0.077962, -0.064066, -0.155032, 0.002694, -0.067716, -0.111364, -0.096614, 0.049908, -0.018387, 0.022117, -0.087767, -0.057742, -0.249950, -0.404029, -0.030987, -0.146365, -0.072428, -0.060754, -0.253104, -0.072711, -0.075650, -0.069412, 0.103105, -0.080384, -0.062607, -0.053561, -0.151231, -0.146169, 0.141473, -0.069679, 0.082209, 0.072563, -0.140807, -0.197798, -0.078638, -0.067482, -0.025578, 0.020232, -0.108368, -0.096009, 0.062425, -0.001265, 0.011628, -0.029279, 0.003690, -0.052461, 0.003654, -0.212724, -0.135171, -0.034176, 0.003913, 0.051528, 0.160232, -0.071372, -0.027640, 0.047018, -0.222003, 0.077678, 0.040101, 0.025710, -0.051502, 0.102754, -0.183327, 0.230094, -0.103791, -0.017950, -0.110133, -0.115620, -0.089205, 0.044010, -0.160656, -0.044631, -0.014066, -0.034984, -0.108490, 0.092778, -0.157460, 0.108773, -0.010499, 0.172993, 0.025566, -0.047663, -0.068401, -0.063880, -0.061531, -0.052073, 0.003184, 0.122894, 0.024199, -0.031167, -0.110054, -0.001847, 0.078525, -0.213086, -0.125073, -0.057582, 0.027851, -0.063991, -0.177390, 0.150160, 0.169934, -0.047770, 0.020972, 0.022142, -0.136097, 0.030945, -0.213219, -0.019003, -0.051223, -0.110276, -0.050912, -0.081939, -0.054116, -0.081214, -0.195780, -0.111825, -0.120425, -0.001497, -0.196042, -0.096759, -0.046516, 0.036125, -0.093075, -0.039457, -0.058748, -0.089228, 0.041119, -0.183880, -0.031203, 0.088522, 0.104324, -0.152806, 0.208652, 0.154008, -0.048479, -0.053163, 0.038033, -0.038239, -0.041711, -0.106097, -0.061641, 0.075893, -0.054235, -0.015551, 0.036950, 0.004684, -0.020378, -0.105345, -0.102548, -0.012891, 0.022730, -0.051507, -0.030914, -0.032270, -0.190488, -0.003415, 0.091554, -0.080116, -0.084885, -0.107405, -0.163357, -0.165116, 0.029349, -0.074412, -0.016617, 0.034014, -0.073233, 0.069844, -0.103312, -0.125821, -0.227593, -0.055248, -0.024878, 0.048168, 0.029524, -0.149570, -0.077667, 0.016792, 0.014795, 0.044661, 0.102830, -0.019020, 0.057727, 0.042373, -0.194784, -0.078137, 0.013874, -0.134571, -0.144024, 0.083011, -0.118330, -0.166605, -0.148850, -0.354237, -0.021149, 0.140367, -0.230823, -0.120628, -0.135702, 0.036596, 0.056655, -0.058366, 0.007183, -0.113938, -0.161364, -0.167124, -0.061334, -0.079468, -0.099890, -0.113397, -0.109680, -0.148189, -0.083978, 0.043200, -0.096755, -0.132222, -0.052810, 0.073243, -0.118705, -0.054610, -0.041336, 0.012539, 0.032622, -0.065444, 0.074664, -0.036939, -0.099833, 0.092368, -0.025407, -0.066949, -0.112678, 0.020089, 0.177919, 0.098682, -0.020289, -0.161415, 0.049939, -0.109872, 0.061725, 0.118122, -0.038285, -0.161179, 0.055812, -0.094701, -0.131986, 0.000466, 0.111665, 0.001596, -0.030231, -0.117810, 0.068117, -0.389480, -0.010836, -0.209171, -0.141422, -0.055193, -0.229727, -0.035104, -0.095660, 0.115707, -0.086791, 0.058180, -0.093619, 0.148127, -0.100919, -0.061794, -0.151518, 0.052623, -0.016048, -0.126933, 0.013116, 0.057105, -0.157348, -0.167042, -0.071960, -0.295957, -0.078734, -0.034170, 0.034289, -0.068071, 0.063896, -0.015239, 0.029679, -0.121732, 0.074485, -0.124483, 0.055538, -0.088048, -0.148653, -0.148786, 0.077783, -0.039465, 0.066607, -0.047082, 0.218696, -0.101927, -0.146325, 0.018054, 0.040616, -0.066027, 0.126605, 0.055040, -0.057195, 0.051524, -0.053999, 0.059755, -0.196759, -0.198131, 0.136743, -0.128796, -0.116560, -0.123655, -0.064663, -0.182099, -0.073187, 0.057066, -0.059876, -0.186620, 0.004194, 0.024385, -0.100427, 0.066598, -0.112768, 0.138287, -0.220866, -0.060256, -0.015224, 0.043732, 0.156147, -0.003610, -0.005256, -0.094841, -0.005304, -0.111463, 0.020349, 0.044272, -0.073969, 0.059760, -0.008064, -0.054724, 0.057083, -0.043335, -0.038643, -0.097182, 0.108132, -0.034154, 0.159665, 0.009355, -0.168645, -0.051704, -0.041225, -0.061538, 0.005697, -0.103109, -0.081605, 0.010629, -0.110609, -0.055867, 0.121522, -0.121942, 0.057804, 0.003777, -0.069485, 0.011980, 0.081867, -0.039687, 0.059028, -0.059658, 0.031176, -0.067510, -0.051672, 0.057875, 0.113158, 0.000754, -0.111254, -0.049635, -0.023181, -0.034778, 0.008992, -0.101643, 0.027176, -0.018160, -0.129376, -0.007044, 0.141083, 0.165707, -0.025046, 0.073884, -0.173783, 0.054294, -0.038023, 0.024366, -0.123977, -0.062625, -0.056799, 0.088956, -0.063130, -0.052550, -0.025273, -0.019012, 0.065259, -0.105049, -0.120125, -0.065944, 0.078764, -0.063077, -0.097489, 0.067107, 0.088185, -0.189830, -0.229324, -0.055581, 0.019841, -0.144098, -0.016770, -0.004263, -0.023567, -0.014049, 0.043917, 0.014499, 0.079846, -0.111170, 0.038934, -0.052659, 0.073643, -0.019298, 0.000168, -0.082789, 0.009268, -0.127910, 0.006000, -0.048993, -0.061357, 0.072547, -0.010597, 0.009002, 0.107096, -0.053144, 0.005752, 0.070420, -0.066860, 0.033131, -0.143614, -0.021828, -0.107915, -0.076512, 0.104527, -0.092807, 0.021723, -0.120802, 0.031273, -0.121354, -0.052740, 0.036376, 0.075518, 0.107145, -0.118919, 0.020815, -0.024484, -0.023267, -0.064083, -0.120193, 0.014700, 0.037170, 0.030620, -0.057052, 0.046440, -0.011608, 0.025061, -0.015121, 0.037365, 0.086973, -0.111984, 0.092766, -0.068833, 0.062362, 0.019851, -0.024905, -0.136386, -0.057594, -0.127203, 0.102308, -0.179121, 0.025646, -0.161674, 0.042172, -0.089339, 0.016387, 0.032825, 0.059582, 0.091298, -0.138461, -0.033707, -0.165972, -0.196156, -0.074439, 0.093994, -0.080662, -0.020863, -0.113671, 0.060983, 0.036472, -0.123035, -0.165540, 0.040381, -0.084947, 0.047534, 0.179812, -0.045855, 0.170211, 0.157748, -0.061987, 0.019128, 0.009146, 0.002058, -0.018923, 0.022114, 0.066733, -0.081776, 0.027223, -0.044211, -0.036465, 0.185767, 0.023922, -0.061111, -0.115233, 0.062234, -0.006498, -0.073598, -0.001204, -0.232634, -0.020473, 0.088411, 0.004240, -0.066343, -0.078447, -0.100859, -0.136248, 0.015320, -0.017964, 0.091984, -0.036878, -0.235961, 0.090018, -0.056764, 0.023565, -0.025739, -0.020281, 0.001504, -0.259082, 0.001180, -0.090385, -0.029754, 0.009561, 0.131493, -0.083524, -0.126946, 0.072839, -0.071890, -0.086984, -0.077749, -0.067903, -0.052821, -0.016187, 0.090745, 0.061580, 0.009418, 0.060103, 0.042592, -0.102485, 0.031276, -0.059654, -0.108145, -0.096573, -0.078747, -0.087043, -0.168885, -0.062120, -0.025944, -0.112890, -0.039501, -0.021113, 0.013483, 0.060808, -0.104816, 0.047797, 0.031158, 0.060076, 0.028142, -0.126616, -0.109990, -0.131040, -0.012514, -0.124861, -0.074998, -0.061571, -0.027523, 0.053477, -0.146815, -0.092301, -0.035604, -0.089934, -0.139329, 0.022943, -0.076867, -0.113450, 0.010409, 0.001736, 0.016330, 0.038294, 0.048388, -0.139871, -0.000719, 0.037420, -0.014403, 0.042261, 0.081328, 0.101609, 0.040780, -0.057332, -0.157130, 0.173619, -0.067125, 0.023265, -0.025238, 0.038872, -0.134102, -0.080613, -0.130309, 0.071321, -0.071233, -0.019210, -0.004254, 0.038617, -0.073750, -0.102487, -0.115753, -0.148662, -0.008889, -0.094370, -0.069168, 0.073174, -0.029669, 0.024503, 0.074689, 0.032607, 0.104649, -0.044263, 0.059584, 0.048603, 0.205938, -0.042374, -0.101070, -0.012017, -0.024295, -0.007738, -0.096439, 0.088546, 0.081982, 0.213603, -0.195858, 0.030802, 0.073155, 0.050617, 0.070126, 0.028275, -0.104473, -0.139720, 0.042989, 0.095888, 0.025599, 0.126689, -0.047630, 0.171674, 0.001608, -0.030202, -0.048715, -0.107650, 0.078652, 0.064910, 0.150963, 0.044346, -0.236689, -0.166603, 0.011557, 0.028269, 0.020971, -0.091153, -0.081443, -0.200198, 0.006479, -0.107009, -0.065909, -0.139722, 0.073990, 0.080846, 0.107731, -0.028531, 0.024136, -0.080429, -0.065560, 0.035005, 0.037238, 0.106520, -0.118427, 0.160374, 0.072644, 0.074262, 0.039754, -0.040897, -0.056887, -0.116201, -0.123065, -0.082067, -0.149158, 0.143460, 0.026940, -0.116097, -0.030477, 0.049275, -0.082040, 0.012777, -0.131263, 0.088732, -0.012086, -0.076023, 0.048771, -0.153118, -0.114197, -0.156603, 0.065479, 0.131993, -0.053664, 0.082953, -0.073494, 0.076493, -0.069863, -0.123426, 0.034565, -0.076753, -0.013982, -0.087931, -0.027184, -0.145931, -0.042212, -0.073043, 0.060277, -0.165524, -0.056325, 0.056671, 0.061145, 0.075738, -0.180033, 0.052600, 0.189218, -0.152602, -0.166874, -0.066490, 0.013671, 0.061756, 0.084575, -0.082671, -0.129206, 0.208485, -0.123320, -0.141993, 0.083678, -0.075610, -0.081373, -0.001964, 0.064513, 0.044300, -0.001235, 0.053514, -0.041669, -0.036280, 0.098427, 0.020601, -0.031054, 0.028637, -0.131600, 0.059919, -0.100427, 0.067431, 0.000596, 0.004466, 0.146659, 0.075841, -0.021436, -0.024107, -0.108212, -0.011323, -0.047685, -0.062694, 0.039604, 0.039600, -0.111623, 0.025345, -0.055238, 0.026640, -0.004225, 0.061585, 0.073656, -0.019384, 0.142653, -0.037647, -0.045780, -0.080417, -0.096711, -0.029979, 0.025470, -0.013088, 0.183163, 0.127820, 0.052134, -0.133734, -0.119828, -0.029864, -0.060990, 0.044486, -0.078620, -0.024878, -0.083129, 0.104036, -0.086215, 0.070821, -0.009084, 0.142012, 0.156385, -0.171795, -0.039296, -0.011877, 0.084781, 0.057474, 0.021367, -0.094050, -0.148175, 0.043327, -0.048877, 0.043399, -0.116454, -0.066121, -0.055067, 0.104682, 0.163119, -0.119757, 0.153878, -0.032269, -0.088453, -0.030632, 0.063780, 0.000341, -0.037530, -0.015678, -0.010097, -0.073062, -0.099273, -0.060789, 0.029258, -0.018211, 0.056033, -0.037817, -0.110193, -0.044650, -0.034709, -0.242480, -0.103599, -0.002857, -0.092957, -0.071846, 0.164591, -0.136080, -0.003917, 0.148538, 0.039432, 0.005217, 0.006280, -0.105234, -0.027021, -0.231378, -0.128732, 0.114081, -0.069845, 0.104970, -0.040116, -0.187937, 0.010303, -0.201239, -0.181151, 0.062788, -0.030400, 0.024192, -0.086029, -0.021977, -0.001824, -0.059366, 0.077257, 0.052586, -0.010066, -0.261479, -0.017243, -0.096858, -0.115455, -0.130517, 0.059575, -0.111235, 0.029912, -0.160074, -0.067987, 0.032968, -0.118360, -0.281927, 0.006104, 0.101565, 0.084086, 0.032211, 0.177986, 0.100935, -0.069298, 0.044844, 0.008318, -0.125508, 0.032770, 0.021770, -0.068913, 0.008069, -0.014594, -0.013691, 0.069364, -0.034967, -0.081574, 0.012978, -0.061151, -0.068572, 0.022141, 0.047905, -0.094759, -0.048792, -0.106624, -0.282648, -0.078797, -0.015901, -0.062440, 0.143288, -0.144040, -0.244868, -0.027195, -0.146923, -0.007910, -0.028992, -0.033442, 0.083749, -0.081980, 0.020252, 0.073143, -0.128464, -0.100074, -0.075401, 0.040149, -0.047994, -0.004953, 0.086936, -0.108151, 0.000007, -0.211767, 0.000863, -0.025687, -0.041811, -0.086540, -0.081219, -0.010120, -0.185070, -0.092976, 0.121783, -0.134851, -0.061693, 0.036709, -0.048452, 0.008359, -0.039270, 0.024104, -0.077773, -0.014128, -0.050781, -0.094788, 0.128016, 0.084162, -0.097619, -0.133667, -0.027683, 0.003173, -0.038315, -0.127990, -0.098593, -0.134002, -0.080821, -0.150475, 0.013243, 0.180392, -0.101063, -0.063447, 0.054778, -0.124957, -0.149130, -0.028406, -0.033197, -0.071766, -0.023737, 0.129630, 0.154663, -0.139058, -0.103449, -0.022624, -0.017636, -0.049942, -0.109726, -0.081020, 0.157948, -0.009723, -0.003254, -0.109720, -0.118293, -0.002897, -0.207838, -0.177746, -0.060274, -0.113474, -0.066450, -0.033715, -0.106370, 0.050591, -0.109252, -0.001791, -0.023642, -0.125515, -0.158358, -0.120231, 0.081733, 0.144655, -0.108028, -0.048122, -0.091661, 0.101862, 0.029320, -0.107805, 0.027723, -0.076489, -0.001322, -0.131859, -0.064155, 0.042623, 0.013979, -0.107023, 0.015584, -0.017210, -0.008751, -0.067163, -0.145952, 0.086046, -0.010275, -0.037842, -0.153456, -0.029945, -0.100356, -0.121449, -0.044256, 0.009396, -0.022782, 0.051113, -0.169155, -0.167747, -0.116693, -0.212301, -0.358594, 0.036895, -0.122653, -0.134577, -0.063230, 0.114199, -0.051756, 0.048781, -0.156885, -0.125464, -0.197703, -0.075396, -0.130035, -0.087249, 0.000550, -0.136167, -0.111565, -0.159015, -0.098005, -0.101535, -0.042105, -0.014777, -0.245145, 0.074903, 0.002716, 0.019414, 0.001091, 0.122359, 0.176440, 0.051469, -0.055881, 0.037340, -0.158272, 0.047847, -0.241522, 0.080232, -0.043366, 0.041007, 0.030317, -0.065132, -0.145010, -0.163012, 0.075438, -0.011122, -0.134859, -0.081078, 0.017925, 0.045803, -0.115851, 0.099408, 0.050047, -0.109664, 0.098941, 0.090264, 0.092266, -0.158222, 0.061245, 0.162190, -0.096535, 0.043904, -0.110846, -0.095636, -0.034788, 0.069044, -0.049934, -0.048823, -0.060150, -0.023812, -0.166272, 0.013419, 0.145833, -0.217301, -0.019545, -0.035568, 0.123773, 0.051194, 0.019890, -0.090114, -0.070661, -0.248855, 0.102732, -0.075836, 0.024860, 0.095107, -0.060794, -0.193302, -0.068863, -0.087854, -0.141927, -0.149679, 0.063718, -0.151452, 0.014585, 0.034931, 0.088642, -0.221427, -0.108577, 0.005358, -0.130151, -0.090404, -0.019443, -0.163885, 0.066872, -0.029056, -0.288585, -0.164653, 0.050302, -0.049633, -0.036391, 0.039832, 0.207236, -0.077583, -0.084813, -0.031877, -0.112793, 0.056873, 0.126332, -0.134284, -0.275617, 0.009743, -0.111099, -0.078352, -0.080592, 0.044980, 0.089160, -0.061798, -0.032594, -0.013215, -0.036046, 0.041346, -0.095473, -0.010611, 0.004900, 0.063249, -0.062402, 0.025476, -0.004861, -0.096544, -0.011546, -0.060325, 0.195116, 0.054468, -0.064079, 0.055890, -0.035914, -0.072055, 0.138405, -0.087291, -0.044778, -0.097859, 0.100209, 0.037078, 0.095477, -0.053249, -0.167719, 0.099746, -0.112250, -0.212256, 0.029107, -0.153492, -0.230159, -0.030014, 0.002156, 0.113195, -0.036298, -0.014107, -0.173704, -0.044473, -0.155862, -0.060472, 0.064478, 0.047712, -0.098227, 0.030374, 0.045742, -0.081369, 0.047294, -0.038726, -0.062619, -0.069899, -0.164217, -0.065875, 0.077497, 0.088128, -0.083034, -0.059700, -0.131472, -0.054484, -0.114116, -0.182593, 0.142773, 0.074675, 0.111072, -0.064121, 0.075457, -0.005635, -0.024853, 0.096848, -0.138742, 0.035129, 0.022633, 0.132991, 0.085112, -0.115220, 0.037029, -0.143307, 0.042942, -0.064224, -0.099072, -0.123119, -0.072526, -0.024651, -0.067044, -0.062592, -0.077242, 0.148293, -0.047216, -0.032999, 0.047752, -0.012969, -0.074900, 0.038836, 0.048290, -0.056367, 0.190603, -0.061603, 0.061078, 0.014860, 0.036371, -0.004128, -0.102458, 0.182637, 0.101718, 0.023527, -0.102194, 0.022059, 0.065645, -0.004495, -0.022070, -0.099555, 0.052846, 0.011481, -0.114902, 0.014209, -0.107365, 0.014308, 0.027596, 0.130825, 0.020732, -0.094501, 0.005131, -0.087750, -0.133951, -0.077515, -0.008795, -0.228419, -0.096107, -0.031991, 0.045627, 0.036550, 0.027750, 0.092930, -0.036439, 0.153156, -0.009787, 0.055489, 0.037875, 0.023379, 0.042287, 0.033141, -0.106792, -0.074038, -0.081855, -0.112793, 0.089519, -0.093419, -0.107405, 0.038585, -0.069083, -0.114564, -0.078193, 0.140713, -0.173437, -0.043854, 0.026374, 0.077357, 0.096528, -0.068819, 0.049358, 0.149759, 0.011609, -0.010898, -0.133765, 0.001330, -0.008324, -0.031733, -0.060317, -0.018467, 0.210988, 0.077892, -0.155741, 0.141410, 0.121298, -0.079532, 0.252668, 0.013033, 0.041414, 0.102859, -0.000917, 0.008056, -0.054280, 0.053817, -0.040849, -0.093510, 0.012020, -0.036188, -0.117543, -0.011305, 0.093352, 0.111912, -0.058695, -0.071428, 0.002237, -0.011085, -0.011948, -0.057742, 0.047392, 0.074877, 0.037155, -0.011100, -0.009286, -0.120886, -0.043759, -0.049038, -0.021822, 0.141148, 0.050887, -0.056596, 0.049479, 0.051775, 0.043669, 0.019809, -0.132449, -0.083306, 0.014701, -0.084516, -0.090948, -0.008328, -0.010839, -0.170631, -0.012724, -0.038536, -0.099331, 0.071733, 0.141655, -0.132094, 0.105457, 0.080695, 0.084015, -0.025647, 0.236398, 0.029817, -0.067536, 0.114279, -0.082486, -0.119532, 0.020352, 0.025229, 0.107475, 0.056398, 0.019071, 0.069063, 0.076900, -0.057832, 0.072453, 0.004738, 0.116797, 0.082363, 0.040679, -0.095312, -0.075663, 0.044095, -0.142776, 0.036365, -0.097419, -0.104000, 0.047444, -0.060991, -0.111030, -0.006021, 0.000403, -0.053408, 0.030824, -0.194854, -0.019633, 0.025873, -0.120869, 0.083248, -0.057371, -0.162773, -0.157638, -0.047191, 0.116624, 0.111447, -0.054414, 0.129379, 0.091672, 0.086075, -0.111393, 0.002609, -0.010925, -0.192332, 0.072143, -0.038396, -0.027539, -0.027886, -0.083356, -0.030632, -0.120604, -0.049753, -0.064290, 0.005276, -0.137934, -0.057823, 0.038199, 0.136055, 0.065534, -0.098776, -0.029641, -0.076348, 0.046976, 0.080904, -0.261458, 0.024510, 0.014425, 0.010760, 0.096902, 0.031921, -0.127347, -0.065352, 0.164764, 0.097733, 0.181460, 0.096300, 0.016140, 0.065838, 0.028069, 0.051744, -0.158598, -0.056041, 0.015602, 0.101188, -0.031648, 0.048682, 0.026168, -0.106453, -0.002760, -0.019143, -0.064889, -0.161276, 0.090030, -0.047703, 0.091863, 0.018590, -0.098250, -0.054191, 0.065271, -0.024307, 0.073420, -0.008803, 0.030998, 0.068520, 0.034874, 0.056914, -0.063518, 0.010393, 0.054401, -0.050932, -0.172785, 0.100863, 0.069703, -0.097762, -0.007384, 0.004635, -0.010273, -0.207278, 0.073302, 0.108342, 0.130598, -0.054729, -0.016827, -0.102132, 0.122546, 0.078612, 0.043842, -0.042267, 0.200914, 0.074404, 0.024297, 0.105427, -0.104375, 0.055619, 0.057069, -0.001851, 0.065964, -0.001195, 0.022729, 0.022073, -0.029320, -0.070153, -0.161268, 0.047858, -0.147964, 0.045465, 0.067289, -0.069831, 0.092197, -0.154009, -0.010195, -0.056671, 0.054727, -0.008106, -0.135846, 0.034321, -0.081701, -0.078264, -0.117005, 0.160638, -0.191100, 0.033678, 0.048149, -0.061018, -0.017497, -0.027466, 0.088274, 0.003973, -0.154826, -0.077601, -0.002950, 0.041953, -0.130916, -0.107686, -0.156367, 0.015014, 0.084984, -0.195726, -0.046842, -0.061948, -0.061929, 0.061295, 0.077241, 0.132601, -0.031612, -0.062854, -0.064064, 0.050765, -0.019975, 0.136289, -0.047616, 0.033680, -0.006266, 0.013726, -0.120194, -0.075373, 0.121046, 0.017635, -0.073954, -0.063736, 0.140284, 0.059805, -0.102996, -0.097415, 0.020804, -0.052096, -0.134464, 0.090456, -0.016046, 0.003695, -0.073162, 0.016027, -0.000303, 0.065191, -0.029423, -0.105069, -0.135284, -0.027289, -0.098499, -0.026312, -0.137966, -0.021413, -0.069606, 0.003022, 0.084591, 0.068589, 0.130092, -0.029718, -0.079548, -0.027851, -0.088684, 0.070488, 0.042541, 0.034984, -0.120701, -0.166404, 0.029823, -0.023113, 0.048852, 0.010380, -0.037443, 0.095632, 0.076273, -0.082703, -0.039044, 0.032747, 0.039960, 0.077181, 0.142945, 0.128489, -0.045940, -0.126169, 0.021836, -0.143711, -0.067021, -0.024431, 0.090031, 0.109441, -0.060247, -0.166991, 0.119620, -0.081608, 0.018503, -0.103343, 0.079820, 0.304362, -0.000739, -0.088315, -0.087640, -0.109793, 0.098481, -0.044406, 0.157180, 0.099373, -0.154507, 0.056355, 0.067070, -0.024038, 0.120250, 0.024307, 0.169660, 0.065804, 0.095565, -0.020777, 0.154547, -0.130848, 0.061449, -0.114338, -0.277576, -0.053885, -0.072571, -0.190717, -0.057994, -0.021943, 0.067859, 0.111579, -0.056074, -0.131732, 0.032730, -0.170150, 0.040556, -0.070479, 0.008931, -0.120708, 0.015269, -0.138083, -0.109805, 0.000865, -0.097317, -0.021767, 0.045443, -0.071256, -0.087648, 0.068254, 0.071868, 0.170344, -0.009927, 0.061820, 0.172824, -0.030321, -0.020377, 0.029003, -0.086170, -0.046015, 0.149099, 0.149587, 0.150123, 0.003857, -0.031742, -0.164714, 0.183648, -0.023489, 0.035888, -0.017664, -0.007932, 0.102735, 0.011830, -0.019398, -0.073007, 0.002036, 0.057906, 0.146759, -0.036056, 0.051205, -0.003888, -0.014566, -0.007951, -0.102988, -0.141405, -0.044773, 0.073747, 0.037438, -0.054663, -0.109474, -0.049189, -0.189124, -0.120972, -0.047123, -0.080835, 0.030850, 0.087799, 0.020110, -0.007487, -0.009820, -0.134029, 0.029948, 0.173388, 0.011504, 0.153716, -0.091824, 0.154322, 0.088436, -0.044886, 0.073344, 0.016022, -0.083670, 0.152777, -0.162827, -0.190493, -0.010321, 0.127390, -0.003687, 0.190250, -0.106072, -0.147913, 0.013457, -0.085461, -0.062108, 0.116386, 0.106956, 0.101804, -0.020163, -0.173254, -0.207904, 0.014855, -0.162786, -0.022880, 0.016213, -0.007525, -0.176715, -0.241784, -0.112541, -0.057487, 0.111572, -0.039052, 0.110763, 0.005046, 0.050448, -0.043885, -0.110655, 0.098413, -0.039950, -0.020884, 0.026153, 0.122392, 0.088595, -0.117351, 0.091926, 0.001811, 0.106406, -0.030490, 0.022052, 0.028914, 0.039856, 0.050225, -0.269035, -0.012347, 0.068012, 0.023381, 0.066536, -0.216054, -0.047693, -0.149744, 0.018547, -0.068146, 0.050893, 0.001489, 0.172605, 0.104889, 0.033876, -0.014600, 0.012505, 0.056733, 0.019886, 0.014079, 0.020885, -0.058805, 0.071955, -0.047827, 0.083058, -0.066707, -0.177586, 0.081370, 0.072562, -0.120563, -0.026902, 0.053876, 0.038732, 0.030035, -0.015949, -0.042467, -0.089358, 0.023694, 0.022045, 0.005519, -0.054179, -0.130268, -0.086068, -0.062635, -0.046299, -0.171343, 0.127543, 0.045988, 0.052155, 0.024745, -0.048960, -0.098882, 0.061385, 0.010606, -0.112526, 0.133479, -0.147400, -0.044122, 0.031200, -0.053560, 0.113472, -0.026449, 0.107031, -0.115872, -0.033762, 0.142640, 0.020138, -0.051080, -0.177988, 0.114117, -0.057666, -0.025811, -0.021948, 0.002548, -0.019361, 0.005077, 0.170039, -0.091954, 0.001795, -0.084601, 0.010650, -0.057050, 0.010883, -0.010705, 0.065631, -0.044156, 0.064659, 0.121103, 0.194152, -0.019848, -0.018387, -0.041258, 0.023628, -0.065773, 0.090696, -0.080665, 0.072205, 0.016863, 0.054325, -0.007763, 0.084395, 0.084755, -0.059993, -0.021547, -0.013007, -0.023395, 0.051583, -0.144969, 0.128073, -0.117076, -0.121677, -0.076913, 0.086685, 0.055837, -0.179420, -0.060421, -0.069833, -0.170655, -0.071029, 0.004294, -0.054059, 0.084237, -0.130324, -0.140159, 0.077370, -0.101795, 0.070417, 0.118061, -0.047481, -0.063400, -0.108128, -0.088090, -0.012494, 0.137341, 0.064419, -0.220813, -0.055061, -0.057388, 0.124846, -0.048439, -0.095277, 0.025084, 0.025341, 0.011504, -0.011614, -0.027005, -0.108342, 0.172922, 0.205698, 0.049919, 0.056374, 0.026850, -0.030416, 0.007564, 0.080025, -0.181077, 0.010126, 0.015377, -0.051846, 0.021096, -0.036149, 0.093578, 0.009445, 0.064730, 0.032929, -0.036312, 0.082161, 0.043837, 0.125773, 0.140191, 0.136059, 0.162146, 0.055364, -0.189778, -0.027121, 0.031415, 0.050562, -0.195290, -0.065707, -0.114995, 0.047474, -0.111554, -0.111235, -0.077907, -0.046859, -0.129531, -0.029520, -0.133611, -0.068378, 0.104291, -0.011180, 0.008072, -0.236179, -0.092536, 0.284131, 0.091880, -0.104658, 0.035369, -0.030930, -0.148208, -0.083417, -0.036487, 0.148977, 0.053650, 0.062709, -0.066371, -0.098806, -0.038112, 0.054154, -0.093856, -0.056671, -0.258148, -0.081355, 0.051070, -0.121231, -0.030955, -0.004252, -0.038402, -0.008297, -0.086987, -0.192995, -0.040629, -0.011182, -0.001034, -0.099052, -0.025642, 0.057768, 0.027779, -0.016143, -0.136071, -0.089523, 0.100375, -0.075392, 0.031812, -0.069426, -0.120098, -0.054370, -0.170946, -0.037783, 0.019682, -0.107906, 0.051187, 0.080240, -0.145358, -0.131524, -0.109819, -0.160454, 0.006837, -0.087884, -0.128334, 0.029056, 0.100818, -0.086485, -0.102571, 0.024929, 0.092840, -0.064172, -0.043248, -0.032490, -0.046312, -0.032316, -0.013323, 0.103629, -0.004941, -0.018913, -0.018550, 0.050446, -0.036296, 0.041374, 0.140193, -0.050405, -0.062587, -0.197799, -0.028484, 0.041897, 0.021977, -0.010021, 0.009603, -0.017631, -0.039182, 0.008287, 0.100917, -0.008547, 0.115426, -0.179964, -0.165274, -0.018747, -0.067302, -0.038887, 0.125155, -0.085911, -0.208581, -0.083852, -0.128129, -0.032871, 0.117500, 0.024178, -0.024256, 0.075277, -0.173654, -0.101746, -0.114663, -0.003843, -0.154603, -0.031158, -0.076191, -0.131225, -0.060274, -0.156385, -0.051910, -0.026891, 0.066860, -0.075316, -0.116080, 0.108318, 0.066218, 0.000474, 0.103536, 0.025882, 0.085026, -0.089233, -0.017536, -0.039995, 0.141361, 0.038330, 0.061986, -0.070948, -0.099496, -0.049018, -0.170534, 0.041431, -0.083013, -0.118958, -0.134527, 0.116145, -0.029886, -0.040649, 0.010040, -0.063496, 0.091040, 0.020789, 0.002517, -0.139581, -0.267783, -0.072724, -0.011540, 0.024365, -0.067577, 0.103389, -0.058059, -0.299851, 0.027281, 0.200481, -0.018562, -0.149547, -0.040051, -0.040360, -0.116034, -0.097727, -0.135392, 0.195073, -0.067346, -0.100693, 0.083943, 0.106606, -0.090283, -0.147942, -0.253815, 0.005812, -0.017152, -0.135016, -0.081264, 0.030916, 0.018225, -0.078498, -0.180701, -0.062109, -0.140708, 0.011224, -0.055406, 0.002020, 0.010346, 0.128722, 0.086081, 0.170851, -0.005650, -0.015302, 0.097834, 0.067995, -0.034793, 0.008565, -0.024966, -0.123186, -0.155797, -0.030480, 0.112718, -0.033473, -0.220132, 0.028741, -0.016849, -0.057554, 0.074471, -0.022651, -0.028401, 0.013850, -0.073497, -0.135020, -0.138805, -0.094844, -0.081216, -0.095806, -0.041066, -0.024316, 0.015025, -0.102894, -0.151340, -0.067436, -0.168642, -0.143026, -0.071198, -0.044927, 0.094819, -0.091707, -0.039109, -0.119267, -0.000165, -0.129543, -0.044937, 0.102472, 0.001229, -0.021883, 0.120354, -0.203862, 0.094812, 0.025533, -0.015492, -0.156981, 0.020201, 0.150784, -0.147255, 0.077002, -0.083897, -0.023223, -0.125252, 0.096460, -0.063696, -0.142226, -0.080164, -0.048889, -0.044924, -0.071760, -0.003329, 0.101764, -0.161483, -0.024940, -0.042850, -0.014706, -0.006859, -0.066840, 0.058298, -0.106100, 0.018921, -0.105262, 0.035572, 0.006494, 0.009985, -0.010718, 0.004212, -0.050844, -0.168188, -0.034972, -0.141004, -0.034203, -0.120681, -0.319309, -0.041597, -0.057602, -0.222112, 0.033803, 0.120377, -0.014401, -0.103432, -0.151814, 0.013925, -0.139068, -0.121930, -0.083696, -0.042199, -0.075973, -0.056710, -0.026159, 0.004719, 0.046037, 0.016237, 0.044006, -0.142508, -0.043062, -0.207246, -0.120620, -0.072167, 0.081131, 0.004051, -0.154869, 0.017978, -0.071422, 0.035287, -0.043925, 0.009850, -0.003046, -0.075018, 0.033483, -0.085791, -0.011126, -0.156479, 0.136852, 0.019890, -0.049169, 0.000743, -0.221086, 0.199349, 0.078513, 0.024106, -0.028631, 0.069280, -0.110526, -0.154725, 0.013494, -0.378482, -0.039673, -0.005582, -0.073322, -0.028036, 0.009864, -0.079217, -0.202428, -0.078402, -0.010662, -0.101309, -0.180034, -0.122283, -0.082564, 0.016870, 0.038700, 0.039100, 0.035088, 0.060239, -0.112454, -0.213548, 0.042872, 0.093673, -0.055406, 0.096242, -0.013973, -0.117144, 0.064599, 0.009156, 0.037185, 0.064935, -0.025390, -0.016524, -0.067462, -0.135419, -0.104718, 0.000211, 0.130642, 0.035470, -0.020150, -0.121937, -0.019161, -0.159500, -0.083870, 0.051832, -0.019668, -0.102030, 0.082597, 0.047534, -0.175549, -0.164982, -0.095557, 0.140897, 0.122877, 0.021999, -0.022165, -0.020787, -0.195129, -0.011048, -0.022848, 0.071313, 0.010023, -0.046359, -0.005642, 0.073547, -0.092517, 0.088180, -0.016027, -0.176424, -0.052290, 0.072374, 0.078596, 0.056039, -0.040175, 0.146569, -0.153748, -0.077229, -0.084700, -0.078877, -0.093896, 0.109786, 0.066308, 0.095264, -0.006687, 0.000986, 0.079594, -0.051314, -0.071748, -0.112973, 0.183692, -0.126369, -0.076733, -0.080710, -0.026773, 0.065181, -0.090354, -0.119469, -0.041268, -0.055099, -0.132023, -0.121945, -0.048868, -0.096516, -0.022561, -0.041601, -0.058839, 0.058982, 0.037105, 0.121511, 0.055036, 0.017907, 0.013465, -0.133079, 0.044917, -0.107338, 0.069788, -0.059331, -0.000269, 0.052566, 0.020002, -0.208756, 0.054666, 0.008397, 0.041033, -0.055155, 0.006903, -0.089982, 0.094523, -0.159485, -0.102109, -0.140937, -0.036310, 0.132878, -0.013564, -0.121098, -0.035779, 0.078070, -0.098578, -0.177471, -0.132714, 0.012960, -0.045249, -0.105978, 0.042884, -0.129916, 0.025686, -0.030968, 0.126901, 0.196863, -0.085754, -0.211509, -0.016662, -0.030209, -0.068158, 0.008360, -0.132218, -0.196799, 0.075038, -0.020584, 0.045712, -0.024262, -0.135267, -0.256894, 0.046432, -0.253218, 0.076902, -0.059271, -0.049020, 0.132346, 0.010840, -0.084499, 0.039594, 0.044123, -0.080026, 0.100347, 0.010708, 0.045260, -0.092541, -0.196826, 0.023411, 0.075059, -0.096561, -0.139021, -0.017327, -0.123012, -0.044057, -0.104219, -0.184909, 0.091194, -0.064767, 0.035041, -0.134745, -0.010636, 0.018286, -0.111232, 0.013941, 0.106446, -0.057117, 0.050420, -0.016774, -0.072920, 0.077085, -0.066063, -0.098309, -0.063067, -0.073802, -0.127381, -0.083910, -0.061841, -0.171208, -0.171880, -0.012462, -0.280780, -0.044407, 0.027088, -0.131164, -0.011889, 0.109857, 0.014954, -0.058511, 0.005255, -0.223855, 0.050030, -0.089408, -0.237182, -0.116953, -0.055392, 0.028595, 0.157695, -0.202568, -0.054566, 0.015386, 0.048843, -0.031179, -0.103587, -0.063674, -0.159328, -0.017545, -0.016153, -0.105060, -0.173595, -0.091837, -0.038155, -0.003142, -0.119841, -0.122898, 0.092435, 0.120992, -0.037498, 0.045078, 0.002410, -0.116222, -0.073777, -0.037734, -0.037936, 0.186291, 0.134175, 0.077840, -0.156529, 0.076321, 0.000137, -0.035409, -0.031892, -0.314562, -0.089587, 0.080608, -0.062329, -0.181437, -0.035629, -0.024343, 0.005296, 0.071568, 0.080073, 0.066019, -0.116987, 0.061047, -0.124772, 0.065116, -0.167206, -0.022888, -0.106431, -0.161381, -0.124693, -0.123596, 0.108010, -0.003946, 0.026989, 0.024859, -0.101557, -0.055949, 0.013219, -0.049445, -0.137562, 0.101912, -0.081760, -0.023664, 0.083341, 0.041400, -0.117209, -0.029276, -0.036183, 0.027867, 0.193400, -0.193240, 0.199320, -0.114093, 0.104547, -0.178747, -0.144323, -0.148116, -0.080043, 0.002647, 0.004244, -0.072806, 0.103658, -0.099839, 0.089529, -0.055262, 0.012902, -0.000124, 0.071406, -0.042644, 0.027850, 0.110417, -0.031163, 0.056521, -0.070428, -0.189596, -0.032362, 0.006931, -0.015353, -0.007941, 0.014488, -0.082399, -0.006470, 0.118984, 0.198011, 0.091893, -0.082019, -0.039022, -0.057911, 0.014011, 0.043440, -0.173210, 0.258197, 0.075201, 0.004832, -0.078500, -0.115774, 0.087577, -0.095415, 0.028220, -0.075956, -0.005124, -0.144974, -0.082231, -0.194153, 0.012516, 0.027541, 0.176413, 0.037370, -0.081512, -0.131621, -0.114681, -0.262999, 0.020799, -0.036732, 0.046226, 0.019815, 0.034797, 0.016980, -0.186174, 0.181158, 0.049719, -0.193899, 0.031973, -0.102193, -0.091709, 0.090501, -0.091315, 0.108138, 0.036726, 0.104124, -0.284190, -0.149219, -0.021372, -0.008079, -0.114393, 0.206595, 0.019034, 0.070974, -0.004355, -0.155624, -0.038794, -0.091919, 0.058539, 0.042084, -0.118877, -0.000010, -0.053590, -0.089735, -0.023466, 0.034750, 0.036240, -0.101153, -0.107969, -0.189410, -0.028603, 0.192672, 0.028176, 0.251168, -0.004084, 0.034764, -0.013059, 0.048330, 0.056339, 0.034477, -0.077349, -0.164685, -0.007058, 0.078193, -0.087214, -0.001644, -0.087307, 0.020520, -0.154071, 0.075594, -0.024478, 0.121804, -0.122032, -0.189940, 0.068172, -0.025245, -0.092125, -0.028241, -0.022689, -0.027826, -0.077916, -0.044923, -0.013387, 0.025319, -0.106895, 0.005723, 0.107792, -0.006191, 0.095099, -0.086669, 0.060708, -0.092774, 0.004546, 0.055588, -0.078149, -0.040334, -0.112472, 0.045824, 0.042291, -0.124697, 0.023570, 0.065973, -0.039407, -0.041178, -0.096204, -0.151488, -0.015991, -0.158186, 0.130067, 0.165403, 0.007993, -0.109372, -0.073080, -0.006958, -0.047595, 0.192117, -0.081889, -0.012843, -0.055801, -0.003453, -0.055445, 0.040581, 0.035870, -0.155257, 0.058279, -0.031364, -0.181726, -0.000129, -0.040300, 0.023280, 0.007229, -0.051018, 0.051329, -0.068347, 0.030671, -0.143485, 0.096195, -0.032895, 0.046643, -0.130552, -0.096340, -0.109895, -0.135703, -0.143743, 0.031090, -0.027566, -0.201639, -0.051135, -0.031039, 0.087457, -0.217040, -0.059423, -0.073841, -0.038827, -0.047118, 0.075770, -0.027289, -0.093998, -0.027441, 0.032789, -0.020441, -0.114609, -0.040974, -0.016084, 0.157173, -0.006091, 0.078173, -0.140550, -0.117376, -0.089889, -0.031772, 0.019197, 0.094607, -0.085366, -0.180401, 0.073425, 0.052086, -0.132816, 0.082132, -0.101334, -0.003392, 0.002604, 0.129204, -0.100042, 0.000446, -0.005719, 0.035864, -0.131343, 0.096145, 0.015973, 0.081704, -0.026542, -0.106127, 0.170729, 0.019946, -0.166742, -0.065198, 0.110073, -0.037195, -0.129518, -0.061864, 0.100651, 0.051915, 0.194671, 0.012427, 0.047252, -0.000949, -0.232124, -0.150063, 0.025034, 0.041911, -0.041240, 0.104327, -0.023419, 0.033507, -0.159644, 0.108542, 0.020363, -0.148185, -0.157225, -0.111234, -0.083409, -0.006036, -0.125978, -0.017992, -0.132664, 0.030890, -0.057339, 0.037076, 0.005061, -0.066264, -0.039938, -0.054129, 0.036562, 0.011009, -0.061883, -0.125414, 0.035846, -0.141985, -0.087452, -0.197674, -0.173450, 0.071800, -0.049251, 0.012122, -0.072411, 0.027283, 0.095733, -0.010555, -0.118282, -0.014294, 0.027264, -0.132671, -0.074359, -0.079945, 0.058698, 0.046462, 0.051126, -0.114908, 0.060929, 0.002220, 0.144432, 0.036250, -0.027579, -0.104975, -0.114780, -0.123971, 0.006914, -0.060544, -0.123619, -0.127841, -0.048138, -0.026188, 0.028426, 0.043898, -0.214727, -0.081492, -0.057601, -0.025105, -0.017982, -0.065096, -0.097976, 0.039835, -0.007328, 0.166665, -0.067824, -0.122148, -0.212343, 0.092158, 0.070616, -0.086876, 0.061871, -0.086836, -0.227264, 0.002750, 0.089956, 0.001237, -0.001756, -0.096357, 0.173404, -0.090497, 0.037170, -0.128945, 0.024416, -0.224205, -0.122241, -0.064860, -0.028234, -0.121362, -0.096524, -0.026974, 0.014464, 0.074088, -0.043067, -0.082520, -0.182446, 0.020093, 0.098136, -0.009991, -0.042030, 0.218444, -0.065728, 0.019162, -0.165899, 0.011949, 0.122303, 0.133231, 0.038064, 0.050325, -0.049397, 0.052859, -0.210986, 0.107510, 0.019825, -0.037315, 0.021129, 0.064835, 0.040162, -0.186431, 0.239511, -0.129153, -0.161751, -0.110391, 0.232633, -0.225097, -0.142007, -0.036935, 0.050589, -0.067242, 0.021706, 0.031060, -0.050255, 0.025457, -0.048994, -0.186538, -0.099548, -0.103262, -0.006868, 0.031371, -0.089947, -0.112852, -0.095936, -0.104903, -0.031669, 0.005828, -0.050652, 0.019287, 0.042833, -0.215877, 0.046981, -0.098712, -0.207228, -0.027620, -0.155148, -0.068342, -0.108371, 0.005003, 0.167736, -0.159596, 0.299959, -0.161814, -0.214913, -0.058239, 0.047420, -0.285691, 0.130326, -0.263803, -0.036265, -0.244631, -0.051431, -0.053726, 0.006492, 0.157091, -0.093317, -0.155342, -0.004737, -0.191155, 0.018780, -0.053255, 0.004869, -0.032725, -0.227056, -0.080566, 0.006602, -0.063916, 0.042122, -0.189034, 0.183401, -0.284667, 0.073005, -0.129852, 0.039850, -0.022040, -0.081519, 0.014266, -0.165442, -0.118120, -0.135059, -0.279448, -0.185290, -0.089473, 0.047070, -0.083012, 0.138411, -0.083990, -0.201883, 0.060758, 0.017768, -0.021071, 0.035572, -0.012883, -0.014287, 0.022687, -0.057283, -0.142093, 0.087759, -0.036439, -0.007635, 0.103280, -0.139088, -0.195493, -0.097972, -0.138853, -0.198486, 0.072295, -0.007573, -0.071494, 0.057969, 0.120895, -0.065535, -0.063487, -0.223646, -0.310239, -0.138297, 0.118049, -0.238934, 0.110140, -0.146819, -0.254879, -0.301785, -0.057738, 0.075879, 0.048036, -0.005191, -0.045233, 0.158160, 0.007994, -0.007708, -0.028887, -0.115474, 0.008101, 0.063772, -0.122489, -0.200870, -0.100250, -0.076180, 0.068350, -0.198919, -0.042432, -0.138631, 0.027904, 0.061593, 0.218638, -0.092270, 0.035397, 0.013298, 0.084401, -0.202406, 0.028811, -0.100420, -0.000491, 0.148000, -0.027692, -0.068440, 0.156369, -0.155839, -0.092847, -0.109599, -0.068542, -0.098277, -0.087771, 0.102906, 0.053480, -0.367666, -0.033980, 0.026812, -0.090853, -0.068090, 0.082581, -0.023172, -0.041314, -0.018082, -0.120442, 0.132475, -0.095224, 0.038280, 0.072004, 0.082093, -0.069866, -0.200850, -0.021175, -0.140015, 0.060462, 0.119439, 0.020924, -0.116870, 0.102249, -0.080027, 0.058083, 0.070071, -0.003054, 0.020244, -0.065724, 0.048788, -0.076762, 0.273161, 0.031777, 0.024658, -0.088068, 0.011325, -0.061992, -0.169331, -0.137906, -0.023852, -0.060705, -0.185912, -0.019231, -0.046922, -0.204446, -0.015023, -0.044050, -0.006028, -0.087648, -0.107681, -0.104436, 0.197933, -0.001628, 0.104896, -0.088427, -0.057475, 0.071489, 0.096057, -0.074640, -0.082973, 0.027476, 0.170519, 0.036761, -0.099969, -0.042120, 0.004555, 0.108101, 0.173222, 0.095746, -0.084823, 0.152619, -0.073104, -0.103434, 0.008120, -0.016193, -0.003015, -0.121952, -0.089847, -0.123671, 0.040398, -0.008902, -0.058003, -0.129881, 0.029323, -0.032152, -0.134021, 0.156634, -0.358395, -0.183213, -0.087929, -0.003844, -0.042923, 0.011143, -0.099330, 0.033786, -0.120881, 0.008037, 0.000480, 0.048964, 0.005625, 0.075523, -0.108431, -0.054367, 0.071786, -0.139296, -0.127759, 0.072397, 0.004030, -0.078633, 0.041121, 0.114727, -0.079720, -0.060923, -0.154871, -0.113185, 0.004997, 0.112168, -0.153224, 0.054041, -0.170847, 0.128028, 0.089565, -0.135854, -0.089579, 0.010812, 0.013063, 0.011685, -0.106976, -0.191497, -0.024460, -0.182285, 0.063490, -0.012845, -0.016515, -0.162134, -0.074916, 0.041498, 0.094095, 0.059889, -0.114763, 0.200828, 0.065744, -0.120326, -0.218675, 0.019039, -0.004904, 0.040818, 0.000700, 0.259753, -0.053142, -0.033328, -0.028503, 0.085110, -0.003987, -0.083058, -0.095314, -0.018836, 0.113986, -0.028967, -0.142865, -0.018659, 0.066684, -0.114522, -0.037037, -0.145573, -0.132890, -0.024258, -0.152389, 0.059548, -0.048170, -0.037833, -0.140266, 0.152503, -0.000560, 0.034090, -0.232422, -0.003846, 0.025922, -0.026679, -0.028050, 0.107457, 0.017409, -0.081024, -0.028165, -0.097079, -0.122174, -0.100243, -0.121466, -0.164251, 0.015984, 0.073585, 0.087516, 0.022320, 0.147233, -0.097287, -0.173420, 0.010302, -0.019682, -0.123732, -0.054623, -0.231490, -0.079383, -0.106602, -0.149907, -0.004011, 0.130401, -0.031269, 0.016657, 0.111006, 0.004459, -0.083693, -0.012789, -0.044920, -0.067513, 0.083708, -0.080504, 0.004792, -0.062134, -0.055899, -0.080518, 0.057413, 0.011656, 0.047751, 0.040297, -0.101556, 0.071683, 0.079608, -0.036934, -0.190369, -0.002838, -0.146288, -0.006756, -0.161119, 0.037847, -0.166515, 0.028490, -0.053618, -0.109750, 0.164105, 0.048337, -0.050280, -0.122197, -0.081554, -0.008902, -0.159988, 0.050331, 0.033430, -0.009680, -0.059745, 0.055723, -0.012819, -0.198752, 0.066051, 0.015845, 0.023755, 0.005744, -0.016556, -0.072923, -0.088961, -0.072156, -0.086554, -0.158910, 0.001916, 0.101978, -0.004437, -0.006649, 0.016205, 0.183314, 0.196583, 0.052571, 0.013423, -0.038834, 0.071198, 0.103979, 0.044197, 0.015927, -0.024476, -0.086507, -0.114047, -0.069223, -0.053408, -0.057524, -0.132471, -0.114594, -0.058085, 0.022662, -0.110305, -0.024002, 0.051766, -0.067050, 0.025612, -0.251654, 0.072556, -0.128968, 0.109450, 0.021107, 0.103897, 0.035797, 0.098522, -0.015085, -0.137849, -0.001878, -0.024145, -0.027091, -0.010199, 0.078938, -0.185624, -0.100281, 0.054682, -0.045525, 0.037726, -0.024407, -0.106881, -0.075841, 0.025545, -0.062744, -0.009445, -0.156588, 0.073552, -0.078310, 0.048327, -0.154077, 0.031755, -0.059042, -0.222568, -0.102296, 0.056639, -0.235403, 0.102125, 0.016831, -0.073258, -0.042271, -0.160862, -0.169609, -0.114813, 0.052822, -0.062168, -0.044090, -0.025387, 0.041153, -0.144508, -0.058151, 0.062478, 0.119840, -0.052599, 0.020888, 0.035530, -0.037294, -0.073300, -0.136131, -0.047695, -0.063863, -0.037064, -0.054413, 0.088684, 0.025330, -0.089203, -0.036286, -0.085310, -0.109071, -0.229601, -0.057774, -0.210718, -0.160436, -0.042919, -0.212820, 0.005601, -0.056141, -0.000944, -0.105159, 0.025511, -0.129836, -0.259899, -0.064081, 0.018541, 0.100740, 0.127829, -0.030294, -0.031313, -0.181377, -0.060977, 0.091646, 0.064552, -0.110888, 0.024389, -0.037981, -0.068293, -0.031343, -0.063883, 0.021001, -0.046672, 0.046085, -0.034547, 0.059195, -0.134493, -0.128941, -0.223127, -0.004493, -0.017984, -0.081263, -0.150013, 0.045436, -0.037758, -0.130395, -0.103221, -0.089009, -0.005124, -0.179004, -0.134245, -0.043614, 0.040713, -0.067645, -0.117998, 0.002762, -0.172847, -0.099550, 0.024798, -0.110581, -0.253001, -0.317557, -0.188628, -0.013775, -0.010445, -0.088948, 0.116397, -0.044017, -0.038227, -0.060118, -0.035426, -0.000057, -0.095274, 0.048118, -0.201053, -0.120251, -0.030030, 0.019741, -0.014379, -0.164914, 0.084146, 0.096121, -0.096041, -0.170454, -0.176967, 0.047421, -0.111176, -0.031927, -0.075504, 0.012242, -0.010974, -0.071796, 0.055812, -0.093269, 0.085406, -0.110919, -0.085478, 0.091538, -0.094092, -0.225122, 0.084768, -0.086278, -0.104837, -0.100839, -0.078579, 0.049791, 0.118971, 0.059798, 0.176076, -0.025831, -0.020497, -0.114905, -0.098744, 0.071090, -0.138439, -0.065516, -0.042916, 0.058498, -0.110176, 0.078299, -0.039376, -0.011369, -0.091972, 0.028069, 0.059427, -0.338496, -0.021833, -0.157079, -0.036995, -0.007839, 0.048936, -0.027965, -0.060289, -0.027113, 0.043871, -0.018958, 0.026984, -0.083462, -0.035223, 0.092553, -0.108198, -0.149017, 0.007484, -0.050572, 0.043059, -0.072945, -0.036069, -0.101053, -0.039579, -0.190722, -0.061125, -0.218640, -0.023052, 0.026015, 0.049153, 0.062712, -0.142582, -0.298809, -0.067474, -0.150005, 0.134263, -0.081913, -0.113859, 0.053384, -0.248530, -0.078128, -0.216699, -0.015437, -0.120984, 0.070991, -0.197057, -0.106145, -0.239389, 0.009400, -0.202647, -0.039370, -0.041000, -0.123890, 0.069021, -0.145255, -0.093419, 0.058336, -0.052642, -0.112674, -0.138818, -0.225829, 0.074233, -0.178967, -0.067837, 0.032981, -0.137003, -0.150903, -0.083215, -0.040813, -0.171570, -0.066632, 0.011712, -0.089729, -0.080069, -0.062494, -0.080735, 0.060433, -0.032847, -0.086358, -0.094631, -0.275007, -0.014590, -0.117605, -0.047526, 0.114720, -0.214795, 0.020912, 0.128601, -0.058182, -0.313141, -0.188715, -0.030937, -0.142796, -0.157943, -0.296165, -0.011177, -0.204084, -0.103469, 0.038103, -0.153143, -0.103282, -0.081243, -0.103091, -0.110842, -0.226803, -0.202591, -0.132665, -0.162207, 0.132483, -0.073700, 0.107497, -0.193824, -0.143472, 0.043858, -0.270416, 0.203441, -0.068231, -0.068434, 0.006524, -0.054939, -0.050565, 0.021790, -0.015581, -0.225032, -0.003544, 0.070741, 0.079423, 0.079569, -0.150546, -0.008703, -0.101418, -0.102450, -0.143068, 0.117838, -0.096700, -0.145971, 0.166703, -0.043307, -0.023980, 0.043231, 0.121327, 0.019951, -0.151755, 0.068101, -0.201589, 0.084528, 0.030807, -0.028752, -0.102831, -0.167638, -0.125759, -0.098120, 0.011728, -0.038721, -0.039703, -0.154478, -0.016005, -0.135870, -0.127998, -0.232847, 0.020034, -0.128379, -0.128865, -0.084580, -0.084017, -0.187578, 0.007349, -0.131670, -0.183697, 0.046101, 0.054147, -0.317096, -0.213572, -0.121061, -0.174116, -0.201282, -0.015382, -0.103396, -0.030334, -0.366691, 0.004868, -0.203288, -0.104590, -0.124327, -0.193726, -0.210315, 0.289319, -0.026530, -0.034682, -0.061645, -0.099577, 0.166530, -0.200773, 0.084102, -0.126887, 0.222590, 0.142822, -0.053938, -0.141680, -0.230770, -0.150539, -0.241777, -0.062453, 0.116260, 0.043142, -0.073688, -0.003357, 0.016843, -0.030473, 0.118773, -0.140363, 0.003578, -0.058730, -0.037686, -0.115768, -0.016780, 0.152128, -0.077551, -0.141165, 0.040915, -0.106454, -0.082330, -0.116265, 0.015938, -0.134528, -0.069585, 0.066283, -0.129533, 0.051664, 0.023063, -0.054898, -0.312810, -0.062407, 0.034540, -0.069223, -0.080429, -0.064051, 0.004822, -0.093319, -0.184938, -0.151217, -0.189819, 0.057102, -0.038602, -0.194632, 0.091520, 0.026081, -0.025814, 0.029976, -0.288125, -0.130287, -0.046980, -0.166430, -0.036963, -0.092937, -0.111653, -0.018995, -0.141066, -0.001147, -0.255235, 0.019495, -0.015580, -0.062754, 0.034443, -0.208505, 0.026198, -0.166115, -0.145869, -0.070249, -0.035755, -0.046433, 0.033049, 0.120558, 0.021522, 0.134921, 0.110642, -0.070102, -0.010559, 0.053570, -0.094858, -0.074518, -0.157581, -0.113765, -0.075657, 0.029092, -0.227277, -0.111356, 0.043079, 0.100017, -0.011837, -0.120461, 0.123722, -0.125368, -0.081320, -0.017118, -0.004643, 0.096641, -0.061441, 0.106153, -0.028496, 0.033296, 0.065222, 0.055240, 0.007011, 0.133556, 0.037852, -0.082130, -0.108495, 0.015963, 0.098175, -0.124318, -0.182369, -0.115522, 0.118131, -0.044097, 0.104416, 0.048686, -0.174191, 0.031551, -0.128994, -0.029895, 0.144859, 0.106907, -0.097289, -0.041700, -0.093899, 0.124034, -0.072160, 0.033067, 0.005836, -0.030646, -0.112258, -0.125877, 0.068076, -0.005737, -0.175710, -0.028043, 0.107053, -0.120416, -0.074664, -0.015964, -0.101466, -0.140745, -0.105895, -0.170885, 0.088677, -0.160670, -0.067838, -0.146220, 0.013930, 0.206636, 0.072344, 0.039244, 0.125601, 0.066657, -0.202078, -0.069020, -0.111247, -0.010756, 0.006542, 0.072791, -0.086471, -0.006872, -0.056868, -0.148918, -0.017150, -0.273401, -0.102820, 0.011968, -0.043657, -0.021389, 0.140507, -0.083034, 0.010868, -0.046441, -0.047332, 0.089474, 0.024118, 0.059532, 0.108455, -0.086501, -0.096302, -0.004460, -0.122639, -0.111519, 0.110423, -0.186281, 0.124346, -0.148434, -0.037792, -0.086090, -0.090418, -0.141573, 0.052495, -0.143926, 0.040658, -0.090959, 0.016650, 0.002185, -0.165503, 0.173081, 0.123671, -0.108912, 0.076946, -0.102159, -0.067308, -0.142295, -0.013560, 0.135209, -0.083610, 0.011827, -0.231330, 0.096939, 0.051197, 0.025423, -0.071925, -0.143626, -0.227922, 0.059193, -0.009670, -0.134329, -0.110014, -0.167106, 0.090227, -0.087972, -0.076646, -0.124080, -0.043346, 0.066009, 0.004488, 0.011320, -0.200771, -0.150558, -0.034996, -0.068613, 0.031641, -0.214585, 0.057406, -0.043372, -0.057998, -0.170581, -0.019404, -0.207591, -0.038017, 0.101244, -0.216310, -0.127162, -0.016690, -0.020230, -0.161708, 0.144944, 0.064828, 0.115100, -0.144568, -0.013266, -0.252206, 0.018383, -0.044807, 0.038711, -0.041164, -0.246369, -0.046144, -0.123214, -0.032766, -0.098037, -0.095351, -0.049355, 0.070309, -0.107021, -0.146538, -0.017378, -0.031289, -0.126201, 0.053332, 0.164193, -0.080510, -0.031915, -0.041079, -0.010839, -0.057808, 0.169594, -0.149379, -0.147921, 0.074333, -0.073788, -0.063642, -0.099694, -0.067868, -0.022523, -0.123825, -0.055525, 0.071997, -0.039878, -0.008982, -0.094150, -0.064025, 0.135358, 0.087107, 0.059219, 0.036540, 0.214481, 0.166670, -0.116016, -0.143679, -0.136706, 0.101818, 0.152818, -0.038243, -0.098080, 0.047393, -0.098311, 0.002591, -0.008494, 0.002600, -0.012833, -0.003149, 0.101603, -0.143179, 0.071653, 0.064600, -0.048406, 0.037493, -0.023601, -0.031961, -0.012215, -0.043447, -0.000088, -0.071666, -0.037566, -0.041187, -0.028975, 0.026898, 0.007957, -0.124335, 0.045560, 0.041194, 0.033225, 0.043576, -0.198075, 0.041991, -0.038160, 0.068094, -0.071488, -0.052659, -0.110265, -0.052309, 0.045972, 0.063102, -0.199078, -0.100556, -0.096015, -0.040017, 0.032379, -0.060681, -0.057418, 0.055170, -0.124515, -0.442210, -0.028586, -0.019294, -0.093941, -0.043193, -0.168526, 0.007431, 0.051279, 0.076467, -0.057877, -0.052088, 0.104380, 0.052018, -0.272110, 0.005665, -0.024033, -0.167829, -0.061371, 0.001161, -0.114331, 0.007212, -0.132596, 0.075799, -0.108288, 0.053408, -0.046300, 0.027241, 0.069681, -0.100017, 0.116517, -0.127969, -0.128292, -0.043819, -0.011778, -0.131431, -0.076162, 0.074678, 0.139991, -0.143218, 0.029670, 0.026785, -0.104289, 0.058512, -0.033456, -0.061659, -0.006407, -0.130506, 0.025145, 0.038709, -0.114906, -0.003295, -0.006639, -0.033812, -0.105668, -0.135040, 0.062021, -0.068231, 0.112039, -0.117247, -0.032513, -0.043074, -0.282077, -0.180649, 0.073194, 0.024171, -0.010542, -0.135457, -0.186995, 0.035268, 0.077107, -0.077328, -0.161547, -0.024326, -0.116706, -0.053137, -0.030382, 0.084122, -0.153727, -0.116124, -0.033031, -0.030659, -0.083773, 0.048182, -0.042349, -0.128219, -0.058662, -0.007578, 0.030227, 0.178599, -0.081777, -0.077169, 0.119899, -0.126671, -0.132352, -0.033175, -0.107670, -0.008380, 0.089361, 0.008111, -0.177184, -0.113730, -0.022137, -0.009464, -0.079538, -0.194033, 0.007528, -0.128258, -0.029871, 0.105926, -0.088999, -0.142424, -0.037205, -0.087674, 0.140695, 0.140555, -0.150117, 0.071113, -0.030335, -0.040650, 0.231397, 0.037538, 0.094914, -0.005786, -0.270026, 0.163949, -0.137601, 0.095608, -0.071822, -0.152619, -0.054028, -0.146208, 0.045541, 0.019123, 0.182964, -0.049919, 0.039042, 0.041546, 0.052762, 0.008571, -0.223418, -0.032320, -0.095951, -0.157011, -0.102530, 0.141209, 0.115808, 0.133502, -0.070737, 0.039796, 0.032698, -0.108645, -0.167186, -0.026274, 0.038665, -0.269882, 0.013543, 0.013578, 0.005514, -0.169987, 0.118358, 0.097492, -0.033764, 0.090773, 0.117534, 0.104731, -0.218014, 0.224219, -0.018530, 0.048568, 0.006757, -0.026406, -0.044572, 0.056270, 0.029043, -0.020568, -0.026750, 0.003465, -0.043032, 0.035817, -0.058472, 0.018884, -0.032658, 0.041770, -0.104788, -0.041239, 0.255034, -0.040495, 0.026119, -0.037637, -0.181564, 0.088804, 0.067232, -0.069384, 0.015212, -0.065457, -0.115590, -0.162527, -0.076227, -0.123899, 0.058157, 0.049822, -0.012776, 0.033265, -0.018157, -0.247890, -0.115591, -0.120727, 0.130552, -0.066335, -0.040972, -0.062282, -0.043222, -0.048162, -0.083565, -0.044727, 0.117857, -0.142414, 0.161050, 0.064470, 0.031004, 0.128139, 0.027950, -0.016679, -0.136226, 0.101024, -0.025829, -0.035360, -0.207353, -0.099878, -0.239537, 0.065014, -0.147278, -0.092810, -0.040352, -0.017110, 0.084006, -0.037813, 0.110981, -0.119578, -0.070354, 0.118278, 0.106208, 0.048141, -0.140024, 0.088749, -0.008125, -0.117271, -0.233766, -0.076661, -0.142281, -0.118289, -0.111592, -0.136956, 0.194969, -0.049358, -0.172965, -0.134111, -0.150761, 0.142860, 0.111915, 0.053385, -0.031928, 0.039079, -0.140399, -0.163029, -0.032378, -0.084074, -0.084231, 0.028275, 0.049473, 0.155145, -0.111478, -0.096801, -0.061291, 0.118494, 0.046945, -0.043483, -0.104104, -0.057625, -0.091022, 0.062599, -0.015105, 0.049464, 0.154570, 0.101447, 0.047388, 0.052484, 0.048542, 0.009914, -0.031005, -0.089840, 0.123603, -0.042480, -0.328093, 0.023814, -0.079097, 0.062549, -0.124070, 0.093475, 0.005966, 0.063865, -0.043735, -0.060457, 0.046918, -0.071535, -0.029020, 0.092402, -0.006788, 0.045067, 0.016266, 0.042471, -0.145939, -0.009645, 0.206575, -0.036372, 0.050235, 0.018615, 0.001174, -0.007066, 0.041973, -0.028442, 0.030848, -0.063840, 0.120457, -0.060283, -0.003688, -0.103413, -0.079604, 0.041151, -0.040618, 0.057419, 0.089978, 0.041155, -0.102569, 0.062587, 0.112777, 0.053299, -0.101019, 0.057724, 0.041480, -0.019897, 0.028515, -0.200851, -0.065658, -0.052666, -0.102024, -0.151931, -0.088357, 0.027571, 0.073328, 0.081327, 0.021530, 0.188177, -0.103126, -0.042821, 0.091477, 0.051598, -0.018914, -0.004137, -0.065633, 0.087704, 0.005653, 0.268261, -0.034925, -0.046203, -0.024108, -0.007113, 0.056439, 0.108912, -0.072613, -0.143521, 0.158838, 0.169516, 0.062593, 0.072433, 0.142935, 0.190626, -0.038709, 0.000126, -0.132907, -0.192268, 0.081422, -0.086519, 0.052337, 0.192407, -0.006755, -0.021974, 0.064198, -0.099124, -0.107474, -0.006143, 0.042024, 0.227668, -0.092579, 0.021494, 0.119977, 0.079441, -0.082294, -0.014176, -0.117550, 0.038603, 0.077356, 0.004786, 0.068164, 0.021303, -0.001576, 0.011788, 0.014040, 0.024215, -0.023952, -0.130248, -0.025207, 0.072400, -0.090933, 0.096239, -0.000126, -0.126587, 0.007267, -0.053093, -0.139487, -0.110832, 0.191887, -0.118758, 0.033068, 0.027524, 0.167369, -0.030523, 0.045911, -0.113458, 0.073496, -0.246999, 0.029344, 0.011007, 0.017994, 0.033210, -0.125035, 0.021767, -0.120438, 0.030030, -0.184470, 0.032325, -0.135146, -0.024644, 0.131049, -0.054377, -0.053634, -0.013256, 0.101624, -0.013015, -0.107712, 0.031939, 0.137379, -0.073813, -0.032689, -0.049828, -0.083212, 0.026137, 0.167743, 0.034698, 0.006738, -0.004483, -0.045914, 0.006484, -0.015429, -0.042880, -0.021523, 0.050307, 0.222664, 0.069132, 0.005886, -0.133332, 0.077401, 0.065246, 0.066960, 0.055472, 0.055087, -0.073146, 0.004020, -0.017526, 0.031164, -0.150450, 0.122602, 0.102606, -0.110788, 0.149482, 0.004407, 0.042420, 0.214760, 0.122977, 0.143685, -0.038605, 0.043683, -0.032923, -0.097494, 0.170746, -0.087356, -0.039094, 0.001184, -0.022729, 0.003225, 0.046162, -0.072199, -0.011280, 0.207409, -0.111453, -0.107994, -0.016733, -0.029588, 0.095434, 0.008704, -0.117800, 0.129408, -0.099176, 0.013107, -0.070949, -0.091330, -0.003796, 0.021579, 0.060386, 0.049683, -0.136666, -0.017506, -0.017655, 0.012702, -0.087432, -0.052076, 0.023241, -0.062531, 0.015498, 0.024510, -0.061477, 0.085329, 0.128621, -0.006324, -0.190141, -0.073316, -0.014300, -0.021231, -0.055816, -0.011991, -0.068223, -0.006668, -0.120381, 0.115878, -0.034345, 0.023790, -0.092656, 0.024306, 0.108706, -0.052800, -0.021444, 0.089790, 0.012379, -0.075952, -0.034582, 0.152334, 0.109856, -0.020560, 0.168608, -0.001634, -0.085670, 0.069779, -0.051637, -0.135192, -0.082813, -0.015428, 0.056553, 0.052404, 0.218124, -0.108295, -0.078747, -0.049933, 0.019072, 0.037976, 0.052120, 0.007398, 0.116835, -0.140742, -0.071222, 0.041988, -0.033098, -0.075759, -0.066147, -0.031270, -0.085516, -0.010901, -0.150823, -0.178391, 0.083699, -0.042407, 0.017517, -0.001683, -0.092927, -0.055061, -0.074748, 0.097853, 0.090266, -0.030140, -0.084443, -0.112408, -0.041116, -0.071044, -0.095332, -0.008164, 0.018481, -0.072650, -0.132295, 0.008647, 0.156598, 0.075697, -0.016603, -0.038884, -0.060629, 0.136098, -0.119714, -0.006067, -0.133970, -0.077915, -0.167316, 0.153001, -0.081720, 0.036344, 0.095969, -0.030352, 0.077044, 0.056533, 0.091012, 0.037306, -0.030482, -0.014527, -0.112834, 0.036857, -0.029891, -0.215195, -0.051652, 0.005394, -0.000769, -0.071290, -0.139909, -0.088678, 0.109333, 0.031721, -0.034737, -0.023321, -0.098007, 0.187967, 0.050030, -0.203190, 0.024169, 0.143164, 0.134861, -0.115096, -0.067046, -0.001817, -0.149922, 0.077590, -0.023559, -0.173918, 0.028038, 0.006208, 0.236414, -0.047157, -0.115196, 0.041254, 0.031154, 0.053235, 0.112157, 0.013485, 0.053232, -0.043587, -0.117773, -0.016338, -0.173317, 0.159853, 0.065806, 0.135034, -0.055219, -0.079416, 0.158325, -0.002260, 0.088523, -0.064872, -0.101351, 0.042363, 0.090688, -0.048518, -0.110268, -0.059717, -0.104193, -0.074488, -0.123310, -0.027266, -0.064861, 0.033804, -0.007288, 0.022970, -0.048597, -0.049142, 0.108557, -0.043785, 0.064863, -0.093374, -0.030771, -0.249076, -0.171171, -0.150191, 0.165696, -0.028811, -0.083749, -0.017608, -0.012782, 0.042869, -0.036941, -0.117571, -0.133073, -0.007499, 0.108215, -0.065739, 0.087491, 0.021730, -0.127748, -0.006363, -0.121411, -0.105073, -0.315914, -0.022765, 0.007690, 0.099982, 0.101420, 0.147188, 0.090874, 0.108933, 0.035279, -0.049512, 0.021875, 0.034695, -0.148833, -0.088689, -0.112720, -0.011542, -0.160989, -0.109315, -0.251373, -0.068871, -0.111011, -0.030127, -0.026648, -0.073859, 0.048350, -0.031524, -0.106804, -0.061243, 0.048530, -0.027073, -0.110453, 0.193959, -0.019973, -0.101817, 0.025764, 0.053087, -0.043234, 0.071182, -0.149352, -0.195861, -0.159304, 0.027748, -0.030367, -0.157580, 0.110373, -0.225392, -0.148966, 0.143434, 0.116526, 0.194409, -0.080505, -0.014888, -0.053022, 0.015967, -0.036483, -0.130443, 0.049618, -0.136442, -0.156172, -0.091701, -0.085794, 0.070613, -0.267142, -0.058667, -0.056816, 0.095079, -0.166588, -0.268938, -0.051983, 0.035435, -0.111635, 0.003555, -0.122874, 0.090623, -0.006589, -0.179115, 0.052751, -0.071274, -0.117713, 0.024670, 0.102909, 0.246344, 0.028224, -0.083995, -0.096026, -0.124928, 0.116205, -0.089863, 0.080344, 0.008705, -0.007929, 0.172648, -0.024322, 0.003752, -0.165519, 0.084981, -0.040836, 0.044203, 0.122635, -0.109542, -0.059820, -0.003197, -0.035226, -0.093214, -0.004123, 0.027874, 0.176464, 0.004209, -0.031144, -0.068636, -0.177605, -0.111524, -0.048778, -0.126856, 0.027967, -0.086051, -0.120192, -0.074432, -0.093254, -0.067565, -0.040958, -0.025646, -0.135444, 0.054505, 0.029185, -0.188362, -0.007335, 0.004951, 0.100286, 0.007818, -0.064171, 0.097564, -0.053638, 0.062231, -0.173665, -0.077156, 0.026076, -0.060690, -0.182474, -0.049005, 0.021145, -0.080703, -0.003160, 0.118147, -0.245967, 0.034739, -0.110083, -0.067656, 0.105221, 0.045056, -0.085775, -0.115718, -0.112291, -0.021178, -0.015345, -0.086034, -0.041232, -0.041474, -0.111443, -0.026968, -0.030757, 0.040496, -0.020220, -0.008413, -0.038502, -0.005205, 0.032057, 0.046193, -0.044713, 0.004011, 0.071863, -0.065448, 0.038259, 0.066567, 0.001453, 0.161954, -0.050723, -0.054000, -0.131840, 0.181133, -0.109312, -0.089919, 0.145300, 0.144842, 0.120759, -0.100774, -0.035852, -0.086338, 0.000641, -0.002963, 0.117933, -0.152698, 0.079652, -0.083893, -0.064471, -0.216394, 0.011515, -0.112178, -0.117178, 0.197594, 0.156747, -0.016600, -0.012648, -0.173751, 0.081377, -0.022291, -0.107914, 0.004152, -0.151973, 0.065781, -0.022203, -0.026391, -0.012050, 0.013742, -0.071692, -0.126754, -0.031159, -0.061168, 0.047975, 0.068789, -0.086390, 0.108836, 0.141575, 0.126633, -0.060161, -0.157398, -0.182378, -0.003537, -0.152681, 0.054282, -0.201889, -0.129038, -0.071822, 0.093924, 0.019111, -0.146600, -0.070746, -0.037524, -0.087249, -0.082789, 0.159890, 0.107385, 0.069994, -0.125598, 0.067421, -0.074085, 0.105610, 0.006482, -0.075154, 0.149667, -0.099059, -0.033344, -0.042296, 0.007989, -0.051144, -0.038015, 0.027585, 0.033178, -0.011812, -0.065347, 0.098332, -0.057643, -0.040938, 0.069607, -0.076291, 0.052531, -0.190654, 0.055021, 0.002617, 0.156015, 0.024479, 0.068101, 0.062592, 0.028439, 0.022029, 0.004032, 0.115887, 0.114265, -0.056220, -0.062561, 0.097927, 0.029074, 0.034799, -0.173787, -0.014999, -0.015789, 0.059694, 0.113057, -0.008059, -0.048405, 0.157586, -0.031565, -0.105501, -0.054663, 0.016578, 0.168539, -0.042692, -0.066229, -0.011002, 0.006278, 0.152517, -0.010699, -0.062938, -0.129276, -0.130796, 0.054334, -0.031461, -0.020322, -0.061863, -0.017902, 0.036192, -0.266152, 0.006209, -0.029106, -0.014665, 0.016082, -0.027500, -0.015445, -0.016836, 0.075976, -0.112164, 0.214892, -0.057798, -0.102994, 0.100317, -0.009883, -0.011138, -0.028186, 0.118172, -0.062113, -0.170218, -0.021737, -0.104577, 0.034010, -0.067139, -0.222145, 0.212909, -0.043841, 0.061825, -0.108610, -0.105388, 0.085274, 0.023294, -0.067480, 0.056708, 0.161212, 0.077287, -0.047113, 0.038842, 0.130118, -0.037912, 0.134183, -0.020092, 0.024762, 0.038315, 0.010419, 0.102280, -0.053996, -0.008889, 0.000764, -0.183089, -0.095921, -0.064591, -0.143277, -0.129270, -0.153964, 0.042799, 0.016016, 0.134972, 0.031311, -0.312111, -0.077233, -0.040005, -0.109627, 0.039140, 0.007234, -0.133608, -0.085972, -0.097715, -0.076997, -0.075594, 0.007028, -0.057237, -0.239508, -0.123948, 0.069429, 0.163685, 0.036929, -0.160868, -0.169395, -0.114597, -0.115751, -0.091053, -0.060400, 0.067821, 0.144153, 0.132019, -0.121562, -0.215781, -0.135158, -0.114949, 0.129591, 0.007426, -0.150770, 0.104883, -0.055898, -0.116148, -0.014033, -0.115661, -0.151382, 0.022568, 0.066930, 0.082830, -0.104657, -0.153416, -0.096655, -0.008559, -0.136368, -0.056433, 0.021403, 0.023651, -0.025558, -0.163072, 0.053725, -0.047198, 0.008052, 0.031127, -0.094185, -0.011264, -0.139642, -0.084853, -0.043300, -0.063191, 0.075187, -0.067488, -0.027889, -0.093439, 0.012233, -0.062308, -0.000756, -0.005080, 0.000222, 0.030307, -0.172609, -0.192623, 0.053044, -0.003245, -0.131028, 0.026132, 0.040326, 0.109084, -0.143978, -0.196973, 0.146575, 0.101468, -0.144427, 0.070830, 0.038363, -0.029374, -0.210822, -0.014200, 0.017204, -0.016821, -0.041697, 0.063953, 0.005922, -0.028839, -0.038378, -0.394938, 0.048958, -0.183215, -0.217314, -0.041148, -0.191355, -0.091649, -0.115266, -0.016999, -0.058485, 0.067134, -0.063879, -0.105151, 0.026729, -0.011734, 0.004218, -0.026165, 0.127728, -0.126673, -0.046794, 0.034425, -0.076752, 0.111983, 0.004581, -0.210351, -0.204567, 0.056670, -0.006775, -0.167200, 0.000019, 0.026451, -0.149050, -0.090853, -0.089131, -0.094656, -0.093403, -0.031001, -0.028681, 0.023772, 0.126474, 0.088194, -0.132567, -0.028160, -0.090261, 0.063427, 0.006505, 0.063987, -0.057951, -0.043484, -0.015106, 0.012584, -0.140878, -0.005560, -0.108101, -0.028458, 0.103267, -0.204323, 0.042848, -0.103790, -0.171509, 0.109017, 0.109992, -0.013748, 0.015687, 0.059537, -0.114245, 0.029090, -0.122885, 0.022265, -0.026376, -0.024221, 0.095049, -0.175109, -0.013453, 0.044993, -0.056094, -0.215022, -0.007812, -0.132254, -0.102332, 0.096706, 0.207768, -0.115265, -0.114925, -0.201132, -0.007182, 0.067029, -0.137812, 0.005168, -0.006961, -0.020794, -0.046648, -0.132116, -0.040318, -0.230655, -0.050666, -0.085052, 0.146401, -0.206507, -0.015381, -0.121159, -0.038881, 0.047402, -0.174327, -0.055665, -0.071584, 0.127484, 0.063647, 0.024398, -0.075751, -0.005655, -0.010370, -0.034079, 0.118864, 0.122564, 0.015608, 0.109511, -0.134150, -0.092401, -0.151053, -0.001388, 0.029381, -0.029165, 0.050231, -0.043443, -0.160328, 0.017937, -0.136200, 0.079261, -0.109399, -0.018539, -0.002950, -0.020649, 0.028684, 0.013506, 0.015669, -0.002649, 0.079547, 0.049583, 0.109039, -0.074567, -0.030830, -0.120750, 0.006241, -0.008622, -0.007539, 0.034243, 0.005502, -0.143947, -0.086839, 0.062640, -0.059563, -0.055134, 0.061047, -0.017857, -0.013690, 0.050273, -0.117497, -0.232094, 0.009935, -0.148579, -0.028493, -0.045629, -0.035663, -0.111834, 0.001821, -0.135393, -0.093947, 0.011369, -0.143318, -0.084329, -0.085459, -0.079285, -0.024742, -0.002997, -0.060999, 0.053049, -0.170000, -0.143206, -0.064530, 0.125493, -0.100174, 0.093276, -0.070517, -0.091718, -0.121696, 0.011138, -0.075774, -0.166890, -0.129733, -0.000295, 0.149983, 0.016908, -0.005948, 0.006269, -0.213603, 0.068243, -0.098296, 0.077585, 0.081334, -0.019777, -0.066966, -0.113370, -0.046785, -0.009583, -0.009870, -0.088502, -0.120125, -0.160068, -0.138138, 0.061591, -0.124891, -0.061637, 0.080544, -0.060810, -0.075052, 0.086513, -0.116099, -0.213514, -0.168196, 0.112932, 0.024139, 0.044200, 0.048236, -0.023796, -0.033069, -0.186392, 0.030800, 0.034833, -0.128701, -0.243361, -0.100876, 0.028121, -0.046352, 0.066099, 0.090666, -0.071198, 0.035115, -0.073675, -0.042346, -0.046082, 0.023658, -0.074510, 0.006956, 0.084002, 0.034657, -0.083783, 0.000634, 0.016675, -0.005387, 0.017514, -0.028896, -0.047780, -0.034604, -0.149868, -0.010960, -0.098245, 0.090854, -0.004148, -0.071747, 0.006076, -0.072805, 0.065022, 0.018813, -0.082207, -0.093771, 0.000353, 0.109510, -0.058698, -0.106059, -0.126777, -0.156781, 0.000611, 0.054106, 0.069460, -0.092583, -0.005714, -0.050136, 0.104519, 0.074661, -0.037266, -0.116246, -0.144223, -0.007601, -0.024597, -0.048853, -0.025553, 0.017304, -0.016361, -0.036639, -0.018004, -0.142550, 0.025353, -0.061898, -0.013529, -0.012071, -0.103970, -0.099104, 0.002642, 0.055262, 0.021561, -0.045603, -0.112036, 0.067356, 0.035881, -0.006767, -0.088828, 0.037021, -0.137600, -0.118281, -0.019758, 0.000422, -0.018415, -0.044755, -0.093424, 0.043537, -0.017035, -0.020834, 0.034421, -0.011181, -0.067299, -0.104182, -0.081453, 0.061552, 0.060433, 0.015663, -0.033849, 0.024676, -0.109997, -0.020203, -0.014209, -0.020718, 0.054611, -0.035109, -0.006201, -0.136809, 0.075710, -0.085297, -0.106585, -0.083763, -0.126454, 0.048720, -0.025818, -0.087855, -0.136786, -0.000662, -0.000832, -0.163821, -0.016359, -0.086828, -0.024135, 0.005262, 0.042012, -0.067846, -0.023317, -0.140769, 0.012293, -0.035212, -0.070339, 0.026303, 0.013691, -0.053194, -0.098246, -0.060776, -0.051510, 0.030277, 0.064551, -0.167256, -0.100860, 0.067397, 0.005061, -0.111391, 0.080897, -0.077222, 0.096614, 0.051054, 0.017623, 0.006714, -0.145824, 0.030931, -0.109226, -0.113076, -0.043264, 0.069659, -0.015159, -0.016959, -0.119577, 0.059987, -0.007545, 0.164871, -0.178215, -0.020156, -0.006880, -0.008039, 0.168732, 0.054661, 0.055049, 0.089445, 0.092125, -0.043501, 0.033850, 0.123987, -0.070662, -0.015445, -0.033653, -0.102806, -0.104483, -0.140883, 0.032283, -0.014025, 0.017133, 0.028500, -0.069607, -0.098021, -0.060538, -0.010115, -0.008227, 0.108072, -0.100245, 0.138193, -0.028097, 0.027327, -0.038005, 0.137640, -0.048409, -0.030424, -0.059278, -0.023511, -0.165785, -0.184085, -0.166871, -0.089859, 0.059096, 0.150706, 0.042200, 0.006399, -0.081862, -0.100058, -0.049365, -0.068263, -0.096522, -0.045429, -0.170809, -0.090073, 0.061684, -0.113549, -0.051997, -0.019618, 0.023939, 0.046631, 0.056797, 0.006206, -0.032168, -0.129923, -0.006077, 0.090844, -0.142979, 0.034182, -0.094065, -0.076553, -0.086705, -0.046548, -0.085139, 0.082820, -0.053477, -0.109257, -0.107919, -0.076493, -0.132548, 0.042857, -0.077154, -0.146520, -0.079550, 0.030416, 0.035348, 0.062055, 0.069670, -0.115162, -0.002854, -0.147792, 0.032789, -0.087374, -0.016855, 0.075100, 0.066412, 0.085670, -0.152495, -0.112928, -0.113986, 0.073483, -0.202942, -0.114838, -0.082949, 0.052516, -0.095854, -0.005997, 0.019388, 0.002759, 0.120895, -0.156853, -0.057292, 0.057837, -0.013090, 0.057168, -0.087874, -0.065939, -0.010881, 0.041237, 0.130573, 0.045813, -0.051741, -0.188601, -0.021050, -0.015702, 0.024079, 0.026703, -0.017392, 0.035659, -0.105213, -0.117430, -0.081519, -0.151303, 0.051120, -0.043803, 0.101718, -0.002939, -0.161444, 0.003457, 0.073334, 0.045483, -0.075426, -0.025854, -0.046104, 0.250167, 0.094958, -0.006111, 0.061536, 0.036668, -0.172796, 0.050142, 0.039115, 0.020336, -0.054195, -0.011560, 0.020544, 0.051546, -0.015950, -0.078721, -0.151870, 0.047631, 0.097421, 0.051678, -0.090672, -0.060404, 0.052199, 0.015891, 0.060557, -0.118766, -0.071258, -0.127083, -0.166365, -0.007769, -0.157822, -0.168691, -0.010145, 0.059842, 0.019810, -0.020838, -0.134594, 0.036198, -0.153485, -0.038667, -0.045879, 0.001924, -0.103901, -0.134965, 0.002859, 0.021384, -0.038127, -0.136621, -0.062895, -0.066012, 0.067669, -0.061461, -0.001237, -0.032453, 0.001870, -0.037399, 0.083828, 0.026226, -0.044692, -0.020478, 0.041993, -0.055840, 0.007978, 0.014430, -0.123201, -0.017959, -0.028547, 0.073040, 0.052153, -0.086668, -0.202699, -0.025745, -0.112547, -0.018114, 0.025375, -0.135810, -0.073711, -0.119112, 0.020938, -0.000089, -0.029914, 0.075723, -0.009164, 0.030042, -0.007005, 0.023572, -0.002674, -0.040381, -0.072924, -0.062264, -0.151144, -0.067335, 0.082397, -0.066790, -0.142529, -0.112966, -0.040472, 0.103290, -0.094637, 0.034678, 0.003285, -0.100616, 0.115250, -0.016859, -0.046460, -0.071704, 0.027739, 0.021897, -0.143725, 0.051473, -0.010150, 0.004289, -0.130885, 0.037414, -0.118046, -0.062863, -0.016052, -0.100112, -0.137082, 0.046010, -0.117231, -0.125465, -0.090434, -0.061468, 0.062527, 0.135838, -0.106173, -0.070717, -0.049267, 0.047096, -0.101740, -0.153127, 0.062560, -0.082060, -0.157556, 0.129820, -0.084881, -0.120953, 0.068747, 0.112557, -0.080562, -0.017443, -0.027502, -0.144805, -0.028341, -0.007889, -0.072237, 0.081385, 0.019706, 0.051381, 0.008085, 0.042344, 0.017038, 0.110147, -0.060396, 0.050365, -0.140826, -0.146293, -0.101916, 0.064790, -0.049643, 0.023685, -0.139293, -0.073554, -0.029394, -0.032753, 0.043729, 0.043749, 0.117182, -0.040966, 0.144990, -0.129600, 0.111576, -0.018164, 0.061688, -0.047513, -0.037041, -0.069994, 0.001708, 0.048826, 0.048584, 0.085076, -0.016297, -0.123460, -0.063315, -0.111595, -0.054026, -0.036846, -0.084717, -0.070325, 0.059200, -0.004668, 0.071493, 0.055626, 0.015416, -0.039685, -0.057187, 0.035305, -0.177211, 0.047484, -0.129393, -0.249386, 0.057174, -0.147246, 0.065168, -0.001256, -0.060545, 0.027675, -0.070815, 0.052601, -0.164170, 0.074378, 0.055087, 0.026302, -0.059446, -0.138350, -0.181576, 0.089484, 0.099279, -0.030497, 0.195346, -0.071608, -0.074335, -0.280353, -0.076279, -0.075073, 0.038025, -0.240784, -0.037179, -0.132946, 0.140312, 0.059861, 0.015005, -0.116603, 0.019391, -0.057016, 0.091232, -0.099044, -0.269772, -0.013925, -0.034097, -0.055830, -0.184001, 0.040300, 0.045681, -0.116302, -0.170992, 0.023004, -0.031721, 0.028657, -0.109784, -0.026474, 0.114603, -0.158460, 0.071954, -0.146382, 0.183542, -0.083915, 0.097065, -0.162784, 0.007165, 0.111056, 0.085973, -0.030248, 0.041155, 0.066624, 0.033229, -0.060372, 0.103747, 0.096510, -0.120529, 0.046396, 0.015468, -0.060840, 0.016666, -0.094071, 0.199359, 0.059778, 0.007744, -0.074381, -0.048514, 0.052665, 0.111234, -0.040742, 0.002256, 0.094625, -0.115741, 0.055073, -0.030110, -0.189383, 0.050292, -0.058225, 0.001262, -0.054226, 0.054126, -0.101918, -0.073435, -0.223862, -0.070528, 0.049332, 0.087659, 0.013461, -0.096705, -0.012674, 0.095976, -0.036781, 0.143048, 0.048210, 0.049428, -0.166918, 0.065587, 0.050356, -0.036781, 0.013410, -0.057440, -0.074150, -0.035183, 0.113350, -0.027853, -0.059010, -0.073445, -0.023270, 0.057904, 0.122558, -0.137268, -0.047921, -0.075946, -0.065115, -0.163687, 0.058779, -0.060253, 0.148161, 0.001213, 0.021911, 0.003715, -0.008802, 0.239290, 0.169314, -0.132672, -0.137972, -0.025396, -0.160871, -0.041585, 0.078807, -0.115711, -0.095125, -0.071074, -0.071739, 0.003994, -0.108202, 0.146434, 0.033370, -0.039487, 0.070185, 0.018054, -0.062368, 0.045169, -0.051988, -0.021586, 0.015119, 0.080216, 0.049772, -0.113294, -0.121293, -0.020525, -0.162923, 0.109469, -0.044126, -0.003076, 0.026487, -0.119247, -0.141305, -0.056630, 0.058862, -0.065958, 0.115450, -0.007363, -0.099002, -0.008380, -0.039203, 0.036759, -0.006507, -0.147973, 0.022365, 0.094555, -0.099839, -0.031687, 0.082173, -0.126378, -0.075653, 0.121101, -0.222985, 0.040924, -0.031961, 0.054727, -0.074743, -0.072351, -0.064997, 0.067329, -0.092790, -0.045843, 0.076794, -0.010529, -0.038401, -0.067844, -0.143684, -0.060390, -0.025635, -0.080102, -0.017691, -0.145730, 0.113963, -0.013478, -0.012486, 0.103136, 0.064785, 0.083160, -0.058007, -0.006563, -0.132216, -0.226364, 0.035451, 0.022713, 0.018599, -0.044258, -0.024229, -0.030399, -0.099722, -0.115895, -0.036544, -0.173395, -0.016583, -0.120036, -0.037578, -0.147025, 0.030973, -0.069296, -0.096503, -0.005539, -0.106656, 0.007447, -0.086637, 0.067879, 0.042965, 0.083424, 0.094062, 0.120966, 0.108649, 0.179096, -0.035639, 0.085192, 0.087117, -0.053979, -0.056925, -0.035446, 0.145312, -0.005606, -0.024900, -0.107811, 0.084954, -0.027720, 0.018908, -0.128826, -0.182368, -0.103605, -0.088546, 0.014185, -0.080249, -0.230498, -0.028909, -0.129482, 0.052941, -0.074701, -0.081246, -0.077731, -0.129628, -0.037602, -0.014599, 0.011963, -0.027925, -0.008442, -0.058601, 0.011118, -0.060032, 0.046800, -0.092579, -0.012368, -0.035810, -0.061257, 0.031693, -0.107239, -0.077754, -0.123133, -0.071007, 0.053820, 0.008853, 0.005243, 0.036442, -0.016083, -0.038925, 0.008787, -0.087659, -0.009856, -0.117998, 0.096711, -0.023190, 0.062874, -0.096450, -0.056009, -0.096594, -0.114379, -0.099835, -0.022087, -0.042725, -0.046531, -0.032108, -0.059165, -0.111028, 0.056814, -0.098655, 0.017832, 0.060134, -0.077763, -0.010346, -0.085392, 0.029299, -0.078973, -0.106634, -0.077720, 0.006093, -0.030253, -0.066054, -0.082985, 0.048307, 0.007340, -0.066841, -0.007212, 0.110366, -0.046212, 0.026518, 0.068355, -0.147290, 0.005281, 0.048951, -0.105598, 0.073331, 0.077620, -0.120632, -0.138130, -0.021679, 0.035618, 0.039467, -0.013495, -0.065657, 0.037684, -0.031594, 0.033064, 0.045801, -0.168088, 0.113769, -0.087720, -0.087739, -0.066799, -0.144477, 0.208280, 0.089675, 0.101462, 0.023994, -0.119786, 0.071165, 0.035918, -0.181156, -0.098001, 0.171515, 0.041430, 0.027495, -0.001000, 0.100818, 0.036853, -0.009020, -0.053467, -0.051423, -0.042202, 0.004261, 0.027975, 0.008570, -0.230604, 0.016644, 0.056851, 0.042126, 0.025783, 0.109654, 0.083604, -0.052260, -0.061549, 0.151190, 0.022221, -0.045563, -0.096668, -0.031675, -0.146833, 0.007339, -0.029045, 0.080612, 0.046680, -0.015058, -0.060251, 0.039983, -0.003482, -0.051996, -0.017026, -0.014562, -0.037065, 0.019310, -0.168659, 0.043711, -0.208882, 0.033571, -0.071807, -0.077137, -0.111138, 0.055613, 0.156116, -0.128374, 0.040579, 0.098915, -0.082687, -0.082330, -0.072119, -0.108712, 0.072664, 0.033439, 0.057784, 0.103735, 0.020427, 0.174596, -0.000163, 0.060901, 0.118798, 0.066827, 0.164229, 0.067554, -0.024778, 0.084611, 0.235916, 0.073540, 0.054253, 0.009681, -0.004989, 0.007516, 0.091052, -0.060312, 0.079626, -0.023869, 0.068642, 0.041102, -0.106328, -0.018706, -0.087731, 0.017396, -0.133611, -0.079406, -0.086697, -0.069688, -0.044234, 0.059643, -0.056414, -0.081905, 0.076002, 0.058908, 0.088377, 0.056908, -0.048129, 0.015750, 0.095042, 0.010080, 0.022002, 0.074985, -0.182433, -0.036118, -0.116145, -0.069004, -0.127161, -0.029668, -0.112119, -0.085980, 0.056309, 0.148816, 0.027945, -0.138086, 0.178568, -0.029127, -0.066154, 0.056752, -0.023537, -0.010119, -0.077204, -0.072150, -0.002608, -0.019286, 0.024144, 0.020020, -0.074722, 0.119429, -0.028389, 0.230122, -0.068982, 0.123281, 0.044308, 0.010979, -0.000165, 0.013637, -0.061842, -0.063384, 0.085443, 0.024084, 0.082826, -0.123831, -0.023217, -0.086497, 0.025792, -0.078563, 0.020476, 0.193445, -0.005141, -0.098221, -0.082281, 0.095938, 0.045511, -0.059979, 0.058637, -0.201512, -0.010404, -0.023820, -0.000435, -0.047664, -0.195836, -0.088135, 0.068934, -0.010124, -0.069170, -0.023301, -0.029881, -0.064577, -0.136678, -0.142195, 0.171773, 0.132389, 0.052187, -0.026161, 0.167304, 0.136237, -0.044622, -0.109196, -0.175536, -0.103894, 0.029569, 0.013442, 0.082235, -0.041401, 0.014286, -0.145687, 0.000653, 0.024088, 0.113097, 0.057207, -0.038540, 0.098082, 0.103404, -0.066404, 0.118982, -0.043605, -0.062578, -0.080189, 0.028478, -0.227105, -0.198524, -0.131768, 0.073300, -0.056673, -0.088128, -0.089447, 0.008031, -0.153737, -0.045709, -0.107715, 0.016444, -0.182028, 0.035936, -0.085042, 0.004110, -0.149459, -0.227653, -0.076441, -0.144213, -0.116496, -0.094603, -0.129568, -0.008741, 0.006558, -0.009322, -0.131242, -0.031838, -0.106744, 0.009309, 0.120170, -0.048628, 0.114859, 0.067513, -0.005770, 0.014038, -0.091763, 0.110884, -0.039031, -0.171433, -0.210430, -0.101487, 0.052184, -0.126430, -0.036605, -0.052994, -0.006072, 0.051719, -0.016216, -0.071416, -0.041359, 0.012007, 0.084656, -0.083831, -0.056303, -0.125950, -0.018342, -0.027392, 0.069368, -0.032142, 0.044999, 0.027914, -0.050264, -0.138030, -0.036672, 0.008389, 0.038634, 0.114108, -0.060147, -0.274457, -0.056945, -0.092656, -0.041278, -0.041540, -0.072814, 0.012455, -0.139141, -0.131693, -0.079803, -0.140814, -0.298090, 0.107119, -0.158335, -0.016712, -0.061553, -0.058579, -0.081262, -0.054171, 0.120912, -0.010834, -0.221479, 0.109195, -0.113612, 0.059440, -0.173484, -0.080804, 0.208621, -0.008770, -0.086663, 0.022000, -0.016174, -0.009680, 0.046040, 0.001341, -0.078206, -0.070069, -0.003192, 0.010387, 0.025958, -0.080031, -0.054274, -0.046168, -0.099043, -0.111166, -0.045045, -0.042671, -0.117107, 0.016633, 0.101610, 0.197905, -0.009198, 0.061220, -0.155751, 0.008762, -0.060109, -0.038536, 0.026279, -0.229633, -0.079314, -0.018434, 0.062764, 0.009817, -0.153060, -0.166417, -0.095618, 0.024848, -0.110382, 0.054729, -0.076345, -0.072270, 0.032688, -0.065124, 0.095779, -0.037966, 0.104301, -0.050805, -0.073454, 0.070531, 0.026446, 0.019300, -0.058059, -0.035844, -0.042913, 0.055712, 0.015054, 0.000891, -0.245412, -0.061572, -0.100891, 0.148809, -0.314346, 0.016689, -0.066376, -0.300216, 0.112239, 0.048092, 0.095277, -0.029494, -0.003905, -0.139879, -0.013146, -0.074076, 0.035819, -0.167039, 0.033349, -0.349845, -0.013177, -0.075665, 0.015956, -0.095365, 0.115758, -0.153874, -0.243331, 0.035533, -0.160267, -0.118767, -0.027059, -0.092553, 0.064590, -0.079095, 0.027039, -0.172184, -0.163336, -0.116022, -0.035109, 0.297735, -0.064080, -0.011405, -0.020605, -0.005939, -0.173502, -0.155222, 0.087179, -0.061505, -0.066256, -0.063145, -0.203344, -0.030590, 0.014133, -0.009595, -0.127894, 0.071135, -0.038925, -0.008408, 0.053228, -0.063221, 0.012299, 0.128464, -0.078871, -0.030202, 0.086567, -0.044282, 0.110487, 0.061161, -0.093802, -0.122253, 0.034295, -0.049642, -0.108700, 0.010393, 0.058036, -0.096589, 0.018993, -0.024453, 0.116995, 0.135421, -0.047965, -0.054556, -0.006804, -0.187042, 0.162696, 0.046328, 0.128447, 0.118221, 0.054481, -0.164329, 0.003167, 0.102233, -0.125449, 0.050190, 0.028850, -0.114217, -0.003602, 0.018664, -0.091796, -0.434414, -0.090518, -0.096930, -0.061796, -0.072217, -0.034295, -0.196853, 0.042523, -0.054459, -0.054183, -0.150214, -0.033314, -0.154321, 0.043854, 0.089156, -0.145225, 0.090898, 0.038740, 0.077110, -0.043618, -0.082285, 0.200662, 0.020806, -0.006232, -0.118114, 0.045669, -0.090796, -0.077409, 0.211521, -0.004308, -0.127790, -0.158419, 0.222572, -0.125652, 0.145233, -0.084423, 0.129958, 0.067044, 0.021733, -0.083157, 0.179133, 0.052931, -0.090668, -0.088333, 0.014447, 0.029266, -0.259841, -0.095884, -0.043976, 0.117906, -0.155420, -0.033065, -0.093155, 0.067246, -0.019129, -0.002000, -0.153061, -0.229062, 0.104068, -0.192380, -0.011651, -0.002346, -0.252012, 0.011180, -0.324709, -0.125759, 0.101356, -0.089823, 0.063342, 0.015731, -0.057132, -0.002828, -0.260994, -0.037187, -0.123856, 0.075064, -0.098025, -0.118518, 0.127290, 0.002194, -0.107185, 0.059813, -0.205168, -0.171980, -0.152703, -0.150903, 0.041138, -0.277319, -0.121382, -0.113464, 0.086036, -0.094393, -0.206729, -0.117303, -0.195145, -0.096943, 0.003614, -0.031714, 0.055012, 0.096844, 0.073072, -0.044472, 0.055993, 0.000899, -0.006958, 0.018457, -0.074636, -0.011490, -0.180614, -0.120120, -0.045428, 0.003380, 0.124533, 0.025319, -0.125360, -0.209269, -0.015677, -0.046134, 0.039399, 0.068729, -0.017903, -0.123143, -0.133799, 0.038098, -0.019442, 0.070243, -0.050013, 0.064597, -0.088034, -0.045302, 0.075975, 0.015425, 0.018252, -0.135353, 0.047426, -0.054702, -0.234901, -0.062426, -0.034964, 0.000295, -0.115879, 0.027389, 0.027928, -0.107112, 0.042530, -0.101335, 0.083280, -0.091848, 0.066253, -0.261683, -0.072630, 0.050634, -0.074930, 0.144325, -0.000976, -0.094524, -0.033322, -0.000171, -0.005050, -0.103494, 0.059872, -0.062285, -0.122841, -0.115786, 0.061708, -0.028742, 0.014342, 0.052456, 0.009823, 0.102569, 0.059656, -0.022265, 0.062231, 0.010834, -0.004278, 0.192530, -0.098894, -0.128283, -0.074329, 0.037042, -0.062316, 0.017556, -0.172978, 0.055892, 0.098666, 0.055744, 0.126940, 0.105741, -0.006136, -0.078843, 0.077481, 0.005758, -0.133180, -0.128704, 0.084610, 0.075500, -0.259561, 0.154910, 0.114283, 0.062311, -0.185992, -0.062943, -0.286213, 0.011525, -0.010639, -0.209634, -0.156427, 0.067745, 0.009622, 0.087996, 0.068872, 0.136684, -0.086609, -0.194344, 0.022642, -0.102270, 0.011065, 0.065363, -0.004647, -0.397334, -0.148144, -0.105005, 0.074224, -0.053787, 0.031204, 0.220918, -0.195159, -0.070500, -0.097969, -0.135300, -0.076930, 0.038107, -0.158058, -0.110190, -0.009068, -0.165306, -0.302885, -0.058600, 0.013975, -0.148461, -0.185913, 0.108416, 0.002641, -0.203127, -0.062463, -0.182013, -0.011069, 0.026151, 0.045043, 0.002815, -0.052553, -0.123320, -0.138330, -0.136340, -0.057874, -0.014058, 0.105941, -0.120548, -0.110280, -0.007812, -0.243077, 0.041930, -0.122283, -0.120697, -0.005344, -0.143094, 0.018032, -0.134278, -0.134617, -0.123660, -0.175345, 0.108093, 0.049749, 0.049668, 0.027092, 0.087432, 0.031823, -0.243276, -0.137235, -0.058067, 0.123507, 0.132382, -0.024515, -0.007315, 0.069884, 0.003869, 0.165826, -0.051705, -0.048881, 0.018758, 0.038887, 0.101287, -0.078906, 0.062002, 0.047360, 0.182061, 0.017613, -0.227564, -0.137294, -0.089591, -0.110889, 0.022109, 0.117321, 0.016938, 0.034929, -0.124403, -0.151349, 0.072093, -0.088243, 0.017915, -0.145111, -0.034258, -0.116637, -0.091803, -0.020433, 0.104092, 0.063917, -0.045417, 0.035980, 0.023577, -0.178420, -0.075415, 0.053286, -0.102139, -0.208257, -0.050567, -0.235402, -0.141605, -0.071333, 0.000721, 0.014639, -0.068167, 0.026542, -0.148422, -0.267910, -0.126836, -0.106282, 0.036794, -0.001877, 0.122332, -0.030332, 0.021241, -0.020832, -0.022291, -0.233678, -0.027215, -0.144049, 0.082887, 0.002253, 0.066991, 0.047753, 0.088270, -0.228495, -0.080941, -0.203726, -0.108397, 0.050967, -0.084531, -0.104977, -0.041803, 0.015468, -0.012553, 0.016533, 0.090656, -0.009974, -0.084743, -0.049727, 0.063210, -0.120026, 0.003749, 0.164630, 0.080907, -0.005208, -0.167614, 0.018920, 0.049949, -0.042633, 0.302108, -0.163759, -0.011840, -0.126113, 0.013072, -0.054209, -0.063138, 0.000710, -0.045714, -0.012816, 0.023638, -0.083559, 0.161987, -0.040200, 0.097409, -0.024086, -0.091961, -0.086014, 0.041834, 0.108626, 0.075057, -0.152771, 0.122554, -0.001515, -0.051740, -0.217705, -0.094828, -0.091065, -0.139765, 0.134990, -0.121110, 0.057494, 0.087112, -0.007743, -0.081827, -0.055436, 0.039349, -0.183878, 0.041346, 0.063767, 0.118846, -0.149220, 0.001159, 0.040194, 0.056220, -0.088376, 0.090335, -0.124117, 0.096827, 0.006342, 0.000998, 0.057866, 0.057910, -0.063053, -0.176552, -0.175055, 0.029595, -0.046145, -0.088072, -0.038660, -0.008767, -0.050873, -0.003306, 0.006270, 0.031840, -0.066405, 0.024956, -0.001143, -0.166575, 0.057557, 0.098314, 0.031349, 0.100997, 0.091789, -0.041701, 0.046465, -0.026324, -0.241910, 0.057723, -0.276172, 0.032408, -0.008253, -0.123853, 0.114917, -0.007677, -0.034426, -0.031262, 0.041463, 0.095656, 0.059515, 0.126060, -0.003316, -0.056387, -0.077166, -0.064688, -0.131127, 0.011004, -0.067938, -0.009409, 0.026847, -0.123661, 0.059797, -0.082475, -0.032437, 0.023672, 0.118099, -0.113500, -0.147215, -0.028275, 0.038605, 0.045743, 0.118949, -0.027397, -0.099315, -0.089435, -0.024213, 0.126677, 0.104378, -0.077688, 0.231710, -0.139155, 0.100351, -0.023684, -0.075703, -0.112733, 0.132503, 0.111363, -0.104170, -0.034364, -0.050520, 0.105596, 0.052498, -0.024544, 0.015754, -0.053246, 0.005268, -0.009522, -0.052806, 0.041325, 0.061655, -0.124384, -0.119193, -0.138990, 0.006371, 0.187548, 0.078385, -0.212335, 0.030460, 0.049768, 0.045856, 0.017842, 0.058355, -0.017492, -0.068573, -0.122512, -0.136114, -0.149518, -0.068272, -0.112481, -0.015888, -0.030768, 0.030774, -0.173485, -0.028118, -0.108420, -0.060957, 0.115317, 0.091527, 0.103866, 0.106072, -0.087824, -0.075364, 0.094952, 0.016072, -0.045483, -0.011346, 0.029547, 0.046714, 0.058523, 0.070342, 0.054730, 0.115607, -0.018809, -0.059960, -0.175178, -0.139351, 0.140447, -0.165268, -0.061533, -0.018630, -0.029451, 0.095593, -0.093508, -0.065167, 0.080115, -0.009687, -0.084897, -0.019409, 0.032809, 0.028101, -0.004757, 0.027390, -0.186223, -0.043376, -0.039173, -0.128870, 0.071574, 0.207600, 0.239058, -0.019399, -0.218449, 0.029216, 0.085979, -0.057551, -0.023627, -0.023202, 0.004803, -0.003504, 0.104317, 0.079433, -0.027330, 0.012400, -0.153557, -0.070710, -0.014740, -0.028438, -0.046415, -0.211059, -0.180244, -0.054970, -0.015123, -0.080934, -0.013008, -0.049470, -0.244959, 0.204567, -0.147449, -0.001297, 0.011021, 0.031001, -0.074338, 0.057228, 0.016403, 0.072926, -0.065760, 0.031633, -0.120051, -0.061770, -0.240044, 0.020516, 0.049325, -0.095355, -0.190882, -0.060042, 0.027001, -0.065211, 0.067188, 0.079095, 0.135263, -0.007892, -0.105054, -0.108175, -0.040269, -0.055570, -0.203389, 0.024020, 0.096003, -0.074282, -0.138407, 0.022491, -0.097667, 0.041994, 0.076768, 0.134967, -0.166755, -0.006565, 0.089069, 0.156837, -0.017735, 0.040221, -0.102891, -0.001886, -0.078941, 0.068729, -0.060030, 0.022049, 0.011720, -0.048167, 0.055501, 0.003690, -0.038797, 0.020332, 0.018427, 0.111684, -0.078287, -0.073337, 0.036260, 0.029414, -0.163856, 0.052863, 0.015253, 0.071898, -0.070490, -0.043045, -0.094456, -0.046148, -0.104983, -0.006070, 0.065275, 0.017658, -0.028080, 0.019701, -0.046577, -0.021035, -0.019473, -0.097182, -0.119315, -0.034772, -0.064194, -0.076303, -0.018434, -0.037674, -0.030424, -0.005148, 0.025940, -0.032261, -0.058015, -0.172679, -0.112101, 0.036858, -0.069307, 0.100350, -0.012289, 0.202587, 0.100946, -0.142325, -0.162014, 0.158907, -0.054249, -0.009809, 0.093780, -0.088725, -0.128247, 0.067229, 0.102042, -0.010686, -0.118825, -0.160370, -0.139666, 0.054414, 0.017472, 0.032111, 0.017794, 0.015864, -0.056455, 0.101918, -0.161686, -0.110958, -0.122129, -0.196465, 0.180613, 0.089768, -0.092938, -0.179381, -0.158884, -0.039821, 0.010055, -0.006106, -0.045653, -0.055738, 0.051028, -0.107023, -0.042490, 0.019491, 0.001590, -0.040090, -0.015411, -0.104679, -0.278613, 0.093223, -0.017426, 0.077010, -0.186564, -0.092442, 0.041118, -0.083895, 0.014859, -0.121207, -0.023309, -0.042089, 0.073055, -0.068680, 0.033399, -0.068437, -0.015117, 0.075738, -0.008502, 0.011595, 0.083512, 0.036111, 0.034631, -0.012089, -0.167275, 0.035244, -0.051799, -0.104531, -0.080301, -0.103602, -0.081681, 0.181539, 0.032769, 0.061152, -0.038814, 0.065908, 0.044239, 0.027647, -0.070721, 0.094727, -0.191709, 0.010335, 0.027388, -0.053923, -0.030030, 0.074809, -0.179671, -0.028357, 0.026903, 0.211239, -0.075187, -0.043744, -0.020139, 0.045220, 0.012489, 0.057707, -0.031138, -0.038696, -0.014056, 0.057743, -0.131688, 0.002772, -0.036190, -0.219572, 0.017150, -0.100274, 0.222748, -0.032882, 0.114255, 0.046193, -0.199053, -0.093609, -0.059852, -0.072864, -0.057696, -0.113337, 0.096660, 0.015992, -0.174794, 0.081647, 0.022361, 0.130787, -0.134001, -0.036873, -0.039753, 0.004854, -0.085773, 0.096393, -0.043720, 0.000788, 0.003722, 0.040080, 0.144878, -0.084010, 0.068261, -0.057341, -0.090079, -0.097149, 0.041649, -0.009540, -0.024638, -0.047432, 0.073698, -0.068103, -0.113925, -0.089421, 0.084342, 0.035463, -0.156829, -0.105415, -0.101689, 0.037280, -0.059109, -0.097243, 0.192449, -0.013756, 0.041569, -0.099253, 0.082396, -0.183388, -0.034749, -0.033847, -0.253259, 0.044426, 0.036026, -0.002734, 0.013033, -0.134119, -0.091668, 0.020713, 0.117087, -0.089988, -0.087447, -0.180903, 0.010403, -0.140362, -0.036270, 0.004972, 0.050032, 0.058866, 0.099612, 0.024996, -0.120502, -0.131421, -0.055495, -0.136748, -0.073380, 0.040585, 0.201858, 0.022506, -0.075789, 0.017284, -0.033429, -0.038251, 0.001981, -0.053349, 0.036635, 0.023561, 0.001031, -0.069752, 0.053537, 0.097820, 0.002555, -0.025135, 0.098512, 0.026901, 0.025552, -0.022900, 0.039833, 0.044539, -0.038849, 0.052431, 0.044064, -0.185545, 0.057721, -0.005120, -0.010373, -0.065854, 0.098963, 0.027148, -0.049490, 0.168463, -0.024612, 0.052873, -0.074747, -0.014686, -0.058146, -0.222742, -0.150061, 0.139675, -0.051050, -0.108890, -0.179742, 0.081270, -0.011750, -0.123366, 0.093209, -0.075875, 0.113333, -0.077838, -0.084943, -0.063109, 0.121067, -0.010752, 0.051612, 0.050595, -0.045367, -0.117334, 0.003104, -0.044989, -0.012566, -0.046600, -0.213750, 0.208828, -0.051877, 0.001808, -0.010559, -0.082499, -0.043269, -0.075075, -0.167302, -0.156207, 0.011066, 0.012192, -0.015147, 0.161946, 0.041740, -0.019250, -0.020861, -0.058715, 0.022127, 0.009455, 0.019162, 0.023732, -0.037664, -0.055874, 0.014716, 0.024105, 0.040908, -0.109053, -0.173040, 0.027802, 0.028047, -0.200483, -0.009391, 0.070176, -0.165184, -0.039852, -0.090504, -0.136428, -0.004722, -0.138089, -0.074819, 0.057701, -0.074891, -0.043014, -0.169973, -0.039559, -0.079804, 0.036433, 0.017808, 0.075957, 0.051762, -0.003504, -0.077647, -0.199960, -0.062733, 0.067948, -0.084374, -0.010585, 0.075495, 0.015075, -0.141548, 0.081915, -0.113862, 0.104865, 0.158465, -0.152924, 0.081528, 0.080311, 0.037055, -0.097254, -0.056039, 0.025643, -0.034546, 0.108141, 0.121459, -0.139965, 0.057549, -0.146974, 0.078782, 0.001352, -0.091746, -0.031641, -0.143146, -0.012351, -0.088307, 0.030683, 0.003712, -0.096946, -0.187117, -0.028938, -0.171721, -0.051407, 0.037397, -0.048240, -0.051359, -0.129828, -0.077682, -0.140448, 0.019471, 0.028218, 0.074746, 0.002215, -0.091275, -0.003751, 0.095512, 0.052515, -0.172887, -0.093262, -0.090194, -0.131669, -0.172820, -0.133029, -0.102334, -0.140678, -0.117636, -0.065705, 0.116968, 0.108993, -0.135983, -0.088854, -0.061853, -0.072562, 0.022186, 0.069690, -0.049725, -0.090727, 0.009472, 0.101574, -0.005250, -0.091360, -0.086698, -0.007494, -0.004976, -0.120712, -0.063050, 0.002348, 0.057430, -0.055158, 0.009859, -0.061294, 0.040596, -0.175861, -0.093101, 0.057519, -0.019300, 0.047653, -0.004630, 0.091603, -0.090637, -0.051237, 0.032697, -0.036023, -0.039074, 0.003244, -0.050393, -0.015099, 0.012983, 0.081599, -0.196057, -0.117705, -0.021703, -0.008510, 0.059765, -0.131374, -0.180741, -0.075861, -0.104504, -0.107968, -0.123209, -0.052155, -0.014345, 0.003794, -0.031149, -0.017336, -0.100110, -0.014474, -0.038336, 0.092595, 0.008222, -0.041387, -0.171935, -0.010100, -0.000119, -0.058582, -0.117947, -0.011083, -0.022847, -0.228012, -0.183218, 0.051968, -0.008118, 0.009054, -0.044358, 0.078473, -0.064402, -0.082949, -0.011641, -0.046741, -0.088232, 0.078228, -0.058968, -0.094942, 0.019694, -0.035140, -0.119815, 0.025225, -0.017010, -0.050056, -0.028037, 0.023546, -0.011450, -0.057907, 0.200384, 0.045135, 0.070906, 0.047776, -0.134901, 0.014408, -0.036790, 0.223034, -0.104238, -0.101045, -0.016241, -0.091502, 0.148021, -0.040939, -0.025147, -0.160740, 0.037313, -0.262183, -0.192009, 0.087846, -0.029232, 0.120777, -0.085966, -0.086151, -0.039068, -0.190534, 0.002480, 0.004113, 0.051940, -0.142600, -0.072945, -0.062936, 0.055899, -0.168630, -0.205972, 0.002135, -0.112931, -0.038044, -0.209325, -0.123948, -0.111404, -0.192845, -0.026719, 0.024658, -0.150637, -0.106929, -0.028636, -0.181025, -0.264138, 0.010932, 0.124453, -0.081252, 0.027982, 0.060752, 0.023427, -0.325035, -0.017635, -0.092204, 0.085484, 0.114739, -0.019504, 0.115567, 0.055330, -0.231269, -0.093358, -0.117302, -0.088390, 0.008402, -0.022636, -0.057537, -0.117447, 0.011473, -0.159469, 0.078853, 0.045084, 0.007001, -0.309220, -0.075181, -0.105455, -0.029204, 0.066589, -0.069219, -0.056813, -0.033701, -0.068815, -0.045257, -0.033089, -0.201649, 0.065824, -0.008091, -0.157651, 0.115925, -0.020675, -0.072274, 0.008482, 0.001916, 0.007231, -0.039103, 0.021706, -0.037135, -0.036862, -0.114302, -0.076014, -0.051272, -0.014375, -0.144067, -0.004595, -0.038014, -0.085913, -0.047913, -0.023614, -0.075593, 0.066597, 0.006241, 0.048080, -0.106840, 0.030157, 0.048269, 0.021723, -0.017521, 0.133678, -0.138713, -0.003044, -0.001916, 0.008520, 0.069667, 0.098400, -0.021650, -0.127962, -0.146466, -0.122121, 0.065911, 0.102983, -0.029653, -0.103998, -0.056947, -0.018629, -0.142359, 0.043225, -0.073225, -0.162901, 0.086918, -0.055290, -0.079972, -0.050271, -0.000265, -0.038542, 0.051949, -0.008031, -0.013301, 0.113932, 0.008302, 0.094063, -0.126880, -0.072445, -0.095464, -0.072733, 0.051677, -0.219750, 0.037991, 0.008383, -0.087085, -0.164267, -0.050154, -0.056435, -0.010428, 0.048161, -0.107693, 0.029832, -0.011115, -0.084461, -0.074436, -0.076743, 0.068052, -0.015054, -0.079348, 0.046484, 0.014007, -0.007270, -0.105133, -0.090610, 0.041298, 0.053449, -0.044286, -0.013770, 0.026053, 0.053400, 0.088829, 0.021865, 0.012477, -0.150926, 0.052054, 0.048767, 0.121828, 0.084253, -0.052815, -0.178735, -0.025416, -0.095299, -0.017088, -0.076164, -0.105926, 0.106431, 0.000853, -0.053073, 0.017364, 0.048324, -0.003664, -0.115764, -0.192848, -0.019459, -0.109212, 0.035058, -0.227546, -0.077406, -0.121400, -0.090561, 0.019749, -0.024144, -0.125730, 0.011034, 0.067873, -0.063616, -0.105617, -0.068435, -0.172062, -0.008656, -0.048916, -0.020623, 0.009606, 0.012958, 0.022084, 0.068134, -0.138246, -0.021532, 0.034889, -0.036786, 0.034718, 0.062097, -0.068127, -0.009942, -0.146297, -0.049699, -0.120110, -0.064292, 0.017209, 0.018662, 0.008311, -0.067736, -0.005631, -0.077510, 0.031009, 0.072934, 0.013752, -0.078550, 0.076478, 0.036744, 0.026624, -0.110724, -0.085069, 0.049875, -0.018631, 0.100263, 0.078442, -0.006863, -0.070171, -0.025779, -0.042056, 0.008621, 0.004605, -0.068528, 0.052749, -0.007998, 0.082957, -0.012184, -0.065187, 0.035243, 0.121238, -0.007839, -0.028215, -0.112405, -0.108244, -0.049914, -0.069312, 0.061223, 0.053603, -0.008826, 0.072332, -0.148294, 0.037153, -0.005567, -0.106635, 0.142033, -0.150832, -0.133857, 0.120182, 0.111972, -0.128849, -0.078088, -0.196285, -0.054753, -0.077286, -0.068519, -0.037416, 0.040072, 0.168804, 0.066489, -0.116145, -0.069193, -0.136441, -0.152188, -0.115355, -0.116444, -0.053766, -0.001907, -0.076158, 0.024802, -0.115490, -0.151738, 0.041210, 0.041324, -0.000742, 0.063943, -0.105252, 0.004160, 0.045537, 0.002318, -0.106384, -0.162123, -0.119846, -0.150237, 0.078139, -0.018489, 0.038303, 0.033986, -0.086966, 0.088983, -0.121998, 0.013737, 0.030177, -0.084168, -0.006263, -0.117229, 0.008614, -0.051335, 0.078283, 0.016321, 0.000179, -0.055561, 0.065369, -0.046941, -0.077899, 0.068133, -0.058959, -0.047971, 0.114664, -0.155423, -0.002579, 0.035591, -0.094061, -0.058062, -0.044108, -0.229780, 0.086326, -0.196991, -0.136759, -0.198792, 0.057767, -0.049656, 0.069706, -0.015906, 0.030002, 0.062652, 0.045720, -0.091546, -0.140281, -0.101454, 0.082932, -0.084213, 0.009663, -0.096115, -0.063205, -0.040710, 0.058044, -0.268206, -0.087285, -0.096841, -0.117279, 0.044641, 0.087186, 0.259887, -0.069268, 0.099866, -0.017935, -0.067978, -0.086307, 0.126402, 0.042792, -0.196570, 0.042727, -0.152224, 0.049320, 0.017017, 0.026719, -0.262618, -0.108888, -0.199796, -0.057792, 0.018508, 0.109688, -0.172313, 0.046896, 0.132784, 0.051539, -0.049796, -0.194127, -0.050474, -0.191154, 0.018188, -0.159084, -0.028630, -0.057603, -0.119146, -0.095357, 0.072858, 0.027424, 0.012903, 0.010047, -0.071052, -0.065537, 0.270823, -0.056099, -0.022573, 0.072804, -0.176393, -0.004156, 0.032450, -0.074083, -0.006849, -0.124248, -0.163062, 0.121845, 0.031421, -0.117502, 0.148223, 0.111827, 0.042336, 0.014476, -0.100456, 0.035437, -0.102211, -0.183130, -0.002971, 0.048583, -0.063703, -0.094139, -0.105781, -0.162451, -0.008729, -0.215287, -0.051707, -0.011544, -0.168398, -0.189929, -0.056316, -0.106798, 0.057411, -0.233756, -0.065946, 0.025907, -0.044695, -0.112525, -0.120324, -0.039344, 0.021525, -0.085938, -0.143884, 0.075155, -0.020421, 0.065911, -0.044800, 0.051797, -0.031367, -0.221139, -0.130375, -0.108411, -0.192291, -0.235790, -0.058657, -0.187307, -0.008742, -0.041936, 0.119947, -0.079252, -0.070659, -0.157955, -0.002352, -0.059637, -0.146315, 0.145036, -0.037262, -0.022770, -0.161942, -0.059815, 0.074715, -0.186685, -0.111785, -0.100029, 0.028296, -0.101840, -0.186933, -0.002408, -0.093544, 0.018395, -0.071339, -0.041517, -0.156759, -0.108611, 0.020766, -0.122790, 0.016803, 0.062014, -0.174976, 0.114742, 0.083049, -0.194603, 0.018813, 0.023417, -0.034152, -0.142146, -0.182401, -0.147678, -0.213601, 0.071376, -0.215259, -0.058226, -0.041427, -0.219914, -0.096808, -0.098754, -0.154464, -0.121903, -0.112442, -0.022756, 0.115272, -0.024160, -0.123413, -0.028202, 0.052943, -0.055372, -0.182752, -0.045750, -0.033722, -0.229996, 0.092028, -0.124788, -0.086060, 0.026078, 0.149154, 0.035149, -0.107949, -0.043027, -0.047057, -0.049582, -0.069815, 0.106591, -0.027948, -0.191001, 0.095326, 0.014380, -0.039764, 0.000589, -0.215178, 0.006535, -0.144192, 0.035971, -0.219127, -0.142913, 0.078318, -0.032087, -0.224298, 0.131704, -0.072768, -0.171091, -0.032780, 0.003461, 0.106727, -0.002682, -0.032128, 0.129506, -0.025440, -0.114209, -0.138029, 0.062652, -0.101051, 0.023027, 0.039508, -0.026180, -0.144341, -0.094476, -0.097224, -0.079122, -0.020001, -0.066524, 0.070039, -0.008741, -0.332817, 0.002069, -0.138013, -0.057050, -0.199622, -0.158505, -0.087164, -0.169630, -0.077679, -0.071714, 0.015127, -0.151197, 0.010714, 0.011435, 0.052871, -0.179792, -0.099860, -0.165632, -0.022888, 0.053046, -0.046050, -0.229657, -0.048851, -0.163322, -0.073438, -0.167641, -0.054326, -0.040303, 0.052291, 0.016743, -0.050087, -0.064149, -0.097669, -0.045354, -0.189615, -0.060548, -0.129865, -0.098439, -0.000170, -0.113368, -0.097785, -0.021120, 0.088296, 0.105389, -0.020244, -0.250389, 0.067390, -0.232880, -0.103813, -0.046680, -0.087636, -0.150270, -0.238645, -0.132662, -0.238248, 0.028771, -0.004555, -0.076236, -0.125719, -0.055865, -0.227546, -0.088398, -0.089686, -0.148081, 0.027855, 0.009440, -0.203992, 0.020700, -0.088542, -0.082777, -0.172679, 0.060121, -0.210724, -0.180674, -0.103853, -0.039215, 0.033926, 0.020470, -0.027728, -0.157078, -0.030505, 0.030657, 0.131967, 0.137307, -0.145393, -0.075991, 0.020752, 0.088197, 0.066786, 0.103840, 0.086652, 0.151581, -0.129904, 0.004395, -0.003671, -0.037860, -0.145458, -0.228325, 0.061900, -0.306053, -0.114616, 0.096464, 0.019048, 0.038692, -0.109234, -0.019063, -0.088204, 0.027472, 0.093422, -0.060539, -0.084761, 0.083679, 0.041504, 0.183996, 0.037524, 0.034065, -0.135286, 0.010064, 0.000603, -0.088118, -0.058920, -0.011835, -0.038578, -0.062039, -0.069191, 0.059606, 0.051316, -0.023510, 0.042423, 0.055032, -0.219737, 0.083349, -0.035839, 0.130430, -0.079611, 0.104018, 0.094794, 0.097598, -0.036984, 0.002941, -0.056371, 0.072524, -0.006397, -0.159007, 0.077437, -0.005987, 0.071942, -0.018536, -0.066996, -0.114908, 0.007759, -0.028909, -0.095161, -0.075607, 0.003061, 0.031671, 0.156829, 0.027816, -0.070331, -0.008892, 0.055009, 0.076142, 0.003627, -0.082158, -0.163587, 0.075681, -0.052391, -0.106771, 0.033032, 0.020392, -0.127835, 0.065562, 0.023562, -0.022500, -0.057994, -0.121820, 0.085418, 0.174063, 0.000052, 0.069160, 0.014944, 0.001086, 0.008664, 0.222824, 0.145833, -0.154925, 0.157984, -0.087144, -0.131691, -0.095151, -0.051683, -0.203896, -0.044726, -0.031083, 0.000060, -0.210537, -0.255797, 0.024412, -0.201307, -0.029747, -0.073330, 0.003745, 0.068202, -0.130787, -0.039779, 0.081570, -0.106402, -0.030823, -0.048376, 0.051429, 0.016617, -0.163747, -0.230018, -0.087963, 0.037831, 0.099559, -0.044564, -0.019514, 0.070241, 0.010924, 0.001628, 0.127350, 0.007032, -0.088167, -0.019513, -0.099216, -0.191704, 0.033218, -0.180459, 0.090662, -0.270130, 0.127024, 0.070237, -0.247875, 0.119021, 0.073414, -0.129609, -0.050320, 0.024670, 0.101164, -0.159840, 0.024106, 0.097351, -0.019848, -0.030125, -0.060774, -0.084771, -0.095129, -0.090480, 0.067548, -0.069248, 0.040870, 0.042579, 0.003700, 0.136370, 0.092905, -0.132522, -0.088057, -0.108258, -0.024469, -0.041030, -0.130526, -0.135973, 0.070965, 0.130834, -0.164202, 0.004880, -0.042217, -0.133042, -0.123938, -0.078062, -0.158363, -0.151152, -0.104163, -0.107608, -0.050500, 0.056474, 0.027148, 0.058331, -0.027920, -0.060833, 0.119183, -0.106840, -0.088958, 0.019971, -0.003406, -0.093114, -0.005018, -0.120476, 0.000892, 0.087427, 0.139219, -0.126208, -0.122987, -0.094452, 0.029473, 0.053039, -0.117467, 0.020854, -0.111123, -0.068567, -0.089542, -0.134441, -0.017885, -0.066303, -0.015825, 0.142990, -0.085874, -0.077276, -0.122480, 0.098478, 0.091253, -0.051116, -0.090014, 0.093978, 0.003814, -0.037739, -0.147091, -0.053943, 0.000919, 0.072881, 0.109153, -0.109764, -0.044410, -0.108408, -0.081759, 0.064884, 0.045303, -0.012070, -0.046717, -0.117630, 0.103667, -0.149598, 0.078620, -0.111427, 0.021058, -0.014931, -0.026198, 0.090705, 0.011041, -0.038059, -0.062247, -0.097273, -0.034697, -0.140595, -0.113895, 0.048172, -0.093500, -0.037128, -0.102923, 0.014936, 0.060049, 0.074965, 0.009806, -0.089403, -0.029282, -0.043089, 0.057495, -0.002589, 0.056348, 0.061575, 0.010783, 0.011714, 0.054997, -0.002073, -0.047787, 0.169686, 0.085024, -0.049856, -0.037929, 0.000593, -0.106130, 0.042712, -0.056165, -0.102720, -0.090704, 0.021784, -0.003485, -0.033991, -0.037551, -0.034111, 0.129986, -0.142506, -0.006813, -0.034785, 0.074856, 0.095805, -0.060003, 0.050456, 0.093065, 0.005926, -0.195404, -0.098432, 0.106519, 0.078895, -0.012565, -0.071586, -0.098668, -0.119659, -0.004766, 0.024480, 0.055396, -0.137531, 0.019407, -0.134613, -0.039781, -0.020498, -0.024894, -0.091648, -0.104594, -0.008841, 0.158590, -0.051582, 0.067648, 0.005482, -0.183746, 0.113853, 0.022271, -0.032432, -0.125623, -0.119461, -0.023050, -0.135896, 0.012387, -0.071310, 0.038052, -0.102893, -0.002298, -0.136720, -0.056335, 0.062744, -0.084420, 0.071916, 0.059839, 0.025248, -0.005824, -0.019080, -0.140400, -0.058920, 0.141018, 0.007022, 0.041603, -0.068860, -0.116297, -0.028664, 0.004230, 0.061862, -0.030163, -0.068234, 0.024764, 0.053067, -0.024471, -0.071711, 0.008107, 0.076259, 0.053946, -0.018397, -0.048663, -0.045426, -0.023298, -0.037971, -0.017719, -0.146930, -0.011250, 0.090920, -0.054357, 0.018149, -0.081567, -0.078925, 0.110962, 0.191193, -0.020375, 0.139740, 0.127379, -0.079376, -0.076989, -0.040376, -0.156180, -0.064762, -0.069173, -0.086976, -0.214060, -0.009955, 0.096086, -0.113111, -0.066370, 0.062445, 0.094272, -0.082217, 0.053822, -0.049291, 0.129616, 0.109353, 0.057948, -0.017282, -0.133406, -0.083368, 0.087209, 0.008347, -0.169435, -0.119538, 0.020738, -0.133938, 0.083452, -0.013232, 0.203008, 0.038320, -0.111459, 0.018534, -0.179049, 0.079737, -0.024103, -0.019370, -0.027199, -0.094156, 0.013706, -0.042807, -0.131098, -0.073020, -0.067800, -0.073378, 0.047535, 0.163215, 0.032938, 0.022811, 0.098999, 0.003607, 0.016279, 0.140777, -0.132813, 0.092104, 0.064756, -0.097717, -0.048257, 0.045245, -0.016621, -0.103148, 0.036454, -0.143780, -0.092501, -0.074182, -0.120335, 0.170751, -0.011835, -0.170368, 0.000211, -0.097063, -0.112551, -0.162989, -0.046707, -0.068051, 0.084907, -0.041847, -0.065914, -0.173615, 0.053249, 0.071742, -0.102555, 0.006855, -0.209369, 0.087008, 0.067038, -0.048203, -0.108181, -0.043878, 0.096467, -0.113366, -0.150303, 0.043612, 0.212061, 0.020196, -0.006987, -0.098946, 0.016963, -0.055567, 0.143320, -0.042339, 0.020995, 0.019594, 0.094637, -0.042165, -0.023204, -0.182039, -0.114292, 0.013496, 0.021379, -0.026868, -0.108388, -0.266269, 0.160929, 0.048617, -0.078955, 0.035106, -0.055910, 0.071420, -0.072860, -0.009414, -0.131712, -0.031084, -0.140786, -0.045710, -0.005846, 0.050730, 0.060969, -0.162676, 0.035435, 0.103142, -0.237069, -0.040054, 0.017622, -0.082521, -0.068336, -0.109198, -0.066592, -0.059017, -0.025928, -0.013957, -0.049053, -0.084905, 0.109170, 0.092728, -0.136729, 0.136182, -0.005270, -0.180701, 0.129139, -0.017198, -0.084279, 0.011578, 0.023601, -0.076741, 0.100448, 0.041491, -0.036055, 0.026722, -0.169879, -0.108467, 0.082822, 0.045708, 0.090172, 0.048026, -0.202752, 0.009325, 0.001655, 0.124853, -0.004386, 0.001322, 0.031811, 0.052999, -0.161608, 0.047673, 0.135771, 0.131542, 0.014760, 0.004858, -0.100572, -0.058963, 0.039826, 0.015347, -0.092098, 0.144306, 0.054197, -0.092995, -0.097823, -0.016626, -0.006181, -0.102560, 0.067853, -0.267500, -0.195885, -0.048117, -0.029163, 0.038944, 0.070522, -0.319053, 0.179717, -0.091251, -0.174661, -0.435454, -0.089082, 0.067564, -0.172087, -0.032084, -0.164083, -0.023588, 0.181847, 0.008281, 0.062587, 0.060308, -0.122497, -0.113632, -0.115364, -0.296068, -0.268116, -0.081933, -0.168085, 0.115864, -0.082824, 0.177594, -0.058857, -0.257729, -0.213224, -0.159826, -0.030758, -0.194165, -0.069115, 0.084598, -0.032577, -0.056459, -0.184533, 0.097622, -0.162353, -0.025787, -0.252319, -0.035415, -0.221438, -0.158318, -0.073159, 0.095429, -0.197148, 0.041976, -0.032186, -0.252871, -0.157085, 0.100673, 0.002254, -0.085338, 0.003846, -0.132161, -0.088344, -0.103131, -0.085740, 0.025679, 0.048844, 0.040174, 0.086364, -0.054431, -0.077778, -0.012895, 0.007129, 0.034941, 0.101263, 0.070759, -0.082308, 0.160223, -0.282003, 0.051059, -0.069357, 0.138068, -0.082995, 0.037431, 0.044407, 0.057991, -0.202285, -0.047006, 0.141287, -0.211574, -0.103200, 0.189886, -0.200671, 0.070170, -0.096357, -0.229827, -0.428962, -0.291173, -0.281660, -0.088916, -0.231939, -0.138552, -0.301003, -0.009535, -0.172115, -0.328289, -0.006151, -0.036269, -0.101433, 0.123231, -0.102877, -0.151140, 0.073501, -0.117081, 0.042882, -0.032259, -0.033525, 0.152721, -0.019480, -0.049708, -0.125957, 0.024993, -0.006005, 0.021452, 0.023095, 0.098534, -0.064069, 0.101981, -0.134227, -0.018657, 0.071026, -0.243196, -0.019465, 0.124266, 0.017363, -0.077227, 0.162229, -0.021498, -0.017435, -0.051386, -0.009670, 0.173873, -0.047935, -0.215999, -0.078973, -0.059782, 0.098294, -0.065527, -0.153574, 0.127454, -0.056426, -0.092767, -0.035940, -0.025413, 0.018092, -0.135840, 0.110320, 0.036084, -0.086341, -0.251437, -0.253009, -0.155141, 0.016127, -0.179855, 0.159829, -0.138067, 0.193042, -0.208479, -0.135449, -0.056848, 0.008373, -0.132108, 0.012713, -0.133263, 0.140545, -0.016418, -0.152121, -0.109078, -0.118307, -0.130369, -0.140219, 0.015312, -0.091000, -0.113787, -0.030739, -0.232721, -0.037941, 0.130297, -0.140204, -0.012924, -0.031383, -0.046042, -0.028586, 0.020476, 0.079548, -0.166819, -0.043469, -0.130579, 0.038741, -0.074537, -0.125647, 0.064681, 0.103563, -0.032031, -0.039343, 0.082439, -0.011424, -0.109661, 0.001598, 0.044465, -0.070005, -0.086358, -0.136995, 0.010861, 0.100883, -0.022707, 0.201211, -0.115345, -0.026083, 0.005026, -0.118744, -0.163265, -0.010858, -0.067379, 0.082500, -0.090216, -0.088336, -0.027592, -0.085385, 0.050486, 0.048240, -0.017086, 0.000432, -0.051666, -0.072917, -0.000645, -0.057159, -0.018556, -0.033492, -0.017204, -0.147985, -0.075875, -0.060038, -0.047733, 0.033871, 0.200974, -0.112030, 0.057186, 0.108671, -0.043868, -0.052161, -0.045125, 0.177257, 0.275658, -0.007151, -0.011075, 0.002008, 0.069919, -0.090169, -0.046327, -0.066261, 0.128003, 0.053096, 0.040705, 0.108055, 0.010922, 0.035097, 0.049167, -0.080477, -0.067413, -0.017612, -0.148640, 0.012151, 0.043093, 0.050311, -0.042725, -0.018459, -0.093347, 0.062527, 0.206588, 0.017988, 0.054837, -0.068877, -0.108071, -0.095807, -0.058109, -0.125179, 0.055581, -0.034695, -0.086689, 0.072152, 0.127252, 0.109967, 0.117945, 0.042284, 0.178459, -0.073177, 0.023417, 0.153849, 0.032601, -0.041433, -0.223185, 0.106359, 0.166570, 0.037390, -0.102813, 0.044346, -0.038964, -0.070533, 0.107117, -0.122701, 0.040651, 0.101887, 0.025657, -0.088202, 0.035174, -0.247586, 0.020991, -0.018984, 0.042628, -0.025992, 0.020338, -0.151857, -0.184043, 0.108072, 0.063584, 0.070611, 0.055786, -0.164776, -0.071169, -0.105938, 0.033848, -0.152374, -0.108969, 0.022230, -0.083749, -0.061719, 0.015114, 0.027103, 0.148639, 0.041188, -0.177375, 0.016439, 0.123583, 0.137730, 0.017628, -0.041160, 0.078899, 0.072238, 0.090395, 0.027665, -0.245385, 0.199521, 0.149550, -0.214155, -0.079680, 0.111648, 0.140296, -0.246754, 0.139239, 0.053093, 0.181491, 0.054302, 0.040134, 0.050186, -0.174573, -0.265285, -0.030821, -0.054843, -0.009411, -0.161036, 0.084913, -0.126708, 0.033856, 0.001187, 0.113019, -0.120294, 0.144959, 0.070103, 0.101135, -0.146355, 0.104842, 0.037133, 0.055443, 0.025776, -0.035043, 0.001175, -0.041538, -0.018517, 0.029375, -0.019908, -0.051783, -0.039971, 0.021118, -0.102089, 0.005099, -0.100198, 0.068156, 0.019664, -0.049365, -0.023093, -0.106837, -0.081247, -0.072971, -0.100182, -0.063486, 0.099426, -0.084681, -0.155432, 0.052309, -0.034908, -0.007981, 0.014145, 0.049152, -0.062679, 0.070932, 0.001995, -0.090149, 0.071056, 0.007941, -0.144564, 0.129118, -0.010190, -0.004135, -0.017709, -0.129758, -0.207350, -0.076816, 0.039484, -0.087395, -0.037305, 0.065577, 0.009031, -0.025807, -0.145888, -0.067127, -0.054545, -0.081712, -0.080970, 0.008849, -0.180051, -0.020793, -0.047157, -0.203093, -0.131726, -0.126905, -0.211743, 0.109008, -0.020943, -0.161304, -0.081877, 0.020637, 0.000139, 0.006070, 0.092990, -0.072432, -0.013247, 0.015552, 0.047027, 0.010818, -0.105269, 0.005215, -0.037501, -0.006649, -0.072171, -0.092405, -0.071070, 0.025878, -0.086222, 0.067114, -0.023072, -0.062620, -0.072908, -0.099221, -0.100820, -0.050921, -0.156027, 0.048047, 0.027705, 0.008874, 0.050820, -0.022182, -0.096005, -0.003258, 0.010055, 0.042951, 0.019940, -0.082034, -0.053918, 0.060969, -0.040328, -0.048475, -0.034581, -0.048915, 0.058013, -0.090266, 0.149421, -0.085566, 0.073043, 0.112818, -0.117732, -0.131818, -0.009860, -0.111742, -0.020721, -0.014390, -0.031680, -0.023217, -0.165007, -0.320458, 0.018972, -0.080950, -0.012220, -0.116500, 0.024678, -0.144892, -0.177371, -0.137938, -0.079593, 0.003932, 0.047863, -0.041444, 0.064758, -0.045239, -0.077975, 0.040542, -0.053457, -0.087280, -0.020268, -0.057985, 0.090488, -0.059357, -0.018214, -0.084230, -0.188434, -0.036112, -0.123939, -0.030309, -0.120930, 0.045743, -0.066995, -0.077689, 0.010187, -0.076964, -0.032591, 0.105162, -0.061735, 0.051663, -0.053834, -0.020514, 0.008221, -0.160315, -0.098005, -0.047395, 0.030614, -0.031317, 0.074674, -0.130146, 0.072514, 0.072376, -0.076315, -0.087994, -0.140947, 0.015131, 0.009252, -0.067014, 0.035374, -0.158039, -0.096967, -0.000271, -0.099540, 0.050529, -0.081489, -0.142857, -0.035224, 0.147970, -0.094349, -0.157043, 0.017052, 0.109400, -0.023731, 0.135802, 0.136932, -0.000695, -0.044814, 0.027279, 0.147976, 0.090681, 0.054258, 0.066643, -0.103095, -0.121630, -0.183378, 0.085567, 0.293945, -0.111438, -0.104217, -0.037080, -0.075731, 0.011387, -0.036005, 0.092156, -0.131206, 0.003777, 0.114747, -0.007716, 0.143649, 0.128954, -0.057941, 0.164756, -0.029324, -0.058382, 0.042995, 0.080620, 0.134985, -0.031629, -0.282219, 0.040387, 0.007966, -0.000915, -0.217002, 0.130720, -0.124712, -0.040526, 0.120526, -0.140246, -0.084807, -0.097977, -0.051868, -0.008593, -0.082093, 0.090893, -0.022362, 0.044957, -0.098569, -0.109834, 0.080344, -0.107738, -0.082325, -0.129004, 0.066345, -0.014170, 0.016460, -0.127995, -0.122534, 0.096690, -0.267126, -0.042133, 0.033444, -0.187448, 0.150946, 0.068114, 0.027747, -0.052293, -0.224387, -0.109840, -0.091139, 0.087443, -0.111495, 0.184282, -0.114936, -0.012401, 0.284928, 0.108246, -0.033146, -0.123417, -0.064339, 0.003842, -0.035732, 0.236813, -0.195109, -0.058219, -0.082019, -0.012507, 0.084543, 0.008199, 0.050977, -0.140399, -0.113599, 0.124699, 0.144645, -0.071423, -0.165008, 0.097516, -0.060495, 0.039050, -0.183390, 0.116078, 0.010753, 0.099272, -0.036542, 0.110364, 0.062703, -0.037800, 0.015743, 0.032042, -0.052795, 0.137977, -0.125671, -0.192222, 0.071310, 0.032790, -0.102359, -0.017722, 0.058992, 0.214033, -0.130491, -0.041113, 0.106669, 0.163699, 0.039384, -0.117237, -0.014262, 0.048813, -0.257744, -0.156469, 0.073723, -0.117613, 0.131459, -0.009507, 0.088637, 0.026440, -0.198298, 0.064998, -0.235009, 0.103410, 0.047430, -0.116574, -0.065207, 0.015130, -0.054451, 0.018255, 0.006457, 0.112921, -0.078700, 0.141556, -0.079282, 0.003979, -0.107195, 0.078428, -0.069874, -0.005195, 0.073601, -0.088687, 0.200097, -0.123059, -0.122667, 0.042644, 0.042131, -0.062083, -0.166644, -0.143966, -0.046140, 0.057427, 0.043682, -0.020336, 0.005035, 0.118551, 0.033706, 0.104947, -0.018241, 0.024316, 0.020705, -0.132635, -0.031465, 0.120343, 0.021840, 0.128521, -0.052414, -0.227583, -0.047885, 0.013961, -0.149004, 0.175569, 0.220025, 0.050051, -0.082405, -0.181405, 0.022593, 0.099480, -0.128112, 0.043213, -0.073251, -0.197915, 0.119147, -0.053910, 0.241466, 0.076329, -0.128563, 0.058578, -0.150223, -0.187116, 0.143647, -0.005062, -0.110154, -0.184509, -0.090118, -0.024195, -0.046820, -0.077948, -0.071393, -0.183386, 0.143415, -0.014588, -0.132936, -0.082817, -0.218421, -0.058558, 0.023210, -0.051832, -0.096326, -0.069977, -0.113695, -0.010011, -0.105443, 0.020502, -0.041686, -0.179788, 0.041678, -0.180895, 0.128711, -0.036760, 0.012394, -0.064658, 0.029815, 0.070882, -0.131892, -0.180470, -0.150151, 0.176324, -0.134824, -0.077133, -0.034972, -0.196510, -0.092682, -0.007501, -0.030844, -0.067427, 0.026527, -0.079523, -0.094904, -0.074009, -0.053589, -0.177054, 0.150869, 0.077063, -0.227394, 0.111328, -0.147490, -0.096045, -0.096569, 0.155781, 0.010647, -0.078464, -0.036048, 0.012501, 0.062799, 0.006844, -0.047125, 0.142456, 0.053979, -0.086873, -0.053560, -0.026439, -0.065660, -0.097065, 0.005389, -0.318542, 0.033392, -0.188363, 0.077718, 0.057514, -0.167755, 0.001854, 0.095619, 0.073375, -0.076836, -0.038822, 0.066109, -0.039514, -0.086004, -0.017788, -0.004852, -0.004630, -0.045367, 0.166758, -0.157723, -0.041698, -0.062253, -0.008645, -0.150874, 0.059655, 0.061741, -0.128869, -0.039013, 0.102949, 0.095248, -0.060154, -0.057396, 0.042016, 0.052245, 0.076707, -0.087250, -0.057279, -0.036985, -0.029637, -0.099104, -0.017564, -0.119531, 0.236064, -0.116087, -0.013249, 0.098533, -0.027676, 0.096121, 0.148362, 0.103975, -0.041831, 0.020813, -0.112517, -0.215787, -0.058329, -0.030795, -0.163582, 0.068148, -0.174672, -0.183174, 0.023318, 0.086293, -0.063765, -0.102037, -0.284059, 0.017206, -0.113902, -0.141529, -0.065289, 0.024573, -0.079146, 0.135707, -0.189691, -0.072259, -0.123849, 0.047071, -0.020145, -0.111950, 0.103704, -0.019168, -0.135045, -0.197114, -0.055158, -0.070263, -0.062823, 0.038581, 0.001950, -0.249141, 0.084586, -0.131427, -0.169594, -0.026332, -0.031506, -0.166994, -0.120593, 0.007842, 0.027234, -0.104105, 0.059085, -0.063412, 0.022992, -0.062297, -0.246811, 0.043541, -0.045977, -0.022453, -0.088950, -0.089724, 0.010460, 0.013023, 0.055060, -0.072087, 0.044288, -0.017595, 0.168310, -0.048867, 0.060594, 0.088964, -0.182987, 0.007847, -0.090021, -0.148529, -0.083344, 0.172411, -0.026227, 0.090401, -0.086568, -0.047022, 0.019489, 0.057414, -0.061341, -0.064528, -0.038632, -0.096966, -0.035493, -0.143426, -0.037660, 0.045050, -0.164830, -0.089794, -0.024427, -0.078072, -0.043106, -0.067201, -0.020378, 0.153956, 0.010352, -0.034353, 0.001107, -0.067823, 0.101828, 0.027612, -0.033742, -0.143031, 0.036885, 0.029744, -0.081718, 0.151545, 0.089715, 0.015376, 0.003658, 0.141647, -0.161251, 0.085479, 0.026663, 0.085221, 0.027759, -0.136333, -0.115033, 0.097846, 0.014748, -0.021651, 0.093137, -0.043425, -0.126370, 0.000733, -0.166966, 0.028172, 0.047446, 0.012851, -0.088811, -0.099462, 0.092368, -0.009435, 0.143585, 0.090868, 0.041192, -0.019597, -0.109534, -0.047768, 0.059951, -0.013958, -0.114673, 0.057678, -0.127818, -0.029101, 0.231799, 0.104539, 0.001712, -0.101536, 0.007033, 0.226337, 0.085902, 0.031082, 0.043889, 0.078443, -0.046592, -0.008681, -0.051699, -0.005923, 0.047942, 0.029046, -0.008449, -0.095941, -0.073742, 0.099288, 0.030109, 0.073822, -0.040408, -0.045253, -0.025129, -0.127312, 0.025730, 0.035722, -0.078394, -0.086228, -0.071665, -0.079481, 0.065162, -0.051588, -0.209788, 0.052465, -0.038662, 0.130271, -0.100260, -0.178708, -0.152462, 0.072247, -0.127251, -0.004066, 0.081176, 0.015035, -0.103838, 0.063000, 0.015412, -0.074954, -0.118940, -0.039039, 0.014352, 0.053317, -0.135792, -0.094953, -0.095235, -0.183415, 0.001641, 0.011245, 0.132021, 0.075763, 0.000156, -0.048924, -0.030406, -0.002602, -0.092448, -0.082720, -0.004483, -0.090317, -0.048076, -0.125601, -0.039240, 0.023791, 0.112728, -0.064250, 0.089258, -0.061371, 0.006444, 0.054269, 0.097483, 0.160578, 0.097031, -0.018909, -0.146846, 0.001415, -0.017420, 0.020813, 0.032416, -0.135623, -0.127698, 0.130726, -0.002431, -0.137736, -0.067001, -0.070600, -0.098201, 0.057792, -0.094804, 0.063997, 0.147811, -0.136786, -0.131217, 0.085333, -0.092890, 0.073633, 0.085126, -0.000408, -0.048128, 0.008897, -0.117624, 0.044787, 0.025327, -0.094185, 0.084262, -0.095999, -0.032319, -0.030107, 0.030882, -0.125738, -0.050468, -0.200503, 0.067816, 0.079299, -0.154036, -0.083262, 0.017647, -0.082367, -0.071736, -0.016503, 0.096388, -0.082734, -0.078123, -0.119414, -0.059310, -0.060944, -0.032431, -0.018067, 0.088929, 0.052640, -0.047194, 0.112633, -0.014793, 0.158738, 0.142430, 0.069288, -0.154628, 0.081312, -0.136159, -0.024614, -0.042114, -0.019907, -0.044002, -0.042654, -0.052490, -0.077018, -0.011234, -0.046710, -0.118560, 0.085608, 0.119733, 0.056618, -0.023886, 0.074863, -0.016976, -0.028376, -0.044275, -0.108962, 0.059913, 0.048099, 0.018059, 0.116109, 0.096673, -0.089301, 0.023715, -0.073514, -0.066683, -0.095634, 0.046505, -0.076310, -0.017509, -0.063077, -0.071110, -0.048464, 0.195337, -0.116846, 0.008006, 0.023888, 0.088921, 0.015501, 0.095719, -0.110054, 0.010548, 0.079920, -0.080905, 0.106867, 0.110437, 0.047405, 0.022129, -0.234585, 0.014356, 0.112195, -0.004834, -0.111541, 0.130303, 0.081086, 0.096891, -0.044965, -0.003120, 0.216873, 0.099178, -0.062803, 0.183344, 0.081040, 0.045307, 0.010955, -0.030306, 0.040192, -0.049723, 0.140444, 0.034599, -0.109515, -0.041322, -0.037501, -0.078266, -0.081348, -0.036325, -0.116812, 0.100095, 0.008598, -0.277077, -0.105057, 0.262163, 0.010269, -0.056659, -0.058080, -0.020558, 0.034676, 0.024314, -0.023202, 0.085992, -0.027906, -0.036971, -0.140906, -0.060440, -0.182594, -0.118448, -0.079565, -0.097806, -0.025332, -0.124572, -0.052885, -0.115781, -0.063342, -0.046303, -0.035667, -0.144608, 0.074024, -0.099493, 0.107792, -0.087719, 0.006820, 0.012568, -0.099864, 0.022606, 0.036683, -0.114542, -0.058621, 0.020221, -0.146802, -0.043024, -0.089251, 0.117378, 0.077602, 0.014370, -0.139559, 0.116962, -0.008108, -0.173840, -0.121226, 0.086315, 0.054531, -0.011754, -0.115549, 0.069258, 0.089073, -0.111193, -0.031850, 0.040133, -0.072448, -0.004639, 0.098172, 0.029247, -0.029934, 0.152096, -0.068992, -0.196500, 0.001955, -0.056543, 0.051603, 0.088252, 0.083777, 0.057448, -0.087571, 0.016141, -0.060511, 0.047731, -0.035539, 0.219764, -0.113229, -0.094508, -0.172110, 0.027480, 0.011553, -0.182941, 0.130823, 0.030095, 0.086267, 0.037758, 0.220705, -0.071017, 0.018584, -0.172856, -0.043614, -0.001098, -0.026748, 0.059527, 0.062266, -0.042238, -0.008013, -0.016931, -0.068593, -0.078598, 0.030182, -0.157815, -0.008681, 0.066157, -0.048303, 0.015288, 0.044978, -0.106113, -0.077315, -0.025990, 0.102891, 0.185130, -0.024001, -0.010731, 0.065850, -0.102013, -0.062593, -0.045022, -0.067648, 0.143518, 0.064728, -0.111680, -0.000678, -0.073053, -0.048245, 0.069004, 0.017312, 0.075816, 0.004365, 0.041039, -0.062942, -0.000994, 0.002364, -0.003930, -0.065815, -0.021435, -0.127028, 0.029801, -0.018776, 0.042286, -0.042674, 0.034875, -0.106628, 0.047392, -0.164591, 0.030209, 0.034968, 0.190763, -0.004525, -0.009334, -0.049266, -0.052241, 0.009606, -0.007048, 0.011288, -0.071196, 0.049360, 0.119268, 0.057273, 0.039797, -0.109759, 0.106813, 0.062194, -0.050170, 0.059410, 0.004025, 0.067662, -0.044801, -0.034547, 0.173425, 0.020804, -0.080763, 0.022400, 0.049921, 0.198659, 0.035762, 0.036016, -0.029587, 0.105716, 0.094531, -0.038007, 0.061646, 0.065111, -0.039000, -0.076035, -0.078452, -0.102687, -0.020787, 0.027515, -0.119890, 0.039630, 0.199840, 0.159765, -0.080057, -0.010321, -0.153983, 0.118333, -0.086668, -0.013253, -0.010273, -0.026068, -0.046951, 0.031283, -0.014099, 0.053988, -0.112020, 0.118297, 0.143158, -0.030463, -0.158456, 0.050865, 0.023516, -0.012050, -0.230532, -0.136868, -0.102858, -0.009007, 0.001384, -0.033973, 0.015545, 0.023551, -0.156680, -0.072417, -0.103981, -0.033869, 0.069268, 0.020545, 0.162654, -0.117278, -0.059098, -0.194392, -0.139446, -0.062951, -0.177986, 0.144243, 0.074950, 0.111486, 0.006458, 0.058028, -0.085482, 0.026816, -0.121819, 0.053485, 0.124496, -0.075293, -0.169254, -0.089232, -0.091340, 0.048659, -0.062464, -0.064748, -0.131208, 0.088860, -0.052224, -0.086826, -0.051607, -0.077246, -0.055202, -0.108556, -0.056065, 0.057743, 0.096160, 0.183382, -0.027552, -0.077426, 0.023819, -0.089717, -0.000287, 0.028362, 0.076649, -0.104372, 0.036818, -0.000284, 0.102812, 0.036891, 0.018373, 0.043983, -0.174909, -0.017138, -0.020778, -0.007440, 0.130258, -0.015996, 0.098470, 0.088445, 0.070540, 0.091078, -0.094918, -0.035589, -0.155721, -0.074278, 0.119377, -0.095980, -0.141145, -0.018824, -0.060941, 0.065115, 0.034791, -0.004524, -0.157128, -0.085779, 0.167321, -0.002849, 0.036952, -0.000690, -0.100427, -0.093155, -0.000595, 0.060434, -0.093525, -0.131561, 0.023042, -0.083169, -0.057200, -0.173415, -0.038030, 0.104060, -0.068385, -0.037860, -0.026217, -0.194319, 0.013596, -0.041440, -0.017567, -0.045592, -0.045328, 0.081599, 0.092636, 0.195843, 0.044393, -0.215519, -0.039122, -0.013979, 0.001782, -0.034136, 0.071835, 0.047769, 0.202204, 0.206101, 0.162418, 0.074673, 0.021281, 0.058341, -0.025996, 0.003251, 0.123176, 0.014245, -0.028691, -0.087977, 0.070472, 0.012808, -0.087742, -0.114825, 0.063134, 0.006560, 0.052915, -0.048833, -0.058214, 0.089203, 0.064754, 0.167779, 0.065672, -0.022501, 0.123159, -0.052463, 0.096079, 0.084980, -0.075104, -0.051009, -0.069814, -0.024832, -0.158930, 0.036759, -0.035282, 0.012737, 0.063307, -0.114126, 0.136741, 0.024727, 0.033257, -0.080859, 0.188860, 0.007356, -0.002874, 0.082870, 0.009247, 0.082538, 0.065677, 0.009335, 0.113776, -0.072680, 0.100042, 0.072351, 0.066236, -0.110771, 0.119118, -0.082499, -0.007195, -0.145682, -0.067721, -0.027950, -0.117367, 0.130041, -0.088705, 0.114205, 0.004906, -0.030890, -0.044834, -0.217532, 0.015586, 0.103068, -0.056596, -0.096351, 0.046487, -0.024606, -0.165342, 0.003603, -0.072857, -0.125640, 0.021471, 0.102385, -0.349159, -0.098234, -0.049371, 0.179120, 0.075915, 0.034455, -0.173416, 0.092346, -0.085002, -0.022238, -0.081746, -0.058369, 0.162597, -0.029004, 0.192093, -0.006156, -0.114625, 0.022180, -0.087859, -0.106775, 0.002555, 0.045459, 0.066634, -0.089777, -0.010161, -0.110789, -0.086646, 0.062401, -0.002030, 0.170004, -0.061804, -0.037666, 0.103670, 0.007029, 0.009093, 0.096768, 0.022014, -0.000049, 0.031919, -0.065071, 0.045387, 0.113546, 0.115533, 0.110929, 0.037197, -0.122872, 0.075704, 0.136735, 0.086049, 0.018735, 0.072545, 0.051108, 0.220528, -0.088495, 0.086708, -0.208721, 0.079494, -0.077365, -0.003567, 0.068002, 0.124672, 0.085595, 0.039445, -0.136187, 0.034498, -0.095102, -0.002012, 0.020351, 0.024322, -0.016566, 0.042334, 0.071651, -0.045505, -0.121090, -0.005466, 0.108713, 0.126225, -0.016264, 0.013659, 0.037933, -0.134372, -0.015036, -0.025013, 0.142639, -0.021065, 0.011891, 0.049168, -0.065338, -0.010880, 0.038194, 0.183204, 0.126851, -0.054300, -0.155704, 0.088390, 0.045472, 0.027505, 0.044534, 0.048762, 0.033702, -0.077891, 0.075945, -0.090189, -0.018068, 0.034855, 0.121652, -0.117966, -0.145060, -0.031106, 0.016688, 0.145647, -0.066215, 0.124659, -0.066882, 0.109424, 0.271280, -0.236841, -0.092408, 0.018421, 0.223000, -0.069206, -0.081095, 0.122125, -0.010705, 0.119318, -0.376613, -0.059694, -0.029527, 0.105506, 0.032740, 0.087789, -0.037009, -0.055790, 0.009216, -0.066952, 0.090736, -0.071344, 0.119258, 0.023688, -0.012298, -0.129942, 0.146300, 0.003655, -0.196985, -0.075604, -0.073782, 0.040885, -0.038359, -0.018675, 0.068187, 0.132270, 0.076096, -0.025440, -0.005342, 0.118800, -0.078055, 0.216559, -0.108134, 0.088340, 0.110640, -0.199844, -0.020017, -0.015299, 0.015696, -0.023999, -0.114543, -0.108246, 0.003353, -0.155637, 0.137333, -0.097897, 0.038011, 0.013143, 0.147057, 0.010603, 0.061409, -0.072840, 0.012783, -0.009604, -0.075175, -0.067381, 0.093187, 0.097050, 0.186000, -0.136772, 0.131703, -0.017543, 0.119426, 0.062284, 0.038054, -0.082453, -0.022614, -0.234076, 0.044949, -0.016465, 0.183214, -0.060020, -0.078275, 0.015523, 0.111485, -0.046588, 0.151854, -0.096033, 0.027353, -0.321650, 0.019673, -0.268757, 0.098480, 0.062022, 0.060382, 0.044953, -0.047448, 0.028484, 0.094250, -0.105764, -0.124701, 0.000994, 0.008364, -0.062564, -0.130445, 0.006007, -0.141124, -0.021927, 0.196742, 0.001567, -0.034311, 0.014492, -0.051848, -0.014753, -0.110847, -0.089917, 0.018262, -0.060307, 0.147882, -0.045439, 0.070775, -0.019436, 0.017795, 0.034064, 0.059687, 0.034353, 0.050628, 0.010886, -0.008428, 0.183321, -0.034535, 0.034827, -0.125095, -0.149053, 0.274201, 0.087116, -0.216636, 0.094110, 0.099162, -0.052779, -0.038214, -0.106054, 0.024743, 0.029725, 0.202675, -0.106283, 0.020957, 0.015405, 0.097521, -0.099243, 0.133554, -0.091130, -0.092612, 0.005784, 0.016687, -0.118171, -0.004479, 0.038904, 0.001635, -0.159247, -0.015392, 0.117856, 0.011779, -0.060985, -0.143476, -0.088226, 0.061801, 0.077662, -0.022336, -0.067142, 0.110964, -0.015645, -0.017550, -0.176668, 0.040566, -0.127545, 0.183712, -0.009899, -0.022472, 0.148941, 0.214817, 0.040666, -0.099456, -0.049091, 0.107094, -0.110691, -0.120432, -0.145378, -0.054641, -0.085762, 0.069187, -0.137930, -0.043198, -0.095536, -0.249990, -0.062480, -0.046070, -0.028894, -0.071563, 0.031134, -0.037096, -0.154284, 0.026777, 0.001730, -0.102041, -0.061574, -0.088461, -0.003272, 0.009866, -0.228555, -0.067671, -0.015911, -0.077538, 0.090665, 0.148352, 0.064468, -0.109324, -0.101338, 0.034953, 0.111654, 0.066164, -0.038720, -0.025573, -0.066585, 0.049455, 0.077520, -0.021850, 0.175285, -0.052673, 0.102417, 0.109297, 0.011757, 0.100593, 0.084977, 0.013717, 0.036016, -0.106271, -0.111136, -0.047958, -0.041176, 0.034476, 0.073370, -0.027490, 0.042882, -0.094896, -0.024596, 0.118946, -0.060494, -0.162125, -0.074944, -0.043944, -0.015838, 0.003803, -0.066670, -0.046287, 0.096139, 0.033481, 0.104161, -0.018057, 0.039932, 0.010110, -0.141101, -0.108458, -0.043373, -0.134799, -0.180732, 0.192478, 0.050448, -0.032863, -0.084447, -0.099214, 0.088612, -0.120709, -0.091295, 0.069868, 0.012616, 0.135437, -0.077355, -0.042537, 0.005445, 0.003142, 0.046659, -0.093801, 0.065226, 0.024403, 0.135293, 0.062255, 0.402985, 0.091129, 0.048034, 0.043006, -0.053728, 0.097698, 0.016740, 0.035966, 0.007481, -0.069694, -0.024622, 0.111955, 0.173263, -0.014686, 0.120432, -0.004321, -0.039923, 0.107830, -0.081696, 0.051994, -0.028190, -0.016473, -0.008562, -0.012551, 0.042145, 0.056163, 0.128186, -0.046090, 0.002434, -0.127549, -0.056991, -0.009277, 0.034906, -0.063698, -0.080574, 0.013652, -0.225782, 0.014953, 0.062681, 0.019795, -0.072723, 0.069185, -0.180760, -0.028796, -0.126987, -0.110180, -0.078701, -0.033729, -0.065309, -0.039364, -0.018729, -0.147758, -0.082006, -0.144001, 0.062542, -0.035789, -0.112815, -0.082250, 0.022239, 0.019698, -0.127321, 0.026959, -0.063142, -0.050954, 0.063463, -0.131642, -0.134509, -0.000176, -0.035242, -0.106152, -0.016039, -0.024376, -0.035536, 0.007644, -0.106280, -0.023021, -0.050988, -0.116049, -0.050861, -0.019918, -0.167507, 0.118363, -0.163410, 0.022640, -0.127934, -0.001288, 0.097011, 0.064380, 0.032419, -0.141363, 0.046521, -0.151667, -0.018633, -0.004756, -0.024741, 0.084641, 0.105051, -0.102636, -0.177343, -0.141356, -0.012796, -0.036715, 0.037245, -0.075281, -0.079598, -0.032344, -0.057914, -0.142945, -0.120416, -0.206885, 0.112706, -0.006944, -0.048717, 0.077067, -0.069518, -0.055780, 0.076700, -0.056640, -0.011831, -0.101034, -0.160825, 0.002176, 0.007754, -0.013002, -0.141796, -0.159902, -0.030505, -0.074532, 0.025311, 0.107833, -0.152444, -0.005837, 0.074735, 0.017942, 0.095200, -0.045587, -0.124575, 0.058515, 0.090247, 0.029468, 0.026922, -0.044305, 0.024524, -0.145730, -0.021494, -0.130208, -0.084475, -0.147309, 0.088179, -0.096273, -0.071430, 0.017702, -0.033076, -0.102194, -0.129904, -0.015815, 0.051535, -0.027505, 0.060059, 0.012144, -0.082843, -0.010642, -0.259532, -0.117512, -0.037379, 0.114181, -0.025326, 0.089258, 0.078019, 0.030967, -0.010373, -0.061233, -0.075952, 0.058150, -0.141331, -0.062398, 0.025082, -0.058456, -0.047697, -0.039654, -0.197237, 0.073034, -0.063244, -0.056539, -0.017244, -0.145043, -0.093944, 0.016616, 0.016695, 0.006178, -0.017390, 0.074570, -0.122857, -0.133419, -0.153489, 0.007803, -0.117168, -0.129875, 0.115395, -0.224141, -0.064623, -0.086557, -0.113050, -0.040435, -0.104128, 0.024478, -0.094467, 0.016406, -0.109071, 0.049591, -0.042494, -0.038972, -0.097336, 0.043492, -0.080185, -0.123533, 0.037348, -0.091011, -0.098395, -0.081488, -0.106942, -0.033650, -0.035744, -0.096591, 0.100684, -0.033210, -0.159718, -0.115744, -0.018633, 0.061016, -0.057053, -0.044072, -0.113548, -0.045267, -0.036350, -0.106492, -0.107135, 0.071992, 0.022221, -0.105242, 0.067790, -0.037667, -0.148035, -0.252628, -0.012037, -0.116148, -0.139975, 0.184322, -0.103553, 0.116415, -0.020555, -0.035162, -0.045387, -0.084307, -0.106745, -0.160494, -0.034336, -0.092605, -0.212006, 0.039605, -0.010672, -0.151007, 0.156620, -0.051276, -0.047386, 0.109268, 0.127695, -0.162426, -0.146408, -0.065947, -0.097681, 0.015445, -0.105342, 0.026790, 0.083023, -0.059390, 0.040521, -0.140106, -0.097507, 0.046457, -0.096502, -0.181112, 0.071770, 0.051537, 0.050295, 0.098748, -0.082852, 0.021215, -0.081641, -0.006244, 0.072581, -0.085840, -0.097139, 0.048634, -0.098063, -0.039296, -0.077730, 0.050141, -0.008218, 0.231450, -0.046559, 0.063561, 0.093078, -0.176698, -0.012820, -0.118668, 0.035863, -0.041321, -0.109152, -0.090523, -0.070253, 0.082278, -0.025125, 0.020133, -0.086047, -0.085828, 0.055242, -0.114241, -0.077038, 0.074504, 0.020895, -0.130578, -0.254695, -0.126348, -0.021394, -0.134171, 0.012252, 0.062329, -0.057485, -0.012889, -0.063010, -0.091053, -0.063359, -0.039009, -0.097169, -0.039613, 0.011355, 0.098925, 0.083592, 0.192314, 0.080824, 0.048113, 0.099763, 0.023808, 0.120720, -0.054475, 0.131189, -0.124270, 0.014444, 0.012271, -0.169929, -0.007729, 0.033052, 0.098825, -0.018556, 0.071007, -0.002619, -0.035846, -0.032665, -0.187364, 0.036990, 0.037743, -0.162469, -0.067437, -0.243498, 0.050567, -0.206336, -0.097391, 0.024106, -0.042568, -0.015225, -0.099339, -0.020301, 0.028783, 0.040398, -0.089442, 0.084383, 0.063017, -0.007024, -0.140748, -0.092928, -0.094470, 0.059939, -0.058935, 0.008218, -0.062519, -0.065203, -0.076088, -0.089426, -0.183828, 0.052770, 0.203602, -0.011581, -0.045396, -0.032463, -0.149040, -0.046479, 0.052659, 0.114449, 0.006921, -0.028044, -0.017367, 0.023014, -0.095321, 0.019176, -0.089983, -0.030397, -0.078233, -0.153997, 0.012180, 0.086310, 0.023393, -0.032796, -0.120537, -0.060967, 0.028762, 0.086869, -0.100049, -0.007324, -0.106408, 0.040427, -0.243895, -0.117082, -0.046273, 0.102738, 0.005852, 0.007075, -0.032604, -0.193993, -0.130197, 0.129241, -0.116838, -0.072585, 0.079729, -0.078080, -0.041999, 0.029594, -0.072779, -0.126294, -0.055659, -0.079019, -0.028837, -0.095580, -0.147193, 0.074517, -0.118586, 0.015103, -0.089322, -0.058657, -0.135960, 0.005646, -0.092775, -0.091004, -0.103888, 0.120119, -0.090599, -0.112464, 0.003882, 0.135997, -0.065740, -0.004524, 0.006437, 0.055991, -0.131307, -0.223452, -0.142006, -0.057358, 0.036869, -0.015637, -0.011653, -0.063010, -0.015287, 0.072202, 0.104521, 0.045976, 0.077859, -0.038655, -0.003854, 0.149065, 0.010886, -0.232655, -0.001900, -0.123595, 0.034773, -0.009831, 0.301042, -0.117149, 0.000571, 0.082511, -0.058698, -0.079616, 0.072731, 0.108994, 0.023971, -0.066944, 0.061585, 0.069256, -0.055561, -0.076621, -0.008350, 0.045620, 0.056412, 0.099333, -0.230948, 0.148187, -0.042395, 0.056823, 0.037645, 0.013312, -0.045816, 0.011055, 0.098643, -0.110136, -0.100716, 0.081780, -0.197037, -0.088115, 0.091025, -0.192107, -0.053802, 0.008341, 0.098239, 0.085699, 0.048397, 0.190262, 0.030442, 0.130937, -0.205156, 0.176640, 0.024022, -0.088851, -0.059209, -0.095086, -0.008886, 0.180888, 0.024851, 0.010996, -0.036539, 0.050505, -0.145126, -0.074018, -0.009234, 0.108677, -0.062938, -0.047595, -0.017960, 0.122506, -0.006201, -0.018038, -0.114332, -0.048185, -0.053222, -0.058988, 0.044114, -0.011181, -0.145789, 0.117762, -0.087272, 0.073601, 0.086473, 0.014948, 0.065414, 0.000650, -0.087873, -0.128354, -0.052442, -0.123583, -0.056420, -0.004889, 0.174509, -0.013745, -0.007221, -0.003066, -0.078879, 0.006186, -0.107709, -0.030281, 0.142835, 0.046912, -0.048745, -0.050122, 0.065671, 0.039466, -0.025110, -0.189800, -0.226480, 0.053123, 0.017773, -0.095201, 0.097794, -0.063037, 0.002734, -0.022990, -0.122947, 0.088302, -0.018393, -0.180220, -0.067203, -0.051048, -0.065333, 0.019381, -0.140444, 0.056243, -0.004398, -0.182621, -0.159037, -0.167475, -0.008418, 0.068923, -0.056844, -0.147843, -0.116210, -0.085442, 0.079195, 0.099822, -0.144327, 0.094009, -0.081384, -0.060649, 0.016998, 0.199694, -0.042141, 0.198868, -0.095948, -0.075815, 0.179953, 0.011689, 0.239326, -0.032547, -0.032780, 0.010052, 0.037207, 0.089992, -0.045948, -0.187183, 0.072086, 0.017030, -0.035836, -0.087403, 0.180662, -0.069168, 0.006276, 0.038186, -0.056878, 0.142921, 0.099657, -0.045116, -0.087419, -0.148103, -0.038162, 0.019169, 0.077388, -0.056695, -0.037493, -0.020136, 0.099914, -0.121570, 0.054703, 0.064205, 0.050489, -0.010780, 0.027524, 0.075874, -0.048080, 0.069841, -0.102417, -0.065552, 0.033640, 0.027987, -0.025155, -0.156780, -0.023284, 0.111467, -0.006417, -0.086030, 0.053714, 0.020301, 0.016194, 0.068523, -0.051493, 0.081536, 0.158297, 0.034957, 0.006358, 0.018162, 0.020640, 0.016813, -0.010568, -0.205984, -0.061011, 0.001346, 0.008443, -0.092324, -0.006090, 0.015777, -0.027835, 0.033577, -0.051585, -0.055377, 0.027594, 0.031313, -0.148366, 0.014201, 0.010493, 0.048482, 0.077125, -0.012654, 0.092549, 0.008562, 0.030199, 0.023611, 0.069142, 0.053781, -0.163049, -0.000133, 0.013251, -0.035728, 0.022747, -0.105374, -0.045028, -0.196962, 0.131006, 0.006144, 0.029290, 0.126556, -0.015543, 0.150530, 0.045414, 0.121202, 0.050837, -0.171679, -0.081481, 0.029984, 0.048014, -0.033187, 0.021817, 0.031392, 0.016965, 0.078594, 0.067741, 0.081425, -0.159921, -0.171153, -0.097354, 0.022828, -0.157540, -0.009406, 0.071360, -0.000631, -0.119206, 0.111214, -0.066469, -0.086637, -0.045492, -0.114606, -0.052633, -0.007726, -0.047747, -0.022396, -0.028426, -0.126415, 0.049195, 0.002687, -0.141847, 0.022937, 0.036684, -0.068669, -0.101835, 0.064099, 0.007240, -0.018940, -0.100798, 0.009113, 0.000790, -0.097238, -0.114498, 0.192273, -0.045079, 0.103229, 0.007704, -0.011364, -0.012104, 0.087041, -0.015927, 0.090098, -0.059222, 0.081910, 0.091572, 0.086598, -0.046616, -0.035103, 0.156540, -0.061884, -0.072908, 0.076041, 0.129412, -0.001335, -0.055022, -0.041472, 0.085036, 0.238408, -0.172411, -0.029131, -0.043338, 0.098533, 0.097420, 0.068324, 0.003369, 0.144564, -0.113110, 0.036866, 0.065085, -0.140976, -0.015457, -0.264892, -0.172538, -0.086837, -0.140052, -0.092725, -0.123459, -0.064725, -0.144898, -0.114623, -0.044515, 0.051203, 0.095951, -0.000326, -0.098625, 0.068854, -0.101823, -0.025034, -0.086198, -0.128810, 0.177864, -0.111816, -0.039242, -0.209717, -0.080555, -0.118023, -0.194040, -0.102224, -0.030017, -0.020062, -0.055747, -0.056429, 0.033666, -0.073263, -0.127430, -0.057474, 0.038633, -0.128287, -0.082419, -0.146422, -0.125450, -0.052868, 0.028005, 0.149110, -0.315630, -0.042470, -0.030175, 0.004027, -0.226357, 0.076013, -0.013174, -0.287556, -0.119980, -0.135386, -0.050776, -0.114635, 0.028044, 0.000797, 0.068625, -0.126666, -0.204986, -0.059138, 0.013259, 0.054025, 0.100576, -0.144145, -0.000765, -0.130619, -0.080602, -0.005661, 0.025844, -0.026360, -0.166356, -0.011122, -0.025210, -0.044296, -0.000850, -0.007747, -0.039806, 0.000258, -0.027734, 0.019946, -0.079739, -0.099749, 0.069578, -0.131105, -0.063909, -0.013895, -0.187603, -0.101891, -0.090393, -0.134948, -0.055964, -0.057362, 0.049546, -0.083203, -0.138827, 0.004827, 0.062894, -0.118345, -0.073324, -0.231309, 0.098363, -0.001489, 0.086925, -0.005904, -0.114342, 0.133563, -0.027399, -0.196428, -0.122504, -0.119819, -0.080955, -0.103332, 0.198657, 0.012993, -0.047007, -0.133247, -0.005522, -0.130070, -0.061727, 0.024574, -0.093496, 0.007829, -0.223803, -0.210533, -0.147446, -0.064746, -0.043863, -0.098864, -0.114110, 0.012128, -0.335506, 0.044120, 0.063288, -0.233319, 0.127914, -0.061419, -0.129713, -0.039740, -0.254166, -0.157280, -0.150327, 0.085651, -0.021889, 0.118274, 0.043685, -0.160147, -0.006466, -0.234645, 0.006519, 0.037762, 0.046426, -0.086013, -0.114231, -0.048374, -0.063302, 0.006059, -0.008285, -0.077581, -0.054618, -0.111957, -0.070109, 0.138427, -0.032128, -0.072798, -0.000997, -0.119978, 0.026256, -0.115372, -0.140777, 0.072710, -0.187723, 0.159242, -0.063665, -0.119789, -0.053590, -0.277490, -0.030447, -0.356573, -0.064897, 0.020795, -0.126058, 0.045316, 0.052066, -0.180215, -0.005607, -0.043249, 0.028323, 0.009398, -0.033063, -0.063835, -0.122906, -0.095392, -0.110710, -0.101390, 0.037460, 0.226113, 0.018186, -0.072250, -0.033365, -0.080758, 0.009399, 0.102396, 0.024591, -0.087461, -0.104540, -0.116771, -0.104996, 0.132594, 0.082293, -0.009524, 0.053096, -0.149920, -0.200166, -0.001056, -0.051728, 0.090337, 0.103921, -0.077180, -0.301861, 0.025497, 0.019407, 0.073053, 0.101174, -0.037411, -0.298862, -0.134744, -0.141794, -0.022005, -0.152719, 0.045792, -0.261877, 0.083849, -0.128341, -0.017284, 0.025739, 0.029738, -0.185518, -0.208471, 0.103180, -0.013372, -0.330900, -0.074685, 0.003270, 0.065553, 0.035559, -0.130103, -0.023056, -0.139922, 0.101591, -0.158741, 0.055080, -0.231822, -0.079650, 0.094480, -0.051409, 0.045299, 0.042256, 0.026897, -0.046367, -0.099795, 0.007227, -0.022356, -0.011282, -0.112858, 0.018873, 0.067624, -0.056585, -0.081169, -0.165148, -0.114437, -0.232415, -0.036487, -0.196164, 0.087172, -0.042976, 0.064888, 0.102172, 0.303409, -0.172843, 0.046969, -0.166481, -0.084826, -0.027090, 0.171673, -0.046504, 0.029131, -0.017574, -0.053770, -0.175839, -0.043938, 0.016024, -0.180871, -0.010848, 0.200308, -0.180069, 0.005208, -0.128836, 0.002064, -0.252170, -0.216304, -0.207724, -0.018993, 0.065012, 0.061515, -0.137856, -0.011988, -0.309465, -0.315914, -0.108109, 0.002665, 0.011536, 0.075810, -0.024385, 0.014519, -0.039672, 0.124800, -0.014547, 0.021928, -0.038864, 0.138569, 0.004848, -0.059984, 0.010576, -0.025638, -0.099210, -0.041970, 0.215588, -0.194097, -0.048943, -0.013924, -0.068870, -0.220416, 0.142586, -0.146905, 0.153360, -0.067491, -0.112759, 0.022120, 0.106932, 0.044462, -0.029418, -0.202806, -0.114809, 0.200607, -0.072902, -0.214482, -0.001648, 0.086889, -0.013317, -0.013571, -0.077062, -0.168446, -0.054463, -0.051107, -0.151939, 0.032932, 0.189319, -0.024154, -0.114375, -0.112284, -0.328119, -0.014826, -0.145405, -0.087581, 0.080569, -0.146653, 0.154748, 0.159002, -0.086460, -0.007152, -0.097908, -0.008685, 0.058138, 0.208937, -0.119715, -0.017410, -0.005376, 0.003257, -0.088573, 0.091213, -0.111207, 0.039732, -0.096027, -0.123630, -0.097022, -0.187856, -0.003266, -0.063513, 0.116632, 0.042576, -0.132306, 0.035968, -0.158526, -0.190426, -0.003912, 0.020829, 0.122510, -0.052195, 0.146484, 0.087997, 0.044001, 0.073593, -0.108813, -0.075088, 0.095388, 0.037019, -0.273792, 0.026839, -0.073442, -0.210495, 0.019129, -0.232859, 0.146815, -0.046741, 0.017320, 0.020348, -0.050299, -0.054666, 0.046460, 0.060872, -0.077042, 0.098824, 0.040760, 0.022170, -0.078218, 0.051636, -0.012001, -0.085569, 0.044185, 0.115231, -0.081864, 0.011335, 0.014685, 0.089162, 0.036745, 0.062234, -0.051472, -0.037219, -0.029971, -0.231880, -0.000241, 0.036978, 0.073333, -0.098013, -0.053810, 0.124634, 0.157997, 0.088890, -0.127623, 0.019619, 0.041730, 0.024505, -0.014573, -0.125266, -0.022212, 0.219509, 0.005506, -0.127630, -0.027247, -0.096824, -0.025556, 0.083390, -0.021076, 0.042209, -0.125901, 0.011533, -0.063594, -0.130421, -0.185136, 0.131994, 0.106266, -0.030181, 0.085502, -0.093897, 0.124968, -0.082045, -0.068846, 0.043847, 0.105334, -0.113730, 0.053401, 0.063131, -0.089535, 0.093130, 0.048204, 0.104308, -0.142424, 0.027159, -0.110598, 0.052054, 0.001367, 0.032786, 0.160327, -0.087648, 0.067394, 0.035020, -0.065429, 0.048780, -0.041647, -0.040351, 0.121424, 0.148209, -0.193111, 0.066293, -0.006282, -0.111747, -0.005000, -0.146356, -0.095410, 0.094269, -0.111642, -0.050712, 0.022213, -0.017634, -0.145786, 0.072267, -0.150918, 0.034268, -0.090332, -0.040167, -0.156023, -0.074330, -0.083086, -0.123274, -0.024438, 0.141351, -0.005383, -0.044570, -0.061290, -0.119689, -0.055002, -0.083614, -0.052771, 0.052133, -0.097950, -0.043821, -0.106170, -0.096665, 0.012634, 0.082648, -0.021326, 0.144572, -0.049131, -0.107077, -0.020586, 0.072495, 0.098553, -0.051630, 0.063362, -0.054651, -0.131793, 0.061277, -0.047336, 0.037379, -0.020771, 0.036366, 0.036593, -0.048478, -0.027250, 0.104620, -0.108648, -0.158777, 0.110846, -0.005068, 0.008111, 0.045939, 0.053768, 0.040048, -0.096292, 0.054286, -0.114353, 0.010208, 0.106353, -0.144829, 0.020434, 0.074855, 0.119019, -0.053286, -0.008488, -0.103839, 0.036764, -0.000070, -0.035142, 0.009090, -0.014071, -0.128918, 0.005766, -0.032582, 0.034803, -0.006882, 0.133174, 0.044744, -0.068487, 0.022517, 0.049658, 0.072306, -0.004770, -0.087140, -0.063559, 0.008583, 0.049436, 0.051727, -0.031735, -0.029976, -0.070912, -0.034001, -0.037397, 0.044040, 0.207507, 0.020507, 0.095356, 0.056654, 0.039653, -0.060179, -0.119750, -0.115024, -0.094896, -0.132547, -0.101931, -0.038158, -0.073108, 0.072212, -0.123874, 0.111975, 0.088059, -0.124721, 0.143998, -0.025335, -0.126462, 0.099949, -0.016275, 0.086109, -0.004575, -0.025938, -0.076762, -0.053855, 0.094594, -0.012556, 0.087268, -0.050210, -0.047327, 0.039121, 0.078019, -0.005885, 0.042432, 0.007261, -0.023861, 0.224663, 0.142011, -0.016769, -0.007429, 0.164840, -0.152078, -0.014466, 0.002572, -0.115958, 0.098253, -0.011385, -0.044056, 0.009027, 0.129893, 0.061922, -0.022035, 0.186615, -0.000073, 0.141756, 0.084808, 0.003508, -0.081698, -0.035101, -0.116988, 0.042002, 0.009418, -0.013718, 0.047286, 0.025344, -0.063428, 0.088763, -0.123346, -0.111451, 0.054829, 0.031355, -0.081177, -0.182718, 0.034034, 0.059490, -0.006843, 0.142535, 0.111406, -0.012147, 0.055432, -0.054504, -0.135127, 0.112777, 0.004268, -0.061062, 0.043770, -0.044478, -0.098413, 0.073492, 0.319674, -0.014689, -0.034863, 0.131306, 0.139425, 0.103436, 0.088272, 0.235512, 0.023117, 0.090608, -0.010494, 0.005047, -0.084895, -0.048561, -0.038816, -0.114244, -0.109486, -0.068393, 0.113406, -0.090134, -0.016923, -0.029299, 0.017868, 0.040263, 0.019540, -0.150504, 0.169218, -0.017004, 0.020849, -0.112316, -0.184766, 0.057643, 0.056987, 0.033227, 0.023021, -0.123774, -0.154481, 0.042191, 0.000653, -0.097147, -0.050058, -0.026749, 0.064931, 0.069953, 0.046502, 0.044236, -0.167552, -0.060823, -0.110611, -0.159662, -0.049604, 0.031204, 0.079793, 0.002569, 0.036423, 0.058794, 0.117131, -0.050037, 0.057604, -0.008873, -0.028066, 0.064386, -0.063293, -0.061512, -0.072607, 0.098283, 0.052157, 0.001221, 0.059973, -0.005298, 0.043624, 0.047253, -0.048420, -0.031213, 0.042534, -0.149944, -0.052202, -0.002280, 0.046402, 0.012315, 0.115900, 0.073398, -0.166132, -0.124693, 0.099770, -0.011429, 0.039417, -0.120794, -0.158759, -0.122621, 0.009395, 0.029634, -0.156439, -0.135071, -0.128133, 0.115241, -0.144677, -0.021830, -0.112742, 0.032523, -0.262314, 0.034590, -0.033029, 0.035494, -0.038533, 0.079640, 0.008694, -0.051302, -0.044283, 0.064450, -0.031807, 0.053055, 0.097237, 0.042648, 0.000384, -0.094690, -0.166451, 0.046412, 0.070720, 0.073316, -0.084634, 0.047709, -0.239416, -0.124602, -0.067630, 0.020254, -0.023486, 0.036692, -0.055375, -0.077138, 0.129559, -0.141131, -0.047192, 0.062662, -0.195406, 0.088210, 0.017168, -0.022314, -0.052856, 0.153003, -0.056973, -0.066251, 0.066309, 0.062606, 0.078728, -0.297286, -0.081967, 0.023710, -0.033878, -0.058844, 0.054432, 0.067807, -0.087084, -0.083485, 0.143145, -0.114645, 0.023530, 0.048225, -0.136428, -0.079731, -0.074615, -0.178922, -0.123255, -0.047962, 0.013337, -0.051563, -0.054193, -0.050811, -0.162173, -0.121398, -0.183156, 0.187894, 0.008621, -0.153930, -0.118663, -0.038507, 0.161521, -0.069295, -0.149330, -0.224511, -0.003808, -0.029747, -0.289938, 0.032667, -0.053238, -0.154684, 0.000453, -0.073604, -0.001724, 0.047152, -0.125736, 0.012341, 0.002597, 0.041347, -0.070002, -0.048247, -0.093059, 0.042576, -0.073749, -0.016040, 0.060410, -0.195470, -0.085548, -0.119734, -0.159171, -0.319789, -0.018487, -0.626564, -0.016003, 0.088327, -0.085532, -0.018246, -0.051617, 0.071317, -0.063225, 0.122775, -0.172504, -0.091489, 0.049888, -0.075953, 0.134867, -0.144049, 0.108604, 0.047871, 0.087818, -0.041900, 0.031292, -0.002934, 0.036808, -0.056041, -0.059825, -0.038628, 0.002603, -0.008547, -0.105059, -0.206157, -0.098739, -0.193445, 0.086864, 0.059251, -0.066920, 0.023428, -0.103385, -0.097081, -0.059656, -0.169270, -0.039941, -0.105427, 0.132769, -0.126796, -0.035689, -0.157995, 0.063593, -0.029832, -0.224695, -0.100722, 0.061674, -0.083221, -0.067585, 0.094120, -0.226442, 0.138540, 0.030094, -0.001416, -0.164976, 0.102223, 0.015459, -0.012040, 0.166538, -0.142366, -0.062807, -0.011126, 0.102174, -0.083752, 0.042821, -0.119965, -0.029805, -0.083186, -0.041284, -0.127005, -0.077351, -0.148377, 0.020705, -0.051571, 0.031844, 0.054288, 0.057469, 0.069216, -0.050238, -0.043341, -0.097071, -0.104340, -0.017767, 0.041043, -0.012445, 0.045976, 0.055746, -0.062553, -0.047000, -0.056158, -0.131645, 0.057907, 0.005742, -0.061001, -0.147506, -0.031342, 0.051445, -0.065412, 0.027596, -0.077090, -0.092711, -0.002430, -0.000444, -0.082416, 0.043164, -0.123388, -0.046560, -0.079136, 0.011618, -0.095979, -0.058403, -0.069843, -0.096465, -0.017204, -0.038658, 0.089457, -0.021161, -0.027565, -0.065393, -0.262026, 0.012883, -0.101654, -0.120478, -0.038934, -0.040409, -0.011444, -0.071711, -0.102037, 0.013506, 0.081680, -0.082036, -0.085067, -0.086826, 0.033351, -0.015285, -0.083640, -0.187659, -0.122888, -0.022320, -0.029890, -0.166167, -0.028456, -0.168796, -0.071603, -0.180286, 0.012693, -0.016465, -0.000063, -0.146358, 0.173835, 0.064508, 0.076978, -0.201600, -0.137956, -0.119975, 0.009569, -0.158353, -0.067119, -0.062812, 0.156281, -0.015490, -0.018155, -0.123895, -0.041568, -0.139720, -0.096152, -0.034203, -0.128847, 0.048350, -0.064013, -0.207451, 0.004381, 0.080400, -0.141267, -0.063710, -0.122039, -0.035976, 0.096996, -0.010773, 0.046690, 0.088024, 0.046785, 0.038018, 0.117536, -0.011783, -0.003247, 0.043259, -0.060701, -0.050550, 0.007811, -0.063064, -0.041960, 0.205912, -0.063435, 0.109991, -0.106448, 0.068030, -0.031924, -0.001924, -0.057255, 0.015473, -0.011475, -0.141963, 0.010375, 0.048496, -0.001422, 0.074690, -0.118031, -0.101558, -0.081115, 0.015006, -0.081355, -0.076941, -0.062571, 0.009652, 0.003217, -0.084683, 0.097153, 0.013865, 0.021300, 0.032038, 0.021048, 0.049479, 0.039318, -0.063665, -0.202813, -0.086950, -0.024727, -0.017493, -0.007479, -0.143613, 0.027621, -0.056599, -0.051189, -0.051507, 0.052340, -0.020270, 0.035039, -0.060797, 0.026651, 0.038132, 0.021531, 0.032477, -0.057881, -0.017224, -0.055117, -0.108346, -0.216217, -0.013075, 0.009472, -0.003296, -0.089656, 0.025249, -0.114271, 0.066570, 0.038608, -0.017282, -0.177246, -0.119507, 0.059125, -0.067722, -0.009919, 0.056962, -0.067141, -0.101812, -0.029608, 0.032694, 0.068243, -0.000433, -0.086981, 0.039530, -0.095010, 0.056209, 0.076421, -0.119419, -0.039165, -0.059588, 0.002516, -0.076253, -0.016761, -0.046063, -0.060866, 0.075955, 0.013156, 0.062908, -0.027570, -0.135372, 0.001713, 0.094290, -0.054661, 0.119489, -0.131187, 0.025826, -0.119147, 0.046337, -0.001914, 0.044719, -0.037244, 0.127645, 0.040080, -0.014423, -0.143227, 0.090531, -0.178846, 0.021590, 0.040406, -0.079063, 0.026601, -0.010506, 0.014926, -0.119470, 0.038131, -0.048186, 0.002609, -0.023055, -0.155723, -0.055834, -0.113579, -0.048969, -0.029402, -0.036580, 0.026898, -0.046316, -0.157280, 0.044270, -0.059158, 0.015900, -0.073120, 0.046763, -0.102147, -0.063723, 0.055292, 0.024823, -0.028145, -0.043777, -0.093944, -0.133037, -0.062470, 0.008701, -0.052159, 0.030944, -0.051699, -0.051668, -0.015958, -0.031047, -0.059058, -0.147072, 0.046258, -0.000174, 0.048761, -0.011584, 0.051253, -0.096969, -0.118455, 0.069695, 0.142756, 0.027470, -0.080092, 0.100967, 0.064689, -0.160315, -0.081796, -0.086795, -0.049915, 0.002290, -0.014488, 0.062998, -0.035992, -0.009296, 0.165448, -0.004495, 0.065724, 0.107353, 0.051067, 0.071488, -0.020762, 0.080545, -0.118882, -0.119751, 0.024417, 0.027475, -0.018608, -0.044010, -0.002760, 0.097684, 0.045337, -0.136637, 0.108691, -0.143127, -0.122969, -0.015272, 0.041429, -0.054743, -0.141258, -0.034097, -0.103939, -0.057863, -0.084833, -0.074406, -0.059474, -0.011251, -0.073537, -0.144648, -0.058479, 0.092989, -0.035178, -0.043441, 0.111912, -0.109631, 0.020343, 0.016698, -0.062098, -0.128051, -0.064220, 0.030055, -0.056820, -0.039329, -0.168408, 0.057078, 0.033860, -0.069066, -0.123978, -0.116058, -0.085135, 0.088791, 0.086112, 0.098614, -0.005947, -0.046083, -0.089463, 0.034754, -0.156966, -0.006916, 0.041890, -0.059181, 0.016779, -0.049161, -0.109398, -0.054211, -0.090455, 0.076875, -0.037148, 0.002375, -0.033930, -0.093772, -0.022852, 0.018437, 0.130475, 0.054919, 0.013709, 0.011967, 0.077303, 0.012336, 0.078669, -0.129750, 0.102932, -0.023189, -0.031697, 0.035111, 0.092974, 0.089535, -0.083402, -0.013156, 0.054999, -0.130631, 0.024679, 0.001906, 0.025523, -0.051373, 0.136428, 0.128548, 0.008477, -0.022303, 0.073909, -0.074735, -0.033012, -0.122059, -0.169483, 0.009366, 0.012172, -0.002931, -0.091137, 0.089818, 0.033664, -0.037643, -0.131350, 0.095172, -0.038716, -0.130252, 0.004223, -0.102319, -0.036268, -0.127171, 0.046265, 0.097091, -0.034949, 0.025319, -0.065355, 0.055124, -0.123838, -0.037531, -0.136009, -0.140880, 0.088014, -0.056641, -0.056317, 0.049937, 0.012152, -0.052769, -0.062792, -0.039326, -0.047608, 0.017642, 0.050527, -0.027137, -0.009560, -0.042909, -0.030200, -0.067567, -0.119840, 0.017457, 0.005499, -0.007811, 0.187889, -0.003186, -0.046063, 0.041159, -0.102694, 0.122644, 0.042180, 0.107466, 0.090559, -0.006209, 0.030193, -0.067974, -0.044065, -0.130097, -0.040443, -0.122496, -0.136276, -0.000649, 0.116848, -0.016801, -0.028447, 0.013389, -0.043188, -0.036511, 0.028283, -0.062417, 0.027036, -0.120594, -0.002333, 0.070967, -0.054388, 0.018201, 0.015261, 0.025636, -0.059295, -0.025982, -0.084231, 0.043152, 0.019074, -0.087492, -0.013312, -0.092845, -0.070769, 0.059219, 0.033459, 0.162598, 0.064315, 0.183785, 0.031006, -0.006333, -0.003131, 0.046204, -0.110215, -0.099539, -0.098509, 0.030745, -0.161797, 0.016614, -0.000388, 0.015044, -0.119548, 0.108370, -0.397339, -0.012778, 0.052810, -0.024348, 0.095160, 0.196797, -0.056869, 0.025944, 0.173588, -0.052163, -0.213647, -0.025256, -0.025646, -0.123423, 0.053126, 0.107599, -0.034810, -0.080587, -0.120472, 0.058810, -0.184728, 0.024865, 0.044790, 0.042009, 0.048896, -0.085552, -0.110579, 0.038470, -0.016227, -0.008406, -0.202112, -0.119611, -0.161826, -0.058248, 0.150939, 0.059193, -0.191560, -0.004286, -0.259217, -0.082246, 0.041865, 0.023771, 0.109477, -0.060882, 0.026517, 0.069648, -0.007305, 0.105324, -0.093030, -0.182956, -0.144427, -0.096240, -0.230159, 0.079684, 0.129366, 0.003366, -0.057048, -0.008006, 0.092950, -0.082185, 0.130175, -0.241085, -0.091307, -0.039872, -0.014155, 0.036317, 0.157002, -0.006737, 0.106762, 0.092124, -0.133884, -0.055496, 0.069691, 0.178231, -0.134189, 0.074596, 0.122251, 0.022753, 0.004061, 0.079788, 0.036350, -0.097318, -0.164269, 0.097166, -0.132568, -0.108078, 0.037892, -0.177671, -0.015179, -0.073252, 0.030956, -0.132980, -0.125278, 0.196279, 0.016370, 0.017795, -0.049607, -0.131027, 0.033830, -0.013042, -0.097533, 0.013605, 0.078480, 0.035547, -0.044169, 0.003490, -0.095766, 0.068880, -0.085376, -0.050713, -0.118229, 0.016630, -0.018520, 0.062152, -0.077559, 0.077275, 0.017308, -0.140532, 0.041092, 0.014014, 0.037244, -0.175109, 0.090930, 0.013060, -0.109352, -0.043978, -0.081565, -0.072914, -0.111879, -0.102173, 0.015045, 0.106707, 0.000068, 0.070332, -0.160778, 0.055912, -0.006693, 0.000020, 0.000077, -0.036832, 0.028168, 0.056064, 0.093591, 0.111056, -0.090609, -0.055889, -0.068857, -0.035164, 0.036351, 0.054321, 0.018916, -0.122858, -0.009357, 0.050623, -0.172289, 0.121567, 0.062455, 0.003870, 0.129442, 0.084123, -0.063105, 0.028788, 0.135756, -0.007792, -0.003796, 0.030584, 0.070598, -0.029652, -0.037425, -0.066969, 0.014291, 0.009750, 0.071065, -0.050245, -0.136927, -0.030345, 0.060301, -0.175132, 0.029869, -0.216435, 0.094437, 0.146192, 0.030263, 0.064947, 0.145231, 0.183106, 0.126476, 0.006988, -0.018450, -0.085893, -0.127645, -0.056796, -0.113121, -0.101139, -0.027167, 0.047222, -0.080871, 0.074965, 0.036502, 0.176833, -0.064102, -0.041790, -0.047969, 0.088304, -0.119337, -0.090329, 0.163074, 0.018248, -0.070720, 0.024215, -0.016098, 0.021752, -0.095479, -0.122623, -0.024726, -0.038904, -0.101323, -0.067171, 0.045864, -0.100362, -0.124543, -0.090657, 0.106668, 0.020179, -0.149289, 0.087140, 0.049306, 0.233262, 0.012233, 0.005295, 0.149258, -0.020395, -0.127182, 0.008304, -0.125530, 0.002086, 0.186914, 0.034930, 0.122771, -0.007437, 0.031366, -0.229437, -0.052303, 0.212441, 0.126160, 0.056481, -0.024820, -0.024745, 0.002341, 0.022120, -0.009208, 0.031914, 0.203713, 0.275215, -0.200065, 0.018702, -0.019419, 0.074721, -0.088488, -0.072263, 0.031979, 0.005109, 0.010994, -0.066002, 0.029295, -0.032066, -0.082980, -0.133413, -0.107219, 0.073397, -0.000443, 0.085402, 0.026227, 0.105194, -0.146557, -0.037184, -0.108570, 0.128444, -0.097772, 0.049894, -0.122560, -0.003005, 0.076969, -0.013453, 0.027080, -0.061665, 0.045820, -0.169484, -0.014029, -0.116217, -0.028079, -0.106242, -0.084458, -0.279807, -0.067807, 0.096201, -0.066272, 0.050224, -0.039634, -0.154735, 0.092728, -0.027871, 0.024026, -0.045299, 0.138388, -0.097102, -0.129354, 0.076796, 0.078089, 0.005222, -0.003454, -0.148204, 0.005941, 0.115183, 0.013401, -0.123154, -0.045274, -0.049612, 0.041300, -0.043549, -0.145589, 0.079408, 0.016954, 0.065091, -0.063699, -0.089196, -0.086750, 0.051602, -0.036011, -0.071652, 0.090572, -0.216039, -0.030570, 0.048123, -0.104164, -0.037933, -0.037210, -0.063680, 0.064813, 0.001923, 0.025099, -0.067784, -0.246227, -0.026268, -0.020930, -0.012415, -0.147000, -0.019543, -0.020581, -0.074924, -0.011693, -0.047584, -0.041623